(* IEC 61131-3 sources: ml2plc/benchmarks/st (part 6) *)

    weights_3_u : ARRAY[0..4095] OF REAL := [-0.726234972, -0.82971102, 0.359873623, 0.467501462, -0.795098782, 0.642522633, -0.834418893, -0.800529778, 0.752689779, 0.406455636, 0.616274774, 0.617786705, -0.741933465, 0.632032633, -0.739187837, -0.503853142, 0.545782745, 0.567466497, -0.337621212, -0.339030087, -0.389321893, 0.674896181, 0.789721549, -0.746486127, -0.669301271, 0.820195556, 0.72258997, -0.971024632, -0.772712708, 0.568969786, 0.828069806, -0.664833724, -0.332123041, -0.638633251, -0.857070208, -0.492956102, -0.802621424, 0.136594638, -0.361942023, -0.667052031, 0.616791487, 0.744978189, -0.954466581, -0.57189548, 0.74708873, 0.656679034, 0.282293171, 0.660095751, -0.696134508, 0.818064272, 0.902193606, -0.636808872, -0.692610443, 0.638984621, -0.867889166, 0.462693274, -0.667061865, -0.625101268, -0.593671858, -0.351741135, 0.234290212, -0.588220656, -0.595141947, -0.701019764, -0.372747988, -0.607375026, 0.464761764, 0.530245066, -0.573789001, 0.530546367, -0.433061302, -0.461016506, 0.59694773, 0.0462750606, 0.332048684, 0.404971868, -0.498975754, 0.562286198, -0.327837288, -0.52094245, 0.35660404, 0.363930374, -0.340805382, -0.0284396466, -0.445062369, 0.1347083, 0.55759269, -0.618813932, -0.599301457, 0.350034744, 0.372941881, -0.528004527, -0.534632623, 0.234335199, 0.397439361, -0.0195646528, -0.0915857852, -0.0818935558, -0.397882402, -0.0978519842, -0.491226345, -0.166510537, -0.00829036627, -0.282786936, 0.626897216, 0.404613793, -0.491245329, -0.337422758, 0.430924863, 0.278444827, 0.0179173294, 0.231050387, -0.347322822, 0.3725501, 0.48292917, -0.507511616, -0.393044561, 0.602047801, -0.562717617, 0.321077079, -0.230540395, -0.587909281, -0.0499534346, -0.369197726, -0.169617653, -0.41201207, -0.260386378, -0.412834316, -0.803556919, -0.740769684, 0.440442294, 0.568141937, -0.475784481, 0.644459307, -0.596662343, -0.940275252, 0.656770587, 0.322523296, 0.875917017, 0.875438809, -0.816106558, 0.825712204, -0.592998028, -0.347098321, 0.495246083, 0.658055961, -0.403978735, -0.0876639634, -0.502450585, 0.64121145, 0.575357795, -0.643270314, -0.996893167, 0.557650566, 0.867267251, -0.850942194, -0.756620347, 0.329067886, 0.669194162, -0.383174628, -0.0802536532, -0.551262677, -0.718719363, -0.598996222, -0.631955266, -0.0989504158, -0.0885992125, -0.713463306, 0.518353522, 0.730688989, -0.800943017, -0.605422258, 0.701749504, 0.95046109, -0.0751864091, 0.87148875, -0.567332923, 0.663198709, 0.649199545, -0.935164213, -0.753644347, 0.803934813, -0.580185413, 0.378011674, -0.636774302, -0.702305377, -0.344566911, -0.367477775, 0.00891227275, -0.607614458, -0.661959112, -0.687778234, -0.625213504, -0.534323871, 0.356132567, 0.448352844, -0.662155986, 0.502999783, -0.572085738, -0.688427746, 0.490987062, 0.707427204, 0.605727017, 0.829243064, -0.728774309, 0.576677978, -0.878341854, -0.301144749, 0.548745811, 0.666547835, -0.0080199372, -0.474185884, -0.431044191, 0.850138128, 0.552011251, -0.779790699, -0.770057082, 0.645845652, 0.763373435, -0.612323225, -0.813291967, 0.79515928, 0.696035445, -0.785743177, -0.688787401, -0.600066721, -0.71572578, -0.727747619, -0.471354902, 0.656914413, -0.512712061, -0.605490208, 0.525177181, 0.528167665, -0.758861125, -0.702212036, 0.415254414, 0.783526659, 0.741826832, 0.719366014, -0.687756479, 0.683343053, 0.737960219, -0.525721431, -0.455234349, 0.570235014, -0.521014452, 0.321572721, -0.731491745, -0.51282382, -0.718585134, -0.164967939, 0.67603749, -0.509025753, -0.7481004, -0.456257671, -0.669510841, -0.814430475, 0.570815623, 0.526050806, -0.529686749, 0.621858954, -0.670453012, -0.304120302, 0.726401627, -0.0356775187, 0.260329664, 0.624240518, -0.748086572, 0.772515833, -0.125408188, -0.57220155, 0.498111188, 0.0558861159, -0.435518563, 0.303609818, -0.723968267, 0.32118696, 0.692383528, -0.775559604, -0.599537134, 0.294759721, 0.716790199, -0.824359059, -0.780710399, 0.106178224, 0.59846735, -0.206296533, 0.128306508, -0.146541059, -0.224539533, -0.0289100092, -0.765631378, -0.220809624, 0.142412528, -0.384071648, 0.592445076, 0.540259898, -0.638875484, -0.205305457, 0.619496822, 0.442066103, -0.0485938378, 0.466518402, -0.158942863, 0.672467291, 0.807129443, -0.740897119, -0.669203401, 0.666509151, -0.744766951, 0.648471951, -0.381909788, -0.573550165, 0.188253239, -0.540039003, -0.318327606, -0.523213089, -0.323695183, -0.519757688, -0.785824299, -0.818390846, 0.508213222, 0.483413875, -0.783533275, 0.773789883, -0.734820127, -0.79764092, 0.595962107, 0.348774403, 0.728198171, 0.80280596, -0.905285239, 0.696726441, -0.556371629, -0.303590208, 0.505447924, 0.654682875, -0.246009961, -0.223182008, -0.24971877, 0.70417136, 0.801208556, -0.83401686, -0.837068319, 0.727295339, 0.710075676, -0.732324839, -0.919261158, 0.631765366, 0.908012867, -0.489900053, -0.275408089, -0.695942461, -0.762747347, -0.440948963, -0.733398139, 0.183654517, -0.027274197, -0.62028116, 0.811902761, 0.743571997, -1.0051589, -0.525409877, 0.59080416, 0.890070081, 0.162616029, 0.72517395, -0.71613127, 0.769188046, 0.83349818, -0.766713858, -0.669896007, 0.711548209, -0.647645533, 0.33983916, -0.509689867, -0.800435543, -0.344411999, -0.346289754, 0.314366817, -0.663431704, -0.645073771, -0.560695171, -0.580787599, -0.820379198, 0.494530648, 0.398333371, -0.511259377, 0.692627907, -0.654955804, -0.870129108, 0.622329593, 0.41138804, 0.681844473, 0.7009812, -0.699940562, 0.538193107, -0.626960039, -0.446550846, 0.611533403, 0.669651389, -0.173716933, -0.318383664, -0.307127029, 0.626539707, 0.756940067, -0.76652962, -0.840944767, 0.790242732, 0.646067619, -0.767073929, -0.862344623, 0.598574519, 0.593686044, -0.577582955, -0.0423634201, -0.574055374, -0.77169019, -0.707057357, -0.778539598, 0.205691278, -0.00679121865, -0.854793429, 0.703709006, 0.763270438, -1.00914109, -0.775699973, 0.657759905, 0.725754857, 0.0530802906, 0.774340749, -0.833031714, 0.78519094, 0.71297121, -0.876600504, -0.740658998, 0.718503237, -0.687330544, 0.385003448, -0.725991547, -0.754310906, -0.279794812, -0.459310025, 0.188008204, -0.733313024, -0.775156617, -0.419203967, -0.273565292, -0.338725805, 0.221741572, 0.281494081, -0.342794389, 0.295483947, -0.291649103, -0.420268297, 0.387898266, 0.168785974, 0.339827657, 0.513234437, -0.494564533, 0.233384728, -0.230191156, -0.308273941, 0.325547248, 0.405156314, -0.0751813129, -0.066444248, -0.128334582, 0.244734526, 0.429480523, -0.436590225, -0.505181551, 0.468694657, 0.35836184, -0.543859482, -0.418227315, 0.220673606, 0.348470032, -0.428927124, -0.277986884, -0.291793585, -0.206854329, -0.250032306, -0.438212544, 0.218785331, 0.0412712507, -0.282670617, 0.316561878, 0.467533499, -0.459543943, -0.365904897, 0.383837134, 0.291643828, 0.1889994, 0.21689266, -0.294608653, 0.276400536, 0.293337226, -0.420555532, -0.405189395, 0.228911266, -0.250243455, 0.240290195, -0.447692513, -0.475426018, -0.201851323, -0.297056526, 0.137493655, -0.48626101, -0.345898688, -0.396780074, -0.780549526, -0.823537588, 0.542945087, 0.354397655, -0.507387161, 0.698669791, -0.818379283, -0.727007926, 0.678681433, 0.212808281, 0.604210854, 0.803043723, -0.779703319, 0.685046077, -0.663781881, -0.521312237, 0.596160948, 0.652478755, -0.35376817, -0.15544413, -0.422452629, 0.534026861, 0.805908442, -0.847195268, -0.851938188, 0.799646616, 0.857016563, -0.839247882, -0.884811521, 0.510792196, 0.88849473, -0.392984003, -0.261963129, -0.586921692, -0.646880448, -0.462142944, -0.818890929, 0.035946276, -0.281571209, -0.74871695, 0.613813758, 0.680141926, -0.949269414, -0.684969604, 0.565539658, 1.00042653, 0.150313571, 0.684495986, -0.722136557, 0.778911769, 0.782094896, -0.730289161, -0.794239044, 0.885579526, -0.69606334, 0.444901079, -0.845269442, -0.598321259, -0.542192876, -0.288296878, 0.215937302, -0.722411454, -0.702072799, -0.705431938, -0.71226716, -0.786647379, 0.531604886, 0.609665036, -0.597535908, 0.666882694, -0.793303609, -0.787642837, 0.698806942, 0.348492414, 0.540394783, 0.626096666, -0.706491232, 0.829213083, -0.538429081, -0.65759629, 0.687242925, 0.430694371, -0.264121145, -0.216645733, -0.692179024, 0.672817349, 0.805104256, -0.622378051, -0.844789565, 0.451787233, 0.719521761, -0.836445928, -0.842959404, 0.355159968, 0.653186679, -0.37796697, -0.291634262, -0.63452822, -0.671194732, -0.504214764, -0.844722986, 0.306022525, -0.0711536258, -0.702196002, 0.737235725, 0.809727132, -0.613162577, -0.383354962, 0.606713057, 0.591403484, 0.339256108, 0.54715246, -0.473906338, 0.783900678, 0.663366318, -0.75187254, -0.493442833, 0.800020874, -0.789069772, 0.564043283, -0.611755073, -0.86263907, -0.336834759, -0.462656617, 0.237991378, -0.707368851, -0.405766249, -0.630902052, -0.821267247, -0.829749942, 0.509847701, 0.460671842, -0.807606995, 0.74302882, -0.736985207, -0.782585621, 0.754141986, 0.416912496, 0.794934273, 0.86178571, -0.872833729, 0.614410043, -0.788762808, -0.349991858, 0.646541595, 0.541881561, -0.174803972, -0.426443964, -0.381490558, 0.821741939, 0.750299513, -0.836915433, -0.74960041, 0.727819622, 0.92942059, -0.863370955, -0.941732585, 0.573167384, 0.670918107, -0.577338278, -0.318402857, -0.76259917, -0.771713018, -0.665239751, -0.721295357, 0.246406525, -0.497510284, -0.683297992, 0.660865605, 0.732286155, -0.704380989, -0.739708781, 0.889108539, 0.684882641, 0.533998311, 0.649343133, -0.691442072, 0.747027636, 0.723184109, -0.669957519, -0.683325231, 0.681482494, -0.914686978, 0.17408444, -0.640013218, -0.716807425, -0.482498884, -0.154035002, 0.310868859, -0.874958694, -0.748723865, -0.56742239, -0.887781858, -0.652014136, 0.452641785, 0.549586773, -0.645061731, 0.63546443, -0.579267085, -0.748191714, 0.554392397, 0.467173159, 0.758127451, 0.917132854, -0.757915795, 0.769090831, -0.851054728, -0.255667329, 0.637966394, 0.573545754, -0.222050503, -0.438768119, -0.314697772, 0.606786788, 0.856207848, -0.851828158, -0.720914125, 0.806266189, 0.729975462, -0.809783995, -0.858449399, 0.63611263, 0.791059971, -0.416043282, -0.307958245, -0.517980218, -0.714065015, -0.545959234, -0.723166049, 0.29447791, -0.254560858, -0.749505579, 0.825292349, 0.793439567, -0.854955912, -0.56521672, 0.660036385, 0.849229217, 0.315747947, 0.638653874, -0.577628732, 0.616680264, 0.968390405, -0.862338424, -0.541128039, 0.630861163, -0.679648817, 0.262172341, -0.719775438, -0.644159377, -0.345081747, -0.21565415, 0.271060109, -0.728009224, -0.683839321, -0.481576353, -0.570552051, -0.777552724, 0.622478604, 0.579048872, -0.596874118, 0.700840712, -0.657557487, -0.895704746, 0.521527052, 0.291102052, 0.669102132, 0.621534884, -0.792802751, 0.641864598, -0.615286052, -0.564382076, 0.658665776, 0.569696784, -0.29823938, -0.0890338346, -0.522620618, 0.498231977, 0.794570863, -0.825930715, -0.709672213, 0.49634099, 0.715287268, -0.878186584, -0.740223408, 0.342125803, 0.71430409, -0.333702475, -0.176821321, -0.435841233, -0.795084834, -0.508588672, -0.649351716, -0.0135515844, -0.00657207659, -0.628678024, 0.758297741, 0.722372234, -0.989041865, -0.492844343, 0.558204472, 0.986102402, 0.104362853, 0.769734919, -0.783679724, 0.814909697, 0.65221858, -0.909674704, -0.94838649, 0.790295839, -0.832857609, 0.358761221, -0.695959747, -0.763435304, -0.301868916, -0.560335457, -0.073698774, -0.803123415, -0.589908421, -0.699640691, -0.89512831, -0.89859134, 0.456811368, 0.526388049, -0.883316159, 0.668905437, -0.864467144, -0.77936691, 0.668658853, 0.686980963, 0.708051503, 0.897727907, -0.782424867, 0.870139658, -0.710069895, -0.290644497, 0.861719429, 0.686867714, -0.0812829584, -0.515805244, -0.619343758, 0.87452513, 0.647835255, -0.735748649, -0.724878669, 0.730390191, 0.706322849, -0.945946515, -0.875465572, 0.565879285, 0.718600035, -0.742332637, -0.467122614, -0.813044608, -0.77358681, -0.570550144, -0.745883226, 0.471848935, -0.442510426, -0.769583106, 0.646922112, 0.724060833, -1.03937078, -0.738261163, 0.878113747, 0.91464299, 0.451797158, 0.864410758, -0.641917169, 0.683274686, 0.916965365, -0.788966, -0.736622751, 0.830067337, -0.689770639, 0.21498701, -0.684152961, -0.942618608, -0.576527417, -0.366254419, 0.413313627, -0.873114645, -0.718489408, -0.583863616, -0.729837894, -0.627582729, 0.446807176, 0.410488844, -0.707820356, 0.574976921, -0.890346527, -0.6144858, 0.741384029, 0.301623613, 0.731503785, 0.6993469, -0.782861829, 0.707979858, -0.698563576, -0.491824239, 0.807846844, 0.705500066, -0.118933909, -0.514284432, -0.541995108, 0.544251263, 0.638027668, -0.623156488, -0.679441869, 0.760259151, 0.714749157, -0.856507719, -0.740746558, 0.407242507, 0.653954327, -0.48238948, -0.237410322, -0.433872312, -0.78880173, -0.499718726, -0.948717713, 0.38727656, -0.382465541, -0.525140166, 0.694271028, 0.800766528, -0.854491174, -0.519459486, 0.69115299, 0.829451561, 0.367598891, 0.702863634, -0.566851914, 0.780456722, 0.797254324, -0.647499442, -0.79959631, 0.792972267, -0.824902415, 0.502618432, -0.768850267, -0.846130311, -0.492772669, -0.54319489, 0.261164606, -0.788439989, -0.598921239, -0.816673398, -0.778527617, -0.844715834, 0.340323418, 0.428646266, -0.54244858, 0.792509854, -0.643731296, -0.842107594, 0.733490527, 0.408700466, 0.724223852, 0.683781266, -0.885363996, 0.572960675, -0.702454209, -0.350052059, 0.623003006, 0.453214765, -0.112270817, -0.282705426, -0.403194994, 0.685073912, 0.766042054, -0.868627787, -0.765646458, 0.69943887, 0.751629233, -0.739947796, -0.768767118, 0.463029802, 0.651656747, -0.593756258, -0.41636619, -0.488620043, -0.625012338, -0.534433126, -0.712874651, 0.208950907, -0.133826539, -0.598224044, 0.815514505, 0.730447471, -0.830714822, -0.623293459, 0.772215545, 0.647283673, 0.318770945, 0.789138079, -0.700474203, 0.864484668, 0.667024732, -0.678884387, -0.587849855, 0.697911382, -0.829990804, 0.179155171, -0.727644086, -0.696924448, -0.538560808, -0.416034847, 0.502129376, -0.694367468, -0.645184517, -0.723423243, -0.49315697, -0.625419617, 0.38362208, 0.653656721, -0.661024809, 0.622956514, -0.517229497, -0.238649622, 0.600716591, -0.0996971205, 0.362163216, 0.714113176, -0.630294204, 0.537375927, 0.00633827038, -0.446282089, 0.578546643, 0.0746347681, -0.4034895, 0.143355817, -0.42931506, 0.271517873, 0.443827868, -0.597008765, -0.408510149, 0.279152721, 0.637251139, -0.680869997, -0.600134134, 0.105825603, 0.446815252, -0.0732483864, 0.131000474, -0.18368794, -0.113074012, -0.129835978, -0.52116704, -0.341600209, 0.373502314, -0.0196969714, 0.633913875, 0.636404634, -0.549856961, -0.143283263, 0.693931937, 0.384506464, -0.140485421, 0.332994014, -0.210686848, 0.494369686, 0.509069741, -0.465097696, -0.556577265, 0.584524512, -0.634896696, 0.527375817, -0.277327806, -0.727154315, 0.244570479, -0.380336553, -0.229002371, -0.681452513, -0.141134918, -0.518900514, -0.655364513, -0.729059339, 0.458059072, 0.374501973, -0.576015532, 0.421382129, -0.445639879, -0.613623679, 0.323306084, 0.220022663, 0.765763342, 0.710305631, -0.466584563, 0.642416716, -0.566652477, -0.159625024, 0.368171424, 0.560183525, -0.0803456977, -0.244403571, -0.230083123, 0.565429151, 0.444226772, -0.678660274, -0.834407389, 0.453305334, 0.794850767, -0.623285592, -0.748075902, 0.327078044, 0.546659946, -0.332765788, -0.0947347432, -0.348671585, -0.549773335, -0.498938233, -0.791302204, -0.0774794742, -0.111681581, -0.462142825, 0.601308405, 0.524632215, -0.952877581, -0.464764923, 0.449773759, 0.883271515, 0.108514138, 0.694043458, -0.71735549, 0.57161361, 0.592660844, -0.839791715, -0.60587889, 0.749918222, -0.508633018, 0.236129105, -0.743721902, -0.476489544, -0.195013925, -0.282672107, 0.0493622757, -0.517781019, -0.535562217, -0.329918176, -0.847776532, -0.732566774, 0.510883033, 0.623402357, -0.765968084, 0.828452766, -0.703445256, -0.628907382, 0.866131842, 0.509048045, 0.585640192, 0.649587214, -0.69290334, 0.82051605, -0.58204633, -0.753176332, 0.677423954, 0.538980126, -0.343862832, -0.418356091, -0.545816958, 0.605414629, 0.631203949, -0.595712364, -0.771879792, 0.87947458, 0.71730864, -0.630509079, -0.781133711, 0.537814319, 0.850713968, -0.634746552, -0.460097373, -0.737617075, -0.642009556, -0.758920729, -0.581466377, 0.621308506, -0.58778739, -0.690724969, 0.78928262, 0.867532611, -0.669017315, -0.833978355, 0.562109888, 0.721790433, 0.676322162, 0.621345937, -0.854133487, 0.876233518, 0.645316303, -0.745479703, -0.547867, 0.74179703, -0.88884449, 0.478366524, -0.884673536, -0.711467445, -0.470088303, -0.41912964, 0.452502936, -0.781383872, -0.814150214, -0.541235626, -0.710442781, -0.681503534, 0.536275685, 0.384036362, -0.749922991, 0.711969078, -0.740409434, -0.725102127, 0.727339864, 0.341918498, 0.818270028, 0.627205968, -0.632465899, 0.722316206, -0.669062614, -0.375851154, 0.657044291, 0.446246296, -0.219635457, -0.43148765, -0.558377326, 0.569771409, 0.593329668, -0.695811629, -0.849102795, 0.527087867, 0.578450203, -0.888826013, -0.785208881, 0.582609951, 0.618132293, -0.591299593, -0.327320755, -0.447967768, -0.604386806, -0.402412832, -0.758327961, 0.391073734, -0.389803439, -0.66774869, 0.692318916, 0.817701697, -0.829085171, -0.63115406, 0.610895157, 0.692555726, 0.369530261, 0.619796872, -0.578089237, 0.65516305, 0.839975417, -0.714050353, -0.745283663, 0.742054462, -0.830090344, 0.18377535, -0.664344668, -0.776352465, -0.420603633, -0.384506494, 0.312064558, -0.62918669, -0.657724321, -0.738200486, -0.94836539, -0.778746307, 0.483145922, 0.703871608, -0.854615748, 0.926780462, -0.809766114, -0.760736287, 0.686831355, 0.42373687, 0.84679538, 0.906513274, -0.940874815, 0.677461803, -0.703147888, -0.676685631, 0.776708007, 0.517841399, -0.369472772, -0.478993565, -0.632530391, 0.686751187, 0.770708263, -0.658292234, -0.901899755, 0.63416034, 0.723803461, -0.916967928, -0.851831198, 0.582687438, 0.92195642, -0.693708897, -0.417580545, -0.636184752, -0.802806199, -0.494223386, -0.753114402, 0.482324481, -0.390217453, -0.83683461, 0.722103834, 0.941145539, -0.733774066, -0.697950721, 0.84744823, 0.903916419, 0.276334882, 0.747675598, -0.871818721, 0.641804755, 0.958486736, -0.652596593, -0.662544787, 0.954618335, -0.931458354, 0.38261348, -0.618713975, -0.795758426, -0.476883709, -0.321306169, 0.372669131, -0.628606498, -0.773585498, -0.705211937, -0.513652921, -0.564952254, 0.429203838, 0.631790817, -0.424225926, 0.703489482, -0.739444435, -0.327212363, 0.65977639, -0.0436902121, 0.294750094, 0.699085772, -0.498512357, 0.707677662, -0.0511214808, -0.666952133, 0.649589896, 0.0616720095, -0.373967946, 0.316006213, -0.487739474, 0.341629297, 0.508030772, -0.795359671, -0.532108784, 0.133212075, 0.792977333, -0.843702078, -0.695294678, -0.0300426763, 0.527421176, 0.148822859, 0.274006784, 0.132002801, -0.177068904, -0.123832136, -0.813948452, -0.385466427, 0.25638929, -0.201113567, 0.684263825, 0.479077369, -0.674763739, -0.0226189308, 0.537450373, 0.612549424, -0.166918933, 0.320700228, -0.0951954722, 0.679965496, 0.61227119, -0.840546191, -0.634014845, 0.692002535, -0.720923662, 0.471729636, -0.273466438, -0.487667233, 0.221207723, -0.483702719, -0.364673913, -0.528105438, -0.20860064, -0.63447243, -0.864778221, -0.824272394, 0.263325602, 0.499057829, -0.529165149, 0.692652166, -0.723354042, -0.789388597, 0.558536112, 0.540036798, 0.613343656, 0.787046909, -0.741134465, 0.784529388, -0.635947287, -0.409773231, 0.533056259, 0.652541399, -0.0424025841, -0.277122438, -0.57015878, 0.5594275, 0.703241646, -0.675032914, -0.726343215, 0.618670523, 0.695467234, -0.891808033, -0.895254016, 0.585447133, 0.828479052, -0.423756212, -0.361082226, -0.632846653, -0.778389513, -0.574056745, -0.610268235, 0.310293734, -0.219143718, -0.781860769, 0.745597601, 0.836865366, -0.806676924, -0.710307598, 0.765738964, 0.700198293, 0.134091407, 0.606047928, -0.828570783, 0.783700168, 0.885118484, -0.847240925, -0.601313412, 0.667737484, -0.857893348, 0.206913203, -0.656649649, -0.590756834, -0.591427386, -0.167132616, 0.210622162, -0.674396753, -0.735662997, -0.550461888, -0.438653499, -0.484567106, 0.0423764028, 0.402782738, -0.39615652, 0.527801216, -0.405160308, -0.540103197, 0.317408293, 0.758783579, 0.668566465, 0.7315467, -0.478771001, 0.391726941, -0.548839748, -0.151168957, 0.532397807, 0.801022947, 0.0191140678, -0.552368999, -0.369526327, 0.842350483, 0.593827605, -0.494756907, -0.704736352, 0.812934518, 0.552430868, -0.62915194, -0.752106965, 0.56200552, 0.59557122, -0.596497178, -0.491576523, -0.77894181, -0.697859466, -0.540353298, -0.392811835, 0.589950562, -0.50101465, -0.765250444, 0.439478427, 0.486397952, -0.583910704, -0.842351794, 0.298052102, 0.800410271, 0.721171498, 0.577043176, -0.711164594, 0.529448986, 0.579870582, -0.761946082, -0.334211707, 0.426836669, -0.544145286, -0.0236858372, -0.72631222, -0.269898385, -0.546507418, 0.150488898, 0.486382157, -0.541724324, -0.581802309, -0.334866315, -0.60239023, -0.679095268, 0.433860898, 0.470565766, -0.718216181, 0.62314868, -0.704164386, -0.857846975, 0.596488595, 0.312603414, 0.859928668, 0.779130697, -0.86165446, 0.697177708, -0.553644001, -0.406514913, 0.730294526, 0.61478579, -0.251439095, -0.25065136, -0.441192597, 0.799790978, 0.852701426, -0.738498449, -0.6936149, 0.683245599, 0.889102221, -0.760666132, -0.890614629, 0.408153266, 0.693063498, -0.6267699, -0.428469628, -0.436086804, -0.851893008, -0.408915699, -0.692253232, 0.288505495, -0.284870684, -0.728752315, 0.845336199, 0.715213299, -0.94300127, -0.678461432, 0.612001181, 0.698265493, 0.415461838, 0.657033384, -0.831675112, 0.581083179, 0.632179201, -0.819402874, -0.801949084, 0.665694177, -0.723644853, 0.517686546, -0.691868901, -0.683371305, -0.526625633, -0.533140421, 0.305379122, -0.800289869, -0.615729034, -0.727103829, -0.730080843, -0.748888373, 0.515534759, 0.503465474, -0.710360944, 0.838060856, -0.988474727, -0.781527102, 0.7566365, 0.654545665, 0.769656599, 0.813188851, -0.902251959, 0.723203838, -0.624532938, -0.469336659, 0.796414196, 0.521895111, -0.162911385, -0.668885231, -0.52628547, 0.751163602, 0.890729189, -0.839278996, -0.962187886, 0.834596097, 0.762223721, -0.883046627, -1.05751264, 0.684665084, 0.961484551, -0.749053955, -0.341711491, -0.637594283, -0.957236946, -0.551831722, -0.882907093, 0.296203643, -0.431090772, -0.767115414, 0.733907461, 0.938528359, -0.9906919, -0.751880229, 0.84377557, 0.96890384, 0.506706834, 0.656855583, -0.781019568, 0.857784092, 0.918415487, -0.857643902, -0.841950774, 0.787070394, -0.750242233, 0.40217787, -0.849638402, -0.753489494, -0.758095026, -0.606765985, 0.335884303, -0.65856272, -0.808486819, -0.885119617, -0.671191096, -0.675404072, 0.322195232, 0.439209133, -0.442668408, 0.53856045, -0.609920025, -0.924227893, 0.699789643, 0.167366132, 0.90906626, 0.814170897, -0.704245687, 0.716417432, -0.437005758, -0.315517783, 0.643189311, 0.343112886, -0.193849027, 0.0624860041, -0.579222381, 0.521086574, 0.524299681, -0.84888345, -0.956672847, 0.606286645, 0.658358991, -0.964612246, -0.787381589, 0.4372302, 0.825733185, -0.355769753, -0.0480801389, -0.540993035, -0.848746598, -0.410088539, -0.820118845, -0.0829904303, -0.0389961936, -0.661750019, 0.672849178, 0.670697868, -1.06788826, -0.460059553, 0.770552814, 0.940687656, -0.152831227, 0.7278862, -0.698670506, 0.82937777, 0.663784087, -0.84242171, -0.728216648, 0.728243887, -0.673153818, 0.513519049, -0.753371477, -0.562419951, -0.0328404419, -0.560846388, -0.160596967, -0.750968993, -0.493129641, -0.480887413, -0.471878946, -0.570706725, 0.190867126, 0.619297624, -0.657996356, 0.641835988, -0.615748346, -0.727557659, 0.42367655, 0.645834148, 0.564158618, 0.677742243, -0.760552824, 0.562094748, -0.760540366, -0.518487215, 0.581878543, 0.531943381, 0.139630035, -0.56694454, -0.510860264, 0.56850177, 0.45130375, -0.611318827, -0.780234337, 0.677732229, 0.788224757, -0.521191955, -0.696267605, 0.604700446, 0.697250664, -0.558842182, -0.64243567, -0.664067626, -0.567382276, -0.541549802, -0.474666208, 0.383841902, -0.483801514, -0.742288053, 0.706105828, 0.699141741, -0.677887678, -0.724218667, 0.462450176, 0.588963926, 0.647865117, 0.79887259, -0.558031619, 0.72386378, 0.548757076, -0.627694726, -0.449682295, 0.678358495, -0.781508863, 0.34308818, -0.572469234, -0.358995378, -0.657875001, -0.091854915, 0.417881787, -0.64309746, -0.650072634, -0.474960387, -0.807871401, -0.87663269, 0.600731075, 0.540997148, -0.502753854, 0.50888139, -0.656033993, -0.746612072, 0.48891297, 0.265826792, 0.717237949, 0.908482969, -0.633575022, 0.726195335, -0.622035325, -0.438288063, 0.762185693, 0.634955287, -0.34310177, 0.0347639322, -0.351194203, 0.716493368, 0.632564485, -0.630600393, -0.802460313, 0.60208261, 0.898235619, -0.893882751, -0.721909344, 0.53441304, 0.595046163, -0.477534801, -0.00178506097, -0.564549625, -0.836093783, -0.445003271, -0.642233789, -0.102366239, -0.127859131, -0.575787961, 0.552174449, 0.811557174, -0.839536726, -0.513024151, 0.73071909, 1.03467178, 0.0279106591, 0.767786324, -0.663220465, 0.635928929, 0.696484566, -0.909432828, -0.634868801, 0.831269205, -0.811127245, 0.419034213, -0.797002971, -0.720269203, -0.443168491, -0.527125359, 0.078103736, -0.729779184, -0.62820518, -0.514111221, -0.945336878, -0.896292031, 0.628046334, 0.775375545, -0.839837193, 0.991284788, -0.87743324, -0.702488542, 0.801653445, 0.591093957, 0.845495939, 0.995687902, -0.867820919, 1.01508343, -0.592688203, -0.701304674, 0.719586432, 0.5491395, -0.42802316, -0.381718159, -0.723167658, 0.615308344, 0.778011024, -0.982355416, -0.971625388, 0.562777638, 1.04408884, -0.874234378, -0.8119753, 0.475267857, 0.857940078, -0.537086546, -0.357432067, -0.619285464, -0.798609316, -0.472768217, -0.919322491, 0.0175475124, -0.268886387, -0.639463007, 0.971882164, 0.976396561, -0.829320788, -0.662895501, 0.989574671, 0.921676993, 0.285999775, 0.725146711, -0.858463764, 0.864225805, 0.83296448, -0.995106757, -0.909235537, 0.770166218, -1.03288674, 0.830250442, -0.810505748, -0.901980817, -0.35455966, -0.747324765, 0.103498332, -1.01383245, -0.698522568, -0.989441216, -0.875591397, -0.758631289, 0.534163296, 0.593221068, -0.766667783, 0.581122577, -0.680642247, -0.748880625, 0.813236117, 0.420501381, 0.509810269, 0.633358181, -0.721417844, 0.870527506, -0.716211557, -0.643129826, 0.594161093, 0.48839438, -0.380239099, -0.440621912, -0.62062639, 0.536787987, 0.760927856, -0.586608708, -0.759728014, 0.663005352, 0.621978164, -0.739436448, -0.795778632, 0.38639766, 0.865861237, -0.483696818, -0.289453, -0.495639235, -0.718874395, -0.537962198, -0.53384608, 0.151461318, -0.205503523, -0.568728864, 0.866042733, 0.695957661, -0.820673227, -0.581232011, 0.865490794, 0.787113965, 0.371780962, 0.685358405, -0.609164536, 0.741983473, 0.676958382, -0.71614629, -0.689819038, 0.870664418, -0.796582878, 0.421531945, -0.676896632, -0.780096352, -0.479086488, -0.28850174, 0.189821914, -0.569561064, -0.613025904, -0.847247124, -0.753034234, -0.821277082, 0.352717817, 0.437189221, -0.591018021, 0.58764863, -0.836360037, -0.888586044, 0.62162894, 0.591918111, 0.696287513, 0.847621679, -0.901061475, 0.817827344, -0.919304192, -0.302406639, 0.495800436, 0.577167511, -0.294019133, -0.506304026, -0.355751038, 0.810717702, 0.767890096, -0.919171154, -0.83949095, 0.7900666, 0.805035353, -0.773693919, -0.883592606, 0.62864089, 0.692126155, -0.61671406, -0.191977829, -0.642546952, -0.862159908, -0.621910453, -0.652162194, 0.276267111, -0.120133847, -0.741554439, 0.571325481, 0.715305507, -0.94157517, -0.67414248, 0.568462908, 0.840916693, 0.100790963, 0.655533969, -0.888875723, 0.739804924, 0.701006174, -0.979101002, -0.886520743, 0.66766119, -0.816392601, 0.455491394, -0.83178401, -0.57834661, -0.482791305, -0.331682682, 0.252267569, -0.64348048, -0.603320003, -0.503108501, -0.673919201, -0.674786091, 0.321125358, 0.282516241, -0.41301924, 0.49846524, -0.644164741, -0.556176603, 0.414570183, 0.0295571964, 0.532456696, 0.744642496, -0.728139222, 0.638748229, -0.241313726, -0.446577042, 0.373588115, 0.214588135, -0.42782855, 0.23797965, -0.436457992, 0.29760024, 0.471895516, -0.613751709, -0.756712735, 0.247900277, 0.544378281, -0.757288158, -0.742842615, -0.00422132853, 0.727512598, 0.127632841, 0.216005534, 0.00528804818, -0.24746415, -0.042836979, -0.481200725, -0.232504398, 0.312444508, -0.129482701, 0.689032257, 0.538662612, -0.663054168, -0.346863031, 0.631804407, 0.696779668, -0.141457081, 0.54328084, -0.213508695, 0.721033394, 0.469021231, -0.680828452, -0.671968102, 0.426979959, -0.451262534, 0.405148834, -0.477650434, -0.577977121, -0.0180714726, -0.595816553, -0.234744281, -0.677820146, -0.210872546, -0.35164547, -0.752111197, -0.592380166, 0.384332597, 0.38259539, -0.623815179, 0.696658492, -0.568687916, -0.668709636, 0.438631833, 0.0161281209, 0.541475534, 0.812331438, -0.739946544, 0.670636892, -0.569358468, -0.539536774, 0.564501464, 0.410508871, -0.434464753, -0.06972415, -0.520966589, 0.541325152, 0.586624146, -0.600775838, -0.951261282, 0.725977182, 0.881927729, -0.653428972, -0.739407599, 0.505920291, 0.819680393, -0.280781657, 0.0477778353, -0.529438376, -0.519729137, -0.478428662, -0.771895468, -0.115888581, 0.041262541, -0.501470804, 0.754126072, 0.655037463, -0.79851985, -0.617849946, 0.508627951, 0.937227786, 0.0741532892, 0.752697289, -0.638364196, 0.679024935, 0.573970377, -0.784812629, -0.628459752, 0.786691964, -0.724843383, 0.5313223, -0.691406608, -0.75389111, 0.0104060043, -0.52564913, -0.188856304, -0.619440973, -0.435179591, -0.541983306, -0.690828145, -0.742705524, 0.616703749, 0.559063494, -0.721412361, 0.819967091, -0.772261322, -0.781257987, 0.631072998, 0.380338579, 0.878968239, 0.641927123, -0.675080061, 0.797613561, -0.481859565, -0.588425994, 0.635215223, 0.529319406, -0.18409355, -0.104161449, -0.584507048, 0.729360759, 0.677086115, -0.91838634, -0.699541748, 0.733176768, 0.760962009, -0.877713263, -0.714370131, 0.56864804, 0.716714859, -0.351008207, -0.0716526881, -0.416153759, -0.674840271, -0.38810128, -0.85689503, 0.106242314, -0.125452623, -0.578308284, 0.581332147, 0.908393562, -0.947099328, -0.463029057, 0.596999586, 0.669750869, 0.124098182, 0.834454834, -0.625547647, 0.756004095, 0.855139315, -0.944711149, -0.826468945, 0.742309391, -0.644201279, 0.416745484, -0.830237687, -0.879375517, -0.241261527, -0.518852293, 0.208572835, -0.896292627, -0.489128619, -0.791282713, -0.693568945, -0.740639925, 0.372672617, 0.433634013, -0.574363589, 0.647077322, -0.755927563, -0.905629396, 0.704541504, 0.472369015, 0.741631627, 0.888307929, -0.764778197, 0.816288471, -0.639776289, -0.400392085, 0.648703933, 0.462509871, -0.321077108, -0.397640973, -0.265255511, 0.60962826, 0.817197382, -0.608798206, -0.813515663, 0.745844901, 0.767741144, -0.782118082, -0.976574183, 0.521064103, 0.811404645, -0.550130546, -0.200923726, -0.801614046, -0.7105757, -0.534501076, -0.834816158, 0.108991764, -0.284213603, -0.598311722, 0.634516656, 0.662789702, -0.961711645, -0.55547899, 0.689463377, 0.925820708, 0.321004957, 0.651610434, -0.788481355, 0.839279532, 0.896962583, -0.826938093, -0.625647545, 0.783975482, -0.765987933, 0.290778339, -0.697226048, -0.772948563, -0.520532966, -0.302889884, 0.307582259, -0.853788257, -0.661415219, -0.415231556, -0.766534269, -0.880717814, 0.779176176, 0.573440909, -0.80526334, 0.675502658, -0.7605474, -0.908923686, 0.559892893, 0.478005707, 0.702541709, 0.698307514, -0.663857162, 0.71693635, -0.757445753, -0.617220759, 0.647994876, 0.76613915, -0.380599052, -0.476907998, -0.581870794, 0.834186792, 0.627154231, -0.657073915, -0.671102643, 0.841464877, 0.697518826, -0.738666475, -0.81698674, 0.449527919, 0.859983444, -0.57618016, -0.373709887, -0.46734497, -0.819586575, -0.523836017, -0.880162895, 0.242388174, -0.180107474, -0.741554737, 0.631468177, 0.889757693, -0.787249923, -0.486703157, 0.765184164, 0.743254244, 0.429390669, 0.710775793, -0.826795936, 0.700413525, 0.743750095, -0.841565013, -0.796144485, 0.741605341, -0.869812429, 0.636555493, -0.769874454, -0.753798962, -0.390066355, -0.462443918, 0.316380143, -0.839541554, -0.594413042, -0.820055544, -0.386250556, -0.766966522, 0.356104404, 0.458123624, -0.598576725, 0.611094415, -0.385008574, -0.720398903, 0.598801851, 0.609170914, 0.564221084, 0.761261463, -0.569838047, 0.671205938, -0.59444052, -0.273799837, 0.431002319, 0.572460234, 0.0684290826, -0.524966538, -0.33802247, 0.701965511, 0.488980323, -0.526777029, -0.605396628, 0.653136611, 0.723090231, -0.658642232, -0.569547355, 0.67019093, 0.650734484, -0.830076218, -0.439730167, -0.690865159, -0.595351458, -0.777168036, -0.59454143, 0.50659126, -0.472202897, -0.82173121, 0.476545066, 0.708236814, -0.645752132, -0.83805418, 0.645649672, 0.63295567, 0.571810722, 0.601033151, -0.722490191, 0.507057011, 0.666704178, -0.780126572, -0.54492557, 0.49361372, -0.570636034, 0.139321253, -0.648267686, -0.601916194, -0.568152547, 0.00459315116, 0.585618138, -0.604337692, -0.612028778, -0.489147723, -0.673163533, -0.82612592, 0.331939816, 0.503432572, -0.595406413, 0.775024772, -0.601431549, -0.774770617, 0.696077585, 0.491742283, 0.826150775, 0.60972935, -0.617925227, 0.681661546, -0.496898532, -0.407171398, 0.738607049, 0.521275997, -0.164188981, -0.427779019, -0.57765162, 0.497248143, 0.58968693, -0.774330497, -0.724048913, 0.561790466, 0.901737273, -0.811422408, -0.920115411, 0.60594362, 0.844089687, -0.510447741, -0.0845303088, -0.505962789, -0.722236633, -0.588820279, -0.905805886, 0.161147177, -0.0675906166, -0.613443792, 0.805045784, 0.740983009, -0.795017958, -0.657744527, 0.771991968, 0.768809021, 0.0715370178, 0.730388463, -0.757172644, 0.610588789, 0.921177149, -0.660802126, -0.704743028, 0.894296169, -0.776598215, 0.40083468, -0.766098022, -0.631082892, -0.482050449, -0.456523091, 0.204471916, -0.742328823, -0.618026674, -0.582585573, -0.582920492, -0.821842253, 0.319727004, 0.406875104, -0.6655913, 0.455741823, -0.710364878, -0.664153576, 0.508424401, 0.288870007, 0.550063491, 0.808270574, -0.626519382, 0.581452131, -0.569593787, -0.476818293, 0.457556635, 0.445561707, -0.0485610664, -0.24738045, -0.444985181, 0.649168253, 0.600435913, -0.82338953, -0.819419324, 0.621534169, 0.59906435, -0.827731371, -0.725520134, 0.373910338, 0.621072352, -0.55123657, -0.122939125, -0.528970182, -0.661496878, -0.421430945, -0.704984426, 0.136317551, -0.129085422, -0.465678006, 0.711385965, 0.720281601, -0.808288276, -0.476439506, 0.492560297, 0.800636828, 0.0788417608, 0.539779246, -0.795838237, 0.750571787, 0.759191751, -0.687685132, -0.687194109, 0.655379653, -0.739059687, 0.418908745, -0.578194499, -0.621934414, -0.250479013, -0.307500094, 0.276355982, -0.756483793, -0.476955831, -0.580926478, -0.880090296, -0.903894961, 0.526468813, 0.438662648, -0.586907506, 0.774678111, -0.848770678, -0.704209864, 0.764953375, 0.166147113, 0.688481331, 0.632664442, -0.728086412, 0.752528667, -0.55796206, -0.527783811, 0.602526486, 0.365419745, -0.382094741, -0.275969684, -0.543003142, 0.763042033, 0.673357308, -0.731986105, -0.954332829, 0.553861737, 0.776516736, -0.868581176, -0.702298999, 0.566449225, 0.738316536, -0.300097197, -0.0250236187, -0.584532082, -0.83366096, -0.365447819, -0.682086706, 0.0813199356, -0.108937353, -0.510033131, 0.831014156, 0.854750335, -1.01503098, -0.408001602, 0.596535981, 0.956232905, 0.0837642699, 0.824545801, -0.576045811, 0.599528611, 0.737659991, -0.831438065, -0.805607975, 0.676522672, -0.821888208, 0.54248637, -0.770706773, -0.587351501, -0.341309696, -0.550333679, 0.254630625, -0.784025252, -0.434925675, -0.583545804, -0.700247288, -0.623690605, 0.747710407, 0.651148736, -0.629630804, 0.811769664, -0.966323435, -0.811420202, 0.80123955, 0.470187068, 0.941537738, 0.727977037, -0.844709992, 0.78723067, -0.710786164, -0.578857183, 0.682575226, 0.577266693, -0.361889452, -0.41349709, -0.478509456, 0.63676703, 0.808829844, -0.806750596, -0.78288722, 0.738270819, 0.718547761, -0.728419125, -0.906690955, 0.564367294, 0.700948358, -0.680756569, -0.20343551, -0.651196122, -0.70710212, -0.679091752, -0.882806182, 0.201177254, -0.296743393, -0.753044188, 0.663322151, 0.83742255, -0.941375911, -0.575195432, 0.874027967, 0.684853911, 0.138523683, 0.814414501, -0.620623648, 0.827720344, 0.946218967, -0.781000137, -1.07697952, 0.815017819, -0.788599968, 0.502321661, -0.839025795, -0.750845373, -0.573712826, -0.620826781, 0.376246095, -0.650368869, -0.546986699, -0.63691777, -0.535458803, -0.661363959, 0.64222914, 0.445760667, -0.650036573, 0.552645326, -0.524723887, -0.470716357, 0.408812314, -0.0521448217, 0.302379608, 0.754069269, -0.734246969, 0.649500787, -0.14728868, -0.611519575, 0.548350036, 0.180664763, -0.329953641, 0.404439777, -0.46179083, 0.233125389, 0.667019188, -0.667292356, -0.578000605, 0.143258646, 0.561079979, -0.572558224, -0.53526473, -0.0906038955, 0.554567277, 0.0830396116, 0.345211923, 0.0422255769, -0.379443973, -0.0188870002, -0.753450751, -0.27103126, 0.269124418, -0.0796215534, 0.622003257, 0.532311082, -0.766920328, -0.0959044099, 0.416122735, 0.438820273, -0.333582342, 0.313035697, -0.136017337, 0.698964596, 0.491872907, -0.490498453, -0.610670626, 0.61041522, -0.681962848, 0.608779311, -0.297278106, -0.602056086, 0.0237780996, -0.524540901, -0.168225974, -0.601503134, -0.0488869548, -0.614751041, -0.709879696, -0.81053257, 0.618391991, 0.481366783, -0.586239636, 0.48582685, -0.760471582, -0.698308468, 0.743673205, 0.227188304, 0.817469895, 0.748536706, -0.744036376, 0.707273901, -0.468130052, -0.512849033, 0.601515889, 0.481829971, -0.287206113, -0.275168508, -0.35080409, 0.626506507, 0.646277785, -0.783339739, -0.864806712, 0.626492918, 0.712349594, -0.698523939, -0.916393638, 0.532894731, 0.861266494, -0.355742395, -0.180526912, -0.492354751, -0.73325032, -0.52450633, -0.812147796, 0.287403464, -0.0731531456, -0.694485307, 0.76377815, 0.586709619, -0.750046194, -0.631363273, 0.649213135, 0.623009562, 0.316970795, 0.730307519, -0.562623203, 0.680675983, 0.778665662, -0.632263839, -0.766701758, 0.748266935, -0.644944012, 0.483556539, -0.655284286, -0.631178498, -0.288947672, -0.524350405, 0.161109626, -0.751300216, -0.568219364, -0.631061614, -0.459654063, -0.453424454, 0.4379327, 0.246354833, -0.393866688, 0.473403245, -0.224508211, -0.136230782, 0.454040915, 0.0736969262, 0.0650235489, 0.224952474, -0.245984912, 0.263276607, -0.10896042, -0.407990217, 0.373538494, 0.0658154264, -0.202472121, -0.0177803878, -0.376174629, 0.212074891, 0.204538375, -0.389253467, -0.273314506, 0.14198412, 0.442196608, -0.42727685, -0.368806392, 0.0250752289, 0.319224954, -0.0275438055, 0.153941676, -0.128593057, -0.0405203588, -0.00136987807, -0.258995146, -0.129632786, 0.0687909126, -0.178865761, 0.272538632, 0.291231513, -0.438901156, 0.0344174653, 0.234318942, 0.240363508, -0.0146555128, -0.0116621116, -0.152764007, 0.43221733, 0.293311298, -0.371143252, -0.293728679, 0.235918984, -0.391553432, 0.233665392, -0.0871992037, -0.456803441, 0.10449788, -0.356044739, 0.00685795257, -0.384432673, 0.0964239314, -0.377044171, -0.885274708, -0.881318748, 0.253104359, 0.446624637, -0.68234092, 0.765807927, -0.643134177, -0.718705595, 0.599717915, 0.561697781, 0.792307496, 0.936580896, -0.690402985, 0.773174942, -0.745944798, -0.402243197, 0.582286894, 0.654970646, -0.142961577, -0.536586404, -0.349747986, 0.59360075, 0.916892231, -0.862155676, -0.807970583, 0.872830153, 0.995110512, -0.833628416, -0.78662163, 0.503455997, 0.867108881, -0.557180941, -0.245067909, -0.628006876, -0.778172553, -0.509984016, -0.902629256, 0.221031204, -0.410905778, -0.60523653, 0.781412959, 0.710905313, -0.821959317, -0.540201783, 0.886811733, 0.900645852, 0.404937506, 0.868565142, -0.854416847, 0.824203849, 0.960867167, -0.978561938, -0.785064995, 0.911447525, -0.702819347, 0.223130912, -0.829280257, -0.814641654, -0.484858781, -0.269801229, 0.268610418, -0.649877191, -0.747808099, -0.815822065, -0.656320214, -0.815543652, 0.276486754, 0.287251383, -0.579886198, 0.543531537, -0.69070071, -0.550088942, 0.576355577, 0.166552976, 0.545751989, 0.793423891, -0.554714322, 0.671759546, -0.616303027, -0.177101985, 0.416990668, 0.419458419, -0.263717473, -0.386263788, -0.426950902, 0.729058325, 0.717306614, -0.584142983, -0.870174706, 0.662294269, 0.703803718, -0.8443048, -0.807497203, 0.302130997, 0.640786469, -0.328456789, -0.208200663, -0.435652047, -0.798655868, -0.473939508, -0.58023721, 0.108643815, -0.151288792, -0.425067931, 0.54358995, 0.489806861, -0.955569923, -0.523314834, 0.548543096, 0.705176771, 0.269364238, 0.721559882, -0.485653043, 0.738701642, 0.556263268, -0.65787977, -0.59525764, 0.704077065, -0.578215659, 0.406451851, -0.627702355, -0.429527014, -0.364257008, -0.394973516, 0.261529177, -0.649741352, -0.676808894, -0.584805846, -0.629884362, -0.771311998, 0.469886601, 0.661175489, -0.873140037, 0.717514813, -0.739519358, -0.585066617, 0.757585883, 0.374872744, 0.537243068, 0.78802067, -0.637313068, 0.84425354, -0.633909047, -0.645332694, 0.598048151, 0.486647695, -0.390491188, -0.397720188, -0.545434415, 0.514657676, 0.814876378, -0.687656522, -0.646742165, 0.669502914, 0.751603901, -0.918543041, -0.719638765, 0.509990275, 0.652769685, -0.355132073, -0.333902717, -0.650711894, -0.57162106, -0.634329498, -0.857199669, 0.319073766, -0.193643615, -0.664176762, 0.715555668, 0.724739909, -0.88206625, -0.446540654, 0.897243142, 0.653189182, 0.292568058, 0.775917113, -0.535787761, 0.790724456, 0.658093572, -0.880992055, -0.838543773, 0.637600482, -0.809378326, 0.59145391, -0.600317597, -0.659047484, -0.531531334, -0.40995428, 0.377802968, -0.835502625, -0.444133312, -0.715831339, -0.659778833, -0.909406066, 0.34459123, 0.36241433, -0.573488176, 0.676793218, -0.925030172, -0.666074097, 0.750683963, 0.34170568, 0.745981514, 0.661837518, -0.658390462, 0.661465526, -0.844284654, -0.362855017, 0.820108414, 0.573328674, -0.245461404, -0.388630271, -0.492695957, 0.665697277, 0.839606345, -0.945376277, -0.834185362, 0.704771042, 0.984751403, -0.802317083, -0.847898126, 0.512270451, 0.934234083, -0.548366427, -0.196056202, -0.769618511, -0.91448462, -0.586469769, -0.686836421, 0.324442148, -0.226726711, -0.699259937, 0.787815928, 0.77986908, -0.906870186, -0.622646213, 0.664633512, 0.965379953, 0.261142105, 0.739521444, -0.882350028, 0.77965039, 0.866730452, -0.685767531, -0.897825956, 0.885700345, -0.851926386, 0.341880292, -0.788809717, -0.90377146, -0.634577394, -0.18189238, 0.202429622, -0.838257372, -0.587727785, -0.792346656, -0.633845747, -0.631282032, 0.230794728, 0.35575673, -0.635922968, 0.522366881, -0.589991629, -0.824365258, 0.563995719, 0.270632148, 0.520304382, 0.719724059, -0.703722715, 0.76465863, -0.446904123, -0.332921058, 0.617324591, 0.460172296, -0.0889797881, -0.414205134, -0.221735567, 0.722010136, 0.666653395, -0.727845311, -0.6857512, 0.691950381, 0.679212689, -0.729128301, -0.873222232, 0.429747105, 0.632395744, -0.502513945, -0.101058438, -0.613713026, -0.658724427, -0.465612978, -0.710263848, 0.206008941, -0.206594348, -0.643254042, 0.460749328, 0.692132831, -0.723083198, -0.489309937, 0.447513372, 0.885030866, 0.076142408, 0.641402721, -0.516031563, 0.681621075, 0.613610268, -0.655405343, -0.622511804, 0.722302198, -0.58512634, 0.152508721, -0.619448543, -0.672749519, -0.371426702, -0.178846836, 0.37492907, -0.680418432, -0.441070706, -0.510757267, -0.880476117, -0.724268019, 0.34619385, 0.431624055, -0.714189768, 0.486258388, -0.851258337, -0.823630869, 0.649866939, 0.534181118, 0.621223152, 0.763567924, -0.879760146, 0.846098661, -0.704669833, -0.378155023, 0.670836568, 0.726910651, -0.0993666723, -0.348512292, -0.376732111, 0.773108244, 0.582655966, -0.71459043, -1.00996244, 0.590018034, 0.840767682, -0.798443496, -0.759210229, 0.501235783, 0.751499772, -0.490923017, -0.199188262, -0.675305605, -0.689773262, -0.431640506, -0.647069097, 0.341923743, -0.18180503, -0.608682752, 0.557936788, 0.64294225, -1.08424616, -0.781532526, 0.771675706, 0.852573812, 0.121008001, 0.86827153, -0.730012476, 0.685991526, 0.905628443, -0.957201123, -0.886822999, 0.832894027, -0.599573195, 0.327064723, -0.733655334, -0.730279922, -0.53496325, -0.240384325, 0.448531389, -0.614097893, -0.794672966, -0.706376314, -0.74544096, -0.773173034, 0.570546448, 0.427514106, -0.444615722, 0.438615471, -0.742748201, -0.663514256, 0.441997886, 0.223081052, 0.768652141, 0.767352939, -0.82819891, 0.591905892, -0.502386332, -0.232138827, 0.458612621, 0.483412117, -0.339043438, -0.297307998, -0.31513688, 0.685150385, 0.517466128, -0.757387996, -0.79981643, 0.646684349, 0.64423269, -0.863603234, -0.77957648, 0.457524031, 0.581705213, -0.500070035, -2.3287168e-05, -0.416274309, -0.822454572, -0.494968981, -0.724004745, 0.151759654, -0.0470242016, -0.458320737, 0.487453431, 0.58742553, -0.985899448, -0.524392545, 0.619049549, 0.672451138, 0.015001921, 0.548505127, -0.609336197, 0.618811011, 0.609387755, -0.616203606, -0.868938386, 0.648502886, -0.706217647, 0.422117949, -0.607814133, -0.69769448, -0.282395065, -0.329915673, 0.270893067, -0.620717227, -0.434449941, -0.541051507, -0.624369562, -0.558936834, 0.36058712, 0.244339034, -0.509721339, 0.602007687, -0.488616526, -0.82423687, 0.558339775, 0.303887308, 0.681071222, 0.791698992, -0.639396489, 0.540880263, -0.672880232, -0.230734691, 0.612652302, 0.298571467, -0.315639675, -0.207863599, -0.476127803, 0.528039217, 0.636137307, -0.730558574, -0.918804824, 0.500870228, 0.709573925, -0.729761302, -0.659218788, 0.32433477, 0.783052802, -0.398996264, -0.198050335, -0.539138496, -0.606561542, -0.257705718, -0.749406338, -0.010693701, -0.0518695638, -0.626358807, 0.694365501, 0.568448782, -0.773178041, -0.513458908, 0.596947312, 0.637067676, 0.0874893591, 0.553110361, -0.563885927, 0.559856832, 0.688722372, -0.619764328, -0.72137177, 0.548958659, -0.621736526, 0.505205154, -0.535925269, -0.674300134, -0.40449509, -0.399067283, 0.189447448, -0.615793705, -0.604717553, -0.589698255, -0.838647723, -0.752080619, 0.788835049, 0.69460237, -0.737440825, 0.753825486, -0.866874754, -0.553911388, 0.60568279, 0.381400913, 0.799542606, 0.658922553, -0.826175392, 0.763886094, -0.750403881, -0.513383687, 0.743360698, 0.473003924, -0.250108391, -0.416798174, -0.682477057, 0.493673325, 0.894135594, -0.72825706, -0.762408912, 0.562559485, 0.661762416, -0.776120186, -0.684534967, 0.593696475, 0.69683367, -0.48964873, -0.251934528, -0.473286778, -0.553586721, -0.571152627, -0.764987946, 0.285947382, -0.152190328, -0.743868053, 0.636850536, 0.654663205, -0.828935623, -0.457564354, 0.71596992, 0.879196167, 0.17749086, 0.76696682, -0.50241363, 0.749014556, 0.827994943, -0.729129791, -0.730309308, 0.760133088, -0.803988159, 0.462360501, -0.660810411, -0.764885366, -0.571637869, -0.578510582, 0.438658893, -0.750849068, -0.506327748, -0.822021663, -0.714650154, -0.825934231, 0.539240301, 0.631770253, -0.681773484, 0.768352687, -0.684669495, -0.826654851, 0.555521011, 0.298306823, 0.615761995, 0.853095591, -0.768198848, 0.748523414, -0.433759421, -0.60152334, 0.576286256, 0.399834365, -0.356214404, -0.0477745645, -0.466592401, 0.760694146, 0.791846514, -0.755647898, -0.994643748, 0.675257623, 0.823906958, -0.849487364, -1.06035781, 0.467603236, 0.874277651, -0.267676383, -0.0789039806, -0.523667037, -0.837654352, -0.370442241, -0.746147215, -0.193121627, 0.109492853, -0.508127868, 0.706793606, 0.760867774, -0.912249506, -0.614453435, 0.621820748, 1.05616903, 0.0724092796, 0.778449535, -0.600701749, 0.685213864, 0.713173747, -0.947834909, -0.92477721, 0.782118082, -0.910845876, 0.557262957, -0.642096281, -0.901124358, -0.165086895, -0.645973027, 0.0933399722, -0.692308605, -0.448648006, -0.55952388, -0.670140684, -0.905963659, 0.306854993, 0.531633437, -0.750165701, 0.758622468, -0.742368817, -0.650009394, 0.735341311, 0.507363021, 0.553088129, 0.789965332, -0.782577038, 0.722765386, -0.613248527, -0.515472889, 0.760704994, 0.620433271, -0.181457773, -0.292714357, -0.51450026, 0.712335289, 0.832214117, -0.617399156, -0.663556159, 0.709122777, 0.762562096, -0.86058712, -0.972798586, 0.637008429, 0.631769896, -0.386212826, -0.238182008, -0.503032207, -0.731764913, -0.542757154, -0.684528172, 0.145795241, -0.26232785, -0.694706678, 0.654279888, 0.848053336, -0.869346499, -0.627607524, 0.800941706, 0.792691588, 0.164885432, 0.642134964, -0.732307255, 0.851825595, 0.661572695, -0.66988337, -0.766816974, 0.838316202, -0.917763174, 0.210481569, -0.714864135, -0.621068001, -0.369671047, -0.29421562, 0.194236115, -0.648427188, -0.541722834, -0.700538337, -0.609870732, -0.713482261, 0.533526957, 0.505420506, -0.761462092, 0.605680764, -0.736602604, -0.675286412, 0.51925087, 0.31862694, 0.556803346, 0.868467152, -0.661071837, 0.84828496, -0.618372321, -0.331619322, 0.755493104, 0.53644377, -0.376695037, -0.236938447, -0.668599784, 0.671508372, 0.717017174, -0.700174928, -0.876824677, 0.544158936, 0.644148827, -0.691998482, -0.885807157, 0.352006167, 0.70680356, -0.399598837, -0.373940706, -0.555352867, -0.686695516, -0.39205569, -0.804119766, 0.0855121389, -0.205437869, -0.432054162, 0.737186611, 0.873384297, -0.78546083, -0.479268819, 0.852739275, 0.745189786, 0.145215303, 0.592113376, -0.56983906, 0.796408176, 0.626489222, -0.890051663, -0.761890113, 0.804768026, -0.804488063, 0.562567174, -0.607810378, -0.657597065, -0.401996285, -0.353776366, 0.306756914, -0.631820917, -0.519993901, -0.519025266, -0.517664015, -0.691131711, 0.36419484, 0.609319508, -0.437314779, 0.45794186, -0.695542932, -0.202282354, 0.521171153, 0.0124146258, 0.248000398, 0.515286684, -0.462535262, 0.584330499, -0.0601333044, -0.483984798, 0.579564869, -0.00630701752, -0.440996796, 0.221724525, -0.497643888, 0.241753414, 0.429231167, -0.594967127, -0.696366668, 0.21122545, 0.76387006, -0.725295663, -0.682499707, 0.136870936, 0.640352666, 0.0971844271, 0.181079447, -0.093014814, -0.118214674, -0.0885042697, -0.630984008, -0.38630563, 0.343149573, -0.0148162777, 0.457977355, 0.722049475, -0.770289063, -0.171033204, 0.526406705, 0.489453018, -0.127697423, 0.378924906, -0.278416127, 0.67813158, 0.445674479, -0.490538061, -0.587413192, 0.50061655, -0.601593077, 0.658657491, -0.124319792, -0.475965083, 0.11623431, -0.622034311, -0.248465717, -0.683995664, -0.246266603, -0.596609175, -0.596734047, -0.608198345, 0.417361289, 0.346513689, -0.668772399, 0.571508229, -0.553525627, -0.786572993, 0.699519455, 0.47918123, 0.805457294, 0.825717449, -0.587299824, 0.721440732, -0.770340621, -0.458128452, 0.456814826, 0.534690917, -0.0717943162, -0.355185479, -0.490397304, 0.768769026, 0.620793104, -0.702713192, -0.69406867, 0.731720805, 0.685039222, -0.709784985, -0.866937339, 0.600554228, 0.894621968, -0.39824304, -0.373409122, -0.528678238, -0.57516098, -0.451306015, -0.687205434, 0.157774508, -0.212319404, -0.774072707, 0.5095281, 0.78033942, -0.855686426, -0.435578614, 0.479955196, 0.731096566, 0.0855724514, 0.790767193, -0.728350103, 0.576205313, 0.839295089, -0.918894947, -0.518834651, 0.634736121, -0.622217238, 0.191857859, -0.624470174, -0.80250901, -0.496632963, -0.225754946, 0.297484487, -0.741780341, -0.711499035, -0.498131931, -0.770092607, -0.841350377, 0.710871935, 0.60860157, -0.634379983, 0.62338388, -0.786254048, -0.743752658, 0.778513968, 0.380605906, 0.741564929, 0.70950824, -0.632787704, 0.81374234, -0.680804193, -0.592398763, 0.656908572, 0.738384008, -0.337080717, -0.0387269668, -0.671773136, 0.562348604, 0.677132905, -0.871127427, -0.902743757, 0.662843525, 0.642007768, -0.722330868, -0.686625183, 0.543022215, 0.852080941, -0.396655589, -0.234145701, -0.704787552, -0.892564118, -0.563664794, -0.700944304, -0.0499284975, -0.100071982, -0.824975193, 0.785685837, 0.733327806, -0.985789955, -0.494533747, 0.569079041, 0.995475829, 0.0173491687, 0.716639459, -0.597337127, 0.716359913, 0.881419241, -0.705274582, -0.763357162, 0.788009644, -0.671955466, 0.600070059, -0.857818961, -0.832677364, -0.356224716, -0.592254996, 0.16872856, -0.698387325, -0.623712182, -0.604543328, -0.763082504, -0.834628224, 0.306040227, 0.354302883, -0.690976858, 0.498179018, -0.558686435, -0.842178226, 0.438858449, 0.357613653, 0.620885849, 0.764080763, -0.636522174, 0.613910079, -0.523531854, -0.403488576, 0.608101547, 0.396393418, -0.371086329, -0.102414593, -0.344746709, 0.537199318, 0.770033062, -0.823680878, -0.7562536, 0.477918386, 0.816444635, -0.855723262, -0.935863197, 0.25004217, 0.567221284, -0.451333195, -0.189253494, -0.313493073, -0.591894507, -0.536549568, -0.795074642, -0.0487271845, -0.081170328, -0.453078747, 0.655549645, 0.607715666, -0.960428238, -0.330212355, 0.587273061, 0.872655749, -0.066790849, 0.751874685, -0.540155113, 0.666716278, 0.634060979, -0.762022197, -0.850647628, 0.606674075, -0.552743554, 0.432056487, -0.705360293, -0.635362208, -0.265966207, -0.312942952, 0.163740516, -0.781231821, -0.646184325, -0.497765034, -0.594749868, -0.651977241, 0.510962903, 0.48331815, -0.711388707, 0.794482172, -0.634144604, -0.600354552, 0.771782517, 0.279378742, 0.664090395, 0.772180378, -0.86859268, 0.664606512, -0.463581741, -0.459145635, 0.745127141, 0.625650525, -0.388047993, -0.26752314, -0.356980205, 0.603207767, 0.558677435, -0.837008119, -0.860293925, 0.733782053, 0.654158711, -0.948712885, -0.706182182, 0.542136014, 0.795793593, -0.578172207, -0.244856983, -0.551398873, -0.859765828, -0.471795768, -0.957506418, 0.00114870397, -0.14141044, -0.672573149, 0.543505609, 0.854262054, -0.974989355, -0.570677876, 0.592236638, 0.753340125, 0.258676648, 0.774816573, -0.561520278, 0.720794737, 0.861506224, -0.818280399, -0.816248298, 0.660308182, -0.783487797, 0.472559541, -0.567909062, -0.769841135, -0.36992982, -0.44512248, 0.211672798, -0.85831058, -0.564784288, -0.736187398, -0.856575489, -0.688995361, 0.528019369, 0.580864489, -0.717701197, 0.575223446, -0.840357184, -0.644141495, 0.560073078, 0.418458194, 0.813837826, 0.743292391, -0.85651195, 0.694204092, -0.666799128, -0.335520416, 0.796116233, 0.490970165, -0.245439738, -0.314309359, -0.502725542, 0.765975296, 0.652717173, -0.740998805, -0.803605855, 0.834221482, 0.872561216, -0.75937748, -0.92128849, 0.614450514, 0.732889235, -0.589897335, -0.390999287, -0.749984324, -0.617868781, -0.692896664, -0.862923086, 0.263996333, -0.164384902, -0.605936825, 0.638017118, 0.914242387, -0.919540823, -0.641202629, 0.672807336, 0.821525395, 0.146091089, 0.731206298, -0.78296268, 0.688082337, 0.840435922, -0.965001762, -0.908083916, 0.851012588, -0.926303267, 0.385692447, -0.648626029, -0.831952035, -0.507010758, -0.316051006, 0.214994669, -0.90746206, -0.628715456, -0.815836489, -0.741105139, -0.597110569, 0.524019599, 0.573146105, -0.56936115, 0.471742421, -0.512584746, -0.495997608, 0.447572201, -0.0882092565, 0.514143169, 0.578645289, -0.544580996, 0.523378611, -0.346962571, -0.357619643, 0.54893893, 0.158550799, -0.386341751, 0.198253721, -0.508448303, 0.405493885, 0.60287261, -0.553333104, -0.846876681, 0.306857377, 0.784080625, -0.839027166, -0.768278539, 0.38080126, 0.679028571, -0.257493436, 0.00781017542, -0.178098157, -0.550591588, -0.229759976, -0.516107321, -0.101500362, 0.332074463, -0.374716163, 0.481380939, 0.503152072, -0.742745996, -0.411417663, 0.519585848, 0.61863476, -0.272574306, 0.530502439, -0.326629937, 0.633793116, 0.552621722, -0.820581615, -0.661003768, 0.581622362, -0.710823774, 0.636210501, -0.430048436, -0.610860944, 0.161980703, -0.536463141, -0.158715799, -0.59583956, -0.228576854, -0.652957439];
    recurrent_3_u : ARRAY[0..4095] OF REAL := [0.0300211906, -0.0726404935, -0.0737517402, 0.158155724, 0.101881593, 0.0459016934, 0.106127605, 0.0329704545, -0.0344988927, -0.0758979842, -0.0294167735, 0.0405295789, 0.0192210935, 0.113318145, 0.0260757133, -0.0657523498, -0.0224163197, -0.134512767, 0.00873535872, 0.0424721651, 0.103415355, -0.0688372254, 0.084060438, 0.0470905825, 0.0343437381, -0.0326196477, 0.0298775509, -0.0407948419, 0.101322442, 0.0656937957, -0.142149746, 0.015102867, -0.0493602864, -0.0175211914, -0.0303692408, -0.197288126, 0.14125213, 0.0856058896, 0.0221487749, 0.0296264663, -0.0948507115, -0.0278902445, -0.0167066362, -0.0772125348, 0.0345653631, 0.113668807, 0.119799644, 0.109393142, 0.0327464528, -0.112259045, -0.132422939, 0.116845936, -0.0464105122, -0.0504373275, 0.148030668, 0.12590833, 0.0312110968, -0.0305655356, -0.00114641618, -0.00481387228, -0.00148997642, -0.0140454788, -0.043380253, -0.0010807598, -0.014458037, 0.0159579515, -0.0403428823, -0.014772784, 0.0942004994, -0.082610406, -0.0322015435, -0.00887908973, -0.0458164886, 0.0110293124, -0.0739976466, -0.0362581946, 0.0755177662, 0.10764505, -0.100206763, -0.0479895957, -0.111544885, 0.11783307, -0.0622494444, -0.0618790276, -0.126783609, -0.111381091, -0.0407576784, -0.130454913, 0.0215890706, -0.0911371484, -0.0917792618, -0.130048037, -0.0297309868, 0.0877916068, -0.000393094262, -0.0588469468, -0.0297936685, -0.0971366912, 0.0301536247, -0.0722011104, -0.0837551877, -0.0260783099, -0.0586579666, 0.108883359, 0.0492240526, -0.16584681, -0.00450916216, -0.0253114011, -0.142470971, 0.0402365401, 0.0252783075, 0.0431143455, 0.0667134449, -0.10590326, -0.0664104894, 0.019558616, -0.0875182301, 0.033093445, 0.0697155371, 0.137690231, 0.0145864999, 0.0742130131, 0.150406629, -0.048722323, -0.0507028066, -0.0139164925, 0.0272116177, 0.0848037228, 0.103041291, 0.133840501, 0.128629327, 0.114150807, -0.0149933994, 0.136328578, -0.00714633893, 0.0632263646, -0.00389948674, -0.0373136587, -0.0361660421, -0.0706003681, -0.0132233119, 0.102651268, 0.0970900208, 0.0556763969, -0.0266075041, 0.16801855, 0.122122914, -0.0653990805, 0.0837429464, -0.0436800718, -0.0256232154, 0.102124937, 0.0752657056, 0.154713422, 0.0260666274, -0.0506237373, -0.0284463856, 0.0192195773, -0.00573915523, 0.0273115728, -0.00244970806, -0.138179153, -0.151856139, -0.0549204648, 0.0667010546, 0.0133919455, 0.0681342036, 0.083140105, 0.0790066496, 0.101608828, -0.0148200337, -0.0527088344, 0.0216680504, -0.126744986, 0.0727042332, -0.0177761577, -0.0781563297, -0.0114615867, -0.101109624, -0.134685636, 0.0576641485, -0.147509247, -0.0655705184, -0.0140403695, 0.099234961, 0.00335595477, 0.0481827967, 0.00108642969, 0.0677736476, -0.0509829633, -0.0663982257, 0.0251895357, 0.0575018488, 0.0351390764, 0.0143772382, 0.0510687828, 0.128724203, -0.0524879545, 0.0846009701, 0.0215634666, 0.0215874463, -0.0228919853, 0.136334121, -0.0845987946, 0.0723666176, 0.0102376565, 0.00383732724, 0.0103866477, -0.0431142226, 0.124460228, 0.200107276, 0.0479671881, -0.0755812079, 0.0902619064, -0.142843604, -0.0545342304, 0.0527493209, -0.0541797392, -0.0768503621, 0.0616208948, 0.0837951601, 0.00714502344, 0.0858522058, -0.0840131864, 0.0268256329, -0.0438843518, 0.0573481992, 0.0930459574, 0.0372035205, -0.143966675, 0.00481981924, 0.0248197056, 0.0165912248, -0.0476145633, -0.0617588572, -0.0879868492, 0.0660810098, 0.100188769, 0.0131307421, 0.0687118918, 0.02752617, 0.0834473521, -0.0857155919, -0.0603220463, 0.0110164033, -0.0817635432, -0.0143848229, -0.0562525913, 0.104724899, 0.0878890306, -0.0319999419, 0.123851545, 0.089456372, 0.028816184, -0.0516834185, -0.0678242892, -0.000487238081, -0.0662352368, 0.0014590444, -0.0246563964, 0.0686305761, 0.00554418843, 0.0282515567, -0.0481138304, 0.109705061, -0.106394254, -0.0443215072, 0.0999002159, -0.139139235, -0.00928665511, -0.0397253111, 0.0938298702, -0.0839995667, 0.0965257809, 0.0854988843, -0.00975783449, 0.0243535042, 0.0170450639, 0.0159549676, -0.100652389, -0.0341138393, 0.109760039, 0.0544666052, -0.118620828, -0.129411712, 0.125624835, -0.00942844898, 0.0457218885, -0.0322152488, 0.154747665, -0.0719875544, 0.0825248212, 0.0222184435, -0.107487805, 0.0240580626, 0.0342749134, 0.0545804426, 0.118475847, -0.0381727219, -0.0196922328, -0.0122831464, 0.0579704605, -0.102477662, 0.0445675552, -0.0130214822, -0.127181083, 0.0127406744, -0.0519533753, 0.0756189078, -0.0517086349, 0.0865597799, 0.108242944, -0.026486462, 0.0976301357, 0.0297792871, 0.089461118, 0.111656331, 0.11560344, 0.0867624208, -0.100683779, -0.0620547384, -0.00687698228, 0.0556412488, 0.0257217046, -0.12562339, 0.0703864098, 0.00830022153, 0.0186630096, 0.0221271738, 0.00233624596, -0.0128272325, -0.107483052, 0.115353957, 0.0140514653, 0.00380971842, -0.0164475031, 0.0248292983, -0.0229293928, -0.0233162344, -0.0321218781, -0.038253095, -0.0523340404, -0.0502889566, -0.0859642029, -0.0186352953, 0.0504419096, 0.212066144, 0.030847637, -0.0039832443, 0.20387359, 0.0830581039, -0.0162938889, -0.052821219, -0.0775873214, 0.0432782136, 0.00630828878, -0.0598597825, -0.0590133592, -0.0160276555, 0.0762145072, 0.0913062766, -0.0763732195, 0.0536984429, 0.126260594, 0.166124925, 0.0996124595, -0.0353368782, 0.0919128805, -0.0817618892, -0.13060537, -0.0492496602, 0.0797692761, -0.0509658232, 0.0341931991, -0.0244456176, -0.144371673, 0.016945241, 0.0437188074, 0.17513822, 0.161979482, 0.0447574817, 0.0721322522, 0.0259358902, 0.0513263829, -0.00340208528, -0.0856347457, 0.0574826561, -0.0435986854, -0.0393212289, 0.0103515256, 0.0027629137, 0.0590720773, 0.161202669, 0.0285558328, 0.042487599, -0.0245804042, 0.0756384581, -0.0490016155, -0.0437188633, -0.0879897624, 0.0908604413, 0.132594928, -0.0411755107, 0.0144351618, -0.0396872498, -0.0632711202, -0.0996934697, 0.079484418, 0.0767583698, -0.0284296796, -0.0203310624, 0.0465131924, -0.0777078941, 0.0394401476, -0.110213131, -0.0243016966, -0.0619608201, -0.00736968173, 0.0807653293, 0.0781108961, 0.0670029446, 0.0359667651, -0.17489022, 0.106508911, -0.0314920023, -0.0596255064, 0.0357943326, -0.0147969089, -0.0322091728, 0.121625692, 0.0630649924, 0.0156011377, -0.154010162, 0.156323478, 0.0521048158, -0.0744174048, -0.0438708104, -0.0274148509, -0.0384579822, -0.0622124374, -0.0403489545, 0.0828858912, 0.0269311965, 0.0437574945, -0.0243850574, 0.0194006916, 0.0877681375, -0.00616865419, -0.0443016589, -0.151599303, 0.0342801288, 0.1373882, -0.118570536, 0.0311327502, -0.0471654721, 0.0557361841, 0.0510144457, 0.167004779, 0.0370514207, -0.176691324, 0.10364899, 0.175244823, -0.0285309106, 0.0586183444, -0.137841046, -0.0251355357, 0.0926762149, -0.00946547836, 0.0714036003, 0.0133831464, -0.0166843832, 0.104796365, 0.0341226198, 0.0298807379, 0.0892409384, 0.0160754696, -0.0776526034, 0.0406826064, 0.00695893914, 0.00179352146, -0.0359312594, -0.0307491533, 0.0842620283, 0.0597327799, -0.058489684, 0.0652802438, 0.120634273, 0.00839943811, 0.0148034543, 0.0289159715, -0.181493834, -0.0612624437, 0.0701209456, 0.124627896, 0.0699967667, -0.0332627669, -0.00146601256, 0.0155480355, 0.0124639738, 0.101679124, 0.0661147386, 0.0655676425, 0.032507211, -0.00537183508, -0.116009071, -0.0426227786, 0.0338342711, -0.133613735, 0.103789069, 0.0237721466, -0.0146712111, 0.00209892727, 0.0812517703, -0.0960010216, -0.0398812182, 0.0841294602, 0.171301529, -0.0616740137, 0.0314620994, 0.0257012378, 0.138789892, 0.07173419, -0.0192908831, 0.0400421247, -0.0696838275, 0.00150038349, 0.0377930924, -0.113104664, -0.134451911, 0.0513372198, 0.00518697686, -0.00657348242, 0.131591082, 0.142681986, -0.166281387, 0.0281995982, 0.0722631142, 0.0553090014, -0.118525259, 0.0537127964, -0.0449562706, -0.0177839696, 0.0959131941, -0.0462499596, -0.0772643313, 0.235673472, -0.0921119079, -0.0824815929, -0.128127351, 0.0130128087, 0.0265209489, 0.00377602875, 0.133012831, 0.019820774, -0.065849863, 0.0459060445, -0.0681104958, 0.176234603, 0.0335450768, 0.000476682559, -0.134560227, -0.068593353, 0.059597306, 0.061161451, 0.089002952, 0.0547687411, 0.0282784533, -0.0931563526, 0.0148324687, 0.0850364491, -0.0328171328, -0.0634967685, 0.0538393185, -0.097870335, 0.0359249488, -0.0242960434, -0.0517275594, 0.0977952927, 0.0730445832, -0.0189512577, -0.030794397, -0.0424824655, 0.084905915, -0.0634760335, -0.0200301968, -0.0350165367, -0.0351203829, -0.0237792451, -0.0402107127, -0.0557167828, -0.0084409751, -0.015320668, -0.0336955488, 0.0718489289, 0.0624024086, -0.0760541111, -0.0849370658, -0.0865568519, -0.022664452, 0.045539435, 0.019727692, -0.00562720094, 0.00124942325, 0.128961012, 0.0534549765, 0.0855579302, 0.135221332, 0.0438616425, 0.0642335489, 0.0753047913, 0.0217456222, 0.0435579643, 0.0114335567, 0.00198130636, -0.0206198171, 0.0332672745, -0.0287975669, -0.0422020666, -0.0687767342, -0.0427560359, -0.136115283, -0.035427317, -0.0615837239, -0.107946299, -0.0263088681, -0.0157322623, -0.148495913, -0.0870623365, -0.0430138223, -0.0760763884, 0.012971051, -0.0292470958, 0.100048348, -0.019314222, 0.043334052, -0.0361490287, -0.125617921, -0.00180942146, -0.0627233908, 0.0159676187, 0.06812042, 0.115724817, 0.0870643035, 0.089640528, 0.0293276422, -0.0362524278, -0.0057851607, 0.079749383, 0.0676407516, -0.0731888264, -0.0598182678, -0.0336906984, 0.134522706, -0.0538420193, -0.0105081927, -0.0904522911, -0.0529807955, -0.115023464, -0.038046483, 0.0693064481, 0.0703464672, -0.101286009, -0.0829353929, 0.0810176209, 0.0267352816, -0.101998039, -0.0210474525, 0.0896722525, 0.0948957875, 0.0764785707, 0.0969453454, -0.044386968, 0.0178281143, -0.0157930516, 0.0637591705, 0.0534478016, -0.081791535, 0.0674777701, -0.0889050141, -0.0679636002, 0.227865309, 0.0386979356, 0.0846257955, -0.0238306765, 0.06915465, -0.0421275944, -0.0846743137, -0.0721803308, 0.0645987764, 0.0114659499, -0.0156908818, -0.0076075457, -0.0451015644, 0.0247296635, 0.0169328228, 0.101324432, -0.0569279343, 0.0550814345, 0.0642896295, 0.0399167463, -0.112161696, 0.000747356564, 0.0287158061, 0.00583758857, -0.0576586165, -0.177706122, -0.0233383477, 0.0158482641, 0.0426830277, 0.0378117561, -0.0384511724, 0.096626699, -0.0304281991, -0.0344576202, -0.068981126, -0.00999236107, -0.145686835, -0.018794328, 0.0549363159, 0.124868475, -0.0528515503, 0.00542497449, -0.00926763751, 0.00520887785, -0.0385200195, 0.105377898, -0.0153157115, 0.0096886605, 0.00409470033, 0.0240849257, 0.0299824476, 0.160701066, -0.00693662558, 0.110601895, 0.00107865594, -0.0841737986, 0.136813968, -0.0556525066, 0.0395123363, -0.0475255772, -0.00245102565, -0.0300234612, -0.0887759477, 0.0292069353, 0.0324145108, -0.0729678869, -0.144896433, 0.0627085492, 0.121023059, 0.101523846, 0.0460572615, -0.0130476011, -0.00442671869, 0.0776944309, -0.0256401189, -0.0258534029, -0.0875134617, 0.0316531472, 0.0134338001, 0.0183724258, 0.0910221785, -0.0448424555, -0.0671966597, 0.0819778144, -0.0927601233, 0.00420876965, 0.158277199, 0.0418164693, 0.029462399, 0.00131501374, -0.0552261472, -0.0408456959, -0.0457095131, -0.0668665469, 0.0422913805, 0.0386807621, 0.0470974259, -0.0555757433, -0.0114802998, -0.0459007248, 0.074424386, 0.0140240137, 0.0515092053, 0.109739125, -0.0375749506, 0.0098653771, 0.0736354217, -0.122812606, 0.0480498485, -0.0437185392, 0.0702512339, -0.0894126296, -0.0827951878, 0.0436093435, -0.0645922944, 0.0789797977, 0.0291797891, -0.0355316103, 0.101332135, -0.198943242, -0.104029313, -0.0112727433, -0.0789091587, 0.0118773729, -0.000342540676, 0.00273814611, -0.0632523596, -0.0654634759, -0.14086774, 0.136601105, -0.00821176264, -0.05583781, -0.0290638618, -0.0186112896, 0.106708393, -0.00524609815, 0.111985132, 0.0159759019, -0.0196489394, -0.0310848951, 0.0919062495, 0.00128706126, -0.0524096899, -0.0410058796, 0.0994544774, 0.0383059569, 0.001709793, 0.0270505175, -0.0850914195, -0.0341122113, 0.0382801443, 0.0187875647, 0.03861361, -0.0111816321, 0.0419666916, -0.00145811588, -0.0587432943, 0.0371218286, -0.00978743471, -0.0155214313, 0.0722185299, -0.0625950396, -0.051668454, 0.00635217084, -1.98557973e-06, 0.0266079903, 0.0965104178, 0.0593874231, 0.0157394018, 0.0291254073, 0.0470053293, 0.0284078233, 0.0667273998, 0.0530054197, 0.0479614139, -0.0406582095, -0.0848233402, -0.00881057326, -0.0390305854, 0.0470714867, 0.0330141634, 0.00621182565, -0.0400558338, -0.0110622616, 0.0188171957, 0.0332569443, -0.0973213315, 0.0514376462, 0.020230297, 0.00126702804, -0.109365977, -0.0354114696, 0.00999673083, -0.0252558291, -0.0149314767, 0.00663108286, -0.0941324905, 0.0610380322, -0.0831719339, 0.140592024, 0.0717088357, 0.0179549288, 0.0568820946, 0.0589482784, -0.00344366487, 0.0709155127, 0.0246975198, 0.0629138201, 0.0472637042, -0.0260836314, 0.0358886868, -0.0351610072, 0.0206064209, -0.0899197832, 0.0360539705, -0.0156198898, -0.0287199263, -0.0237169545, 0.140227064, -0.0215220582, -0.0155000035, 0.0248110592, -0.0333273523, 0.0362003744, 0.120821871, -0.0120896529, 0.0651367903, -0.104569778, -0.0685840696, -0.0592691414, 0.0800046921, 0.0394370072, 0.0483403578, 0.0630822927, -0.0838180184, 0.0636225641, 0.0329086259, 0.0978200436, 0.0213489477, -0.0855389982, -0.0740655288, 0.0161811933, 0.151725888, -0.0902655944, -0.0280115698, -0.0420006812, -0.0466880724, -0.0898003578, -0.141560018, 0.0149214026, 0.039345447, 0.0207163505, -0.0258197337, 0.0121819992, 0.0104798116, -0.019134406, -0.0742832571, -0.0608402789, 0.00371132605, -0.0716577843, -0.0102680735, -0.0282074492, -0.013085071, 0.00696290471, 0.00381721556, 0.052351106, -0.104948543, -0.00349350553, 0.0223676227, 0.00554437935, 0.0151917338, -0.0154319704, 0.0451491438, -0.0366223976, 0.0613482259, 0.00938831456, 0.12777096, -0.111735135, -0.0348628685, 0.0266387966, -0.0848575756, 0.0460705794, 0.00341442367, 0.0079893088, 0.00728575746, 0.0120959003, -0.103442483, -0.0214767233, -0.0122043844, -0.104347214, 0.0350893177, 0.113822937, -0.00995320454, 0.0689455718, -0.0145815704, -0.0428336859, -0.0286409333, -0.0811021999, 0.125193283, -0.0192737803, 0.0276477393, -0.00993182324, 0.0471581817, 0.0231339596, -0.109355502, -0.117305204, 0.144997433, 0.0151157714, 0.0844534338, -0.0343651734, 0.0428620316, -0.00809036475, -0.0672432184, 0.0611731224, -0.0845748857, 0.0148144085, 0.0099927634, -0.109748997, -0.0800439194, 0.0179431085, 0.0386479609, -0.0328162126, 0.0233447067, 0.000507566147, -0.0540861897, -0.0436197668, 0.136744231, -0.0723383427, 0.120576993, 0.0313198715, 0.0151343495, 0.00956058688, 0.0441376679, -0.0929630175, 0.0826271847, -0.0876522288, 0.0497241579, -0.0532637313, 0.0360197909, -0.120650068, 0.0634097308, -0.0932886973, -0.152571946, 0.0495552868, 0.0512149744, -0.0588000938, 0.00934654661, 0.00886407867, 0.120594025, 0.0621935613, -0.0745492056, -0.00351090031, -0.0503250659, 0.0951018482, 0.0218997821, 0.0429161862, 0.00255380943, -0.192196816, 0.00421994459, 0.0331431404, 0.0209429264, -0.0102446675, 0.065385744, -0.00934347603, -0.0778645501, -0.0742510259, 0.0279874597, 0.00824572891, 0.022834558, 0.0787923485, 0.068176806, -0.142575294, -0.0214019455, 0.0431722999, -0.00839523599, 0.0336834826, -0.0530726165, -0.0890816003, 0.0272959881, -0.0813687444, 0.0251530595, -0.0454012901, -0.0119484328, 0.0687285289, 0.0111977039, 0.042694129, -0.0184652433, 0.0290676206, 0.120775983, 0.0462502204, 0.0458604582, 0.0991594046, -0.0471682623, 0.0169123765, -0.0223320536, 0.0584361143, 0.0313238092, 0.0598582178, 0.0452558696, -0.0473417453, -0.0160958096, -0.0382179171, -0.113199547, 0.0429387018, 0.0126064243, -0.141708672, 0.0561275259, -0.0514974706, 0.0028870441, -0.00186583144, 0.0542809814, -0.133144855, 0.13110131, -0.0619775467, 0.0667550638, 0.00407430343, 0.0933402628, -0.0220654439, -0.0276085194, 0.0261877533, 0.0389356427, 0.0085213501, -0.119906865, 0.0741268024, -0.0328141563, 0.0718610287, 0.0872857198, -0.0447113216, -0.110671438, -0.0578399003, 0.0857168809, -0.03271107, 0.0738816559, 0.108883522, -0.0343707502, -0.00753945531, 0.0515688322, -0.0147661353, -0.0524580479, 0.0608402789, 0.0445684753, 0.0285523068, -0.109277993, 0.070337534, 0.0272401553, 0.0353941433, 0.0222975779, 0.0128672598, -0.00301552005, -0.0973205864, 0.10792546, 0.018098237, 0.104823112, -0.0538132042, 0.141909778, 0.0314420238, -0.0277270172, -0.0402160212, -0.015063649, -0.0499392673, 0.090666987, 0.10393694, -0.0378711149, -0.0596093759, 0.0535159633, -0.130450368, 0.0946984887, -0.0148644941, -0.0580188856, -0.0506390184, 0.0958756357, -0.00710751256, 0.04835172, -0.00110983336, 0.0637535378, -0.0741288438, -0.0353915319, -0.0536486879, 0.0236730259, -0.01360323, -0.0201059133, -0.197702736, 0.0104328562, 0.0219679624, 0.0193600822, -0.0580621734, 0.000722768717, 0.020218214, -0.0416449681, -0.0252169892, 0.0284183025, -0.0408081897, 0.0971229225, -0.0989613086, 0.0676739514, -4.57838178e-05, -0.0325548425, 0.124891654, -0.0249339845, -0.0448648669, -0.0860858411, 0.135519788, -0.0126024559, -0.00650942046, -0.0178682227, 0.0157775246, 0.0321179777, 0.0359329842, -0.154746488, -0.0417040624, 0.0106083816, -0.0687999204, -0.04342594, -0.00977691263, -0.114951603, -0.167931125, 0.130631298, 0.180089399, 0.0460239872, 0.00140842423, -0.0103462273, -0.0837078989, 0.203594267, -0.139691621, -0.0553071611, 0.0519921556, 0.0752987489, -0.02307266, 0.0217926558, 0.0384444743, -0.0378084481, -0.00622680411, -0.0154887512, 0.0137523329, 0.02744684, 0.0529851243, 0.00022099771, -0.0210061241, -0.0213450324, -0.00144641288, -0.0338753499, 0.0976678208, 0.0839371234, 0.00644144183, -0.0212083384, -0.00823141076, 0.00303189107, -0.0606096461, 0.0214796457, -0.0091151977, -0.149327904, -0.0816511363, -0.00109600648, 0.160985664, -0.0915080979, -0.0764324665, -0.0513857156, 0.0188563056, -0.0482605658, 0.0110944454, 0.00537128374, 0.00916528888, 0.111269832, 0.0517503619, -0.00489495322, -0.0374845117, -0.00212028786, -0.0960891694, -0.0880883113, -0.0025981334, 0.0541328788, 0.0289277323, -0.0322767906, -0.0763743296, -0.124166809, 0.0541787446, 0.0224841125, 0.10735859, -0.112267554, 0.0613304041, -0.0375550166, 0.0711611584, 0.0157942362, 0.0914436802, -0.0144078666, -0.0181604102, 0.0121784825, 0.00565243559, -0.0955590308, 0.0696517527, 0.0795066208, -0.00259897113, -0.0420458987, 0.0728832036, -0.0184523873, -0.202795371, -0.0350662023, -0.0611995086, -0.0217991471, 0.0101415236, 0.0153950425, -0.0374389775, 0.0952190459, -0.0143837286, -0.0147394054, 0.0437798947, -0.140954733, -0.0967265069, -0.00696234219, 0.00492353737, -0.0288501102, 0.0016134372, 0.00987270288, 0.0545649603, 0.183393598, 0.0611884519, 0.0782967359, 0.0560247451, 0.0338543355, 0.00486933626, -0.0185989141, -0.127538711, -0.112394586, 0.0266220234, 0.0501661748, -0.238818854, 0.075178951, -0.0953118056, -0.0361153409, 0.0358236432, -0.192152649, -0.091668129, -0.0130089419, -0.00927320961, -0.0107419714, 0.0461085662, 0.0165692661, -0.0513927191, 0.00370220933, 0.0259465929, -0.100428723, 0.0388426632, -0.0524522066, -0.025584789, 0.0589909889, -0.00583225675, 0.0193980969, -0.0032009799, -0.0188045986, 0.0178497285, -0.0385144688, 0.081183672, 0.061315082, 0.0825035498, -0.0108325351, 0.0939969048, 0.118712887, -0.110002652, 0.0159510095, -0.0272368379, 0.0272152591, 0.075575456, 0.0401944853, -0.139272094, 0.0121700456, 0.0693234056, 0.067877762, -0.0503801927, -0.0100093447, -0.0268891584, 0.0517582633, -0.0206706841, -0.035483554, -0.0586260855, -0.0300630294, -0.119854912, -0.0620919578, 0.100395717, 0.113561206, -0.0681952164, -0.112974942, -0.0581537336, -0.00899193622, 0.0414297767, -0.0132136792, -0.027603507, -0.022939615, 0.134260103, 0.134957984, 0.020267915, -0.0543925762, 0.00606182963, -0.0194226392, 0.00143498369, -0.180657759, -0.010997694, -0.0365972891, -0.0676313266, -0.137266397, 0.0148993051, -0.133080408, 0.0260280091, -0.00607299339, -0.0297786333, 0.0242825039, -0.0418978855, 0.0773347393, -0.000944940373, -0.0122882165, 0.134246141, -0.181817785, -0.00448207185, -0.0666503161, -0.000194192515, 0.0506850034, -0.182508036, -0.0106826015, 0.0565887913, -0.163172677, -0.000436317176, 9.17259604e-06, 0.00623785146, -0.213638961, -0.11311245, 0.114885837, 0.136188999, -0.0547634289, -0.0319928341, 0.063556686, -0.0383523665, 0.0233660601, 0.0244582798, 0.0156256612, 0.0102286264, 0.110123917, 0.0108919647, -0.00318586268, -0.0345591418, 0.02237924, 0.0220686905, -0.100356959, -0.0868106857, 0.0951698795, 0.0631417334, 0.0195696782, 0.0197948851, 0.046977967, 0.111540154, -0.0389526747, -0.124880537, 0.0932635069, -0.0240721647, 0.0736240447, -0.0713330284, -0.100934051, -0.0332081206, -0.056899704, 0.0142954942, -0.00425576791, 0.0407140888, 0.0232541263, 0.0660687611, 0.055978965, 0.205581218, -0.0522601232, -0.0177105553, -0.0709572136, 0.042501092, 0.136781737, -0.0591489449, 0.10280785, -0.0286009647, 0.0203699283, 0.0684441179, 0.0151023567, 0.00649720803, -0.011614088, -0.0292001143, -0.145675272, 0.0745430589, -0.0365434624, 0.0497663878, 0.0714009777, 0.0432593264, 0.000566895586, -0.0398042239, 0.0387506709, -0.01325492, 0.00306883641, -0.00806504115, -0.0631631538, -0.0358932018, 0.00865605939, -0.00388304912, 0.0228559636, -0.0118870949, -0.0144958608, 0.173925027, 0.0152818449, 0.0460042655, 0.0929632485, -0.11597693, -0.0457302704, -0.00481079146, 0.00812531728, -0.0175451841, -0.0146273216, -0.0324932411, 0.0914042816, 0.0152572189, -0.0973307192, 0.0300447084, -0.0236581732, -0.00614617858, -0.0062218681, 0.0844372511, -0.0257651359, 0.0486652851, 0.0117939711, 0.0269584842, -0.130671054, -0.0907182097, 0.0558942333, 0.0269881673, 0.0672956035, -0.0295029841, 0.0920254141, 0.00585082732, 0.00767091569, 0.0626625121, -0.0814452693, 0.062444672, -0.064830482, -0.153269723, -0.0444657467, 0.004085619, 0.0561959743, -0.0803028196, 0.0606159419, -0.0403594561, 0.0761666894, 0.0986458734, 0.0105678514, -0.0817268714, -0.0271067526, 0.123596549, 0.00231281528, 0.0176865272, -0.0248383991, 0.115191989, -0.0942414999, -0.0389549807, 0.059627112, -0.0159614347, -0.0179036092, -0.132311836, 0.0365776531, -0.00939529575, 0.0188696757, -0.0315882787, -0.138933256, -0.0103765316, -0.00589833222, -0.0435589291, -0.0838890523, -0.0195166953, -0.00982258283, 0.0193074346, -0.0212550163, 0.0524057858, -0.0268558655, -0.0110593773, -0.0858485326, 0.136565596, -0.0338770412, 0.0230880268, -0.0766331553, 0.0936120376, 0.0894639641, -0.00722966157, 0.0693049431, -0.0281773955, 0.0802517757, 0.0316463821, 0.0451297984, -0.117503449, 0.0870215446, -0.00771393441, 0.109934144, -0.0832953006, 0.058644902, -0.0155102331, 0.131189704, 0.0246528871, 0.0168847498, 0.0417052768, 0.0578640252, 0.12534298, 0.00086741522, 0.0603443943, -0.0755436271, 0.018010933, -0.0159134269, 0.0909223482, 0.105587371, -0.0225883648, -0.018136058, -0.00429809093, 0.0648536384, 0.00792603102, 0.100273214, 0.0426818356, 0.0358592942, -0.019300919, -0.099387452, -0.0207134746, 0.0274422728, -0.106460415, 0.0799673796, 0.00366885494, 0.0256798808, 0.0333483554, 0.0427413732, -0.000553729013, -0.0421616882, -0.0394642055, -0.0127464496, -0.00283724372, -0.0142694162, -0.00163088657, -0.105811559, 0.038578026, -0.111376107, -0.0123410979, 0.000582673354, 0.0306444187, -0.0510375798, -0.0955996513, -0.0337491222, -0.0427375436, 0.0668885112, 0.0387860388, 0.0303316265, 0.0527413785, 0.0891910344, 0.0156252384, -0.0414381102, -0.0514662415, 0.0876697078, 0.143676057, -0.00428622402, 0.131740123, 0.0262013078, -0.0214228537, 0.0162912421, 0.0362434909, 0.0137105649, -0.0189073104, 0.0995535105, -0.0660979897, -0.102600813, 0.0476988591, -0.0180132743, 0.0930725336, 0.0458689667, -0.0532454103, -0.000116987154, 0.0197553188, -0.0316911414, -0.0152121885, -0.0904175863, 0.0844524279, -0.165547609, -0.0619317517, 0.12770927, 0.0103618838, 0.066581279, -0.00753936358, 0.0160168111, -0.082596615, -0.0370407775, -0.0138111124, 0.0578644872, 0.0567265712, -0.00937330443, -0.0208524279, 0.00568321673, 0.0352295525, 0.0316374637, 0.0383372568, -0.00410140678, -0.0159495249, -0.119643256, -0.0967994928, -0.00457899366, -0.0840825886, -0.00609358307, 0.189631119, -0.00772488676, -0.0562163219, 0.116063178, -0.0523985811, -0.00439142808, -0.0318450294, -0.0286335051, -0.102702357, -0.0878510252, -0.0354822725, 0.113764897, -0.03534621, -0.104682565, -0.067143932, -0.018403139, 0.0943159834, -0.0787311271, -0.00701456051, -0.0965824127, 0.119348221, -0.0734687448, 0.0549593791, -0.06867522, 0.0889204815, -0.121300004, 0.0857042074, 0.0114896242, 0.125987515, 0.131136298, 0.0701710731, 0.0439608805, -0.047840327, 0.0277401656, 0.0564279035, 0.0779915899, 0.136212945, 0.00460846862, -0.0677497759, -0.0715289786, 0.0150211751, -0.0407311581, -0.0127222119, -0.042455323, 0.0607895777, 0.173657656, 0.104650997, 0.00195117109, -0.0108929705, 0.00134520046, 0.0316501334, -0.0480045862, 0.0740273222, 0.107059404, -0.0139094181, 0.0933045521, 0.0341952369, -0.110332601, -0.0287618712, -0.0501488298, -0.0959062278, 0.0929894671, 0.0538922958, 0.0178117007, -0.072513625, -0.0560367592, 0.0946408361, -0.0176601652, -0.0623949431, 0.11369361, 0.0758318007, 0.00737708248, -0.0665262491, -0.0557445325, -0.108372115, 0.00145903183, 0.124586642, 0.0352536514, -0.0335065126, -0.0505453572, 0.15350382, 0.102788538, -0.0545426793, -0.0371701829, -0.117617652, -0.0163915269, -0.0635081977, -0.0985327736, -0.0312759466, -0.0946389213, -0.101049721, 0.0435979217, -0.00786320865, 0.0426449627, 0.0169741418, 0.0111421272, 0.0265836753, -0.17795454, 0.0141290557, 0.0903434753, 0.0691457242, -0.0120085133, -0.0327966586, 0.00159727596, 0.0406891368, 0.0370729789, 0.0657485276, 0.10091044, -0.0109258816, 0.0501286685, 0.00371955708, -0.0208817869, -0.0126140974, 0.0867753923, -0.0718555823, -0.0448352732, -0.0100010429, 0.0135794897, 0.0442451313, -0.0854981244, -0.0428287387, 0.0145759936, -0.122173212, 0.0869320706, -0.025685735, -0.056249842, -0.039507661, 0.0238149613, -0.14451392, -0.0123944217, -0.0103876553, -0.0339916646, 0.046212513, -0.0512748808, -0.0487293378, -0.0314902849, -0.0570745468, 0.0528965704, 0.0513674095, 0.0355832055, -0.156722128, -0.0745223165, -0.054123722, 0.07634902, 0.0399962068, 0.0753087252, -0.0408569351, -0.0402079448, 0.0424394347, -0.180192992, 0.0247934405, 0.00698059797, 0.0393613018, -0.0503891483, -0.00118991546, 0.00325610489, 0.0749366581, 0.0247755647, 0.0585099757, 0.0318140201, -0.0235114805, 0.0815698281, -0.00935976766, -0.153780609, 0.143829837, -0.000695410185, -0.0505319089, -0.0805246457, 0.0407051295, -0.0339464992, 0.0287359748, 0.0735844597, 0.0347057283, -0.0256676152, 0.0358682089, 0.0351833589, 0.0243087821, -0.0101794899, -0.070938468, 0.0585412085, 0.0242326297, -0.0373695157, 0.0499537587, 0.0148751428, -0.0247470364, 0.0399893373, 0.00381147163, 0.0228822287, 0.0986248404, -0.0894921198, 0.106893569, -0.119953528, 0.0489409491, -0.0408462174, -0.05191724, -0.0571553521, 0.0414567068, -0.047445152, -0.0349077731, -0.0283654295, 0.0597603917, -0.0224978384, 0.030724559, 0.0843390897, 0.0264454894, 0.0966515765, 0.167522177, -0.111903526, 0.00882041454, 0.113430358, 0.0291332863, -0.0260825232, -0.0793373361, -0.0346951112, 0.0396763645, -0.0837606937, 0.00599098578, -0.0700120628, 0.0362895653, -0.201220602, -0.0652408451, 0.0983557552, -0.0305539519, -0.0905546769, 0.0781318843, -0.092222698, -0.103067264, 0.0987830758, 0.045919463, 0.0908412114, 0.00743933767, -0.000903667882, 0.0673883334, -0.00918021053, -0.0279686786, 0.0120513588, -0.0784084052, 0.0919407234, -0.000809054822, -0.0930619985, 0.00232095132, -0.0435902402, -0.066131644, 0.00156507734, 0.00279734842, -0.00235813973, 0.0383707695, -0.0504254848, 0.00257976586, 0.0383168086, -0.0559064522, -0.0534450486, -0.0758779496, 0.0953854695, 0.132303834, -0.0230809674, -0.0412184075, -0.017347794, -0.0476713926, -0.0258203596, 0.167052031, -0.0768064409, 0.0581221543, 0.0832431465, -0.0756253675, 0.073915869, -0.0277787428, 0.0670492351, -0.126199961, -0.0692963228, 0.0618876591, 0.061215423, 0.0948523879, 0.102515221, 0.0105340537, -0.0490158424, -0.066204682, -0.0114222281, -0.0259333961, 0.0268512424, -0.0240285192, 0.0975229889, 0.0199942347, 0.00509725977, 0.0178026408, -0.110453472, -0.145900846, 0.0381931141, 0.0195362102, -0.0643835962, -0.0124122482, -0.0106626721, 0.0120995101, -0.0803319365, -0.0431276858, -0.0610677041, 0.0589038916, 0.00969081745, -0.0979269892, -0.160353616, 0.00215788186, 0.0276951697, -0.00386547297, -0.0402911752, -0.0883995518, 0.0351082012, 0.00981349126, 0.0510662273, -0.0526945964, -0.0314154886, -0.125641719, -0.0229007266, -0.0723547637, -0.0714586675, -0.218625143, 0.0324526206, -0.00133723952, 0.0972320512, -0.0218060166, -0.0243024211, 0.068929255, -0.0148029383, -0.0295722019, 0.00892486051, 0.0101208016, 0.0139173307, 0.00760096917, -0.0666164532, -0.0561370701, 0.0248976778, 0.0537908785, 0.0947454348, -0.0378669389, -0.129367724, -0.171187624, -0.0988218933, -0.0418063924, 0.117174529, -0.08213377, 0.101846017, -0.0128666349, 0.0666807964, -0.0470159426, 0.000867781462, 0.130794257, 0.0302610211, -0.0359856896, 0.0312333647, -0.0520480908, -0.0232087225, 0.126273811, 0.0212589353, 0.00844010152, 0.0702419132, 0.069330968, 0.140420675, -0.0790618658, 0.0982266888, 0.0279324092, -0.021764446, 0.0403622873, 0.0360463038, 0.0522308312, 0.0263859164, -0.0660897195, -0.0260122716, 0.0587906465, -0.0165068898, 0.0118215568, 0.116144128, 0.0262203328, -0.129264325, 0.0846690685, -0.082121931, -0.0407930762, 0.110639967, -0.0203457363, 0.0497394279, -0.076648578, -0.109537818, -0.0968411043, 0.0174954198, -0.0489697829, -0.000839303248, 0.00780601799, -0.0506865941, -0.0235634819, 0.0124392062, 0.0553957298, -0.0309087858, -0.0106674321, -0.0123102777, 0.0587912202, 0.0771834254, 0.0601142459, -0.0440628566, -0.105514377, -0.0222603045, -0.0444181077, -0.118177205, 0.0587717034, -0.0497949123, 0.057883665, -0.0269314721, -5.55440784e-06, -0.0486246347, -0.0606392771, -0.0122536812, -0.180696011, -0.0932258815, 0.0564828068, 0.0683011413, 0.0668136999, -0.106748983, -0.034203209, 0.0697825253, 0.0776619911, 0.0430945531, -0.0202588513, 0.0135798603, 0.0685243011, 0.0470924824, 0.050038483, 0.0260951351, -0.0188981667, -0.05626598, -0.0308555029, 0.00269413646, 0.0321046747, 0.0673542842, 0.0152772674, 0.000534251332, -0.0957631543, -0.0416444466, -0.0481545255, -0.00117808534, 0.0869539008, 0.00363457063, -0.0844588056, 0.146690086, 0.00341843953, -0.0287580416, -0.131334633, 0.128242806, 0.0793444216, 0.0350410119, -0.122858815, -0.0029347213, 0.0196148157, -0.0958061218, 0.139851466, 0.178974509, 0.0849440545, 0.0649157688, 0.161671922, 0.0135882776, 0.102754846, -0.0809206069, 0.0411005467, 0.00458120648, 0.0303182937, -0.00111264363, 0.0546225011, 0.116480209, 0.0340099819, 0.0191972926, -0.0349055603, 0.0488266423, 0.0599862598, 0.0659702495, -0.0212834459, 0.155259833, -0.0356789827, -0.0589237735, -0.012385048, -0.0444460176, 0.0270156488, -0.0360074714, -0.0231806543, 0.0205656234, -0.0253960565, 0.0225299336, -0.0817852765, -0.0741998404, -0.0744033605, 0.08136262, 0.0998105779, 0.0145104919, 0.13637574, -0.0184606779, 0.112999789, -0.0340401269, 0.0372141972, 0.128838018, -0.0560116619, -0.054176271, 0.0386753529, 0.0168194808, 0.106321022, 0.0782190487, 0.0210235976, -0.109597981, 0.114914745, -0.100452952, 0.00199358165, -0.119633958, 0.0552967116, -0.00784056261, 0.085729368, -0.0139441267, 0.0154473465, 0.0230699964, 0.0630311817, -0.0285764374, 0.0794003531, -0.0662526786, -0.0403759107, -0.0215331204, 0.0585868806, 0.0641366914, -0.0714779049, -0.0516804829, -0.115252681, 0.03934066, 0.0521539487, -0.0521697477, 0.0632954016, 0.0472986735, 0.0540311188, -0.079566434, 0.0109893093, -0.0508477949, 0.0969278961, -0.0280641764, -0.0909949988, -0.0146755213, -0.00297376886, -0.00317909941, 0.0654218569, -0.055034548, -0.0476058871, -0.114990205, 0.0453802086, 0.0516088717, 0.131197974, -0.13477245, 0.0250613429, 0.0154938037, 0.0192972422, -0.00781201199, -0.0932095498, -0.115033433, -0.0839962438, 0.118021339, 0.0362724736, 0.0669088662, -0.0141215641, -0.00995045155, 0.0379489101, -0.0162990056, 0.0602151752, 0.099577032, -0.067778185, 0.0149203511, -0.00255671958, -0.113436691, -0.0915586203, 0.0136897275, 0.0411932655, -0.00953338202, 0.0263220593, -0.0732731596, -0.118662558, 0.0749758258, -0.0214597844, -0.0393433496, 0.0138760433, 0.0184391588, -0.208835825, 0.125120178, 0.0977995098, 0.0527613461, -0.120004192, -0.000734303147, 0.00713940524, -0.0657053888, -0.0646293834, -0.0411789007, -0.0304559097, 0.0198378935, -0.0110937105, 0.0679421574, -0.00985591859, -0.00248605758, -0.043492876, -0.0291730724, -0.0291538015, -0.0849319026, 0.0157827307, 0.0133116934, 0.0607607402, -0.0812886655, -0.0553325936, -0.0242931135, 0.117785767, 0.0170826335, -0.0091655273, 0.0149460379, 0.123396315, -0.0602605939, -0.0471653678, -0.0144482926, -0.0235987809, 0.00425107218, 0.0347998813, -0.025054194, -0.0339833088, -0.0931314826, -0.0289532151, -0.100628607, 0.00409202278, -0.0470786206, 0.0112245418, 0.0831836164, -0.0807382613, 0.0457447581, 0.0371434726, -0.00157180824, 0.0330429412, 0.0785487518, 0.117080823, -0.00489734113, -0.0406062566, 0.0132249352, 0.0562938564, -0.127077758, 0.0887920111, -0.00685449317, 0.139241233, 0.0873695537, -0.100828312, -0.0187399201, 0.115055084, -0.0487159081, -0.0302133579, -0.0768338293, 0.109716788, 0.0370821282, -0.0287049375, 0.0339346826, -0.0768983513, 0.0506638214, -0.0337555222, 0.0354681201, 0.11514692, -0.124518529, 0.0959410667, -0.0218171068, 0.024832489, -0.0312339403, 0.129222929, -0.0300681666, 0.0334382914, -0.0897566751, -0.0120510366, 0.0624336302, 0.0457688347, -0.0506006442, 0.137060016, 0.0133634377, -0.0277635027, -0.0519386791, 0.138215795, -0.0255931355, 0.0637193248, 0.0782612711, 0.043704588, -0.0706363916, -0.0867473483, -0.0280122384, 0.0143328644, -0.185355306, 0.050373856, -0.0229333751, -0.066549696, 0.0259219687, -0.0110726804, -0.0339643508, 0.0199308693, -0.0870389342, 0.0375659764, -0.133983865, -0.0622325093, 0.131928563, 0.0606075227, 0.068603076, -0.150959507, 0.0186037701, 0.0163800921, 0.0321337283, 0.00117886369, 0.000826181844, 0.0113856308, -0.0348047912, -0.0119585209, -0.0290229712, 0.0411998257, 0.0409038179, 0.118324578, 0.0484670438, 0.131134927, -0.047241576, 0.0746052638, -0.0132506397, -0.00523084402, 0.0403868295, -0.0415815935, -0.000496421009, 0.0481602177, 0.02978421, 0.0564897209, -0.0941936523, -0.0705231503, 0.0620953739, 0.0165946558, -0.0201972723, 0.00739394873, 0.0693807825, 0.152135521, 0.0163156874, -0.07376571, -0.149465919, 0.0617062971, -0.0557777435, 0.140250653, 0.0829453617, -0.0322103314, -0.0854051635, 0.0221399292, 0.00541131804, -0.119276442, -0.0918929577, -0.0844398737, 0.0397989228, -0.063847065, -0.054408513, 0.0407775901, -0.0566180088, 0.0307342559, -0.0669313669, 0.0502063967, 0.0694551468, 0.0186264273, 0.141365051, 0.208998054, 0.0882838815, 0.0431206562, -0.106544271, -0.025726106, -0.124994293, -0.108791724, -0.00610821694, 0.0892394409, 0.0467048548, -0.0183123369, -0.0259367432, 0.0793271884, 0.0753387809, -0.01059209, 0.150667146, 0.0324033499, -0.0317094512, 0.0576882437, 0.0694558024, 0.109828189, 0.11538896, 0.085645929, 0.031709671, 0.000370375812, 0.112622947, -0.0891636685, -0.0968724787, -0.144358069, -0.0474674366, 0.00848028064, -0.0375958011, 0.0430304445, 0.00660038553, -0.0156454258, 0.056116946, -0.0557026677, -0.0476781391, 0.0235502943, -0.125562862, -0.0046607703, -0.000461176038, -0.00376228988, -0.00742668286, -0.0267891437, -0.0796516612, -0.0622754246, 0.0241216607, -0.00720124412, -0.0482311323, 0.0269438699, 0.0341051444, -0.00857788976, -0.0618463457, -0.0687971115, 0.0168338753, -0.0437239334, -0.0133013222, -0.126889855, -0.0678971708, -0.0325310044, -0.158968776, -0.0658790767, 0.137922496, 0.159343541, 0.0599740259, -0.0736397728, 0.115832753, 0.00552628655, -0.159536272, -0.108788006, 0.0292282421, 0.0619180948, 0.0232697465, 0.0114452057, 0.00564116426, -0.0352590159, -0.0244480371, 0.120290115, -0.173366487, -0.0393587053, 0.131349578, -0.0242320467, 0.0382967778, -0.0374716818, 0.131232351, 0.00148183596, -0.0862775669, -0.0387868658, 0.0471384004, 0.0219578557, 0.025387682, -0.014806807, -0.0119337738, 0.0113282539, -0.0756373405, 0.0581592396, -0.0075218454, -0.068835184, 0.0475200154, -0.0637260675, 0.193392813, -0.0613547042, -0.00515126996, -0.107052475, 0.11569576, -0.119802773, -0.111610524, 0.0550946966, -0.0737449825, -0.045266822, -0.0353542194, -0.105106704, -0.1943589, 0.0179066919, 0.11703974, -0.0468418822, -0.013253523, 0.0484630913, 0.0434607863, 0.0510577559, -0.0305536259, -0.148791358, 0.0887724161, -0.097481668, 0.0422660895, -0.0535485707, 0.00857671537, -0.0413352959, -0.0438640192, 0.0100388546, 0.0508824401, -0.0646590143, 0.057626307, -0.0195472836, -0.0699712262, 0.115772441, 0.0393819921, -0.0359452814, -0.0358799808, 0.067502439, 0.0392773449, 0.0120418202, -0.177543595, -0.0146268904, -0.0204802621, 0.0016590287, -0.0298607051, -0.0187359713, 0.100402273, 0.115794286, -0.0648050606, 0.138902277, 0.0666446462, 0.0184744634, 0.0240013637, -0.0266780537, 0.0688692182, 0.0461845919, 0.0567253493, -0.0309719369, 0.0898457766, 0.0817998946, -0.0356795192, 0.0649556443, 0.106682301, -0.166588888, -0.00919233076, 0.141001731, 0.0420306027, -0.0658727512, -0.00433288515, 0.0317629911, -0.0550467074, -0.00407661311, -0.0857384354, 0.0598526224, 0.00708718784, 0.0864894912, -0.0628462583, 0.0308408234, -0.000600259751, -0.120377198, -0.0287705027, 0.0112019461, -0.0801755488, 0.0116645917, -0.078481406, 0.0767025799, -0.075545013, -0.140401378, -0.0802578405, -0.120694712, -0.0216989685, -0.0317520089, 0.0420968048, 0.070038408, 0.00442051981, 0.0610248409, 0.139262721, -0.0418416671, 0.050451614, -0.0104785236, 0.0406922102, 0.110013396, -0.0490329191, 0.12251652, 0.00627331156, -0.0276043098, -0.0187224839, 0.0982051641, 0.0293273591, 0.0450135656, -0.0379322655, -0.0112920254, -0.107056648, -0.0681236461, 0.118041284, -0.0493883193, -0.00300544873, -0.0748077631, -0.0504209548, 0.0146083888, 0.0419397876, -0.00454512984, 0.0104878852, -0.187521726, -0.0824201331, 0.0579334982, 0.0474240631, -0.0432562158, -0.0197104309, -0.0446122512, -0.0378362015, -0.00945643149, -0.0539182052, -0.00146937557, -0.111218169, -0.0110235699, 0.0074978359, 0.161174268, -0.0650610924, 0.0904625505, 0.0807929561, 0.0915387943, -0.00764246192, -0.0486331359, 0.0369200967, 0.118042879, -0.00210989453, -0.0401251242, -0.12022458, 0.0929566175, -0.0149899637, 0.0888923258, -0.162864044, 0.098613888, 0.0444668122, 0.00797554664, 0.0253885258, 0.0782689527, -0.0126456572, -0.0217401646, 0.132580444, 0.059950754, -0.00834976509, -0.0496116169, -0.037995778, 0.132465795, 0.0355909914, 0.027968524, 0.0530179814, -0.0166351162, 0.0771531537, 0.0245379992, 0.057781186, 0.0145554598, 0.0339131877, 0.188989908, 0.063147679, -0.025067037, 0.0142894313, 0.0364510752, 0.0422343612, -0.00567561947, 0.0124436766, 0.00300999358, 0.00380477495, 0.0679786354, 0.051919803, -0.0499886312, -0.144870698, 0.139361382, 0.0195103325, -0.0856847316, 0.0278958902, -0.00421368703, 0.00291786436, 0.0304587819, 0.0217464864, -0.0125341946, 0.0506761521, -0.0362862945, -0.0923682898, 0.0533040985, -0.00371540152, 0.000961206853, 0.0589806214, 0.000787030905, -0.131475985, 0.054873541, 0.0949562043, 0.0810329914, -0.0336201787, 0.126859963, 0.15160881, -0.0486177132, 0.0335220993, 0.0558877923, 0.0428225473, -0.0423192233, -0.0434767045, -0.0189460516, -0.107544094, 0.000446313992, 0.00141296652, 0.0334832147, -0.204021677, 0.178792879, -0.0609032884, 0.0193695966, 0.0513797626, -0.0362374894, 0.047803212, 0.0560990237, 0.0023830561, 0.0802260116, -0.0867181197, -0.0223791339, -0.047827974, 0.0230495315, -0.0701122582, 0.183097705, -0.0689380169, 0.105148278, 0.0907316059, 0.0237972438, -0.0149131007, -0.0549703613, 0.137934983, -0.0971860141, 0.0100527536, -0.110943921, -0.0569062233, 0.0577629618, -0.0443707705, 0.175148338, 0.0470523536, 0.0229153782, -0.108078659, 0.0912545621, -0.0411299206, -0.0125831012, -0.014442116, 0.0116702914, 0.0116804931, 0.00841268525, 0.00972991809, -0.0457131639, -0.0640593246, -0.0764123499, -0.0467268825, 0.0948646963, -0.110118203, 0.104310952, -0.0200548321, -0.00133190304, 0.112414286, -0.00887494348, -0.0175741073, 0.0546413921, 0.0407879762, -0.137215406, -0.0960658342, -0.0782571658, -0.0324235559, 0.0907090008, -0.0478524938, 0.030605752, 0.0432760715, 0.0325544327, -0.0496563055, -0.034460105, -0.0536670089, 0.00116366334, 0.061855834, -0.0359185711, -0.114783369, -0.0068679899, 0.0400654972, 0.0265578609, 0.0767074376, -0.072686851, 0.132775396, -0.0462088808, -0.0183823705, 0.00448135519, -0.0202818383, -0.065671809, -0.0463726036, 0.0428554304, 0.0909213647, -0.0419094712, -0.106354974, 0.0316834077, -0.0306691602, -0.0556162484, 0.142710477, 0.0494344719, -0.103703126, -0.059927728, 0.0554858632, -0.120031625, 0.0450445749, 0.0475841835, -0.0595748462, -0.00376545638, 0.0586875342, -0.0307709053, 0.0238728747, 0.0150918737, -0.000204436481, -0.00262482837, -0.0332630686, 0.102440573, 0.0357867703, 0.125794888, -0.112869285, -0.0243463106, 0.101468235, -0.12973693, -0.0667174682, 0.00922841486, 0.0572887175, -0.0303817522, -0.0662079304, 0.066669099, -0.129647031, 0.0546359047, -0.128584623, 0.010580454, 0.0101046814, -0.0312611423, 0.0791293904, -0.0426313728, -0.0680926144, 0.0335913859, 0.0148151731, -0.00421966705, -0.0111462269, -0.0224630907, -0.000497120433, 0.0246174708, 0.0833309144, -0.129092276, 0.0678693354, -0.131356567, 0.0588797405, 0.00920473225, 0.0612161979, -0.0848389193, -0.0071021202, 0.080742918, 0.0552304089, -0.0345649272, -0.00250155292, 0.0574286059, -0.0959362164, -0.135212213, 0.00283145555, -0.0284595434, 0.0140521834, 0.0576984659, 0.0464126095, 0.063174352, 0.040335957, -0.118675485, 0.135154814, 0.0202042088, 0.0609128438, -0.135530487, -0.0496266671, 0.00842737779, 0.107638665, -0.0529136173, -0.065190509, 0.0396431759, 0.0686914623, -0.131918639, 0.103470311, -0.016866155, 0.0228836238, -0.180925727, 0.0224847198, 0.0532157496, 0.172246039, 0.0417397097, 0.00659351051, -0.00833398104, -0.027996242, 0.0823713541, -0.0462665185, 0.00943694916, 0.0314624496, -0.0479518138, 0.0495952778, 0.0898738652, 0.00436242763, 0.0604423732, -0.0349833779, 0.0444733836, 0.0104675815, 0.0487625673, 0.0547988042, 0.122417681, -0.103307828, 0.0407392383, -0.0402793512, -0.0260798652, 0.0149922073, 0.0195754189, -0.05040773, -0.0902734175, 0.00871187635, -0.00195848197, 0.0102583338, -0.0978202, -0.0685906112, -0.139993802, -0.0051469449, -0.100025199, 0.00589732686, -0.0337264985, 0.215451062, -0.0984086841, -0.00606664969, 0.0359480307, 0.0565156266, 0.105717048, 0.0267035998, -0.0242278166, -0.00569936121, -0.0918593109, -0.0523912534, -0.0822795704, 0.113297582, 0.014958689, 0.0333733894, 0.117265664, 0.0192012917, -0.0707047284, -0.105211809, -0.0132810213, -0.071634531, -0.0505304076, 0.0251308717, -0.11762315, 0.030193273, 0.00410067569, 0.0369552188, -0.031379018, -0.0473172627, -0.0846178234, -0.0176126845, 0.0762565881, -0.0263493359, 0.0386259109, 0.00295338058, -0.0766040608, -0.0461957157, 0.085407868, -0.0253898911, 0.0454309508, 0.0543058626, 0.15222469, -0.0694000125, -0.150859237, 0.0406388752, 0.0129035041, -0.0507414937, 0.0925635695, 0.0131557621, 0.00173948146, 0.0527211428, 0.0082938252, -0.0199036524, 0.0526379533, -0.0866013691, -0.0417134427, 0.040677879, -0.0628831312, 0.082594268, 0.0365447104, -0.0956738889, 0.014216762, 0.0195986778, -0.0878263563, -0.0386111587, -0.0719939172, -0.0631440058, 0.161196768, -0.0623713508, 0.0674361512, -0.0172760263, -0.117272392, 0.0254153721, -0.189543292, 0.0338623449, -0.0333566591, -0.0785432607, -0.0825426802, 0.0212335829, -0.00181452557, 0.0224282667, -0.0112977102, -0.0815744847, -0.078524895, -0.0774800107, -2.10814178e-05, 0.0677622408, 0.0377039611, 0.043813847, -0.0690885931, 0.0389433466, -0.209852159, -0.00648564193, 0.016548641, -0.0730931088, 0.0825504363, -0.0176654309, 0.0567998029, -0.051393047, 0.0608661249, 0.0974092633, -0.0341625921, 0.0777445063, 0.0798430741, 0.0532468259, -0.066051513, 0.0264353119, 0.163517594, -0.0298399553, -0.0835821703, 0.0212889966, 0.0603696071, -0.0551470481, -0.0349132493, -0.073651202, 0.0817477852, -0.0104334783, -0.0674619302, 0.0600917898, 0.0395211875, -0.0919675902, 0.0394610986, 0.0600610226, -0.0318777189, 0.124784738, 0.0569640696, -0.089247331, -0.0424785838, 0.0129063651, 0.0959335864, -0.105632305, -0.0349580944, 0.124290213, 0.00742910523, -0.0856474265, -0.0649904013, 0.0538651571, 0.102797888, -0.0986762345, 0.0703774765, -0.0206485633, 0.0402970538, 0.0192304533, -0.00283538736, -0.056690678, -0.0873244852, -0.055459749, -0.00415593386, -0.0918343961, -0.0803622529, 0.108468682, -0.157544032, 0.0120868664, 0.0939099938, 0.132997841, -0.00674599037, -0.0179110896, 0.129941925, -0.0587300844, 0.0247610286, 0.0774628744, 0.0160910618, -0.0476965532, -0.102211349, -0.0750115514, -0.00666426728, 0.0836928189, -0.0767372474, 0.00125703483, 0.0226993021, 0.0866479278, -0.0185180958, 0.0609958544, -0.00676918775, 0.00245276652, 0.104882963, -0.0618118271, 0.0347103737, 0.0706075057, 0.0598387346, -0.0084846206, -0.0362102054, -0.108916335, 0.0123542259, -0.0172353536, -0.0278785471, -0.163362816, -0.0573998764, -0.085427314, -0.11744605, -0.103283063, -0.0401511155, -0.0180830099, 0.0555042364, 0.115041502, -0.0738493353, -0.00529451668, -0.00972217508, -0.0345094875, -0.0759169757, 0.103236079, -0.00818775874, -0.067956008, 0.0146953929, 0.13305375, -0.0778180435, 0.0579100139, -0.00344126951, -0.119493879, -0.0432206392, -0.0199865401, 0.0835982263, -0.00647525303, -0.0163019374, -0.0838292018, -0.00633716583, -0.0312179942, -0.0265295058, 0.0268367082, 0.115729399, 0.0971110016, -0.00338013656, 0.0156162735, -0.0879468098, -0.0433894545, 0.0345592611, 0.0536117218, -0.0351378322, 0.0382302962, 0.0127161127, -0.00957513787, 0.11938367, -0.0673539117, -0.0369861275, 0.0134010594, 0.0141588133, 0.105023503, 0.0664163977, 0.029922653, -0.117293611, 0.039896138, -0.0773853213, -0.0897473469, -0.0697960109, 0.0581272244, -0.107994184, -0.0148722082, 0.0915718973, -0.0251923297, -0.0658146143, -0.000552773476, -0.0682300031, -0.144395769, 0.0585696325, 0.0236287657, -0.0936093181, 0.00539004151, 0.0615960807, 0.0584734455, 0.00777017325, 0.0802931711, -0.106316745, -0.0129972901, 0.0404598229, -0.0114201587, -0.0783428848, -0.100179978, -0.0737028867, -0.0314852335, 0.00265409378, 0.0352568403, 0.094788298, -0.0325277448, -0.0307070017, -0.068057254, -0.00465865992, -0.0122316107, -0.0948953703, 0.208852217, 0.0282319412, -0.0256948993, -0.0362353139, -0.00716653233, -0.0289362669, 0.168159798, -0.0553451665, 0.0347298011, -0.0679618493, -0.0605969317, -0.0318555869, -0.0855532736, 0.0666620955, -0.119269513, 0.0350951627, 0.142051041, 0.0425311662, -0.0091514783, 0.0184900872, -0.0630475134, 0.133693263, 0.00296160299, 0.0309478026, 0.0415407345, 0.170553029, -0.0490989387, -0.135096058, 0.126458749, 0.0118405139, -0.0247989483, 0.00372360437, -0.023267014, 0.0483793914, 0.0218263846, 0.00648327172, -0.104708791, -0.0632834136, -0.0144017916, 0.038995266, -0.0494858362, 0.118353747, -0.00793843158, 0.0208233427, -0.08309789, -0.0353376158, 0.0120601878, -0.161479384, -0.0884625912, 0.0657360554, -0.0234829895, -0.0697832555, -0.0651538819, -0.056885317, -0.109124765, 0.0493674688, -0.00817315932, 0.0100291241, -0.0481616072, 0.000424249098, 0.0191879421, 0.0442795306, 0.0166311134, -0.118633807, 0.0365566425, 0.0225939676, -0.00260969903, 0.114157684, 0.0262636915, -0.0418700352, -0.083099097, -0.0560676157, -0.119343206, 0.0361770205, -0.116154544, -0.13569513, -0.0284458604, -0.025453655, -0.0674404427, 0.017628219, -0.0759436861, -0.0249355529, 0.0292041786, -0.0493779406, -0.0167716984, 0.108655222, 0.0311130378, 0.0179302357, -0.135022163, -0.0417784788, -0.0570391379, -0.135354355, 0.0101753296, -0.00823653676, 0.118374012, -0.057753209, 0.0182850026, 0.0976908654, -0.0130774835, -0.0517067276, -0.0648995489, 0.0260742195, 0.0781308338, 0.0817104727, -0.00144365057, -0.00840477273, -0.0647739768, -0.0124128386, 0.123619005, 0.00500325579, 0.126719385, -0.0177009441, -0.0213475171, -0.0480079725, -0.0449275188, -0.0113018146, 0.00201481557, -0.139193699, -0.0132091753, -0.0924841762, -0.0141410977, 0.0912420899, 0.0638051257, 0.0620417744, -0.0886238888, 0.0261636358, -0.189361647, -0.077522859, -0.113367982, 0.19848153, 0.0629237592, -0.0115735661, 0.0534239337, 0.0523569807, 0.0614056997, 0.017402282, -0.0137614813, 0.128127381, -0.0507759713, -0.0122432224, -0.137505561, -0.0140329935, 0.175129205, -0.0474996269, -0.0126683433, 0.0954533815, 0.0182087515, 0.102476642, -0.00505503453, 0.0445043184, 0.0157436822, -0.000684835017, -0.0446982607, -0.0160516407, -0.0268566143, -0.034871392, -0.0723624006, 0.0276829042, -0.106894553, 0.0297245849, 0.148517668, 0.0306119043, 0.024480788, 0.057873264, -0.0542904139, -0.0187257193, -0.0268429592, 0.0347781479, 0.182711676, 0.0387707427, -0.0413666219, -0.0304399971, -0.0249730311, -0.0115301311, -0.0225001946, -0.0538630486, -0.0358827002, 0.153448954, -0.016551502, -0.0279785749, -0.0211092904, 0.0145989303, 0.114712067, -0.0959315822, -0.0200077035, -0.00496096537, 0.0531129092, -0.00461301208, -0.092136547, -0.019290518, -0.0976062939, 0.0286135897, 0.136693239, 0.0312552676, 0.117106304, -0.122289285, -0.0588494167, 0.0291798022, 0.0087381117, 0.0761296526, 0.0589485057, 0.161292061, -0.0534005016, -0.0545016713, -0.0542927757, 0.0473307259, -0.026263196, -0.0648127347, -0.0510592088, 0.122262836, 0.0621393174, -0.00620839931, 0.120539084, 0.143868059, 0.00991750322, -0.00703470968, -0.133466795, -0.0672097951, -0.0992771462, 0.0398608893, 0.0112410393, -0.0732283741, 0.0225866288, -0.0965754241, 0.0600055791, -0.0412300713, 0.0300039612, -0.147102296, 0.145886332, 0.0533294939, -0.087719366, -0.11787077, 0.122798428, -0.0632750094, -0.0133608114, 0.0397222638, -0.120839655, 0.0279717967, -0.0290077776, 0.0442973301, -0.0888298824, 0.0969517604, -0.0830697343, 0.0314744674, -0.0240058973, -0.0318419263, -0.0793337822, -0.145824462, -0.0259806756, -0.056130074, -0.00145428069, 0.0159080252, -0.0695925355, 0.0958659872, 0.067442283, 0.0224857777, -0.0833125859, 0.0308842678, -0.0480967164, 0.253588706, 0.00488279015, 0.00748084858, 0.010573877, 0.105883926, 0.0911075398, -0.0282798465, -0.0420237556, 0.0919920504, 0.0166334547, -0.0042803511, 0.0474388972, -0.0794579312, -0.12708059, 0.0714929402, -0.116839588, 0.0495442934, -0.115805045, -0.0915021449, 0.0321426913, 0.00533871911, -0.149284571, 0.105603233, -0.159845412, -0.0764946789, -0.0513117686, -0.0528372861, 0.0752885342, 0.155340552, 0.00743776234, 0.0421962626, -0.120706692, -0.0271855444, 0.0263345502, -0.0189696793, -0.0801173896, 0.03058137, 0.0575154275, -0.0212100595, 0.0674094707, -0.0577037409, 0.0451060459, 0.00919431448, -0.101748303, -0.127133489, 0.00121978298, -0.0936859027, 0.144394696, 0.0653232187, -0.0212536044, 0.16899395, -0.000152459368, -0.0977137461, 0.0033859238, -0.117419414, -0.0493396297, -0.035705924, -0.024119677, 0.0573134907, 0.0069703497, 0.0261702631, -0.116585165, 0.00808379799, -0.146062806, 0.0126314852, 0.0150787905, -0.132542253, 0.0098644346, -0.0288225487, -0.010356755, 0.0386339724, 0.0684816912, -0.0271345451, -0.0483281352, -0.0399376117, -0.0557099693, -0.100194566, -0.102490455, -0.0575878583, -0.0679349005, 0.0249807127, -0.0806581378, -0.00437785126, -0.0550510548, -0.0687842146, 0.0311038904, -0.00495552784, 0.00638894085, 0.0355049297, -0.0132802539, -0.0234391242, -0.0858439803, 0.0587111451, -0.0252123624, -0.0960020944, -0.0448848084, -0.0496538766, -0.00416004006, 0.016414592, 0.0572075024, 0.0184295736, -0.0296163149, -0.026117295, -0.039015539, -0.137685612, 0.0715054572, -0.0219773948, -0.0229666159, -0.0302200988, 0.0363391303, 0.109770469, -0.0656398833, 0.0457481146, 0.094116956, -0.0773075968, -0.0314593501, -0.159501195, -0.110025816, -0.0458520651, 0.0304925535, 0.0181574859, -0.0170991682, -0.146890998, 0.0161250383, -0.204725102, 0.0404614955, 0.00172442512, -0.0773060024, 0.0338327289, -0.111908913, 0.0843269378, 0.0417656079, 0.0236102529, -0.0767799839, -0.0120361708, -0.0634715706, 0.00617155805, 0.0768341199, 0.15493007, 0.00329212658, 0.029349409, 0.125606447, 0.0361124091, -0.0804133043, -0.137538493, -0.0659092069, 0.0318373069, -0.160256818, -0.0132932011, -0.11344295, 0.0680131912, -0.0408285931, 0.0277636871, 0.0435267016, 0.0119331479, -0.0301122367, -0.0860860273, -0.0477272347, 0.0555923842, 0.0643539429, 0.0257913917, 0.0240713283, 0.148189276, -0.0128130158, -0.120931864, 0.094560191, 0.0486292243, 0.0279901735, 0.0159090422, -0.109461352, -0.00390604138, -0.015810281, -0.0487371013, -0.0140297767, -0.000135540962, 0.0851485655, -0.0680190176, 0.118419319, 0.0645026565, 0.0795653462, -0.0313418992, -0.0489860103, 0.0370845869, 0.0840737447, 0.00726946816, -0.0644930378, -0.0160436202, -0.0734778047, -0.218570292, -0.136610791, -0.0216169842, 0.135029256, -0.00319907814, -0.0150682442, 0.117365927, 0.0704264194, -0.0719463676, 0.0415127277, -0.0872843713, -0.0254714675, -0.0133848153, 0.0679500997, 0.0415262394, 0.0900941938, 0.0285563879, -0.00156569388, -0.0411640517, -0.0303782597, 0.000205819029, 0.00295572542, 0.0670176148, -0.137253135, -0.00285264291, -0.021808045, 0.0313622952, 0.0469728671, -0.0205262154, 0.00927074254, -0.0372303762, -0.0103757288, -0.0714906454, -0.157990828, 0.0343606398, 0.0954145193, 0.123222455, 0.0823525265, 0.117442392, 0.0234946515, -0.00873712823, -0.00445685443, 0.0669916421, -0.0227660593, -0.0154639501, 0.0184325259, -0.0205302611, 0.135972634, -0.06449496, 0.00152645307, -0.0575076118, 0.0527576469, -0.105739474, -0.187588841, 0.0853657201, 0.0738194585, -0.18257232, 0.00380814308, 0.0113347061, -0.0144741945, 0.0401724204, 0.0282401312, -0.0107867429, -0.0162548311, 0.155527055, 0.0126220174, -0.0744252354, -0.0558582246, -0.180569381, -0.123541631, 0.126075476, -0.13872765, 0.0357238427, 0.0408113226, 0.0505880788, -0.00524656894, 0.121458866, 0.228833333, -0.0176178459, -0.0455273241, -0.13362968, 0.109332412, -0.0374373719, -0.00115054101, 0.0354806446, -0.0877593532, 0.139906853, -0.0553748682, -0.0612836853, -0.0690333545, -0.120751485, -0.0274280068, -0.134869367, 0.130242035, 0.109948143, 0.0753683746, 0.0777142346, -0.037511088, 0.0469326377, 0.00097156316, 0.0486398265, 0.00589081924, 0.0846952945, 0.206510618, -0.0853412375, 0.0449974313, -0.0534627996, -0.0558119938, 0.0255994126, -0.0422267132, 0.0211019013, -0.101064906, 0.0302758403, -0.00200177729, 0.0577369705, -0.0173249096, 0.0458261706, 0.116266757, -0.0139172692, -0.0195216723, 0.0236957557, -0.00261176378, 0.102870516, -0.0350448191, -0.0415064879, 0.161883056, 0.10469836, 0.0162769742, -0.126410037, 0.0825980902, 0.0385107286, -0.0513081625, -0.0198488347, 0.0984914452, -0.114959389, 0.115681939, 0.0209397022, -0.0462179631, 0.0214058869, 0.105201021, -0.0764848813, 0.0111919772, -0.0412613116, -0.0272944085, 0.0146023501, -0.0598362722, 0.0309797414, 0.0782676339, -0.00873469189, -0.0515040122, 0.0926494226, -0.0146439606, 0.122180969, 0.0172243491, 0.096255213, 0.0478411429, -0.00864358619, -0.043324858, 0.0806294382, 0.0385359637, -0.110801741, -0.0747344047, -0.0966870263, -0.0405380689, 0.0107716825, -0.138293356, 0.0552434511, 0.0178805068, 0.027309062, -0.046948716, -0.0610931665, 0.088001661, 0.0763297454, 0.104673654, 0.0307341795, -0.0418299511, 0.0517079681, -0.0207884647, 0.117879823, 0.120932519, 0.0588165745, 0.112198956, 0.0273296181, -0.152703375, 0.0917826146, 0.0574529879, -0.127207488, -0.034267921, 0.038627021, -0.109168932, 0.103566602, 0.144766361, 0.0263313949, -0.00911980867, 0.025112465, 0.00483409502, -0.0115482705, -0.144090742, -0.0522341058, -0.0890554339, 0.123037137, -0.14432092, 0.0566201583, -0.0978538245, -0.0754307657, 0.0577240288, 0.115228221, 0.0717470497, -0.169151589, -0.0289260317, 0.0186712164, -0.0132641988, -0.0773575976, -0.13275443, -0.00525302626, -0.0448894016, 0.0724294782, 0.0305841565, -0.105213851, 0.0965616778, 0.0152161764, 0.0214027092, 0.0398187488, -0.124009691, 0.0709653571, 0.128675655, 0.0161593743, -0.0553461984, -0.0716221556, -0.0192435756, 0.0274756961, -0.0260479618, 0.0247825366, -0.0331113636, -0.0272251852, 0.067591548, -0.103237525, 0.00457238592, -0.0378931724, -0.0647895262, 0.111099169, -0.0802518725, 0.0201167539, 0.0551374778, 0.0205719061, -0.0536681078, -0.0430784672, 0.00408056565, 0.125642642, 0.124837883, 0.0629464313, 0.0523719788, -0.0555003472, -0.0356114469, -0.0642954111, -0.0556642935, -0.0128267063, -0.112548143, -0.0343009867, -0.0197926443, 0.032527376, -0.027550457, -0.0483105481, -0.1111186, -0.0533099994, 0.0897685438, -0.176952422, -0.111487359, -1.16974115e-06, -0.0101449145, -0.101750091, -0.0680906251, -0.0606357791, -0.00741220964, 0.130814746, 0.00218121661, 0.00785925984, 0.0854899511, 0.0221307538, -0.0848427489, 0.0814598054, -0.0656011105, -0.00223445706, 0.0759817585, -0.04201537, 0.000538141001, 0.155041024, 0.00807041302, -0.0581379309, 0.0459022969, -0.041241359, 0.175478607, 0.0606626831, -0.152528405, -0.00659666769, 0.0296979882, -0.0253408607, -0.0210521482, -0.00938495249, -0.0788428262, -0.0433672257, -0.0670581684, -0.0472778715, -0.0580407344, -0.0635472536, 0.105501935, -0.025068542, -0.114852771, -0.078055203, 0.0648784712, 0.0575545654, -0.115270779, 0.0121703502, 0.0322844461, -0.0923805609, -0.144185811, -0.0330828764, -0.0184293706, 0.0116816945, -0.13204585, -0.00187658332, -0.0570808128, 0.0447487347, -0.0320288502, -0.00365327112, -0.0644106045, 0.0492683053, 0.107609272, 0.020459529, -0.0907351226, 0.0351800546, 0.0128706573, 0.0705500469, -0.0460589565, -0.055538062, 0.0625325516, -0.00942290761, -0.0372318514, 0.0181166455, 0.0596277937, -0.0327496566, -0.0815372467, -0.143072665, 0.117885664, 0.0493902341, 0.0260507278, -0.0880189314, 0.0991055444, -0.124405935, -0.032854408, -0.018674368, 0.0103320964, 0.095204711, 0.0335261337, -0.0324110873, 0.0762193576, -0.0107756723, 0.0228998549, 0.0467691422, 0.0496879257, -0.00409949198, -0.134445935, -0.048339799, -0.0293532889, -0.0458019264, 0.0628730804, 0.070340015, 0.128977701, -0.0638133585, -0.00630695, 0.0475100204, 0.0443713255, 0.0790372193, -0.0519603938, 0.188868493, -0.0768636093, -0.0245793685, -0.0350950733, -0.0824217573, -0.100060083, -0.0734033883, -0.126760826, 0.145379573, 0.00923496857, 0.0131270029, -0.151082799, -0.042517446, 0.0937817767, 0.0573463663, 0.0198057704, 0.0535882413, 0.130594969, 0.162333325, 0.17903626, -0.0330195092, -0.00909163989, -0.0369175971];
    bias_3_u : ARRAY[0..63] OF REAL := [-1.01581478, -0.887849212, -1.0505383, -1.15503514, -1.07520187, -0.916982114, -0.917284429, -0.731233597, -1.29561114, -0.978517473, -1.07225573, -0.933320463, -1.01116836, -1.08638, -1.18247354, -1.04536152, -0.969618022, -0.833687901, -1.11044276, -0.937979698, -1.06253076, -1.03395391, -1.0668242, -1.07883251, -1.06569052, -1.17800641, -1.06056368, -1.06715477, -1.12462008, -1.39895415, -0.985698521, -1.04860067, -0.951921403, -1.17121184, -1.14114308, -0.945074677, -0.979631424, -1.1202879, -0.966821134, -0.93666774, -1.21267986, -1.05218196, -0.937734425, -0.909563243, -0.509452641, -1.04473948, -0.886089802, -1.02757108, -1.03394639, -0.899240732, -1.0388056, -0.880722702, -0.876731336, -1.037606, -1.27209771, -0.938842952, -0.941654742, -0.963986933, -0.950356603, -1.25041759, -0.941537082, -1.0247581, -1.06483781, -1.16372526];
    weights_3_r : ARRAY[0..4095] OF REAL := [-0.32606411, -0.305181414, 0.853710055, 0.643296003, -0.507959902, 0.360487521, -0.395130873, 0.414017469, 0.52319634, -0.479849488, -0.219426215, 0.15654248, -0.266728312, 0.461980253, 0.425416172, -0.556642294, 0.567818284, -0.549158752, -0.975931108, 0.67720896, -0.512712419, -0.328124523, 0.426616818, -0.443059117, 0.207611114, -0.310299754, 0.239883587, -0.236781195, -0.359037995, -0.36396715, 0.353712529, 0.408867657, 0.591968954, 0.530881524, 0.290289044, 0.594232917, -0.553219259, -0.784148693, 0.648065209, 0.490015626, 0.40664199, 0.315410346, -0.130245835, 0.343178451, 0.620505393, -0.133835554, -0.542454004, -0.264066935, 0.462930053, 0.207760662, 0.291069508, -0.347996682, -0.453460783, 0.382044703, -0.468908966, 0.723257065, 0.391256899, -0.62128371, 0.708973348, -0.712345123, -0.631182015, -0.333737373, 0.533903599, -0.446012765, -0.0378672406, -0.0479045957, 0.586389065, 0.264671922, -0.315799654, 0.208430871, -0.279002279, 0.175511852, 0.18931058, -1.05650055, -0.255715102, -0.00363925798, -0.0582851283, 0.244597003, 0.621904135, -0.331989348, 0.22773771, -0.47247237, -0.619856715, 1.33818412, -0.277933121, -0.213242188, 0.212933451, 0.106559314, 0.170447171, -0.224164695, 0.0732215643, -0.171327472, -0.0792607442, -0.611715198, 0.186487168, 0.723508537, 1.28295064, 0.690890372, 0.263711125, 0.478959203, -0.203083411, -1.04438186, 1.11608183, 0.370813042, 0.261939019, 0.276761144, 0.0417740121, 0.317641348, 0.114977218, -0.247694671, -1.47137809, -0.247703269, 0.447909325, -0.0339002497, 0.260987759, 0.177349597, -0.402403384, 0.156143531, -0.135770425, 0.510051191, 0.266276211, -0.167485476, 0.913470268, -0.461754829, -1.2195636, 0.077979736, 0.337161303, -0.141935438, -0.265271962, -0.035638582, 0.655573785, 0.537032127, -0.366385311, 0.203982592, -0.307501882, 0.381213546, 0.349319398, -1.1813004, -0.298807174, 0.0479753166, -0.37418431, 0.278960109, 0.840693057, -0.64014262, 0.474891245, -0.556242645, -0.614137411, 1.7334156, -0.526385307, -0.572337627, 0.248649359, -0.140956938, 0.119385995, -0.29798314, 0.244529814, -0.295158684, -0.300115496, -0.580093205, 0.226594269, 0.918142796, 1.74169719, 0.820151925, 0.248385459, 0.692447603, -0.396430552, -1.54747987, 1.38017225, 0.565111041, 0.392608315, 0.422911912, -0.119393133, 0.676306248, 0.460222095, -0.212124556, -1.80655181, -0.505402863, 0.301489621, 0.412834406, 0.181648746, -0.250534654, -0.471679151, 0.314968139, -0.233505979, 0.52545321, 0.381838292, -0.353975505, 1.25488007, -0.596149445, -1.74091864, -0.217042983, 0.638933122, -0.469897091, 0.245818049, 0.290093303, -1.08427835, -0.664157927, 0.370533347, -0.185779259, 0.533736944, -0.0601371452, -0.527724266, 0.60000211, 0.149180949, -0.224620834, 0.200513855, -0.258397371, -0.456327915, 0.949554861, -0.421606094, 0.376373112, 1.6443671, -0.485285401, 0.816311598, 0.243153811, -0.471630067, 0.139453158, -0.144242361, 0.317050517, -0.232827887, 0.255592555, 0.15091145, 0.247503817, -0.286755443, -0.362139732, -0.461967707, -0.363402843, -0.109364457, -0.491291016, 0.351950824, 0.639383376, -0.539893091, -0.424525499, -0.2290764, -0.199569568, 0.0934817418, -0.173082545, -0.35091725, -0.0301282555, 0.594287872, 0.188275486, -0.270237386, -0.136253968, -0.155206367, 0.0628562197, 0.550562918, -0.107881248, 0.202634931, -1.20844626, -0.0330623388, 0.419759899, -0.539858162, 1.55076027, 0.473937124, 0.114922389, -0.359740287, 0.358791083, -0.238371491, 0.0309315939, 0.379086971, 0.413848668, -0.293242633, 0.332917243, -0.141442761, 0.232743874, 0.242201135, -1.23438561, -0.296759665, -0.115022659, -0.164160192, 0.163818792, 0.685197115, -0.330099732, 0.304970264, -0.346489012, -0.779386997, 1.42712438, -0.523679256, -0.276608735, 0.150926173, -0.12271972, 0.232150823, -0.36957562, -0.0389995165, -0.138426706, -0.0751603991, -0.493225664, 0.166680902, 0.683986783, 1.75461292, 0.551047027, 0.17739968, 0.486676127, -0.162812993, -1.4567163, 1.28828633, 0.419575125, 0.305336416, 0.287140518, -0.0665183365, 0.310240835, 0.230046228, -0.329168618, -1.68186617, -0.129506499, 0.230660826, 0.191573709, 0.167725205, 0.0199827328, -0.31258601, -0.00548750907, -0.322434396, 0.417515099, 0.352410108, -0.267527252, 1.1229645, -0.469884247, -1.70649111, 0.0533591323, 0.396650195, -0.213872373, -0.247390494, -0.308249265, 0.885731876, 0.648571968, -0.310095698, 0.268737406, -0.389113486, 0.0871751979, 0.343963742, -0.485504836, -0.115139328, 0.23760289, -0.424925536, 0.500883222, 0.316645622, -0.702252448, 0.555773854, -0.386323303, -1.48340034, 0.66543299, -0.705020845, -0.37072435, 0.363651961, -0.446105599, 0.149830148, -0.358513474, 0.396215469, -0.265176088, -0.253546655, -0.286184102, 0.458667219, 0.252435833, 0.38352707, 0.340764135, 0.106404178, 0.436587185, -0.641245365, -0.495529294, 0.632080793, 0.337052464, 0.518227041, 0.220586628, -0.318199962, 0.406555504, 0.530345023, -0.155054793, -0.621839464, -0.295333445, 0.212138698, 0.228294671, 0.316329509, -0.364110976, -0.440465301, 0.486016542, -0.278429061, 1.33248186, 0.18339245, -0.53936249, 0.29928565, -1.45049202, -0.368015051, -0.349973351, 0.438491136, -0.403809279, -0.477971882, -0.304249853, 0.466022611, 0.498331398, -0.467597336, 0.348668754, -0.510163784, 0.410904944, 0.498593748, -1.05407882, -0.255845338, 0.185745597, -0.367634088, 0.333585799, 0.853473485, -0.660563707, 0.329295546, -0.603268206, -0.667021155, 1.56817055, -0.494137198, -0.403352022, 0.44587186, -0.295524448, 0.238873377, -0.393918365, 0.317173779, -0.151768267, -0.37963894, -0.579922795, 0.234902322, 0.674435318, 1.45155692, 0.716528475, 0.271678597, 0.764275908, -0.332182556, -1.46324396, 1.45741057, 0.597791016, 0.335873425, 0.256497473, 0.030166598, 0.484657943, 0.466247529, -0.41871053, -1.51203668, -0.494381219, 0.329711199, 0.293426394, 0.439302534, -0.11895518, -0.503041506, 0.27442047, -0.2831963, 0.558458626, 0.304881573, -0.32383275, 1.03910983, -0.792959034, -1.5608331, -0.257430762, 0.664614916, -0.501426876, -0.281351089, 0.0414545909, 0.447095424, 0.343832135, -0.255541176, 0.0612748638, -0.280172408, 0.177165255, 0.36193496, -0.925673783, -0.16850391, 0.0128063755, -0.0942704827, 0.134742722, 0.680249214, -0.383725584, 0.369982153, -0.395214558, -0.586839259, 1.06134593, -0.446925581, -0.405082673, 0.0176686663, -0.0800010785, 0.340114951, -0.200141653, 0.0898567736, 0.01082341, -0.143583834, -0.3846412, 0.0610680543, 0.750910878, 1.13939989, 0.655028045, 0.41650939, 0.57746464, -0.235219672, -1.15468717, 0.96712774, 0.269759059, 0.0998954624, 0.116918571, -0.0196392536, 0.38387078, 0.117413625, -0.302846849, -1.33640993, -0.398219466, 0.394320697, 0.0167492945, -0.0259594377, 0.0365658924, -0.192624837, 0.0477550216, -0.140257016, 0.48980245, 0.242636696, -0.0990151837, 0.977481246, -0.521247506, -1.034536, -0.171559945, 0.293284655, -0.237343356, -0.313935697, -0.232274383, 0.778067112, 0.62355727, -0.57867223, 0.428997576, -0.640505195, 0.250204235, 0.661255181, -0.649872541, -0.122935608, 0.126976743, -0.333370656, 0.507789612, 0.593846679, -0.838342011, 0.664126933, -0.352723658, -0.909550726, 0.843601286, -0.8069399, -0.315561473, 0.478078306, -0.322076082, 0.273690939, -0.423558116, 0.177327543, -0.399279118, -0.173438579, -0.431111574, 0.160768285, 0.451122195, 0.598117471, 0.364526689, 0.266648859, 0.584997833, -0.595889211, -0.674656212, 0.733342409, 0.516002715, 0.433507383, 0.472957939, -0.183722794, 0.407700777, 0.417470217, -0.197818443, -0.78360039, -0.190586895, 0.252519101, 0.269995302, 0.320930928, -0.201623842, -0.679484725, 0.476249129, -0.337365001, 0.729481757, 0.393714428, -0.458076656, 0.610665083, -0.840719402, -0.656802475, -0.316481829, 0.264371485, -0.371127099, -0.252732307, -0.239085466, 0.266183496, 0.417861938, -0.438964844, 0.221316725, -0.455889136, -0.13639456, 0.258295447, -0.0555382408, 0.164990604, 0.154210657, -0.170295238, 0.262882829, 0.0899999365, -0.248038337, 0.436610639, 0.148447692, -0.615800679, 0.150086999, -0.390931129, 0.154123083, 0.145448953, -0.182117596, -0.20823136, -0.00837396272, 0.134367272, -0.222348854, -0.404675871, 0.174651444, 0.138303235, -0.0794249997, -0.0343393162, -0.130718768, 0.00081770902, -0.0382439457, -0.424111843, -0.119458333, 0.230674118, -0.028081717, 0.415239364, 0.156845033, -0.163451418, -0.121806018, 0.408577055, 0.241918802, -0.0300814416, -0.0074230493, 0.0646340176, 0.324945062, 0.306441814, -0.211217076, -0.170305654, 0.242016852, -0.278236717, 0.575324535, -0.113995463, -0.432759374, 0.114849724, -0.533126533, 0.0167393349, -0.38273707, -0.0428678691, -0.28884092, -0.471949935, -0.268262804, 0.698775351, 0.698765576, -0.415175825, 0.310324371, -0.465906799, 0.294130713, 0.402897477, -0.594575763, -0.276606709, 0.336049944, -0.483903408, 0.384283513, 0.581177354, -0.83756572, 0.441531897, -0.380635679, -1.11072242, 0.831285536, -0.794558227, -0.485136062, 0.480796397, -0.478292763, 0.204729795, -0.229210749, 0.30153206, -0.166791767, -0.234277368, -0.397676736, 0.398091793, 0.483754039, 0.766412258, 0.511118889, 0.171075433, 0.313571274, -0.557242393, -0.641509473, 0.633744478, 0.381214678, 0.45218268, 0.479226977, -0.355552763, 0.230504155, 0.50238204, -0.196017981, -0.771038353, -0.19761245, 0.31358242, 0.489434212, 0.411978036, -0.132157326, -0.518997371, 0.482037663, -0.459952474, 0.861239672, 0.258370727, -0.446846068, 0.452018321, -1.01126957, -0.603265166, -0.195862025, 0.351056933, -0.368395925, -0.504480958, -0.367227137, 0.939662576, 0.660247386, -0.365831763, 0.541688263, -0.460847795, 0.307414412, 0.624971688, -0.344881892, -0.129336655, 0.271847337, -0.217659026, 0.245232657, 0.36421901, -0.855669737, 0.592403769, -0.393725753, -1.20529306, 0.547492087, -0.729086757, -0.410979331, 0.346642703, -0.328289866, 0.237400368, -0.295209855, 0.197553545, -0.485058933, -0.189968109, -0.304942578, 0.487791836, 0.54598552, 0.630286992, 0.37855649, 0.137780443, 0.480451822, -0.39389208, -0.634016931, 0.647453427, 0.214886963, 0.531250536, 0.445005357, -0.208312169, 0.374261469, 0.578697205, -0.139688984, -0.697460771, -0.35923028, 0.434657186, 0.464936823, 0.450845182, -0.302823961, -0.736231744, 0.452758044, -0.506413817, 1.14236045, 0.248236433, -0.505619764, 0.633802891, -1.08701026, -0.525048733, -0.285771459, 0.441548675, -0.56051898, -0.31927681, -0.324115783, 0.643988669, 0.405917078, -0.330453306, 0.375912219, -0.34731546, 0.176775172, 0.385320067, -0.976352394, -0.39451161, 0.302981526, -0.331505746, 0.394162476, 0.700016201, -0.629214704, 0.529205024, -0.680885017, -0.727290213, 1.39126933, -0.598196208, -0.611907423, 0.453459501, -0.260176986, 0.173567802, -0.294734448, 0.349817783, -0.168323874, -0.219119057, -0.633465707, 0.165119141, 0.66164422, 1.34298229, 0.864157617, 0.481791258, 0.551117599, -0.453588724, -1.33108592, 1.32759583, 0.400511742, 0.416378945, 0.210791215, -0.0152973225, 0.598210633, 0.338426322, -0.389807463, -1.30942619, -0.491540879, 0.587278724, 0.2986525, 0.20118694, 0.00159147358, -0.630330503, 0.450823069, -0.408089966, 0.715183794, 0.22981061, -0.406616211, 1.01547182, -0.78458935, -1.39109886, -0.209403127, 0.513578713, -0.506427526, -0.29192251, -0.365352601, 0.821260273, 0.799699843, -0.551483572, 0.347243428, -0.618902028, 0.104906209, 0.384635627, -0.678108811, -0.1532446, 0.366201997, -0.224698484, 0.291296363, 0.267117858, -0.721745253, 0.407198012, -0.250949353, -1.48795342, 0.745735586, -0.698526442, -0.408564717, 0.319990903, -0.258586496, 0.218047649, -0.279926717, 0.209587425, -0.461742342, -0.232960254, -0.45649752, 0.39823553, 0.316946059, 0.499801308, 0.365775526, 0.285763681, 0.410254568, -0.585092723, -0.758430243, 0.793517828, 0.347428501, 0.463376641, 0.282039613, -0.137573525, 0.201987252, 0.574360251, -0.147843152, -0.551913857, -0.105053365, 0.239548668, 0.268206239, 0.277595073, -0.292813897, -0.627250075, 0.332713664, -0.36461249, 1.09503412, 0.278442115, -0.570906878, 0.575401843, -1.14452851, -0.503782451, -0.222146109, 0.25390774, -0.435958177, -0.346188098, -0.287907928, 0.577285111, 0.625171602, -0.485937923, 0.279984206, -0.580171645, 0.304609418, 0.382132024, -0.720344841, -0.334448129, 0.338395119, -0.253193289, 0.320167184, 0.369183391, -0.75026536, 0.365687907, -0.602306545, -0.862038493, 0.716569424, -0.626643598, -0.529524446, 0.27669844, -0.231221542, 0.19715257, -0.364062011, 0.272420794, -0.193196043, -0.26943177, -0.40359816, 0.175001666, 0.61060524, 0.733311117, 0.647010386, 0.300696403, 0.531074643, -0.427513987, -0.991258919, 0.965829194, 0.505575061, 0.464456826, 0.370266259, -0.180219814, 0.514823973, 0.547894955, -0.30526337, -0.775482357, -0.277872801, 0.304864079, 0.438526511, 0.442127705, -0.185165703, -0.408223033, 0.372900993, -0.307785809, 0.803971171, 0.247336209, -0.346430957, 0.561486781, -0.784184873, -0.775968432, -0.33393088, 0.414071649, -0.414346129, -0.424316555, -0.228602037, 0.798046768, 0.589726985, -0.471872777, 0.375852257, -0.523459375, 0.312538296, 0.64948523, -0.564522266, -0.39429161, 0.392420679, -0.331350297, 0.406572282, 0.498701811, -0.538559735, 0.37152037, -0.500432014, -0.88565588, 0.814511836, -0.65060389, -0.32671982, 0.443832159, -0.366107523, 0.323150456, -0.431577086, 0.31207934, -0.443811983, -0.453019857, -0.491461039, 0.260425597, 0.649067998, 0.623069763, 0.515208781, 0.29761672, 0.553334832, -0.419336051, -0.74229908, 0.618693173, 0.562187016, 0.327073514, 0.328121513, -0.152062252, 0.258443296, 0.38306722, -0.219228178, -0.824401379, -0.364127398, 0.281175613, 0.228253767, 0.505391181, -0.260356188, -0.714000762, 0.434605122, -0.283382773, 0.759392858, 0.418259323, -0.480381697, 0.658830822, -0.828426778, -0.594255626, -0.434398293, 0.434758842, -0.475796342, -0.253429919, -0.151888281, 0.464026541, 0.447059274, -0.23363854, 0.234164312, -0.228685543, 0.108610779, 0.417265028, -0.949152887, -0.376021415, 0.127703905, -0.180501074, 0.241112828, 0.734871805, -0.522570789, 0.398032188, -0.564164639, -0.479930878, 1.43935657, -0.37222895, -0.455183208, 0.266491622, -0.0408120714, 0.311739117, -0.388832271, 0.182095289, -0.118631139, -0.00731076393, -0.43673858, -0.0472857542, 0.855252743, 1.33718526, 0.790244818, 0.398922116, 0.565711081, -0.20525077, -1.10990274, 1.13496363, 0.480120897, 0.20322676, 0.107450388, -0.0908780992, 0.300021589, 0.119640276, -0.191865563, -1.46495235, -0.298560351, 0.488960505, 0.0581271686, 0.0770600885, -0.103614494, -0.303027779, 0.0364120677, -0.139285401, 0.683296263, 0.190768391, -0.226745963, 1.05477059, -0.473936111, -1.46578884, 0.078238152, 0.489368916, -0.337299317, -0.444000721, -0.174462199, 0.626759052, 0.392545253, -0.330222338, 0.246465355, -0.421768636, 0.284421295, 0.400160909, -0.558163941, -0.282744735, 0.106122591, -0.385983437, 0.504063666, 0.545476139, -0.622974038, 0.304397136, -0.36480096, -0.651256442, 0.750828683, -0.651343167, -0.32135278, 0.462911516, -0.208699137, 0.344162047, -0.337207288, 0.166761756, -0.157386944, -0.209506616, -0.315502286, 0.185891688, 0.636180043, 0.588617742, 0.512386203, 0.317265481, 0.474550545, -0.591336787, -0.675465286, 0.629930377, 0.497780949, 0.283470303, 0.278181314, -0.152107403, 0.323860735, 0.300083309, -0.237705827, -0.707360804, -0.233611494, 0.298213273, 0.327645987, 0.474210054, -0.220958605, -0.43902716, 0.405127794, -0.285075426, 0.677587867, 0.197221667, -0.526327968, 0.604875863, -0.556873083, -0.553813517, -0.32801944, 0.378549248, -0.587617636, 0.21427089, 0.21984911, -0.875384271, -0.620468438, 0.364588082, -0.312358916, 0.41226685, -0.139815196, -0.175383493, 0.280132443, 0.102841973, -0.131755173, 0.0816493407, -0.245622069, -0.476292968, 0.712404072, -0.346726954, 0.30152601, 1.45562994, -0.407604456, 0.471377373, 0.0670249537, -0.208978981, -0.00896921568, 0.00792890228, 0.160337701, -0.126184568, 0.109025173, 0.0403974764, 0.385903925, -0.0472378358, -0.234496132, -0.592926741, -0.370333821, -0.015724184, -0.372033179, 0.464167625, 0.449376225, -0.561121225, -0.294491768, -0.269805431, -0.23032254, 0.113178119, -0.374025494, -0.24987562, 0.154645085, 0.500742376, 0.0921915993, -0.187845826, 0.00581417372, -0.133517161, -0.0244534146, 0.424528837, -0.286528796, 0.305054575, -1.10627806, -0.224664286, 0.403331935, -0.541942596, 1.32796419, 0.379160345, 0.156610399, -0.148328111, 0.27849111, -0.479717582, -0.416316181, 0.728976667, 0.47371915, -0.340526283, 0.425530344, -0.493184388, 0.196874604, 0.422890276, -0.734140754, -0.428865492, 0.295673072, -0.347783983, 0.275349826, 0.647607803, -0.740972102, 0.359515399, -0.355478734, -0.89868927, 0.693098068, -0.565694273, -0.45446521, 0.521305144, -0.423126072, 0.343195379, -0.36296463, 0.182377294, -0.3046498, -0.230392531, -0.479535222, 0.292608529, 0.443596572, 0.750985682, 0.678646863, 0.341219902, 0.37737909, -0.480458766, -0.824370861, 0.720338881, 0.468586832, 0.401706249, 0.337754607, -0.288740158, 0.38029319, 0.319494545, -0.25374651, -0.610306621, -0.489055008, 0.301279873, 0.242298141, 0.469092429, -0.316974074, -0.482820809, 0.29542467, -0.279328406, 0.800565243, 0.219063267, -0.567258596, 0.586478591, -0.836146533, -0.598628998, -0.277637094, 0.35739249, -0.349981159, -0.212868378, -0.132515892, 0.582968831, 0.245836794, -0.21859476, 0.248592272, -0.436507136, -0.0525316447, 0.219017044, -0.078199558, -0.0697035566, 0.325711846, -0.220956966, 0.382013202, 0.151345342, -0.482834786, 0.230038151, 4.8701273e-05, -0.896882534, 0.167872235, -0.556771755, -0.0531435348, 0.277634442, -0.303767294, -0.0111572994, -0.0296421107, 0.21856828, -0.113810413, -0.360011727, -0.141940147, 0.157705769, 0.144350186, 0.290767372, 0.136084914, -0.179874763, -0.0301123243, -0.427401155, -0.297967046, 0.323375195, 0.045945961, 0.229860306, 0.399075538, -0.240118444, 0.0239243489, 0.305032372, 0.043214988, -0.0338462107, 0.12562266, -0.0240930375, 0.38718912, 0.217619404, -0.29890126, -0.19797644, 0.214872062, -0.149662852, 0.862906933, -0.158315763, -0.35901013, 0.207159743, -1.03316343, -0.0435992517, -0.371495306, 0.0122571802, -0.222766235, -0.335296631, 0.00614431966, 0.442041367, 0.511820197, -0.271431029, 0.251062542, -0.354020029, 0.26408121, 0.380686581, -1.19595873, -0.199459553, 0.0512621887, -0.230785102, 0.121044502, 0.563847125, -0.476866037, 0.282984555, -0.610335827, -0.750677407, 1.48484993, -0.396005511, -0.4459984, 0.15016526, -0.165891528, 0.175520033, -0.253411263, 0.0663821399, 0.0307248328, -0.027399281, -0.577981889, 0.187904432, 0.716747284, 1.71462762, 0.719156265, 0.457143158, 0.491087288, -0.243744597, -1.26668429, 1.36153471, 0.529155016, 0.0915734097, 0.329717249, 0.151948646, 0.425810426, 0.218522847, -0.193444088, -1.54156172, -0.419055372, 0.324922889, 0.101474956, 0.0678244159, 0.0475526936, -0.368958205, 0.0250567012, -0.249778137, 0.567493558, 0.285005659, -0.29450646, 1.22011006, -0.566066265, -1.52908516, -0.0332701094, 0.39348945, -0.435152113, -0.279379427, -0.252164513, 0.88293618, 0.603829801, -0.557003856, 0.4126091, -0.611310482, 0.262114704, 0.39541617, -0.657683015, -0.419031233, 0.334631443, -0.439445496, 0.239912346, 0.594620764, -0.710724235, 0.625857174, -0.281924397, -0.94848001, 0.766416132, -0.573693395, -0.507681251, 0.455642968, -0.344042838, 0.120637521, -0.196149305, 0.187891915, -0.33866787, -0.461829305, -0.431388974, 0.473234236, 0.376484066, 0.671459436, 0.532400489, 0.414870739, 0.612779319, -0.447367132, -0.736575902, 0.608187616, 0.457972795, 0.391607225, 0.391642749, -0.270501822, 0.473758906, 0.371922523, -0.248366505, -0.516390562, -0.178563148, 0.301155925, 0.488553792, 0.470395386, -0.259697437, -0.604833424, 0.439455271, -0.526135087, 0.754391849, 0.213179052, -0.635523617, 0.726304114, -0.92388463, -0.556524396, -0.369461954, 0.522346735, -0.548059225, 0.257865012, 0.0679476708, -0.755721331, -0.416924179, 0.183604792, -0.196284577, 0.381534636, -0.153743476, -0.434020489, 0.365814686, -0.0303360354, 0.00483766757, 0.234462872, -0.1011682, -0.343322188, 0.688691437, -0.311507314, 0.243866593, 1.36334038, -0.447809219, 0.745755851, 0.321573853, -0.16720055, 0.0732166767, -0.0399155952, 0.141015455, -0.313092411, 0.0137336878, 0.160370693, 0.317644477, -0.166301489, -0.494622916, -0.501563907, -0.429580897, -0.0300284959, -0.421272367, 0.521287918, 0.609171689, -0.657234728, -0.159242377, -0.208006412, -0.282181531, 0.0125726322, -0.109527849, -0.450762987, -0.0350307785, 0.4969396, -0.00262273988, -0.0696354359, -0.0597759075, -0.103529476, 0.0310744941, 0.573780298, -0.313798845, 0.202677295, -1.02902234, -0.0767832696, 0.405816942, -0.357142836, 1.42817438, 0.576379418, 0.041038733, -0.40113923, 0.450059474, -0.249666899, -0.324406743, 0.645155787, 0.651951373, -0.335311472, 0.318877369, -0.377464861, 0.278273344, 0.577528358, -0.707005084, -0.454609185, 0.346883327, -0.375036657, 0.408443093, 0.604526222, -0.738248646, 0.488500953, -0.574646294, -0.803916037, 0.758122504, -0.623487353, -0.300931603, 0.519699752, -0.21979551, 0.182568133, -0.535689473, 0.355320454, -0.335205972, -0.333302468, -0.528201103, 0.384286255, 0.590183973, 0.814082682, 0.453687638, 0.449585825, 0.441816151, -0.566304922, -0.855111718, 0.909155846, 0.491852105, 0.46307838, 0.467540711, -0.180398166, 0.49356845, 0.508661568, -0.372565985, -0.889092684, -0.290327221, 0.393947303, 0.43914488, 0.396424651, -0.0341150574, -0.504731894, 0.242020696, -0.3221201, 0.611044109, 0.406554967, -0.525439441, 0.852771521, -0.805656016, -0.788086474, -0.3786515, 0.528430641, -0.327401429, -0.405131936, -0.401135057, 1.03028727, 0.547111273, -0.511407316, 0.484279543, -0.37078923, 0.317534953, 0.497445107, -0.566063821, -0.192737415, 0.17343004, -0.437663138, 0.27078265, 0.370668411, -1.03059494, 0.679856479, -0.484099001, -2.04160094, 0.550596535, -0.936203003, -0.326845407, 0.458781779, -0.330802292, -0.0390953943, -0.148416176, 0.282826245, -0.339116395, -0.44140628, -0.354241639, 0.373801202, 0.561958194, 0.471544474, 0.338501513, 0.190972656, 0.560675621, -0.60877955, -0.806209028, 0.740752816, 0.403585136, 0.44382149, 0.310492158, -0.165237129, 0.467229635, 0.639951468, -0.250467837, -0.719496429, -0.342186749, 0.346429437, 0.472102076, 0.423257083, -0.113565609, -0.611903667, 0.502099693, -0.454853475, 1.47754538, 0.192447752, -0.623071432, 0.622491539, -1.70403862, -0.689736545, -0.311849207, 0.346993446, -0.61403209, -0.32030949, -0.260404497, 0.606727421, 0.378895342, -0.522973001, 0.242676035, -0.503748238, 0.400032282, 0.409070313, -1.04656887, -0.23251985, 0.0598524436, -0.160751864, 0.267909467, 0.585713267, -0.53919065, 0.41407761, -0.638192773, -0.853965998, 1.66303492, -0.484024048, -0.597094715, 0.202447027, -0.31045422, 0.41164431, -0.37736547, 0.236909643, -0.288764238, -0.323797226, -0.65210408, 0.277571082, 0.785428286, 1.53385842, 0.603273511, 0.27001673, 0.734697819, -0.316855073, -1.2592355, 1.29509652, 0.566119313, 0.451303422, 0.450500518, -0.118251942, 0.5555861, 0.517378032, -0.212427497, -1.65542746, -0.387000918, 0.551443279, 0.295913428, 0.357824534, -0.0474563763, -0.501777112, 0.346730024, -0.255087167, 0.65019232, 0.233359382, -0.399132252, 1.20495582, -0.788980126, -1.47384763, -0.298721731, 0.547602355, -0.400281519, 0.415391237, 0.11500933, -0.764448643, -0.526417255, 0.471959233, -0.303978741, 0.411469579, -0.215374574, -0.552919745, 0.464531958, 0.180658236, -0.228912786, 0.307991862, -0.389285654, -0.357774109, 0.677281499, -0.538697839, 0.266804308, 1.55649245, -0.543816209, 0.663670182, 0.205055431, -0.306369811, 0.314960301, -0.0812868699, 0.244915798, -0.0972369686, 0.118134655, 0.228851423, 0.33507967, -0.178763539, -0.542017519, -0.440441757, -0.505637646, -0.00129357539, -0.469659418, 0.369825453, 0.763003647, -0.471925408, -0.229464024, -0.215304658, -0.216859743, 0.120160319, -0.403819114, -0.454149246, 0.198572591, 0.695058703, 0.091226548, -0.0968206972, -0.355034381, -0.354152858, 0.0810929313, 0.477759898, -0.261985332, 0.248434946, -1.40007436, -0.115490466, 0.2606875, -0.557928205, 1.54712737, 0.568113387, 0.0240328442, -0.371635526, 0.468986988, -0.3890315, -0.227186203, 0.558743656, 0.638008714, -0.2325169, 0.325430512, -0.360332191, 0.387367666, 0.388153821, -1.04519343, -0.269344211, 0.165706381, -0.168712839, 0.402218312, 0.652806342, -0.674834907, 0.41147843, -0.499225646, -0.734338701, 1.82643378, -0.444065362, -0.588895082, 0.455570638, -0.21291098, 0.110225089, -0.332531989, 0.181953952, -0.294583291, -0.264316112, -0.515410423, 0.162889913, 0.868188739, 1.86032271, 0.700357616, 0.513032436, 0.765919447, -0.49682951, -1.62329006, 1.45719647, 0.545549512, 0.451227427, 0.28905201, -0.142598704, 0.610706568, 0.444595754, -0.141367614, -2.04516983, -0.381730109, 0.318353266, 0.207129255, 0.14816165, 0.0522552989, -0.550924182, 0.407493293, -0.41661644, 0.614094198, 0.354451597, -0.451580673, 1.33644974, -0.551402748, -1.78111506, -0.0356309898, 0.558322489, -0.308785051, -0.253635705, -0.0270095747, 0.46169883, 0.35802564, -0.205481261, 0.318101376, -0.502353311, 0.353082567, 0.418376744, -1.11887336, -0.111144789, 0.117297441, -0.257290363, 0.253319979, 0.7175529, -0.568437874, 0.234085515, -0.576971769, -0.753595471, 2.22766876, -0.63931638, -0.406852841, 0.176097482, -0.0419444628, 0.108799115, -0.454771698, 0.139979661, -0.00126432185, -0.175606206, -0.553412139, 0.166107267, 0.923081875, 2.3204813, 0.596822083, 0.273973882, 0.590377271, -0.273627281, -1.66828382, 1.68053067, 0.356793612, 0.158161953, 0.292190343, 0.0725176632, 0.514080942, 0.25470531, -0.336534709, -2.26764321, -0.27513203, 0.21084933, 0.238806561, 0.319567502, 0.00441332161, -0.470187545, 0.247312322, -0.301804394, 0.539537251, 0.40202406, -0.321202397, 1.35585296, -0.678141296, -2.18601513, -0.156690359, 0.644770503, -0.447970003, 0.184947133, 0.0586535335, -0.842697203, -0.476564407, 0.326289117, -0.175858513, 0.337102354, -0.150091827, -0.393082768, 0.342845351, 0.0555129908, -0.0486602783, 0.266736895, -0.220026106, -0.269021273, 0.608967543, -0.186941519, 0.279839188, 1.1750114, -0.559024274, 0.393088549, 0.141963348, -0.172769904, 0.121606402, -0.110438086, 0.119224839, -0.16923289, -0.0105624478, 0.0515540726, 0.399702787, 0.0513814129, -0.278160423, -0.349841654, -0.216284662, -0.0206595752, -0.322790265, 0.407239199, 0.418390363, -0.452856183, -0.365659744, -0.303342491, -0.235371232, 0.132295564, -0.27970612, -0.363894314, -0.0102149583, 0.503446877, 0.252181977, -0.201562554, -0.140030086, -0.212522104, -0.102482498, 0.521413445, -0.0599606782, 0.317379594, -0.91857636, -0.0796753466, 0.374061078, -0.407837212, 1.13819242, 0.538435876, 0.0274906904, -0.203527272, 0.221570566, -0.585137784, -0.22554791, 0.897851586, 0.794410348, -0.348831713, 0.427135259, -0.493484974, 0.113772824, 0.674505949, -0.469446868, -0.368993729, 0.295242786, -0.40725553, 0.337209344, 0.473266065, -0.80423677, 0.664289951, -0.449214637, -1.27750874, 0.742842019, -0.766273737, -0.467851818, 0.290394068, -0.465311527, 0.238281116, -0.425370961, 0.435574234, -0.291806579, -0.428470105, -0.44762519, 0.277623832, 0.619269311, 0.458167434, 0.591054261, 0.323538482, 0.396119237, -0.537716269, -0.799658716, 0.515515029, 0.291549206, 0.352653205, 0.560084641, -0.245590121, 0.225990862, 0.502214193, -0.276380807, -0.484679371, -0.15336445, 0.211182415, 0.427163899, 0.443517625, -0.239297152, -0.777251482, 0.447269887, -0.335349888, 1.21866739, 0.410942733, -0.667268157, 0.692402005, -1.24103224, -0.534754515, -0.281618685, 0.307847261, -0.592071176, -0.17489098, -0.057309825, 0.622739553, 0.33250168, -0.18130222, 0.214820161, -0.32339251, 0.378621399, 0.253713369, -1.22676325, -0.325474322, -0.0511168316, -0.237608954, 0.160359859, 0.682873309, -0.438781857, 0.374165386, -0.598473728, -0.586400807, 1.50517404, -0.531930804, -0.505696177, 0.188739181, -0.0759081692, 0.322496235, -0.534777462, 0.0866990909, -0.220319897, -0.220647246, -0.589855194, 0.136748701, 0.710161626, 1.55659211, 0.811731458, 0.392696917, 0.581875682, -0.286527216, -1.25108588, 1.18614066, 0.594158888, 0.238403395, 0.324100316, 0.0939783454, 0.568623304, 0.285499305, -0.149848759, -1.64757788, -0.389623255, 0.426757812, 0.339580208, 0.224090979, 0.0706543475, -0.387865424, 0.149145648, -0.13083519, 0.49459061, 0.21732384, -0.269787997, 1.21367657, -0.599125087, -1.48657, -0.0794282928, 0.483454108, -0.495730668, -0.149702519, -0.12196622, 0.518101096, 0.498079419, -0.440585136, 0.377816558, -0.44399941, 0.298395574, 0.526369333, -1.3361609, -0.184671834, 0.198181227, -0.213837981, 0.227365643, 0.69264257, -0.642421722, 0.253970891, -0.459746599, -0.721164227, 2.0608139, -0.410998136, -0.295992911, 0.381521583, -0.0209507495, 0.356352538, -0.274228454, -0.0050154482, -0.0101287942, -0.149391398, -0.546611249, 0.244803205, 0.957121789, 2.423383, 0.761666834, 0.449197382, 0.818116665, -0.290270865, -1.38992047, 1.68735409, 0.584730566, 0.209530428, 0.390848577, -0.0938457027, 0.381666511, 0.222843274, -0.335909754, -2.28804636, -0.407721847, 0.495959103, 0.0609779879, 0.377927572, -0.000324302353, -0.402243406, 0.0875439867, -0.308821261, 0.752283812, 0.330103457, -0.535354733, 1.26573205, -0.805240512, -1.81103754, -0.212165743, 0.49315542, -0.27250576, -0.26895386, -0.23040916, 0.642885923, 0.658500731, -0.37262395, 0.37434265, -0.349618167, 0.240233302, 0.563242972, -1.00378811, -0.382425368, 0.209850684, -0.395602703, 0.19864963, 0.598141253, -0.55917263, 0.327447176, -0.54477936, -0.677006662, 1.02608597, -0.622659922, -0.374311239, 0.454068393, -0.1352209, 0.139970779, -0.393903822, 0.311810255, -0.347855955, -0.183584973, -0.613458753, 0.294341862, 0.695668757, 0.97671634, 0.629432797, 0.222873241, 0.576654196, -0.576174319, -1.17176938, 1.21802914, 0.463727653, 0.323104858, 0.385295808, -0.0564640015, 0.495977908, 0.560169458, -0.402570993, -1.24606681, -0.30742529, 0.446491867, 0.206024915, 0.378804684, -0.0637932569, -0.548548579, 0.264957011, -0.435918182, 0.714320481, 0.503891647, -0.490187079, 0.92835933, -0.653939903, -0.998602509, -0.234939784, 0.519885242, -0.345346838, -0.438330591, -0.199805692, 0.791778803, 0.772088349, -0.334469944, 0.533462465, -0.613139749, 0.273976594, 0.438189596, -0.5514853, -0.35970071, 0.340049952, -0.453285843, 0.468381822, 0.559531033, -0.710513115, 0.589847207, -0.400875419, -1.59320593, 0.761381209, -0.714087009, -0.386633068, 0.277693152, -0.341802031, 0.180621013, -0.407044262, 0.40718329, -0.343057722, -0.358702391, -0.242539018, 0.427075744, 0.438927263, 0.677350819, 0.34506014, 0.311973274, 0.431390852, -0.481903553, -0.805651665, 0.652924657, 0.382951111, 0.34651202, 0.547604501, -0.228527293, 0.320236057, 0.505470097, -0.118233278, -0.483198285, -0.175483301, 0.31151852, 0.390251815, 0.294036955, -0.243998915, -0.682308316, 0.409372777, -0.539528608, 1.08507121, 0.392528206, -0.633849263, 0.564027965, -1.2653687, -0.708535314, -0.37867108, 0.462343037, -0.63749373, -0.336225659, -0.354143858, 0.538114786, 0.575526595, -0.513737082, 0.226745903, -0.354042709, 0.321344256, 0.533973157, -1.00941694, -0.384838343, 0.116603948, -0.371144712, 0.309847772, 0.680324495, -0.464205742, 0.382111371, -0.518437624, -0.835754752, 1.296188, -0.719237804, -0.336357653, 0.317768604, -0.37401849, 0.148494884, -0.583994448, 0.362303764, -0.160795614, -0.393341154, -0.592710495, 0.422500819, 0.844100416, 1.22041082, 0.815548182, 0.259628803, 0.518015802, -0.441701949, -1.20411873, 1.26204193, 0.557317436, 0.330148011, 0.305774599, -0.166518152, 0.624247551, 0.459448367, -0.399693191, -1.16738927, -0.503780901, 0.536997199, 0.198219493, 0.41484648, -0.156464636, -0.587040901, 0.381635636, -0.46363765, 0.541935325, 0.447267145, -0.478802979, 0.919147849, -0.607068002, -1.34749579, -0.334636748, 0.49500072, -0.340175569, 0.353704125, 0.101251774, -1.02059579, -0.730872273, 0.478754908, -0.210190028, 0.556650937, -0.0836573839, -0.428684831, 0.475618631, 0.26693821, -0.0365147106, 0.349770874, -0.296871215, -0.461401045, 0.932147861, -0.574303329, 0.337240696, 1.84354556, -0.531826258, 0.684611261, 0.230101213, -0.265553534, 0.351761222, -0.155148238, 0.210944265, -0.266109228, 0.320440918, 0.119257875, 0.288138092, -0.342955351, -0.413885891, -0.525543213, -0.563633621, -0.26180914, -0.464125246, 0.587187707, 0.672474265, -0.593278229, -0.299270064, -0.353163183, -0.463583589, -0.00285831909, -0.251852244, -0.532872677, -0.0746277645, 0.717572629, 0.203225821, -0.289940834, -0.307978928, -0.279727012, 0.257997662, 0.563363969, -0.126924291, 0.392226875, -1.30514491, -0.0880905986, 0.494673967, -0.658143938, 1.59869182, 0.759586871, 0.277507126, -0.217861027, 0.398876876, -0.492357105, -0.282907367, 0.813215792, 0.627021313, -0.321904421, 0.363541245, -0.311341137, 0.114971392, 0.586712539, -0.438207448, -0.291453928, 0.183375284, -0.316651762, 0.33620429, 0.418325275, -0.810234189, 0.564028382, -0.281237781, -1.54698515, 0.64791584, -0.66442287, -0.140249655, 0.357892454, -0.271120518, -0.0289524198, -0.137522936, 0.168941945, -0.435024828, -0.443703264, -0.342307836, 0.250819564, 0.352735728, 0.470329642, 0.484651417, 0.17451258, 0.504986525, -0.489991665, -0.452524006, 0.48424527, 0.453603983, 0.420602649, 0.463263929, -0.239898235, 0.244296864, 0.545481205, -0.197661057, -0.449634731, -0.223071486, 0.32376349, 0.377509594, 0.199731633, -0.298727512, -0.554720581, 0.451484352, -0.285018682, 1.16988611, 0.0934815109, -0.358396918, 0.328986198, -1.4225142, -0.614723146, -0.273198545, 0.22736989, -0.557725787, -0.351461083, -0.262877256, 0.811221361, 0.416087955, -0.510921419, 0.461658508, -0.567678869, 0.33768183, 0.472564608, -0.607918084, -0.25393039, 0.224310562, -0.32430318, 0.35536015, 0.607146919, -0.650484383, 0.625925839, -0.362202227, -0.8074193, 0.735684514, -0.70511049, -0.265186429, 0.325658977, -0.412962407, 0.18513383, -0.42445606, 0.303192258, -0.305631042, -0.355679244, -0.420834124, 0.273631752, 0.425167948, 0.594565034, 0.507372856, 0.183894157, 0.542529643, -0.518569767, -0.60572201, 0.685898781, 0.293093473, 0.42061916, 0.299018055, -0.277766168, 0.450671166, 0.341782182, -0.327823669, -0.508060336, -0.290250212, 0.362154663, 0.246053413, 0.241558269, -0.251524419, -0.508265316, 0.250327438, -0.392809272, 0.668544412, 0.436275512, -0.586359143, 0.622453272, -0.81871587, -0.55931741, -0.30781436, 0.328269511, -0.407830954, -0.387682945, -0.0372718908, 0.546487033, 0.632412314, -0.494615287, 0.484569222, -0.335046232, 0.400614917, 0.409777731, -0.785230041, -0.35260576, 0.146089226, -0.41855368, 0.350596845, 0.767834604, -0.553323448, 0.557047486, -0.474052519, -0.851296663, 1.20988882, -0.479504496, -0.47507292, 0.252668232, -0.0768971816, 0.10374929, -0.491340846, 0.167298138, -0.135968253, -0.237201631, -0.539235413, 0.266471863, 0.764274776, 1.06963873, 0.64189136, 0.258160442, 0.773039699, -0.597770989, -1.18434858, 1.07148314, 0.604650915, 0.436439157, 0.245012432, -0.211310655, 0.393630803, 0.334076166, -0.392476201, -1.0658356, -0.247959822, 0.362116396, 0.347162098, 0.382426381, -0.0759491622, -0.601584256, 0.407191366, -0.328497529, 0.781683564, 0.318506658, -0.326974452, 0.927063286, -0.62534368, -1.00211442, -0.233628362, 0.503780782, -0.579641759, -0.510079503, -0.225645274, 0.714158595, 0.562757492, -0.41103372, 0.357707769, -0.349875361, 0.383057445, 0.474146307, -1.10002911, -0.351130009, 0.233985648, -0.387513161, 0.255342811, 0.734385729, -0.669323981, 0.4122141, -0.628313184, -0.787473977, 1.24135518, -0.668933749, -0.559095502, 0.493527651, -0.325537354, 0.203377366, -0.4349356, 0.218989521, -0.266290963, -0.250037432, -0.707569301, 0.145341069, 0.838765979, 1.36045778, 0.589600563, 0.41397813, 0.701046765, -0.613428831, -1.41070533, 1.2054882, 0.640872717, 0.36385268, 0.334897906, -0.143711925, 0.392348975, 0.496713519, -0.244517505, -1.36358345, -0.466609299, 0.50618273, 0.453114003, 0.209123433, -0.0101209115, -0.494866222, 0.45383361, -0.415456951, 0.557616353, 0.488063991, -0.589736938, 0.964533627, -0.786089599, -1.40910828, -0.219961941, 0.69679755, -0.42304343, -0.0751851201, -0.0158687998, 0.524854839, 0.382059753, -0.380647719, 0.296273112, -0.221393883, 0.295532912, 0.207258373, -1.01958632, -0.419472277, 0.119841956, -0.231918409, 0.127797827, 0.693200946, -0.596327722, 0.273448795, -0.444010764, -0.650002062, 1.56623471, -0.508645296, -0.322794497, 0.232511312, 0.0286838915, 0.123914391, -0.478893369, 0.0807095543, -0.0190814249, -0.138284802, -0.594440401, 0.161965251, 0.646832049, 1.39575422, 0.672821045, 0.266411602, 0.6013605, -0.208654016, -1.19242501, 1.31982136, 0.38568151, 0.303202957, 0.202859864, -0.0928090587, 0.347312659, 0.315423042, -0.12567246, -1.46938014, -0.267662674, 0.402740896, -0.0137400124, 0.0410433933, 0.104746483, -0.513144255, 0.184428141, -0.265233636, 0.507298529, 0.334750563, -0.241917416, 1.19321907, -0.509043217, -1.28002822, -0.154179201, 0.46423164, -0.425630748, -0.377833992, -0.308563799, 0.503439784, 0.566137612, -0.329539478, 0.425764769, -0.447303951, 0.275466025, 0.301733613, -0.909776688, -0.281282872, 0.19528611, -0.443917394, 0.446689099, 0.604748964, -0.472025454, 0.362883776, -0.586260378, -0.786115766, 1.10065484, -0.663078666, -0.53651011, 0.513481915, -0.268212765, 0.135437921, -0.293859124, 0.201443642, -0.263526827, -0.191120133, -0.507800221, 0.197312221, 0.61701107, 1.18685925, 0.58754468, 0.339690387, 0.543017268, -0.573801339, -1.25017965, 1.26668549, 0.644240022, 0.227935314, 0.239973575, -0.0955443829, 0.429756433, 0.310308695, -0.327461034, -1.12692904, -0.343368918, 0.404465795, 0.285750985, 0.347576022, -0.193942234, -0.509978712, 0.299390674, -0.408819109, 0.613180876, 0.50600493, -0.383563101, 0.823956847, -0.557829618, -1.04754567, -0.14566049, 0.683749676, -0.417017907, 0.141781881, 0.0743693039, -0.132111654, -0.194817632, 0.239561945, -0.203357652, 0.129579425, 0.243770778, -0.162329704, -0.120766371, -0.304414809, -0.100198939, 0.306472868, -0.205838069, 0.228253603, 0.0499281138, -0.0701815933, -0.350182891, -0.102613375, 0.308618367, 0.0602031201, -0.356271297, -0.215074703, 0.0202723313, 0.339929104, -0.35398379, -0.0955704078, 0.054202728, 0.199776128, -0.264065534, -0.272960156, 0.252726734, 0.197265312, 0.293150187, 0.241630673, 0.224784866, 0.0434284359, -0.270462722, 0.32273671, 0.330430359, -0.057046663, -0.11925932, 0.302505672, 0.173419356, -0.056487646, -0.131198362, -0.121880151, -0.250820816, 0.220319062, -0.0528289527, -0.267461002, 0.34639132, -0.068936266, -0.145081401, 0.209030926, -0.0336397141, 0.296665043, 0.0556676574, 0.282968313, -0.196078867, -0.392456293, 0.0977721214, 0.126284763, -0.0385491028, -0.536525786, -0.216324195, 0.917357683, 0.536329627, -0.551019132, 0.495584935, -0.356248587, 0.0713457093, 0.452945203, -0.551084518, -0.223783389, 0.23693043, -0.475640595, 0.480812252, 0.483833313, -0.90822643, 0.466743559, -0.492364109, -1.43452275, 0.66220808, -0.800147474, -0.287594885, 0.49357149, -0.400070131, 0.0161626022, -0.284491211, 0.356228054, -0.332562715, -0.46980533, -0.303855091, 0.407975286, 0.441551328, 0.45449084, 0.380961061, 0.376776457, 0.403666914, -0.517319918, -0.723441899, 0.774898529, 0.332766831, 0.347670108, 0.34094736, -0.253277391, 0.293842703, 0.526172578, -0.283712655, -0.712753057, -0.20704098, 0.165279225, 0.358801842, 0.494020849, -0.328629881, -0.772424579, 0.380714238, -0.42599535, 1.14401996, 0.355478346, -0.508070111, 0.439177215, -1.32407653, -0.469580084, -0.414156139, 0.241568148, -0.484124035, -0.276388198, -0.261566132, 0.653547585, 0.59162581, -0.422252506, 0.424493521, -0.599047959, 0.258712322, 0.441181451, -0.53624934, -0.186149001, 0.276645988, -0.383999735, 0.443050385, 0.489643008, -0.733591199, 0.614002407, -0.534607351, -0.705386817, 0.529855013, -0.53553319, -0.261432081, 0.310381442, -0.319335639, 0.267668366, -0.359064192, 0.182456613, -0.20163992, -0.45611757, -0.396166146, 0.226411417, 0.597525537, 0.497735977, 0.519696236, 0.393224806, 0.501320422, -0.6284495, -0.796498358, 0.649134874, 0.404830784, 0.374959826, 0.532537162, -0.0843869746, 0.495871365, 0.55207634, -0.153529882, -0.76127553, -0.440744579, 0.39312306, 0.434141517, 0.313946664, -0.260658473, -0.664929032, 0.20010671, -0.28246513, 0.68965894, 0.159476191, -0.541988015, 0.612759888, -0.686699986, -0.721419275, -0.159214392, 0.563255191, -0.451826155, -0.404601485, -0.129923105, 0.768116534, 0.457714319, -0.282415062, 0.518207252, -0.545926452, 0.202296808, 0.334579706, -0.539969027, -0.0623441637, 0.186650351, -0.314906806, 0.295887321, 0.349980056, -0.642017603, 0.412462145, -0.309073955, -1.63875937, 0.440417379, -0.617059648, -0.303727299, 0.303480119, -0.199189305, -0.0904858708, -0.247963756, 0.236305654, -0.32573244, -0.384526402, -0.379666358, 0.305572599, 0.2990233, 0.532991648, 0.44215709, 0.0943114758, 0.460006803, -0.413071066, -0.602228284, 0.655565858, 0.306779355, 0.375284523, 0.392729402, -0.31339851, 0.310526878, 0.321203232, -0.0857086107, -0.340077549, -0.158091217, 0.276746541, 0.313685209, 0.222494602, -0.0896148905, -0.662942171, 0.40668714, -0.226965919, 1.21436954, 0.116670243, -0.460618585, 0.379437119, -1.43157935, -0.497810781, -0.268609434, 0.2691257, -0.4374744, -0.544128656, -0.153738856, 0.806466758, 0.697766304, -0.308749884, 0.279687375, -0.616335094, 0.0378023386, 0.631812394, -0.61610961, -0.324923128, 0.246356532, -0.479753315, 0.498239189, 0.320099026, -0.879978836, 0.413096756, -0.27323848, -1.64678144, 0.718110323, -0.815286458, -0.438307106, 0.39924106, -0.232177705, -0.013364736, -0.314342916, 0.349587202, -0.35428375, -0.342492789, -0.488959461, 0.243335634, 0.580216885, 0.686432123, 0.512776315, 0.37325263, 0.457635701, -0.666968644, -0.518783569, 0.760379374, 0.273760647, 0.537627399, 0.460816681, -0.324044377, 0.370896131, 0.465907395, -0.0126787117, -0.595686376, -0.374347538, 0.222507402, 0.428265959, 0.479308754, -0.270265073, -0.590712905, 0.396659136, -0.344178051, 1.16334081, 0.384546846, -0.527725339, 0.435495198, -1.30978096, -0.696059883, -0.320203543, 0.229033664, -0.650147617, -0.273492187, -0.164835364, 0.668667018, 0.629295409, -0.522264779, 0.330360919, -0.60428226, 0.169723704, 0.471017838, -0.589739799, -0.172625318, 0.290637463, -0.357112855, 0.482530624, 0.596085727, -0.593576312, 0.496339232, -0.396099567, -0.791489959, 0.523505449, -0.698192954, -0.24262999, 0.361119211, -0.375197023, 0.307743907, -0.457079798, 0.203491971, -0.218809396, -0.207070023, -0.5566383, 0.21313338, 0.587665677, 0.590981603, 0.460330576, 0.381497055, 0.31396991, -0.406499654, -0.646273673, 0.782972097, 0.285102636, 0.433285028, 0.391306609, -0.333679378, 0.320724577, 0.434925884, -0.342287928, -0.727689326, -0.217701256, 0.270231545, 0.473350465, 0.303761214, -0.402583748, -0.546936989, 0.436739236, -0.509154141, 0.763270915, 0.269892544, -0.616448164, 0.659267008, -0.929162681, -0.668321013, -0.337674767, 0.440619588, -0.591116369, -0.563047826, -0.26057142, 0.969926476, 0.607192755, -0.409259439, 0.310617298, -0.471728027, 0.339939326, 0.551383674, -0.62580049, -0.172993213, 0.240941212, -0.26740551, 0.305900991, 0.347701877, -0.878069222, 0.515981078, -0.537627876, -1.17052972, 0.755907178, -0.639583409, -0.47517246, 0.346790433, -0.219063297, 0.0348705351, -0.292179734, 0.474882126, -0.386153251, -0.213677242, -0.456836134, 0.324294567, 0.331846178, 0.537104189, 0.436003745, 0.144273177, 0.530209661, -0.426131099, -0.735307217, 0.718763411, 0.453274429, 0.469704777, 0.321545869, -0.21566245, 0.424108654, 0.344189733, -0.0592800081, -0.521855295, -0.107721195, 0.317939609, 0.430018395, 0.457768142, -0.172899276, -0.612234235, 0.406998247, -0.448220253, 1.11257839, 0.191234738, -0.479058534, 0.481455982, -1.12707865, -0.648124576, -0.194276959, 0.345581084, -0.484572679, -0.343308598, -0.12794216, 0.672531426, 0.424719602, -0.302648067, 0.359854698, -0.400834858, 0.473584592, 0.422555357, -0.678353608, -0.261491418, 0.217765197, -0.171049848, 0.285351127, 0.513761342, -0.658162415, 0.46343568, -0.548393846, -0.617358863, 1.1439836, -0.508872807, -0.538265049, 0.477225065, -0.299464107, 0.22175248, -0.313081294, 0.371365666, -0.230835333, -0.145164087, -0.441226751, 0.414759785, 0.584097981, 1.06914091, 0.552144825, 0.320418417, 0.714488447, -0.354277045, -0.928710818, 1.1338594, 0.36863628, 0.266910672, 0.392667323, -0.0111860326, 0.355612755, 0.278948724, -0.428407669, -0.807357132, -0.262119412, 0.42804426, 0.205490455, 0.33340618, -0.288222104, -0.650719345, 0.412516952, -0.491195202, 0.773645103, 0.364975005, -0.519680321, 0.906551361, -0.524672151, -1.01487565, -0.39606598, 0.405813515, -0.563595951, -0.269886643, -0.350732118, 0.606613576, 0.384260803, -0.376138091, 0.508033037, -0.360961974, 0.466318488, 0.277735382, -0.66640687, -0.35502246, 0.109514922, -0.298087895, 0.355182439, 0.646670938, -0.632044554, 0.439749837, -0.382921994, -0.660431385, 0.893898308, -0.540391684, -0.321551055, 0.221916288, -0.160736755, 0.308179349, -0.26730603, 0.206497774, -0.225358516, -0.351685643, -0.558867693, 0.374778271, 0.612612009, 0.978533804, 0.607411861, 0.285413414, 0.51165098, -0.344507605, -0.921458423, 0.888002694, 0.500364721, 0.202447027, 0.380399704, -0.271877974, 0.380116731, 0.526907861, -0.218600065, -0.825426459, -0.240812227, 0.396916181, 0.264241874, 0.365629554, -0.171145856, -0.403258473, 0.408908993, -0.489471793, 0.606956661, 0.459666014, -0.463012695, 0.852094889, -0.780032933, -0.761940658, -0.291623026, 0.498924643, -0.302560419, -0.171400279, -0.33405292, -0.0493575782, 0.17232205, -0.110599153, 0.329337597, -0.357625425, -0.234940618, 0.152215123, 0.319324821, 0.43764329, 0.386182725, -0.177471906, 0.32160902, -0.474107057, -0.00973141473, 0.0944921076, 0.322700441, 0.0120441252, -0.451121688, -0.0308260825, 0.433692187, 0.224495098, -0.292792976, -0.511347592, 0.473475844, 0.262363851, -0.240330055, -0.421176165, 0.369746774, 0.432316303, -0.436458081, -0.277693868, -0.514254212, -0.520781636, -0.385244131, -0.155822918, 0.358417571, -0.188162878, -0.299654812, 0.237457052, 0.241685927, -0.423709124, -0.283290237, 0.1787242, 0.314056337, 0.152405173, 0.388397336, -0.299144179, 0.190873206, 0.425582856, -0.315479517, -0.129302844, 0.184376732, -0.328748405, -0.127442196, -0.323519915, -0.122181714, -0.446838707, 0.0990149751, 0.233083859, -0.313614875, -0.286455244, -0.108938903, -0.173898384, -0.154455885, 0.608990073, 0.639379859, -0.333209395, 0.214992166, -0.297589988, 0.255593807, 0.415786177, -1.06228507, -0.219749421, 0.0616546981, -0.0850304291, 0.217553958, 0.614582717, -0.527022839, 0.334150106, -0.680784225, -0.861281753, 1.82366407, -0.43191725, -0.372459769, 0.387694806, -0.0302853379, 0.131834209, -0.512922108, 0.107565053, -0.224938229, -0.319808245, -0.549067795, 0.112411819, 0.703112602, 1.82133305, 0.7760638, 0.212270632, 0.559252858, -0.326964855, -1.57775831, 1.69533455, 0.496235013, 0.351062626, 0.150329247, -0.0431579985, 0.518127322, 0.488872588, -0.182545111, -1.98710394, -0.428537518, 0.527171254, 0.13654837, 0.316436887, 0.0261419453, -0.339206904, 0.154128537, -0.293990165, 0.695450902, 0.270007789, -0.371297151, 1.1685667, -0.692904472, -1.70720041, -0.161414593, 0.542755067, -0.368743628, -0.271216959, -0.350861341, 0.879380643, 0.389808565, -0.462255955, 0.25825274, -0.287204325, 0.0223016348, 0.572541773, -0.368543565, -0.262212306, 0.345916182, -0.206542492, 0.198395595, 0.438706398, -0.680423021, 0.421501189, -0.225021601, -1.4016006, 0.453847796, -0.717998624, -0.333025008, 0.322651654, -0.387569427, -0.0341551788, -0.28112945, 0.37996915, -0.186973631, -0.203572124, -0.152209431, 0.34419021, 0.34519434, 0.446676373, 0.446126312, 0.0983296484, 0.314393342, -0.616695642, -0.579172671, 0.402942836, 0.259942979, 0.484394908, 0.313688248, -0.130447447, 0.179317132, 0.490951687, 0.0383905619, -0.331919551, -0.27869752, 0.304098934, 0.407192022, 0.405362815, -0.326767892, -0.457747221, 0.379286647, -0.478376925, 1.23467183, 0.119863309, -0.276864558, 0.246494442, -1.32616842, -0.403463274, -0.377959818, 0.28082931, -0.308996797, -0.425722748, -0.193674147, 0.78785944, 0.508327127, -0.248903885, 0.264103949, -0.357186317, 0.0147308437, 0.409206808, -0.194472671, 0.00276197912, 0.258905709, -0.166197851, 0.420497239, 0.329626769, -0.692572415, 0.47229892, -0.0915081054, -1.23548186, 0.432720244, -0.532778084, -0.293897599, 0.351049364, -0.116568863, -0.0321129113, -0.00978968013, 0.194032043, -0.305195987, -0.331068963, -0.151935816, 0.279666692, 0.18866615, 0.430132568, 0.327653021, 0.187172294, 0.219540179, -0.436067939, -0.488186747, 0.306090027, 0.0649880245, 0.295697391, 0.304286689, -0.220163599, 0.218568921, 0.42988044, 0.083551079, -0.21370098, -0.24988465, 0.119232155, 0.42408514, 0.367069811, -0.316671014, -0.37558344, 0.158022285, -0.264873117, 1.1731286, -0.00102446123, -0.327192366, 0.419644058, -1.28937852, -0.396725744, -0.142590478, 0.174560189, -0.52244091, -0.0736855492, -0.00405138312, 0.502723634, 0.257404685, -0.20088473, 0.338655323, -0.30681926, 0.248688862, 0.340052962, -1.18811226, -0.305723131, 0.132275894, -0.0452247262, 0.171353057, 0.583092511, -0.487280637, 0.196598664, -0.483296543, -0.69260937, 1.35671079, -0.436298639, -0.381194085, 0.213245317, -0.139961824, 0.242243573, -0.332228541, 0.162442148, -0.0164368581, -0.134004563, -0.395557404, 0.153602988, 0.805303276, 1.37767732, 0.616612911, 0.365305662, 0.650224328, -0.22939913, -1.2560699, 1.10163033, 0.357846498, 0.065071173, 0.181495398, -0.0377712026, 0.388611585, 0.213618428, -0.107306898, -1.31008828, -0.177096337, 0.321845561, 0.218017265, 0.206176892, 0.00983442646, -0.525239408, 0.240989879, -0.143164024, 0.669313908, 0.247989461, -0.351266146, 1.11758339, -0.531946778, -1.49604833, 0.02928463, 0.581405699, -0.440303475, -0.385143578, -0.396308482, 0.750951886, 0.57296735, -0.446412802, 0.455750138, -0.418437362, 0.0957896784, 0.501497984, -0.44672817, -0.237872884, 0.274565369, -0.42142725, 0.489412338, 0.56970638, -0.710014164, 0.450249612, -0.278510541, -1.0801419, 0.788323283, -0.569819212, -0.344335169, 0.542477369, -0.337672293, 0.236581355, -0.170987174, 0.246147275, -0.266410828, -0.17478773, -0.250558347, 0.252318501, 0.381735712, 0.602397978, 0.616476417, 0.217723235, 0.384022832, -0.377786189, -0.662218869, 0.57415092, 0.349585682, 0.339607358, 0.465482593, -0.295192808, 0.506696105, 0.317660213, -0.0275208782, -0.636613369, -0.173345938, 0.383084655, 0.39059639, 0.437923908, -0.362441689, -0.492392182, 0.304834664, -0.277102828, 0.780932546, 0.358055443, -0.35449028, 0.648201704, -1.02766812, -0.65746969, -0.290710598, 0.266317517, -0.487403065, -0.342292964, -0.214244977, 0.737149656, 0.448120058, -0.230806604, 0.422618449, -0.292649239, 0.168079019, 0.534740627, -1.16855597, -0.432713687, -0.0108646816, -0.126822308, 0.25649479, 0.770150781, -0.645632446, 0.403120458, -0.724118412, -0.859452844, 2.22503901, -0.64947921, -0.367921531, 0.358518481, -0.155806094, 0.193853229, -0.297354549, 0.120156467, -0.0946324617, -0.243912473, -0.472326577, 0.145495683, 0.832385361, 2.19498634, 0.778509676, 0.342008919, 0.848277271, -0.49624604, -1.69642162, 1.71654153, 0.588248074, 0.33258453, 0.344076008, -0.163638383, 0.56731528, 0.247680068, -0.354752421, -2.37261987, -0.398869097, 0.391421556, 0.352473855, 0.115878321, -0.112021856, -0.472907096, 0.381194562, -0.418286622, 0.543751717, 0.30754447, -0.280784011, 1.41610241, -0.798416913, -2.10225344, -0.185180351, 0.510154903, -0.323697358, -0.458895683, -0.348646909, 0.705939233, 0.538262188, -0.513440371, 0.475339651, -0.328043967, 0.384672582, 0.44323957, -0.761635363, -0.270843118, 0.261911571, -0.252113491, 0.381079525, 0.609498322, -0.450055778, 0.356651932, -0.491022676, -0.810506225, 0.82410872, -0.578057647, -0.521694124, 0.423432797, -0.246942252, 0.291828603, -0.274428874, 0.34558928, -0.163658366, -0.2072023, -0.667214453, 0.331220478, 0.769516528, 0.815972626, 0.761667073, 0.519886792, 0.735126495, -0.363234431, -1.01916885, 0.980866015, 0.465000719, 0.297353357, 0.268718481, -0.133869484, 0.596612692, 0.272900581, -0.374923646, -0.764245868, -0.400829643, 0.387301534, 0.411194116, 0.458122432, -0.0897585005, -0.611259997, 0.396098167, -0.514478326, 0.615652442, 0.469147056, -0.551474094, 0.677580595, -0.723048508, -0.958446622, -0.351297438, 0.5369609, -0.466082484, -0.392684519, -0.140763402, 0.738301575, 0.505346894, -0.551214337, 0.488818526, -0.464140445, 0.197854578, 0.394551396, -0.906450927, -0.236846372, 0.0841318369, -0.367447346, 0.449851722, 0.773675323, -0.738755822, 0.441427588, -0.654032588, -0.711928427, 1.18266237, -0.549853086, -0.460477382, 0.219276875, -0.149520844, 0.179480404, -0.431614518, 0.197724342, -0.272667557, -0.340881646, -0.565278411, 0.232482374, 0.804801285, 1.03302395, 0.805033445, 0.504528701, 0.587796926, -0.4402273, -1.21261656, 1.17494059, 0.443305463, 0.264766097, 0.316561788, -0.138892338, 0.65940237, 0.564585388, -0.31081444, -0.90176338, -0.471996456, 0.371961445, 0.158505559, 0.370738208, -0.0978980586, -0.373646945, 0.392568529, -0.308288038, 0.779628813, 0.232412338, -0.372803688, 0.794813037, -0.738244116, -1.15833187, -0.373204678, 0.6222229, -0.539139509, -0.443403453, -0.290466309, 0.819968641, 0.527707577, -0.413294584, 0.274637192, -0.467576206, 0.0177975688, 0.598754168, -0.495468289, -0.163562313, 0.17254664, -0.416864395, 0.243399248, 0.288690567, -0.750119209, 0.554691315, -0.208583638, -1.92795444, 0.496306002, -0.850651801, -0.344283283, 0.44015038, -0.395032018, -0.0522430316, -0.25097248, 0.401277214, -0.398269415, -0.220324293, -0.422234803, 0.186774373, 0.392636329, 0.649317384, 0.484548628, 0.120573297, 0.480113119, -0.571780026, -0.65580982, 0.513943195, 0.472561806, 0.326867461, 0.286692291, -0.303493977, 0.462431997, 0.504831314, -0.20678623, -0.445540279, -0.0930512697, 0.290064484, 0.194492519, 0.420097232, -0.199875414, -0.649175227, 0.197605386, -0.534060299, 1.32834315, 0.113373868, -0.361338526, 0.44961217, -1.64719367, -0.678484142, -0.303245872, 0.287665248, -0.575748205, -0.336794019, -0.0869292989, 0.432107985, 0.486114502, -0.221369773, 0.288731098, -0.318255961, 0.268310964, 0.240426511, -1.1222862, -0.309996933, -0.0533496514, -0.178539693, 0.306757689, 0.708717108, -0.463632852, 0.213827491, -0.629661322, -0.744728744, 1.77040315, -0.515126169, -0.487291873, 0.264207542, 0.00132249307, 0.323194981, -0.497462869, 0.182954505, -0.23436442, -0.187767476, -0.705290735, 0.164230332, 0.66266185, 2.02163887, 0.588158846, 0.303405881, 0.737843692, -0.390376419, -1.43576646, 1.54322898, 0.434838712, 0.145693526, 0.30881536, -0.0685351416, 0.342455328, 0.24507685, -0.27616778, -2.15865946, -0.287609041, 0.460926324, 0.190310925, 0.0574499927, 0.100047357, -0.557812035, 0.199095517, -0.114541799, 0.670535684, 0.32147494, -0.418899715, 1.15679395, -0.762430549, -1.66618228, -0.093862243, 0.486004472, -0.202861622];
    recurrent_3_r : ARRAY[0..4095] OF REAL := [0.00911375321, -0.00202236348, -0.0237983093, -0.0230638143, 0.0748881623, -0.0255280919, 0.032285504, -0.00382772577, 0.110893279, 0.0975007489, 0.0418522805, 0.0609153658, 0.0313407704, 0.0302556343, 0.0175146423, -0.0281471703, 0.0318852216, 0.0426676609, 0.0123656504, 0.1041703, 0.0541706048, -0.000886218622, 0.197626323, 0.0429425202, -0.0799675807, -0.00761905871, 0.00706546754, -0.0571719408, -0.0689751357, 0.0451986678, 0.0201027133, 0.0631553233, -0.129691571, 0.0320937745, 0.0302708726, 0.121609271, -0.112159126, -0.0793186352, 0.0803062767, 0.0614077896, 0.00459189387, 0.0504808798, -0.125838056, 0.176575303, 0.0082402043, 0.0200517774, 0.0343972668, -0.0574389771, 0.110039622, -0.0383961499, -0.114136584, -0.0274701472, -0.0615831465, 0.0620580614, -0.022973517, -0.00469653029, -0.0329369009, 0.0095978938, -0.056178797, 0.0776937082, 0.0561335124, 0.132600427, -0.100108549, 0.0226371828, 0.0583960861, -0.0655008852, -0.00749516673, -0.0113983564, -0.0423510447, -0.0797068775, -0.0199018288, 0.0782541484, -0.0776402503, -0.0815584138, 0.154344261, 0.116309933, -0.0853010118, 0.0429037586, -0.111408979, 0.0519659445, -0.0714104623, 0.0202703439, 0.0431506336, -0.0217190031, -0.0993405879, -0.0339033231, -0.0319767073, 0.0969930366, -0.0934475288, 0.0431513488, -0.0437430516, 0.0551541001, -0.102149546, -0.0419385284, -0.0510420054, 0.104995966, 0.00981811248, 0.054826092, -0.0460422263, -0.14945735, -0.0887676179, 0.0757255033, -0.0682021081, 0.067138575, 0.0527030081, -0.142467126, 0.00623679161, -0.081650205, -0.0217414498, -0.0519152284, -0.0114929061, -0.0353443436, 0.0697723329, 0.0216454808, -0.147972912, -0.0305027403, 0.00866494142, -0.0361279584, -0.0156128649, 0.0648681819, -0.0711312518, 0.0697998106, -0.0817103982, 0.0791503042, 0.167355821, -0.0372648276, -0.0513354391, 0.120582767, -0.0890771151, 0.0257072933, -0.123685598, 0.0827882737, 0.0198066384, -0.0830840692, -0.0058414354, -0.11684899, 0.11155083, -0.0375803076, -0.0860175788, 0.108100832, 0.00140646752, 0.00455251336, 0.00355935167, 0.104866102, -0.183338359, 0.19762516, -0.02773319, 0.0545151457, -0.0323703475, -0.0841021389, -0.020246096, 0.103897557, 0.0332882218, 0.122344576, 0.0356296748, -0.0390966535, 0.0482734516, -0.0153638236, -0.0705761611, -0.0545569919, 0.0216887072, 0.0146980723, 0.134173021, -0.0277683474, 0.108473256, -0.00895685516, -0.000122845173, -0.148091972, 0.00765258633, 0.112680122, 0.0627765208, -0.0699514449, 0.0579327606, 0.167391047, -0.0206126291, -0.0232587494, -0.0227806028, 0.164959013, 0.017952228, -0.029058177, 0.0931209773, -0.0905666649, 0.0297105536, 0.0643432513, -0.0572242662, 0.00399557408, 0.0640901178, 0.0284853913, -0.0532626435, -0.093953222, -0.116984934, 0.00363150612, 0.0778844729, -0.0534194075, 0.0356680602, -0.0513897985, 0.0127216633, 0.0420455039, -0.026197603, 0.047176417, 0.0816618875, 0.00285134348, 0.0223577488, 0.0966080576, 0.00698447414, 0.0076117944, 0.041453708, -0.0264793001, 0.0078772828, 0.0449370891, -0.114559084, -0.0222518574, -0.0767178088, 0.0344772972, -0.0263515487, 0.00535550434, 0.0400021747, 0.0447246432, -0.0108250044, 0.00396102015, 0.0204284508, 0.071688287, -0.0889900625, -0.0552459359, 0.0875648484, -0.0842856988, -0.0550064743, -0.101071484, 0.0326540209, 0.0544580296, 0.0738798827, 0.00837158598, -0.0739922822, 0.031114623, 0.0112157539, 0.047144495, 0.129318848, -0.037200179, 0.118786499, -0.0740327165, 0.0661123395, -0.0531371832, -0.0284307264, -0.108321421, -0.100672431, -0.029302977, -0.101315923, -0.177598029, -0.092394568, 0.0691574663, -0.0419421941, 0.0279376302, 0.158116013, -0.0253254287, 0.0146561749, -0.047278095, 0.033318989, -0.0360458903, -0.0600628331, 0.0303683579, -0.0589155927, -0.0240204073, 0.0839619339, 0.0034722772, -0.0770511553, 0.0292353425, 0.0550547764, 0.00291131251, -0.0408926569, -0.01090765, -0.0305658355, 0.141737267, 0.021275593, -0.123218119, -0.0334331989, -0.0504225008, 0.0127103962, -0.0695255473, 0.0296204053, 0.0265006982, 0.0580648482, 0.0501579717, -0.0626788139, -0.0789386332, -0.0628380179, -0.0720427558, 0.0320159942, -0.0315630734, -0.10637518, -0.0208138376, 0.00724740699, 0.0239238143, 0.0816971362, -0.0362997353, -0.10336107, -0.00830980577, -0.0301181413, 0.0565131381, 0.0499073453, -0.000258012209, -0.0084053874, -0.0921288431, -0.002275832, -0.114925586, -0.0470449179, -0.106850281, -0.0981545299, 0.0292031579, 0.127993435, 0.023694573, -0.0580891445, -0.108017705, 0.0432504714, 0.0474100932, 0.0421978645, 0.0362437442, 0.00868836232, -0.0331392735, -0.0259158984, -0.0993543863, -0.091642648, -0.0400814563, 0.0184793398, -0.0358050019, 0.143999591, -0.023802178, -0.0589483343, 0.0488821268, -0.0130757075, 0.0715813115, 0.0435160547, 0.0556875393, 0.0652761608, 0.000147297047, 0.0398971811, 0.0967640653, 0.0463042036, 0.00411752611, 0.00755714439, 0.0722247064, 0.0147378575, -0.147983626, -0.0114682335, -0.119335331, -0.0348146968, 0.0757440105, -0.0889739841, -0.171713427, 0.0727809593, -0.109121919, -0.0193136204, 0.107689202, -0.031507574, -0.0489449948, 0.0480983704, -0.0117908092, -0.0625669062, -0.0629829913, -0.0509033576, 0.14963536, -0.101753235, 0.0575250536, 0.0423747487, -0.135954604, 0.00802879781, 0.138046563, 0.203562587, -0.0937730521, -0.043450743, -0.0903653726, 0.0496570095, -0.101320013, -0.0425310731, -0.0388302952, 0.0215265229, -0.0114472369, -0.160118356, -0.0577234179, -0.056208618, -0.159860149, -0.130893126, 0.0153518021, -0.0469167009, 0.0170055293, 0.0609783083, -0.0040185065, 0.0274109729, 0.11365439, 0.00275870599, 0.00512488326, -0.0133355847, 0.094586432, 0.102978855, -0.0182318985, 0.0394562408, 0.024214007, 0.00501166517, 0.146497458, 0.0535710938, -0.167801186, 0.0870854333, -0.0367849171, 0.127105713, -0.0133330319, 0.0571585521, -0.131522089, 0.0820833668, 0.0694639385, -0.00270178728, 0.0746649206, -0.0351437517, 0.0531759933, 0.107341737, -0.0166541357, 0.0899687558, -0.135554671, 0.107365236, -0.0745012611, -0.121961415, 0.00332099153, 0.0623820536, -0.0855424553, -0.144670919, -0.00410610996, 0.018668985, -0.0468354598, 0.104753383, 0.116255291, -0.0909991711, 0.0423864201, -0.0167759657, 0.112893499, 0.0140526397, 0.0157002211, 0.025987532, -0.0515090972, 0.0492114387, 0.0286730602, -0.00728053227, 0.0730762854, -0.0576741025, 0.0987064838, -0.12626642, 0.0363303982, 0.00025613606, -0.0854930282, 0.0409880728, -0.0491628014, -0.0495841466, -0.0832021907, 0.109828413, -0.00949191209, 0.025237117, 0.122777909, 0.0256123319, 0.0638817549, 0.00852558389, 0.0977258906, 0.165678307, 0.0380590409, -0.040783532, -0.0961662456, 0.0668946505, -0.0157988425, -0.0765058249, -0.0761791319, 0.127417073, -0.00562030124, -0.0150924847, 0.0162233636, 0.0635270476, -0.121701874, -0.0227665529, -0.0745811015, 0.00387974456, 0.0041704569, -0.0789878815, -0.0486721024, -0.00843084604, 0.0702937096, 0.030550193, -0.0509378761, -0.0183612444, -0.141379282, 0.118152753, -0.0668954402, -0.0372721925, -0.0300644953, 0.0570926517, -0.0313790515, 0.0383626595, 0.12200132, 0.069827117, 0.0511526726, 0.105546087, 0.111735642, 0.0725364089, -0.0557615533, 0.060444653, -0.0400662571, -0.0745078549, -0.0652316064, -0.0708966032, -0.0220151078, 0.0539559312, 0.0375150554, 0.0141001325, 0.0504179634, -0.0686047524, -0.0137163773, -0.0515023954, 0.0290786456, 0.0783781409, -0.0577777997, 0.013601426, -0.037097238, -0.0802973881, -0.0311410725, 0.000239511253, 0.0391602069, -0.102556601, 0.0228124075, 0.0532910526, 0.00637396704, 0.211682871, -0.0590877682, -0.0185743347, -0.116268821, 0.123046994, 0.0638253465, 0.103012592, -0.0295602046, -0.0184217803, -0.126529723, -0.021587871, 0.0466953442, -0.0207868125, -0.0102520138, 0.0223338567, -0.0615631379, -0.0313155428, 0.0144809857, 0.0701513886, -0.0250683762, 0.0702576339, -0.104813933, 0.0414853878, 0.0486246869, -0.0420227423, 0.0235443022, 0.0312029328, -0.0468768179, -0.0021700263, 0.122100636, 0.0458291471, -0.0841060728, 0.0307521727, 0.120696224, 0.0763218403, 0.124105752, -0.0635750741, 0.0466547534, 0.0204870068, 0.0262179971, 0.00880821981, -0.134466439, 0.0516617745, 0.0791150853, 0.158821866, -0.0417293124, -0.0195431169, -0.0592326075, 0.0584496781, 0.0470124222, -0.0392942876, 0.0094333142, 0.0206860416, 0.160820901, -0.00310400408, 0.0299142431, 0.00139450654, 0.062466152, 0.05967924, -0.0433351211, 0.0331435986, 0.0972179025, 0.105120547, -0.0478204675, 0.0743556842, -0.0672744066, -0.046730414, -0.246408552, -0.0541513227, 0.00750867184, -0.0652973503, 0.0212405361, -0.02554431, 0.00203400478, 0.0351974927, 0.0219492614, -0.0213655662, 0.120339364, 0.0119028874, -0.034202572, -0.00784637406, -0.0541388094, -0.0597577617, 0.0158543289, 0.091164723, -7.52375927e-05, 0.0459715798, 0.0581619553, 0.0518091209, 0.00359082595, -0.0237384886, -0.147958845, 0.0622775517, 0.00865327567, -0.0153832324, -0.00439291075, -0.0402460471, 0.0388767943, 0.0856813192, -0.0089630885, 0.0840314776, 0.0315066054, -0.0487823747, 0.0760353208, -0.0752325878, 0.0017796047, -0.0281302053, 0.0624732561, 0.0957097262, 0.0376511998, -0.0715606511, -0.0852134004, 0.037225768, 0.0122167673, 0.0466136895, 0.038283091, 0.0952630118, 0.0974789783, -0.12276344, 0.00118430168, 0.0302159172, 0.00623338297, 0.018055059, 0.0586414635, 0.0171477292, -0.0526880771, -0.118420757, -0.124844752, 0.0284788664, -0.114810653, 0.0275984257, -0.0696739107, 0.0751996264, 0.095859915, 0.0687997341, -0.0259143673, 0.0121420603, -0.0324660055, 0.0405802354, -0.085328877, 0.119429722, -0.100314185, 0.102070868, -0.0252911821, 0.038893953, 0.0412346721, -0.0210889746, 0.129765391, 0.0169580691, 0.0226371624, -0.00887788087, -0.0572359003, 0.0157009233, 0.0193942357, -0.0108801918, -0.0912810713, -0.0476359725, -0.134074837, 0.0126453936, -0.0825806633, 0.0523258373, -0.0237158537, -0.0808548555, -0.091645591, 0.0902565494, 0.0146779232, 0.0990815386, -0.0994295329, -0.0455697812, 0.0555170365, -0.0137906522, 0.0581970885, -0.0395062715, -0.0858608931, -0.0830656365, 0.154364914, 0.14480707, 0.0541687235, -0.0914984494, 0.0245234314, -0.0803825408, 0.0533412918, 0.0108824316, 0.00130331982, -0.0745498165, 0.0868173093, -0.0637374967, 0.135478705, -0.0230534226, 0.0158655085, 0.0483710021, 0.0841864422, 0.135531038, 0.037712846, -0.0691346228, 0.0643537939, -0.00478052162, 0.111542173, -0.0323873013, -0.0721196979, 0.0629153326, -0.03225936, -0.0202114917, -0.0586395785, 0.0703757331, 0.105001338, -0.0352300443, -0.0207109638, -0.00277804397, -0.088710092, -0.00636978261, 0.0597423539, 0.1233472, -0.0532054417, -0.0184984189, -0.0356769115, -0.106631212, -0.078933306, -0.029100934, -0.0164433196, -0.100324057, 0.00681179203, 0.0538881905, 0.0577190667, 0.0235630125, -0.0408950746, -0.0765696466, 0.0572620928, 0.0715509504, -0.0141098583, -0.14256452, 0.0620078668, 0.0513346642, -0.014593279, -0.000190385617, 0.115069576, -0.00733298063, -0.0381898433, 0.0965593979, -0.082215935, 0.037181966, 0.057968311, -0.0169563778, -0.0351036116, 0.104300693, 0.131403923, -0.0407392234, 0.00248470437, -0.0625106692, 0.0529611409, 0.100966096, 0.0189072099, -0.0458419807, -0.0284237247, 0.0446987785, 0.0183654595, 0.0586776659, -0.0624799319, 0.116953477, 0.090016, 0.0165911783, -0.0229423959, -0.0926959291, 0.0235078447, -0.143053502, 0.0780783594, -0.0424500518, -0.0258744825, -0.13351348, -0.0939254463, -0.0294577107, 0.0331923179, -0.0493002273, 0.0673060417, -0.075317204, 0.0199663527, 0.0166395791, -0.0253233835, 0.0714993253, -0.0840470567, 0.116615638, -0.0817578733, 0.0800578892, 0.0296422839, 0.170557499, -0.1654616, -0.0277361833, -0.0246826354, 0.0284979492, -0.0261004046, -0.0193990432, -0.153675005, -0.000156990252, 0.0446386524, 0.00112404674, 0.00340267271, 0.110186473, -0.129498541, -0.0645064041, 0.0497275293, -0.01430069, -0.0417016521, 0.0662118047, 0.0380283259, 0.088968575, 0.0519468486, 0.0699722841, 0.0985773206, 0.01397039, -0.123004794, 0.050001882, 0.0688602924, 0.0884637237, -0.024484409, 0.0231193155, 0.0867063031, -0.117401488, 0.146742731, -0.0245518778, -0.00049746735, 0.107563034, 0.0153732263, -0.00138764642, 0.00719641149, -0.118613921, -0.0699281916, -0.0448083505, 0.0568592809, -0.03438925, -0.0568434261, 0.128248841, -0.0970832705, -0.131126106, -0.0322123691, 0.0494427308, 0.0349712223, -0.0516956002, -0.0108481338, -0.0205307081, -0.0627812296, -0.094834514, 0.0353070721, -0.0258042347, 0.139962509, 0.171861947, 0.00694552436, 0.0189717431, 0.0562504679, 0.0536639579, -0.012175221, 0.0922481269, -0.00224624015, -0.0172267184, -0.00408977456, -0.0315037183, -0.155455768, -0.0409466997, 0.13185519, 0.0294154324, -0.0134966858, -0.0774052441, -0.0542730987, -0.0419860855, -0.012225043, 0.081311509, 0.158177853, -0.0468696058, -0.0932726637, -0.0693122372, -0.00300208479, 0.0683663636, 0.0593294948, -0.0115551008, 0.179554924, 0.0512919687, -0.00133599411, 0.110675007, -0.0401133969, -0.000876663718, 0.151455745, -0.00121552218, 0.0146848718, -0.00242423825, -0.0363500565, -0.116146825, 0.079527013, 0.0865260661, 0.0545096248, -0.12196292, 0.0208703764, 0.0821463987, -0.0134822782, -0.027833946, 0.010675285, -0.0534569211, -0.15372014, 0.0209434144, 0.00385515532, -0.03036635, 0.0187385231, -0.0500814356, 0.00731410086, -0.0450109951, 0.0475450531, -0.0660711229, -0.0576170869, 0.0392976701, 0.0141733531, 0.105263107, 0.105541557, -0.0835994035, -0.0604783595, 0.0700645596, 0.00952682085, -0.060204614, 0.0383245014, -0.0303084739, 0.0449032895, -0.0314889662, -0.0117235109, -0.0435175374, -0.0120741315, -0.0456162468, -0.0304395314, 0.0392664373, 0.0543761477, -0.0223365463, 0.0479622632, -0.0356663093, -0.0946084857, -0.0987185538, -0.00450733677, -0.0622910261, -0.0854664817, -0.11624071, 0.0300633647, -0.0188361872, -0.196206644, -0.0151952319, 0.0356712975, 0.00420160685, 0.00529858842, -0.0407636985, -0.134199858, 0.0454469286, -0.0514911935, -0.0955984145, 0.0996576995, -0.0216490272, 0.0796884149, -0.0338479728, -0.0541275144, 0.114153914, -0.0927425176, 0.0597409792, 0.0275961626, -0.0266114324, -0.00144245848, -0.0843057185, -0.03371007, -0.000822213478, 0.137287915, 0.00845224597, 0.0294579789, -0.0588286072, -0.00748171657, 0.0366862677, -0.0881185085, -0.181755364, -0.0932161659, -0.0302605592, -0.004988058, -0.0171914734, 0.114152938, -0.0937477127, -0.107621804, 0.0418742374, 0.140122101, -0.109398291, -0.060850732, 0.0686470121, -0.000218321104, -0.0639985651, -0.0357726179, 0.110667303, 0.017532561, 0.0799096227, 0.0709084868, 0.0575583391, -0.0957374871, 0.0288257729, -0.0392640568, -0.124348633, 0.0544305295, 0.0763412863, -0.0880652219, 0.097671628, 0.047271423, -0.053128466, -0.0847817063, 0.0605234578, -0.0322612561, -0.0957455635, 0.163376689, -0.113794908, 0.0213765427, -0.0908470526, -0.0491742082, 0.0226370767, 0.0737887472, -0.0319020078, 0.0486837551, -0.0219347104, 0.0116338525, -0.0391337238, -0.0229025614, -0.055400338, 0.0399981774, -0.161445707, 0.0143578146, 0.108743295, -0.0870562717, -0.0278399661, -0.0423922464, -0.0586773343, -0.0430437848, -0.0837854445, -0.00241982192, 0.0739955232, -0.00983252376, 0.0226107929, -0.0281373821, -0.0663822368, -0.10870792, -0.0264889598, -0.0318740979, 0.0360140987, -0.0275817625, -0.0117399385, -0.0622121133, 0.0386478081, -0.138306975, 0.0722252876, 0.0681583658, 0.0357433297, -0.0503761508, -0.0888322741, 0.00609578472, -0.0550457835, -0.00491966493, 0.0018206574, -0.0777870715, 0.147252217, -0.0580721535, 0.00839607045, -0.0367960967, 0.0526871458, 0.112481609, -0.0370250121, 0.100097127, 0.0684277043, -0.0590134449, -0.000272998586, 0.0157443862, 0.0360369533, -0.00823564827, -0.11443729, -0.0748900771, 0.0570345223, 0.136014342, -0.00862678513, 0.0702614263, 0.0514154285, -0.0681594908, 0.0298552141, 0.00540684536, -0.0526974462, 0.0862854049, 0.0461132079, 0.10347601, 0.0749654993, -0.0231539886, -0.112434372, -0.0588796437, 0.0134588666, -0.131307006, -0.0329538956, 0.0385348871, 0.156908885, -0.0546470098, 0.00706227124, -0.00997575559, 0.0139146633, 0.0237259697, -0.00629263464, -0.0165242497, 0.090869844, 0.0364026949, -0.0375510603, -0.143859923, 0.0524707101, -0.0971896201, 0.00969352759, -0.0669112504, 0.100931376, -0.0398303121, -0.0936012641, -0.056639906, -0.0213063024, 0.175421089, -0.0735043213, -0.0395346321, -0.0607963353, -0.029217504, -0.0229287352, 0.042531345, -0.0905115232, -0.00708591565, -0.137183487, -0.0699275136, 0.107452646, -0.0319059044, -0.00441396236, -0.0106489789, 0.00246873125, 0.0293903332, -0.0112364143, 0.0890116245, -0.0172665641, -0.00711072702, 0.0278019793, 0.051202938, 0.054612495, -0.0475451201, -0.144114584, -0.0397719592, -0.113360614, 0.0785803273, 0.248093903, 0.0131256646, -0.0935446024, -0.0747676492, -0.00567668118, 0.00239985064, 0.0283464417, 0.111431696, -0.0532648116, -0.0453556739, -0.0236246549, -0.0972554907, -0.0118487664, 0.0293593854, -0.0276271068, 0.00488677248, 0.0133009003, 0.041428037, 0.0813874677, -0.00393976644, 0.0840215832, -0.0254320111, -0.0392817594, 0.00961663947, -0.085313648, -0.0234975703, -0.0803359449, 0.103493989, -0.0231693909, -0.0406989381, -0.057833001, -0.0455716588, 0.00552285463, -0.00918115489, -0.0363552719, -0.0460190773, -0.0786511749, -0.111753605, 0.0318435878, -0.0275966488, -0.146628007, -0.0202041827, 0.0246242601, 0.018335212, 0.0525075756, 0.0480933674, 0.015275049, 0.0815747604, 0.0505161509, -0.0541922376, -0.0505428798, 0.111340925, 0.0775246918, -0.0652684048, 0.0497954078, -0.202423543, -0.0580477528, 0.020171009, -0.00113054644, -0.0192843638, 0.0420398563, -0.0225126874, -0.00377615076, -0.0362481251, -0.0177948177, 0.0269957781, -0.00571646122, 0.0753164589, 0.0851424038, 0.0344276242, -0.0110771693, -0.0674054474, 0.0238144211, 0.0722684339, 0.127525941, 0.0353774205, 0.0332326517, 0.0574975386, 0.132011339, -0.021666646, 0.0812211335, -0.0385468937, -0.0912349299, -0.0816484094, 0.0864037871, 0.169749379, 0.0938792005, -0.0426299907, 0.0495092198, 0.044266887, 0.0522757173, 0.0168170929, -0.0512816086, 0.0146380551, 0.0567030497, 0.0319734029, 0.0424369946, 0.0125781037, -0.0639688969, -0.0218270272, -0.00753120333, -0.094087109, 0.0415724069, -0.0458106026, -0.191868842, -0.0353733376, -0.0827914998, 0.0222649202, -0.0110880127, 0.0588395298, -0.00075106509, 0.00630116276, 0.0508419052, -0.0973529369, 0.00889941677, 0.0150931329, -0.0762014017, -0.00210261345, 0.0544563234, -0.0157391671, 0.0114466082, -0.0318201222, -0.00051691226, -0.0407840647, -0.00694661075, 0.137765795, 0.0271868668, 0.0586328693, -0.0419846252, 0.0305384435, 0.0598569289, -0.0171761531, 0.0587193891, 0.0230484381, 0.12882179, 0.0120551828, -0.168238074, 0.0669286475, 0.0403562225, 0.0549735874, 0.066484943, -0.0145690329, 0.0632467121, -0.0359894931, 0.0815353915, -0.0462696441, -0.0617114268, 0.0324998535, 0.104943894, 0.0243134871, 0.0348146185, 0.111343443, 0.0185335688, -0.126225591, 0.0969006494, 0.0387630202, -0.197859943, -0.00749284029, -0.102993302, 0.093429096, -0.130881503, -0.0969738141, 0.159489989, -0.0507350154, -0.0478643775, 0.0019461792, -0.0112797022, -0.112410203, -0.00914694369, -0.0477013178, -0.0175735839, -0.0404180251, -0.0811169967, -0.0171765462, 0.0963852555, 0.114861697, -0.0139015261, -0.100321144, -0.0470585749, -0.0460179895, -0.162901118, -0.0248801392, -0.0205437746, -0.0337562151, 0.0522041097, -0.0410371646, -0.0846687555, -0.0636999235, 0.200840011, 0.0945674181, 0.0910367817, 0.0748383999, -0.140553772, -0.0284785368, -0.0362542495, 0.107232265, -0.0338969082, -0.0610294044, 0.0289454386, 0.0942899287, 0.0331130847, -0.0296364836, -0.0157973766, -0.110053211, -0.0952294171, -0.0308468044, -0.0917455107, -0.012321448, -0.026099572, -0.0903289616, 0.149475008, -0.0356912613, -0.0336054303, -0.0462723821, 0.0410968587, 0.0664142892, -0.0442651771, 0.0419820622, -0.00955121219, -0.0328969583, -0.0133415833, 0.0805753767, -0.0440384522, -0.0572364479, -0.0806434304, -0.199577808, 0.230586052, -0.0350115635, -0.0919062197, -0.142132744, 0.168537289, -0.00562704355, -0.0955159962, 0.0648066252, -0.0613829941, -0.0894394368, -0.0347663015, -0.028064115, 0.0362613648, 0.0463579334, -0.0798790306, -0.0732574761, -0.0253687128, -0.0559770465, 0.0480587594, -0.0656372085, 0.0877685621, -0.0300214272, 0.0177654028, -0.0479325876, -0.04533384, 0.00566974469, -0.160316736, 0.0640275702, 0.0861340314, -0.0507358126, -0.0361745469, 0.0520602651, -0.0654230267, 0.05035422, 0.0391078517, -0.0605994686, -0.0294262469, -0.00314886123, 0.0941899493, -0.0902123451, -0.0473316908, 0.03309476, -0.00887358468, 0.0519970991, -0.0706470236, -0.0585814975, 0.0448119715, 0.0293908119, -0.0922531039, 0.0633407086, -0.164037898, -0.0344860554, 0.0450999252, -0.00827317126, 0.0797850564, 0.0878356174, -0.168259695, -0.111685902, 0.0194611624, -0.0502003171, 0.0400763042, -0.000246921554, 0.0347175598, -0.0578241013, 0.0705874041, -0.0547405779, 0.0456695706, -0.0114778504, 0.00666502118, -0.158520162, 0.0391363762, -0.103737898, -0.0202049147, -0.088732928, -0.0948789492, 0.0870066583, -0.0883992463, 0.0831747726, 0.0661358535, -0.00944175199, -0.194340572, 0.00321928412, 0.0783763677, 0.00112029398, 0.0339062437, -0.0166905355, -0.057094533, -0.0835953802, -0.0406135097, 0.0742160231, -0.044803407, -0.174876824, 0.112007923, 0.147358492, -0.0847913846, 0.0327977575, 0.0154416123, 0.0593767762, -0.00806243159, 0.0516847745, -0.0334345698, -0.00635620393, -0.0670741349, 0.139667913, 0.0469381735, -0.0539213493, -0.0244122203, -0.0659745857, 0.0283477679, -0.0295619257, 0.0378655344, 0.0485721529, -0.0206418131, -0.111100182, -0.0611830056, -0.0195047855, -0.000287644565, 0.0513734743, -0.0807389319, 0.0663611367, 0.0745266005, 0.0250715297, -0.074418515, -0.0920155793, 0.0298504829, -0.0113703683, 0.00965473056, 0.00187846646, -0.138389483, 0.083949022, 0.0813331231, 0.0412819758, -0.0259420518, -0.0780557394, 0.0112823695, 0.0292894877, -0.121571183, -0.171000004, -0.082161963, -0.0934179276, 0.032158263, -0.0429277867, 0.0859632492, 0.143906415, 0.0723193884, 0.1921767, 0.0211715698, -0.119239479, 0.00303502637, 0.0327959321, -0.0355542824, -0.0364986621, 0.014449208, 0.0821491703, -0.0108046737, -0.09774068, -0.0262510162, -0.0463821851, -0.025814116, -0.113182858, -0.0296528637, 0.141963795, 0.069177866, 0.011556413, 0.00709964149, 0.0644153059, -0.0336896852, 0.0873855054, -0.0798419714, -0.0273210257, -0.117931627, -0.0242039915, -0.0473055542, -0.049700819, 0.0279959533, 0.120111533, -0.0517931357, -0.0758071691, 0.0162475444, 0.0594417267, -0.165750802, -0.0595090389, 0.024117101, -0.00721539045, 0.02062824, -0.0610174797, -0.047291778, 0.0229518041, -0.0178083591, 0.0143660717, 0.107656598, 0.0646652132, 0.0129710324, -0.0765416026, -0.0067758821, 0.071242258, -0.0673705488, -0.196762294, -0.0317336246, 0.0874641016, -0.0363835618, -0.0167499296, 0.0126019027, 0.0590260327, -0.0619911924, 0.125976726, 0.0454879105, -0.0814923048, -0.160627574, 0.0401536077, 0.11946094, -0.00205735117, 0.0649667308, 0.119357049, -0.0163080599, -0.0327946432, -0.0541737825, 0.103204623, -0.0368971452, -0.00818765908, -0.0605907142, 0.0254717674, -0.0940710902, -0.190521747, -0.102423266, -0.0435902327, -0.0440872647, 0.0942212269, -0.00657942891, 0.00986169092, 0.0419842377, -0.0898573399, -0.13850674, 0.0310922042, 0.110772438, 0.128877789, -0.0391735509, -0.0354640856, -0.0221875757, -0.109102696, -0.131654769, -0.00299015827, -0.0143673187, -0.0724790767, -0.0387414917, -0.0553217307, -0.0794467032, 0.0357225388, -0.0577824861, 0.127521515, 0.030323673, -0.0575866997, 0.0470415689, -0.02680251, -0.13124375, 0.14153403, 0.0602536276, -0.0151671181, -0.0162680708, 0.0525177345, 0.0274184011, 0.0358750187, -0.119836435, 0.0613141358, 0.0407154448, -0.0118777975, -0.0230017081, -0.00926114991, -0.0414987132, -0.0842045993, -0.00167208165, -0.0925509632, 0.0421595834, 0.0608234778, -0.130276754, 0.0267832708, 0.100988097, 0.0781755894, -0.0390111469, 0.0901702121, -0.057276465, 0.0248767994, 0.172336698, -0.020048501, 0.0744086504, -0.0542870872, 0.0197537728, 0.0848038197, -0.0120387282, -0.0234180801, -0.0143575976, -0.0196826849, -0.0373380929, 0.0507742353, 0.0573016703, -0.105674788, -0.0482716076, 0.0154178804, 0.0567820966, 0.0546647832, -0.077160351, -0.0974433571, 0.0261986218, 0.0682947934, 0.142600715, -0.0821557045, -0.0264292788, 0.0293401107, -0.141429424, 0.0557237118, 0.00814896636, -0.0856773034, -0.0153672369, -0.0419892743, -0.0394244827, 0.0818297863, -0.0586152971, -0.0249222666, 0.0107620507, 0.0225159116, 0.0488754958, 0.0784658343, 0.158379465, -0.00325796939, 0.0975780785, -0.0909784883, -0.00240113959, 0.028311016, -0.0576878339, -0.107952863, 0.0455746762, 0.0782887936, -0.0428143069, -0.0966097116, 0.0105752349, 0.147920817, 0.0276091732, 0.0509470589, 0.0948298052, -0.115800686, -0.0791827589, -0.0415750258, -0.0642590597, 0.051787965, -0.0664690211, 0.135570541, 6.43308667e-05, -0.0391023755, -0.0508662984, 0.0224460736, 0.0564484969, 0.053764686, -0.107197657, -0.00115409866, 0.0311301108, 0.0211292151, -0.0459631011, 0.0348635539, -0.0117480159, -0.0270452388, -0.00449803099, 0.109037757, 0.155846879, -0.0825168863, 0.122937411, 0.0165575948, 0.0443798937, 0.0524557307, 0.0123378197, 0.230386585, 0.00925843418, -0.147435188, 0.0187123716, 0.0921274424, 0.0463036858, 0.0319886357, 0.00493047945, -0.0185778253, 0.0484505594, 0.134464771, -0.0519553833, -0.0243367665, 0.106514797, 0.0361147523, 0.0137277758, 0.00527644157, 0.0497434065, -0.00503639504, -0.0432905667, 0.0993102491, 0.136526898, -0.0145881996, 0.130319893, -0.132631332, -0.066883117, 0.0614537522, -0.146018207, -0.0854729265, -0.0106974319, -0.0684075132, 0.000379471108, -0.0152550749, 0.0307253655, -0.0415801778, 0.0565482304, 0.0613053888, 0.0351135246, -0.00204717368, -0.0194362011, 0.119199343, -0.10788542, -0.121140428, -0.0756799057, 0.0656082779, 0.0473917872, 0.110425636, -0.10782776, 0.0833447948, 0.0206291992, -0.0329098925, 0.105064832, -0.027444927, 0.00177714229, 0.0579485819, 0.0476972051, 0.0915832892, -0.0460004956, -0.0286061596, -0.0868751183, -0.00388204306, -0.122030437, 0.0168477185, 0.0854151845, 0.0344677158, -0.109319732, -0.0454696715, -0.0337420478, 0.0016348036, 0.116318591, 0.091471374, -0.0618529841, 0.00717924815, 0.0219491664, 0.027185725, -0.0214611832, 0.00936102122, -0.0100392811, -0.122589931, 0.0584963523, -0.0140657034, -0.0762873739, 0.0760588795, 0.0238103811, -0.0771279335, -0.0201385953, 0.0819055736, 0.0235249512, -0.0114337914, 0.0701106191, 0.0395762213, 0.0140983667, 0.0242828913, 0.0286869016, 0.0211825147, -0.0424613357, 0.0431166589, -0.097460188, -0.00259585679, 0.0190237854, 0.0898538753, -0.0310720168, 0.0507076494, -0.0149203688, -0.0873094648, 0.0690678656, -0.0789354071, -0.0375652462, 0.013849549, 0.0499016792, 0.0156347491, 0.0342558399, 0.0526852161, 0.115731694, 0.113165185, -0.0557963699, 0.0368037485, 0.0216162018, 0.214696974, 0.000794485211, -0.0406426713, -0.0198553521, 0.0373584591, -0.0704259425, 0.029388763, 0.082738027, -0.0326178819, 0.09166722, -0.0369430296, 0.00916040316, -0.0170614962, 0.0870813802, -0.0095146168, -0.065076001, -0.102999263, -0.045840688, 0.0162314083, -0.0649379268, 0.0297924839, -0.0204978622, -0.0241616368, 0.0600432009, 0.159195215, 0.143640861, 0.0745456144, 0.0539212152, 0.00271478156, -0.0936590433, 0.0323141217, 0.0196025074, -0.000803589821, 0.0519903377, -0.120891005, 0.0062912032, 0.0357041061, 0.0307115577, 0.0233878214, 0.0397786349, -0.0911078379, 0.00382280257, 0.0125010032, -0.0251113549, 0.0125831477, 0.0556067452, 0.0666292682, 0.0994372368, 0.0410823897, 0.0671635717, -0.0785583779, 0.0100541897, -0.0105275586, 0.100008905, 0.00607637689, 0.119727626, 0.06037727, -0.0570261627, -0.0179527644, 0.0237348266, 0.0198590662, 0.097318396, -0.0709325224, -0.150020763, -0.0541847646, -0.00585578289, 0.00333797373, -0.028236445, -0.00830273796, 0.0893258899, 0.136049345, 0.0833097324, 0.00150818564, 0.0841375962, 0.044127617, 0.0420588702, 0.0320436023, 0.0824125558, -0.0333235189, -0.0897977799, 0.0601325929, -0.0908033848, -0.0204037391, -0.103487767, 0.084499523, 0.0478009656, -0.0516456328, 0.0319618322, -0.0162731893, -0.0307973847, -0.0242388286, -0.0598752722, 0.0676786974, -0.0532381423, 0.0455306582, -0.0513714179, -0.0223139729, -0.0721026957, -0.0332549997, 0.0154482415, 0.00276384782, -0.00769143552, -0.135057539, 0.0194987282, -0.0791820884, 0.027593242, 0.0468132161, 0.0648820028, 0.141864702, 0.0540276431, -0.0930785388, -0.0342094153, -0.0712071806, 0.0516552515, -0.0519339666, 0.141384766, -0.115820587, -0.0578783303, 0.0993592069, -0.0826922432, -0.0402599946, 0.0600859299, 0.052808255, 0.062896654, -0.0991227105, -0.0308523662, 0.0058810655, 0.0195116568, -0.176231444, -0.0120743476, 0.0466277748, -0.00479177758, 0.132687926, 0.0372997411, -0.0698493868, -0.114647776, 0.0988531783, -0.00462367944, 0.0126146749, 0.0215533301, -0.0302089714, 0.111634687, 0.0171016511, 0.0716648474, 0.0292715598, -0.0343657285, 0.0722840428, 0.00431878865, 0.169528246, -0.0553757697, 0.0625901446, 0.129925251, 0.0075961519, 0.0814568102, -0.000654119998, -0.0866291448, 0.122778445, 0.0197446793, -0.0894370601, -0.0221604332, -0.0719681457, -0.000667473301, 0.0250691995, 0.0285977963, -0.0907365084, 0.07515008, -0.165994599, 0.168218225, -0.137749895, 0.106884032, -0.129251719, 0.0266259871, 0.0769484565, -0.0372937955, 0.0479861833, -0.0484450944, 0.0363472104, -0.0782243684, -0.0511998497, -0.013238335, -0.0329197496, 0.0104758553, -0.0709497258, 0.0391665697, -0.127216831, -0.0404612347, -0.0867774114, -0.046600692, 0.00418355316, -0.0633166507, -0.0414735936, 0.0236057006, -0.0258368962, 0.0678422004, 0.112647943, -0.0324306339, -0.00988782942, 0.0839368254, 0.0120457122, -0.0703958571, -0.0518545657, -0.0366280451, -0.0344718434, -0.0195410885, 0.140279353, 0.0287122019, 0.034899421, -0.0190885291, -0.0903406516, 0.0937678069, 0.0595882423, 0.0444250442, 0.02489971, -0.0289831776, 0.0477713309, 0.160236746, -0.0507163815, -0.02798298, 0.0835297853, -0.145065278, 0.110856101, -0.0219675228, -0.09635894, 0.139262006, -0.0428989083, 0.006609309, -0.0212683361, -0.0233980827, 0.00470141508, 0.0974960998, 0.104721539, 0.0269472525, 0.0124460198, -0.0666405708, 0.00455601886, 0.0233568326, -0.140762657, 0.0594203956, 0.00405210583, -0.180983603, 0.0104133934, 0.00331818778, -0.0334692076, 0.0713636801, 0.0462374873, 0.0826871693, 0.0863402188, 0.134145707, -0.0676784068, 0.0348382145, -0.0834512562, 0.0684894025, 0.0506787188, -0.0485029928, 0.0136228791, 0.164052099, 0.0657436177, -0.000161466189, 0.00585474214, -0.00230954075, -0.0957160294, 0.0718223453, 0.0585715473, -0.0631539151, 0.0948207974, -0.0422124118, -0.0262737256, -0.0412255339, 0.0186428111, -0.13579911, -0.183053255, 0.00305974856, -0.024856139, -0.0873593986, 0.100135244, -0.0249364562, -0.0182432774, -0.0374694169, 0.112602696, 0.0115270391, 0.00774586573, 0.00832534954, -0.0187189281, -0.0247038193, -0.072468698, -0.0127941612, 0.0929326862, 0.0153889861, 0.0401442125, -0.105329812, -0.041904889, 0.0746989921, -0.0426267236, 0.096574001, 0.0588563308, -0.0723425001, 0.0519671626, -0.110282645, 0.023782514, -0.0220482349, 0.0455567315, 0.00126918801, 0.0148957735, -0.0828897879, 0.0330617018, -0.0603466406, -0.0312512703, 0.158161759, -0.064591296, -0.0302896984, -0.0546595864, 0.041126214, -0.0834092349, -0.0379186906, 0.159711421, -0.080117397, -0.0189905092, -0.0189962052, 0.0377800204, 0.0824783742, 0.0999648273, -0.030885186, 0.0940911844, -0.0122155016, -0.0698266551, -0.0508394614, 0.0794238448, 0.0523062013, -0.0470671318, 0.0817164108, 0.0626662672, 0.0733318478, 0.104500718, 0.0606436543, -0.0396260135, 0.0492423661, 0.0252361633, -0.053880997, -0.0710671544, -0.034930598, 0.0249724053, 0.039634496, 0.00128793344, -0.0316855088, -0.0832425132, 0.128735602, -0.107892126, 0.189235479, 0.114530109, -0.0733102486, 0.0611379035, -0.0727086216, -0.00784323364, 0.0649280772, 0.078512989, -0.0140992254, 0.0500521399, 0.0546547771, 0.032995224, -0.0924386531, 0.0342714824, -0.0288704298, -0.0537729412, 0.0160043482, -0.0571973547, -0.0930881575, -0.0060783294, 0.00658744713, -0.00991571881, 0.0334253199, -0.0391148813, -0.0716266036, 0.0784005821, 0.100003406, -0.049674537, -0.136607498, 0.0599353202, 0.00876861438, 0.123580955, 0.11543794, 0.027512813, 0.0601726808, 0.0825635195, 0.0102091115, -0.0660458058, 0.0296149608, 0.00901784003, 0.140400052, -0.140364692, -0.0125178769, 0.0600770488, 0.0589169003, 0.0683401376, 0.0202003792, -0.0620686933, -0.112169608, 0.0258502401, 0.112197705, 0.0135365054, 0.0189605858, -0.086132735, -0.169402003, 0.0953313708, 0.00955498405, -0.0141711263, 0.0974058509, -0.0825876519, 0.0700342059, 0.0554787591, 0.0475979745, 0.113273486, 0.0469833612, -0.095944792, -0.00116587523, 0.107693441, -0.0434525535, 0.0535380021, 0.00395460706, -0.0444919243, 0.109183334, 0.147456348, 0.0826073885, 0.134649783, -0.0860900283, -0.0745515525, 0.0465153717, -0.122678399, 0.0569026023, -0.0684145316, -0.0305911433, -0.0619250238, -0.0482132137, -0.0189730283, -0.0551335625, -0.116009459, 0.02166228, -0.0904422402, -0.0962748304, 0.0397973061, 0.0565618835, -0.0541109219, 0.00912805088, 0.00842884742, -0.00535425078, -0.0266479701, -0.0859368294, 0.0233013704, 0.042687472, -0.018398555, -0.0481752902, 0.0822771192, -0.022317227, -0.118334077, 0.095822528, 0.139224648, 0.0195650458, 0.0683586597, 0.0631345958, -0.0373875722, 0.00341564603, 0.107133001, -0.0751987696, 0.00454649981, -0.0362539589, 0.026337428, -0.0179972276, 6.35553151e-05, -0.0705527738, 0.0230018832, 0.0606943443, -0.038967438, -0.0266847778, 0.0172603615, 0.0308038648, 0.022909835, -0.0310519468, 0.0154562201, 0.0787664652, -0.121662647, -0.0801561549, -0.00359021639, -0.0524999462, -0.00503655523, -0.0436337888, -0.0619397163, 0.0351424366, 0.0792855993, -0.0914481431, 0.054709658, 0.0170378536, 0.0350544453, -0.0636989996, 0.0668064356, 0.0525544137, 0.0519481078, 0.0748329982, -0.0683197007, -0.110261567, -0.0808580518, 0.0433228835, 0.0686655864, 0.0811156705, 0.156877279, 0.0324891731, 0.025431687, 0.102199338, 0.0574450791, 0.141714647, 0.111159399, 0.0125291236, -0.0447607189, 0.130543992, -0.0637754649, -0.0112033971, 0.0106440624, -0.0678310171, 0.0161886699, 0.033586964, -0.0785687715, -0.000732215121, -0.100033045, -0.00619979948, 0.0352816507, 0.00844343752, -0.0454045013, -0.101458229, -0.119886011, -0.0570310503, 0.00495114177, 0.0789650828, -0.0153123513, 0.07088162, 0.00860105455, -0.0862798318, -0.0800941512, 0.0199356303, 0.0428098105, 0.0869083628, 0.0312335305, -0.0582196042, 0.110067889, 0.0443210714, 0.0505822003, -0.0973165855, -0.0469971225, -0.0390720591, 0.151471704, 0.127615348, -0.105041966, -0.164652064, 0.0131918658, 0.029172156, 0.00465614349, -0.0354489461, 0.0173196532, 0.0124960765, -0.200602576, 0.00305063999, -0.011325432, -0.0427099168, -0.0469666794, -0.0288568828, -0.0726884678, -0.00320445118, -0.020172514, 0.0339836776, -0.0170585364, -0.0856021419, 0.000350127928, -0.00189465168, 0.0373253897, -0.0414954796, 0.073211439, -0.0566916279, -0.012231566, 0.0222783666, 0.0329278037, -0.115158595, -0.138853624, -0.0693328455, -0.0101504438, 0.0382712074, -0.00926143676, 0.0709851384, 0.0712291747, 0.0422781147, 0.053045772, 0.054939948, 0.0537798926, 0.0823203847, -0.0454094484, 0.124955572, 0.0222275015, -0.0329840928, -0.097050406, -0.0406842232, -0.0315937251, -0.0451682471, 0.0331139192, -0.111749321, 0.0606486052, -0.076717943, 0.0591437481, 0.0165941566, -0.158840597, -0.00306601822, 0.0333832949, -0.0355267599, 0.111018218, -0.0104070455, 0.0489391163, -0.00862740353, -0.0600290075, -0.0773975477, -0.0431323797, 0.0192667395, 0.105983481, 0.0561273359, -0.091204077, -0.114225745, 0.103793919, 0.012235254, -0.115128316, -0.0581305996, 0.0234019887, 0.0715955943, -0.0840854943, -0.102567874, -0.0818333924, 0.0280918758, -0.0301763713, 0.0228692051, -0.0594820604, 0.0897795111, 0.106658682, 0.0206690338, 0.0726500899, -0.000891397242, 0.0139189754, -0.054154858, -0.0630462244, -0.108763322, 0.126787513, 0.00294042518, 0.0292959437, -0.0553980321, 0.0807077736, -0.0965617076, -0.0890631229, 0.0466582552, -0.00911538024, 0.156839207, -0.0626729354, -0.0245680921, -0.00179294869, -0.056965515, -0.0199423786, -0.115498662, 0.0221503396, 0.0872155279, 0.119776607, 0.0166656077, -0.0399951339, -0.0429340228, -0.0653482974, -0.033989653, -0.0458589531, -0.0407891795, -0.0253337026, -0.0725796819, -0.0302919783, 0.00206887163, -0.100360379, -0.071315363, -0.017575983, 0.0177510977, 0.0351644121, 0.0383973196, -0.0745397806, -0.0709501654, 0.195765108, -0.0271085314, 0.0249852221, -0.0700546056, 0.184820786, 0.158069536, -0.0409562513, -0.0287105516, -0.0858581439, 0.0129066352, -0.030616425, -0.0372961275, 0.0750120357, -0.00228865957, 0.000365508662, -0.0622223467, 0.102390289, 0.0501865447, -0.0586910993, -0.0958363265, 0.0167813376, -0.0460788198, 0.0475374013, 0.073757261, 0.0686880201, -0.016310079, -0.0307487864, 0.012816906, -0.0567861497, 0.117383681, 0.0600756668, -0.0127716083, -0.0240453258, -0.0374855399, -0.032605987, 0.0901284069, -0.133627295, 0.0372318402, 0.180233389, -0.042641554, -0.0745786205, 0.102745302, 0.0446086749, 0.141644612, 0.0281131864, -0.0547536165, -0.0813148469, -0.0966759175, 0.0440410338, 0.0347155966, -0.0452661924, 0.00467441976, 0.143894181, 0.0984901041, 0.000415101647, -0.0614643805, 0.00953144394, 0.0880256295, 0.0648551509, 0.0617447086, 0.152493358, -0.0478570797, 0.104216434, 0.0910557956, -0.065354012, 0.0716719031, 0.0858117864, -0.0790668055, 0.100356698, 0.125176936, 0.00570722762, 0.0199908521, -0.0199188571, 0.0151966773, -0.0859806389, 0.0459887758, 0.229563281, -0.055340413, 0.0785515308, -0.0705481991, -0.0218721218, -0.0860364884, 0.0521545634, -0.0791168362, 0.092071332, 0.0687095225, -0.0352584347, 0.0084028868, -0.0515908487, 0.067410484, -0.0238079429, 0.0491214432, 0.0763769448, 0.0616733208, -0.10592977, 0.0577273741, 0.0236162581, 0.0179329254, -0.0668587163, -0.000917315483, 0.100958973, -0.136879578, 0.0519942529, 0.0552516207, -0.117933288, -0.0284534171, 0.0147698354, 0.0290891677, -0.0483859926, -0.00171393529, 0.0671777129, 0.0262195617, 0.0175510049, 0.0993073359, 0.00920790061, 0.0365526564, 0.118519023, -0.0862539858, 0.0720768198, 0.141677991, -0.018712623, -0.0670909733, 0.0032716766, 0.033690609, -0.000137303025, -0.0312980786, 0.0564908609, 0.115278304, 0.0838204175, -0.106906064, -0.105256386, 0.0039839847, 0.143497258, -0.0308761299, 0.061087437, -0.0215484872, 0.213556752, -0.0191945173, 0.0867439806, 0.0362426117, 0.0124808261, -0.02415636, 0.161512941, 0.071432732, 0.0367532372, 0.0120303296, 0.0474461541, 0.0920784175, 0.0683402717, 0.0278418101, 0.0420726165, -0.051485911, -0.00894092023, 0.0546397753, 0.00826329738, 0.0242030192, 0.0114576034, 0.0699174181, 0.0751249939, -0.0101688132, -0.0607835576, -0.104924619, 0.00508963317, -0.110204637, -0.0232813805, 0.142941684, -0.0581625439, 0.0117709413, 0.019689925, 0.0111599695, -0.0325533599, -0.142398402, 0.0469465777, -0.0962782055, -0.0296663232, -0.0991843939, -0.0907072723, -0.018030135, -0.136653036, -0.00641700998, 0.0690531433, 0.0612690002, -0.127184689, 0.0164758004, -0.0353412777, 0.126112342, 0.0430115089, -0.0611712597, 0.0732707083, -0.0329353586, 0.0160628408, 0.0106481165, 0.0799932927, -0.029079929, -0.111094221, 0.138537467, 0.0436870679, 0.0114703607, -0.111047409, -0.0588934831, -0.143290088, 0.00713616796, 0.00893756747, -0.0305529404, 0.00438396959, -0.00538037438, -0.0742936879, -0.0868203044, 0.0736782998, -0.00870422367, -0.0734259933, 0.0238608457, 0.0103617096, -0.0459689163, 0.0194341168, 0.0505106598, 0.038368959, 0.048780188, -0.0726687014, -0.110066131, -0.067750439, -0.157951459, -0.0285825022, 0.0622866154, -0.031255234, 0.0788101628, -0.00532437488, -0.0541705601, 0.181852654, 0.0464031994, 0.0114014857, -0.115355566, 0.0505047888, 0.0553555712, 0.011652261, -0.0318466201, -0.0325593352, -0.107562304, 0.0409038886, -0.0569218919, 0.037518084, -0.0663177744, -0.010987144, 0.0359393656, 0.0968064517, 0.0664260089, -0.0963557586, -0.0316545814, -0.00830668956, -0.016299244, 0.131724447, -0.0682323277, -0.100451991, 0.0899666324, 0.0605907626, -0.0334617831, 0.00608175248, -0.00132036954, 0.144946083, -0.015863914, 0.130428657, 0.0414888225, 0.03145032, -0.012145143, 0.105927542, 0.0972640514, -0.0331205763, -0.048977606, -0.0166362859, 0.0798452944, -0.0234581437, 0.161201462, -0.0630989969, 0.0775372311, -0.0355709456, 0.104933083, -0.0266663842, 0.0230915528, 0.107127644, -0.124312878, -0.0319105722, 0.0134256873, -0.152985573, -0.116613597, 0.0173692219, -0.0704726353, 0.0289779007, 0.0375288725, 0.0732763112, -0.0757907927, -0.195766464, -0.0980283767, -0.00513102859, 0.0143520981, 0.113044247, -0.0562009402, -0.123434529, 0.0368995182, 0.0028431192, 0.136627197, -0.0138487108, -0.069396466, 0.0879209787, 0.113950782, 0.0165350158, -0.0697787404, 0.0165037923, 0.0319612734, 0.00848966371, -0.0742693692, 0.0245090649, -0.0677825734, 0.02509683, -0.0597349927, 0.131780028, 0.0651398599, 0.0184568018, 0.0326681882, 0.0139567442, -0.00476132333, 0.0173050445, -0.0241064765, -0.0518168993, -0.0752798617, 0.0386652574, 0.0384047478, -0.018362388, -0.101061665, -0.0666311234, 0.101437956, -0.0874377638, -0.0317256749, 0.0850132555, -0.0111166034, -0.0420253798, -0.0590298176, 0.00268510729, 0.104384378, -0.033026509, -0.0944487453, 0.0328986719, -0.0315738469, -0.127896726, 0.0722550005, 0.0570910573, 0.0532291643, 0.00170435198, -0.0596524999, 0.00574701605, -0.0424169526, 0.126607269, 0.0750704706, -0.125349313, 0.0210697092, -0.136739492, -0.0569494255, -0.0609738082, -0.0403983779, -0.0410580374, 0.13844195, 0.0848094821, -0.125428453, -0.112865232, 0.0516311377, -0.0986351818, -0.0494424626, -0.0234178081, 0.044481352, 0.107108541, -0.0497174039, -0.106645383, -0.0507276244, 0.0824460238, -0.151569441, 0.114093393, -0.0665538311, 0.068059355, 0.0118242092, -0.0422057286, -0.173799008, -0.00440534949, -0.0892028213, 0.00304216705, -0.0684691593, 0.0433448181, 0.0295414627, 0.00422838889, 0.13651593, -0.0920076668, 0.0499312393, -0.0532680899, 0.0698095188, -0.0335529149, -0.0184200816, 0.00152085349, -0.0769852102, -0.0194537211, 0.0329587795, 0.084027186, 0.0138547821, 0.078202188, -0.113860883, 0.081746459, 0.1273821, 0.0576579385, 0.0589885786, 0.137488559, -0.0280587077, -0.147009701, 0.0482914932, -0.0349069014, -0.0415082574, -0.0786461309, -0.0904545635, -0.0178104006, 0.0326328538, -0.0779492632, 0.0391764306, -0.00248269504, 0.041821897, -0.00617768522, 0.0309736803, 0.0183068309, -0.0023522526, 0.131349832, 0.0794798583, 0.0397143438, 0.0478656515, 0.0136936139, 0.0489361435, 0.0558214411, -0.00169046316, 0.0115834484, -0.00844283216, 0.0599297397, -0.0403334275, -0.0405900553, -0.0121230781, 0.106669635, 0.110829912, -0.0452369377, 0.0713214055, 0.0187946334, -0.0228895321, 0.0249673799, 0.0452177264, -0.101951599, -0.0477757826, 0.104328498, -0.10797099, -0.0486136638, -0.0292987712, 0.0669425651, -0.0583777986, 0.0370908305, 0.028847212, -0.0660194457, 0.0539241061, 0.0207896139, 0.0580766648, 0.0728344545, -0.0960628167, 0.0166663975, -0.0675754026, 0.0527179092, 0.0253911428, -0.0322320201, 0.000191444531, -0.0626192391, -0.0938816443, 0.0427594446, 0.0444745012, 0.0671123564, 0.116402999, -0.00334139913, 0.0760671645, 0.0691754073, -0.110883355, -0.018052483, -0.0751862302, -0.0639079809, 0.0157645084, -0.149932712, 0.0299264304, -0.17823188, 0.0385304317, -0.132355168, 0.0266840048, 0.0542500056, 0.0666455328, -0.092522651, -0.0835058093, 0.0800313652, -0.0826294273, -0.0597820953, -0.103087187, -0.0524287559, -0.117469326, 0.0530021451, 0.0314180478, 0.0173868798, -0.0561694875, -0.0524752513, 0.107553661, -0.0895222872, 0.035363283, -0.00804894418, 0.0827626139, -0.023751054, 0.0319075957, -0.0241621211, 0.108154953, 0.0550332405, 0.0688145459, 0.0629935786, -0.0339644738, 0.0941599458, -0.0688125864, -0.0261289347, -0.0469831042, -0.0747010112, -0.1975936, 0.10091415, -0.0841339156, -0.0335424654, 0.0286981687, 0.0692808703, -0.0667530447, 0.0430541411, 0.0215135142, -0.0122609325, -0.0251649506, 0.0593507327, 0.176167563, -0.0734691918, -0.0467854515, 0.000647263776, 0.038958177, -0.0285261609, 0.0124273915, -0.0466737039, 0.0187623464, 0.124909841, -0.166239634, 0.0446738228, 0.0110851061, 0.0547700152, 0.0490482748, 0.134703919, 0.0421581641, -0.0794193894, -0.0543411858, 0.0453204773, -0.0109050162, 0.0158124641, 0.0817929879, 0.0832850188, 0.0549521595, -0.00940894336, -0.0147470459, 0.0424956232, -0.0880125538, 0.177774161, 0.127763346, 0.124928072, 0.0601709485, 0.0640123338, 0.0203758813, -0.051416859, 0.057953991, -0.0709685087, -0.00976901688, -0.0335928351, 0.00619953498, 0.0378086716, 0.0417027101, -0.00208918098, 0.00262965634, -0.0185245723, 0.0205108598, 0.042619355, 0.146731392, 0.0441337712, -0.0846837461, -0.00324742123, 0.236852542, 0.0898044258, 0.020407008, -0.15276964, -0.0101641072, 0.0237147808, 0.0172680281, -0.00233229995, 0.131191328, 0.0216754414, -0.0336728096, 0.107479818, -0.0277084317, -0.1844064, 0.00492768548, 0.0109517844, -0.0393908992, -0.00126481801, 0.104402393, -0.0805563256, 0.0671683326, -0.028834559, 0.00854677334, -0.0218764003, -0.0414474383, -0.0489949323, -0.000848490745, -0.113781974, 0.0259864926, 0.00311553292, 0.0160832442, -0.0782885551, 0.0363949053, 0.00709262863, -0.0311835818, 0.056816116, 0.0280716978, -0.110789046, -0.107226349, -0.114018351, -0.112105981, -0.051748991, -0.0294137653, 0.0470993072, -0.0109183677, 0.0952649862, 0.0169891641, -0.029055912, 0.0548034087, -0.0231187064, -0.0509331226, -0.0425397605, -0.0886350796, 0.0664251149, 0.000766177662, 0.0235708579, 0.0986191481, 0.0169718452, 0.0350453779, -0.0181663595, -0.0581547208, -0.0111971665, -0.0658968091, -0.043942187, 0.0744755417, 0.0649959669, -0.00646108575, 0.0577539243, -0.035588719, 0.0617120005, 0.0129959956, -0.00798365474, -0.0934553295, -0.00565501768, -0.0376720279, 0.134627596, -0.0593289584, -0.022235956, 0.0201732926, -0.110076368, 0.0505789034, -0.0523465984, 0.0842581093, 0.0155403186, 0.0820551142, -0.0493090674, 0.225808814, 0.0257120468, 0.00689401105, -0.0957904756, 0.130746499, -0.0968430638, 0.0995664597, -0.054121986, 0.0299899653, 0.0616851412, -0.0309149232, -0.0588663667, 0.00374672562, 0.0229911096, 0.00757680833, 0.0249638297, -0.00211454183, -0.0953999609, 0.0296648555, 0.0276420079, -0.0173467435, 0.0349950381, -0.0239780173, -0.0750618353, 0.0558826625, -0.135295808, -0.0406377763, -0.0228079446, -0.0255099293, -0.0144131482, 0.105348289, 0.0330178663, -0.0323044285, -0.0620107092, 0.131417841, -0.0253877491, 0.0873237997, -0.0394588523, 0.130003497, 0.0544283539, -0.0228096507, 0.0344365835, 0.0589501187, -0.0384093933, -0.0729825944, -0.0472028404, 0.00675820373, 0.0377000533, 0.025417015, -0.150040045, -0.115042344, -0.0164607763, 0.10575477, 0.0255208723, -0.0214468297, -0.00740232365, -0.0733775645, -0.085227862, 0.0887256637, -0.0821226463, -0.0732457265, -0.0800393075, -0.157817408, 0.0516942963, -0.0149588697, -0.0229824521, 0.0223708227, 0.108997419, 0.0898767784, 0.0144321844, 0.000437498093, 0.0885114521, 0.0405967273, 0.0147995763, 0.134369314, -0.0147804739, 0.0423911065, 0.121686779, -0.0199723002, 0.0324794352, -0.0344413184, 0.0108162761, 0.0200632159, -0.0909346044, 0.0907277092, 0.078306593, 0.0123565141, 0.0495449752, -0.0268470664, -0.19156903, -0.0474564806, -0.0203771871, 0.0257022083, -0.0370838679, -0.104858413, -0.0181517266, -0.004468292, 0.00745896623, -0.0022775121, -0.0293494053, -0.0270710811, -0.107970081, -0.0305090789, -0.100271553, -0.10888052, 0.0533380061, 0.10615176, -0.0254803989, 0.0142585365, 0.0874576494, 0.0021774061, -0.0550973043, -0.0375173315, -0.0712005347, -0.0556420982, -0.0178135373, 0.0202902313, 0.116308086, 0.0801922977, 0.0404350646, -0.094611831, -0.0405631363, -0.0629749671, -0.0304389298, -0.0778223425, 0.0274351016, 0.0912509486, -0.101376347, -0.109884903, 0.118219361, -0.117630638, 0.033197917, 0.00980661903, -0.0233400688, 0.0876687616, -0.0866567641, -0.0495598651, 0.154081911, 0.066799514, 0.0663663745, 0.138981178, -0.104617655, -0.134632289, 0.0132512227, -0.0307451282, -0.0717537105, -0.0447786599, -0.0203792769, -0.00305938348, 0.128751531, 0.168384135, 0.134389818, -0.0488407984, -0.000193296, -0.0230348315, -0.0891407803, 0.0645165443, -0.0150886513, 0.0311952345, 0.0172327608, -0.0182059966, 0.0205209963, -0.023462031, -0.0115296096, 0.0937949345, -0.062077418, -0.044753857, -0.00663919561, -0.0111889178, -0.106608666, 0.115085535, 0.00561359525, 0.0392463915, 0.139113545, 0.142638013, 0.0229292717, 0.125224665, 0.0784767196, -0.134339631, 0.00184373744, -0.0163332913, -0.037552651, -0.0847556069, -0.102111034, 0.0670402348, -0.0362388343, -0.143356144, 0.00816862285, 0.171866357, 0.063321799, 0.0515059792, 0.0642708689, 0.0454857424, 0.0236697234, 0.105821952, 0.0092480965, -0.00954593718, -0.0710259974, -0.0341528915, -0.0791757852, 0.0946761966, -0.0109210648, 0.114886783, 0.177807823, 0.119987622, 0.0022838451, 0.00656085368, 0.0229036044, 0.0576986969, -0.0194735266, -0.0557837673, -0.00587408245, 0.00565860048, 0.0221642759, 0.0461966321, 0.00775645301, 0.0414951742, -0.0115494877, -0.0968217701, 0.046022784, -0.0580905527, -0.0181989633, 0.022852499, -0.0723620951, 0.142874643, -0.0302886758, -0.0984666646, 0.0232525952, -0.0980240777, -0.0456527174, -0.00293019903, -0.097713165, 0.113620192, -0.018971812, -0.0219054222, -0.116879433, 0.0463627949, -0.130884036, -0.0317850523, -0.0150047466, 0.040894188, 0.102204598, 0.150269806, 0.0201216973, 0.0339559913, -0.0181002952, -0.104960471, -0.0267044716, 0.0290627331, -0.0245765261, -0.071058929, -0.13309963, -0.00754409656, 0.032728754, 0.120368265, 0.0840021297, 0.121953458, 0.0370791778, -0.016948875, 0.123968489, -0.0218659379, 0.0870331824, 0.011598371, 0.0358568542, -0.0549993739, 0.0354933813, 0.107385799, 0.0247484297, 0.0363589413, -0.0932978243, 0.00257878006, -0.129064277, 0.0111397859, -0.0785455704, -0.0435388722, -0.0460782498, 0.0266925059, -0.0495381057, -0.102360234, -0.0679884255, -0.0235304758, -0.0381551832, -0.0561104901, 0.141988829, -0.078078486, 0.0651649013, 0.0301409364, -0.0386709869, -0.0861276835, -0.06776914, -0.0386363938, -0.0569600686, -0.0936848819, -0.186116084, 0.0288296659, 0.010812805, 0.00793905184, -0.0462868586, -0.0906251371, 0.150258929, 0.0796489045, 0.0377195105, 0.0914610624, 0.00676715001, -0.0510880947, -0.0859677643, -0.0254568122, 0.0497521162, -0.0127981463, 0.0270112157, -0.0329849198, 0.0815009847, -0.0126657169, 0.0565544777, -0.14730446, 0.0399446636, 0.0802432224, 0.0333384946, 0.0544420928, 0.085682556, -0.1993016, 0.0529618785, 0.0273188688, -0.111082606, -0.046358332, 0.0874589086, -0.0264321417, 0.0715716183, -0.0346798263, 0.0223852396, 0.0577339418, -0.0958287045, -0.120151833, 0.00864275172, -0.0160820521, 0.00365970843, 0.0863499194, 0.0390572399, 0.0824703574, -0.00912335794, -0.00690958649, -0.0363679193, -0.0325383544, -0.0292693563, 0.0690342039, -0.0164378732, 0.00357266515, -0.0945315361, 0.00905000698, -0.0426640883, 0.084148258, 0.0307582188, 0.0673260018, 0.0324155875, 0.0248095021, 0.0546956547, -0.169563293, 0.0235199165, 0.208287105, -0.068595916, -0.0589914434, 0.0206119567, -0.00962059386, 0.0512155183, 0.0895944834, 0.0827069134, 0.0629096627, -0.0445563346, -0.0354665592, -0.0346590281, -0.0655499771, -0.0373479873, 0.0698575899, -0.0468572788, 0.00708710589, -0.00173727423, -0.0926145092, 0.104473613, 0.0377659239, -0.0705457777, 0.023749087, -0.0678561479, 0.125114292, 0.055179134, -0.0156256072, -0.00088315492, 0.0195074286, -0.0321733728, -0.136137784, -0.0892990008, 0.074931927, -0.139921665, 0.149736241, -0.00113547593, -0.119224325, -0.138149425, 0.163096026, 0.111989059, 0.0714135095, 0.110901728, 0.0429112762, 0.11657019, -0.160976976, -0.074212864, 0.0048305355, -0.105347976, 0.0909552872, 0.0236025043, -0.0941404924, -0.0795364976, 0.0665476769, 0.0217442717, 0.0755219609, -0.0634106547, 0.0359948166, 0.0906661898, 0.0534381792, 0.0274045356, -0.0940109044, 0.00214707386, -0.0603406392, -0.0384378657, 0.0393172428, -0.0180536099, 0.0640648231, -0.160350576, -0.0605928935, -0.108627155, -0.0328229517, -0.0526959151, 0.0211077407, 0.133559987, 0.0900996923, 0.0283339117, -0.0361762606, 0.0774903893, 0.0309651326, -0.077206187, -0.142700225, 0.0507220514, -0.175183147, 0.0608116277, 0.016379755, 0.144942716, 0.0481477119, -0.117837735, 0.018508248, -0.0424480923, 0.0253082402, -0.0704792961, -0.052820012, 0.0263381302, 0.00419567712, -0.0866010785, -0.0889194682, 0.0321662389, -0.118707448, -0.0977562219, 0.000621002167, -0.118462905, 0.0978502259, -0.0253498629, -0.0458875671, -0.051405862, 0.0701094493, -0.0925895125, 0.0269318074, -0.0387994498, -0.0177200045, 0.0361462906, 0.032940004, 0.0911707282, -0.0253412202, 0.131375626, -0.076097846, 0.0516649634, 0.0129128927, 0.044285655, 0.0269309897, 0.0223179683, -0.0487635061, -0.0733353645, 0.0146101527, -0.00891945511, 0.100568205, 0.0520949662, -0.0144930556, 0.0657366961, -0.0298533905, -0.183018446, -0.0344359316, -0.0526576638, 0.204600394, -0.0510475226, -0.0618838072, -0.0188805908, 0.0744666457, 0.106323443, 0.0069219768, -0.0662630573, 0.123655081, 0.079134956, -0.0166491717, -0.025728751, 0.0176477507, -0.120832592, 0.0348780043, 0.132895634, -0.152824923, 0.0176192392, 0.0983903855, 0.000804595649, 0.0392432623, -0.0858294889, -0.00694064423, 0.0766717196, -0.0207373202, -0.143785551, -0.0299797244, 0.00368108228, -0.02576527, -0.0918034166, -0.0245569218, -0.0020073913, -0.134635925, -0.0244379062, -0.00205026567, 0.0436320864, -0.0382906646, 0.124861129, -0.0658158511, -0.0838000253, 0.0625896007, -0.187241822, 0.0442486778, -0.0854963809, 0.0744676366, 0.015948303, -0.0422934443, -0.0632212684, 0.0303207487, -0.0105451606, 0.0159170292, 0.0608507097, -0.0636942834, 0.0493633822, -0.156775504, 0.00367055833, -0.0044856444, -0.118679613, -0.0614755079, -0.109478787, -0.113873944, 0.0541704595, -0.0759271681, 0.0513200127, 0.0227294788, -0.00442646584, 0.0624753572, -0.0299119651, 0.0340797305, 0.0449048541, 0.065268077, 0.0243841615, -0.0443482772, -0.0178897921, -0.017998118, 0.117099263, -0.0903324708, -0.0930202976, 0.0174601749, -0.0082530342, 0.0238389187, -0.0269895345, 0.00585436868, 0.0552141257, 0.0576381721, -0.155392274, 0.0323198363, 0.124261506, 0.0385111682, 0.0172231607, -0.0813641548, -0.0470695235, 0.0632121563, -0.0595323779, 0.018977534, 0.0495419018, 0.114390008, -0.0611852705, 0.0584638566, -0.05169563, -0.0447621755, 0.0405260995, -0.0654804185, -0.0223629847, 0.0111893751, -0.0597181506, 0.0481003746, -0.0876153484, 0.0571012944, 0.0373661555, 0.00842267741, 0.0424995199, -0.0365535617, -0.103940263, 0.164833188, 0.081475459, -0.0621950999, -0.0220634304, 0.00333214551, -0.103024431, 0.059290383, -0.00829190947, -0.00786833931, 0.0418062247, -0.00335859787, 0.118728697, -0.0206394717, 0.0441573337, -0.0821953714, -0.112937331, -0.0872935355, 0.00823296793, 0.0686616898, -0.00996761862, 0.0819208771, 0.103608765, -0.133317322, -0.143641129, 0.0187726133, 0.0164246075, 0.0107233748, 0.0463518016, 0.119414046, 0.00115352124, 0.106320053, -0.0232305583, 0.145007864, 0.0707367361, 0.0352928489, -0.102848031, -0.0608059093, -0.0658036917, 0.0598252937, -0.0420819595, 0.0859991163, 0.0343810208, -0.0238903575, -0.0279339999, -0.00486056507, -0.0449833646, -0.028704524, -0.0549230054, -0.125461668, -0.0846189857, -0.00544487685, 0.138138548, 0.18346715, -0.10757079, 0.00334860012, -0.0436559319, 0.0171282887, 0.0511732697, 0.0205869693, -0.158152893, -0.0237202868, 0.0500039905, 0.00804132037, -0.178919747, 0.049530372, 0.0231576655, 0.016319206, 0.0968668461, -0.209181368, 0.0242683813, -0.0633693859, 0.143747747, 0.0669897944, -0.0720201135, 0.0511079021, 0.00224748626, -0.0249123648, -0.0882710144, -0.026280582, -0.0307737496, -0.107300185, -0.105721176, -0.11115665, -0.209473535, -0.0533579774, 0.0403167084, -0.137139887, 0.0712546259, -0.0053200461, -0.00831546076, -0.0903995559, 0.0744837746, 0.132631153, -0.0206565894, 0.133443296, -0.123549096, 0.00900856964, -0.0347793065, -0.0173467137, 0.0470211133, -0.0636748075, 0.0644437224, 0.0110963862, 0.010691151, 0.0257252157, -0.121936694, 0.0435509644, -0.00285037979, 0.0418016613, 0.0332998931, 0.0127451979, -0.080453068, -0.00660414994, -0.0891625136, 0.00468665361, -0.0160302259, 0.0267248079, 0.0152133033, 0.108307645, -0.0517366603, 0.0560837314, 0.0401830934, -0.00482201949, 0.0350291207, 0.0949657708, -0.027060559, 0.0701910704, -0.0418955274, 0.0724823996, 0.0422584601, 0.00114974752, 0.0695210099, -0.0699081048, 0.0320460238, -0.079946436, -0.098674804, 0.106608361, -0.0207979083, 0.0518062264, 0.128592819, 0.0216310043, -0.158794522, 0.0481886566, 0.0344376825, -0.103498466, -0.0388584435, -0.00339685567, 0.119976752, -0.121837057, -0.0361002609, -0.0467634946, 0.0227424484, 0.0812298506, 0.0057318625, -0.0632766932, 0.0133693535, -0.115805924, 0.0372774228, -0.128631905, 0.052809976, -0.0637927055, -0.0514348708, -0.0125545496, -0.0759181529, 0.0670369864, -0.129334778, 0.0128213912, 0.154368311, 0.0482923649, -0.105797492, 0.0687054098, -0.0472880341, 0.0421877354, 0.106991515, -0.00419089198, 0.0296891294, -0.0278291311, 0.119926207, -0.0632965714, 0.0724663958, 0.034995757, 0.0958595276, 0.00775001571, -0.0390481502, -0.0269152913, -0.0981106907, 0.0792592466, -0.0565083064, 0.0675349608, 0.0583877675, -0.0413221344, 0.0838775635, -0.0292064138, 0.0683145002, 0.0489856079, -0.00130998157, 0.0536718294, 0.0666105598, 0.031892512, -0.0458434671, 0.0538467243, 0.109850742, -0.00417516986, -0.0509028248, -0.142170504, -0.0366610698, 0.0718423426, -0.0225093924, 0.0383118689, -0.0554144755, 0.122152165, -0.0448820665, 0.116410255, 0.120842285, -0.140279487, 0.0613858178, 0.0650201887, -0.037952818, -0.0877776146, 0.0418614224, -0.187158108, 0.0190712661, 0.0696339682, -0.121901698, -0.104807861, 0.00705167651, 0.0914953873, -0.0124439057, 0.0169791616, -0.0378904678, -0.0500747412, 0.0369469672, 0.0846178979, 0.147575781, 0.0938130915, 0.0561358258, 0.0405266471, 0.00478235073, 0.0182364658, -0.0715994984, -0.0431600213, 0.172556713, 0.0006400235, 0.0317676365, -0.0478407927, 0.0609547161, -0.137460351, 0.0181176532, 0.00583034381, -0.0277956836, 0.0598901697, -0.0803982466, 0.0962693095, 0.0339596942, 0.152170867, -0.0431792364, 0.0741693377, -0.0776144266, -0.101780161, -0.0274014324, -0.0231655389, -0.072895214, -0.000511298655, -0.0507130511];
    bias_3_r : ARRAY[0..63] OF REAL := [0.211404547, 0.289471477, 0.350232184, -0.0113848262, 0.255106032, -0.0505001619, 0.393956006, 0.30565241, 0.215408534, -0.321017623, 0.146971986, 0.0140901972, 0.352487236, 0.073317118, 0.295657784, 0.195680931, 0.273608774, 0.247949466, -0.11806614, 0.244580895, -0.263936877, 0.299780279, 0.184798613, -0.0554735512, 0.345186561, 0.0326451622, 0.373724312, -0.0231367871, 0.362007052, 0.263970047, -0.101536416, 0.10940177, 0.303294301, 0.309194207, 0.367130488, 0.0412951261, 0.368920535, -0.00199001329, -0.0144892968, 0.218033642, 0.367789537, 0.388805985, 0.313740879, 0.32673353, 0.427658528, 0.0293739345, 0.169871822, -0.0308606736, 0.0321528874, 0.117100634, 0.105766714, 0.333601326, 0.314314336, -0.68898499, 0.30870831, -0.0834920183, -0.11542882, 0.321295649, 0.104272589, 0.312997669, 0.332255304, 0.352245361, 0.0179513358, 0.283515096];
    weights_3_h : ARRAY[0..4095] OF REAL := [-0.477327704, -0.223028138, 0.477383763, 0.272099614, -0.331715822, 0.392723799, -0.293869436, 0.293111712, 0.455964506, -0.370485485, -0.169337988, 0.358209044, -0.154706374, 0.319936365, 0.341514915, -0.402719289, 0.434456199, -0.47526449, -0.489136487, 0.58730334, -0.355098248, -0.302809507, 0.400321782, -0.371956021, 0.267092794, -0.463135689, 0.245020077, -0.399190784, -0.3084068, -0.313749343, 0.342046201, 0.564289451, 0.565605402, 0.579033673, 0.30539766, 0.45197311, -0.31735304, -0.48857221, 0.383875638, 0.302260935, 0.181652904, 0.315515608, -0.304400623, 0.285881907, 0.342444241, -0.290956706, -0.347757041, -0.304790974, 0.329997271, 0.307092458, 0.212757081, -0.246385187, -0.675582767, 0.27869159, -0.218399927, 0.649934232, 0.295164227, -0.504191816, 0.348629862, -0.788004518, -0.560513616, -0.37868908, 0.269324958, -0.386194885, 0.193138495, 0.0936199203, -0.371325284, -0.268244445, 0.284468323, -0.12238384, 0.208948225, -0.432277054, -0.20721513, 0.604005039, 0.275245756, 0.13828665, -0.0714443922, -0.0516165309, -0.545582175, 0.20568718, -0.181170657, 0.353475958, 0.459297806, -1.02305448, 0.308819354, 0.284700543, 0.00352787809, -0.0693232417, -0.21972768, 0.467387348, 0.0895780027, 0.0536244921, -0.0766994208, 0.446248025, 0.014726595, -0.51319015, -0.829305232, -0.732334197, -0.230438501, -0.527176559, 0.21426262, 0.720788836, -0.743974924, -0.29229632, -0.188690841, -0.0433681533, 0.0430677794, -0.570068121, -0.18835257, 0.152503192, 0.934911609, 0.225885972, -0.379429728, -0.208068192, -0.13282527, 0.118086673, 0.250476748, 0.0636733547, 0.155737996, -0.326886982, -0.424665511, 0.0709498152, -0.661783159, 0.405686229, 0.873163402, -0.0793672577, -0.4177818, 0.245727047, -0.175405353, -0.182268158, 0.395008862, 0.458469391, -0.411543816, 0.286715537, -0.214017823, 0.484770089, 0.241020083, -0.677324235, -0.476985693, 0.205288187, -0.320069313, 0.388286561, 0.530830264, -0.3388322, 0.462102681, -0.45303601, -0.569363117, 1.00542247, -0.387329727, -0.447940975, 0.195828974, -0.134499982, 0.127954915, -0.40173763, 0.196886495, -0.115446515, -0.0797588825, -0.58165437, 0.143406764, 0.49846068, 0.774460018, 0.545146048, 0.520931423, 0.562419355, -0.409500718, -0.861158252, 0.760374963, 0.581687093, 0.14180471, 0.300121695, -0.163008973, 0.539554894, 0.453706324, -0.350945413, -0.799297988, -0.450918794, 0.507954419, 0.0722613037, 0.14165011, 0.0171291456, -0.451630801, 0.339028627, -0.192155585, 0.502704501, 0.45119524, -0.238778964, 0.932323456, -0.594341278, -0.898570716, -0.0490389168, 0.511603117, -0.467601538, -0.405882061, -0.283297598, 0.739298701, 0.722658992, -0.26715821, 0.479726195, -0.532120645, -0.0237284917, 0.48330611, -0.323726654, -0.208368391, 0.232581526, -0.188637063, 0.318077564, 0.298525453, -0.850645363, 0.539557278, -0.377814859, -1.40523076, 0.465162724, -0.679179311, -0.241804957, 0.490303159, -0.195624158, 0.163719326, -0.237672776, 0.340154707, -0.157789201, -0.323773414, -0.332811028, 0.347858131, 0.352136403, 0.536489844, 0.31132561, 0.12756747, 0.476868987, -0.565818965, -0.488098741, 0.712121427, 0.354632258, 0.260619611, 0.48601073, -0.170348659, 0.188437447, 0.444436491, -0.191516027, -0.509016156, -0.303999394, 0.3035326, 0.426323533, 0.232193306, -0.302694231, -0.538741648, 0.337178558, -0.329310685, 1.2656703, 0.26894775, -0.53832674, 0.606308877, -1.39138579, -0.4849841, -0.118635602, 0.206906736, -0.590465903, -0.199698865, 0.0271727275, 0.279044747, 0.306948125, -0.0775341243, 0.0305152144, -0.290344119, 0.271196783, 0.355138123, -0.756615937, -0.33631447, 0.0121018663, 0.0225032959, 0.218690887, 0.450739831, -0.340195209, 0.321393847, -0.453326762, -0.424223185, 1.29127443, -0.450598478, -0.536069751, 0.133924276, -0.0862702057, 0.0843360797, -0.291461736, 0.162584856, 0.073226057, -0.0175837167, -0.559712708, -0.00935774576, 0.652041018, 1.12887228, 0.769396007, 0.220070481, 0.686632812, -0.390937507, -1.07226002, 1.04997945, 0.410393894, 0.276414692, 0.285110533, 0.187463403, 0.331211299, 0.240157336, -0.359538853, -1.06251729, -0.326777726, 0.335062295, 0.0289323889, 0.247402132, 0.152282834, -0.354610175, 0.138785884, -0.209046245, 0.367701799, 0.449430674, -0.39971137, 1.0538317, -0.411711067, -1.054932, -0.0593135431, 0.621842921, -0.248209327, 0.477279454, 0.215619951, -0.58452481, -0.387168229, 0.317550212, -0.459208816, 0.301971972, -0.190631434, -0.403445691, 0.433657497, 0.27659744, -0.268536121, 0.424349725, -0.477041692, -0.504639149, 0.611898065, -0.271073163, 0.398134053, 0.86002779, -0.541121185, 0.661311209, 0.171835855, -0.268515766, 0.370931357, -0.183438286, 0.413021863, -0.433557153, 0.295048714, 0.286439538, 0.461956412, -0.164179012, -0.331664711, -0.379812568, -0.527498066, -0.22169888, -0.193573356, 0.420137376, 0.509923577, -0.565212548, -0.406003714, -0.435218006, -0.211141258, 0.183033764, -0.326328188, -0.358321816, 0.263253033, 0.572903156, 0.108593255, -0.218963191, -0.393386781, -0.451561987, 0.272487462, 0.42083475, -0.320441037, 0.378210187, -0.800743878, -0.206348464, 0.493317813, -0.446035206, 0.908499122, 0.386151254, 0.357700586, -0.402182609, 0.459070325, 0.140864849, 0.288575321, -0.348540753, -0.425076783, 0.118181348, -0.243356273, 0.150108084, -0.444325507, -0.123226129, 0.473306119, 0.364770591, 0.00148743833, 0.0944404677, -0.306541115, -0.522351444, 0.498851001, -0.291609466, 0.26778546, 0.56175822, -0.910838962, 0.220005333, 0.245392412, -0.0919606686, 0.12009117, -0.270596415, 0.422408104, -0.247022122, 0.254039794, 0.247460261, 0.418485373, -0.0811505467, -0.418760002, -0.589756489, -0.569615185, -0.405208886, -0.295897305, 0.412519485, 0.577107072, -0.615277588, -0.450129092, -0.182284147, -0.281509578, 0.164060608, -0.51912117, -0.171782985, 0.26589784, 0.778394759, 0.445781618, -0.545298815, -0.346169353, -0.38436529, 0.154302657, 0.517731547, -0.123004794, 0.294294149, -0.45413813, -0.482562453, 0.281019598, -0.610744178, 0.363704741, 0.753128231, 0.086575456, -0.298806816, 0.24589105, 0.0509542264, -0.0878675953, -0.361967802, -0.14129588, 0.291017771, -0.0843326002, 0.128758132, -0.258407384, -0.0918218046, 0.707275033, 0.435013413, 0.0250871573, -0.025642937, -0.158087835, -0.674037695, 0.402723223, -0.0601783954, 0.288742483, 0.243659988, -0.825990617, 0.233642012, 0.269061714, -0.00234434125, -0.0981221199, -0.295686483, 0.219935164, -0.079252176, -0.0368116088, 0.0231886599, 0.375911981, 0.0211249851, -0.502770126, -0.684528112, -0.633163512, -0.299694657, -0.558346987, 0.0696757883, 0.671057284, -0.563194811, -0.547928572, 0.0158232022, -0.124067858, 0.0469608977, -0.375115931, -0.0409443192, 0.144540578, 0.627113402, 0.248610184, -0.504922211, 0.0778462961, 0.0162984747, 0.0167965312, 0.235533431, -0.208053276, 0.211524189, -0.272877842, -0.34588179, 0.178460166, -0.770073295, 0.325554669, 0.703614473, -0.0297916122, -0.327837318, 0.14476645, -0.44144997, -0.234786794, 0.529188812, 0.523501515, -0.357796252, 0.424868345, -0.517006397, 0.141995251, 0.379098713, -0.633924782, -0.251206756, 0.303300261, -0.401111096, 0.313024074, 0.616434216, -0.750947535, 0.386095852, -0.386080652, -0.715659797, 0.555656493, -0.676157176, -0.307923377, 0.264926344, -0.165334404, 0.311968446, -0.291944951, 0.305121362, -0.301692277, -0.412759036, -0.418982774, 0.274645507, 0.610886574, 0.565908909, 0.414676845, 0.207962871, 0.588509679, -0.404941797, -0.6643821, 0.66783911, 0.424814522, 0.481505871, 0.24890855, -0.242444739, 0.265006423, 0.439041078, -0.175621569, -0.500849247, -0.224863112, 0.277053595, 0.169953287, 0.346366912, -0.169367328, -0.483527571, 0.376635015, -0.450908452, 0.827903807, 0.32844761, -0.474182993, 0.488985538, -0.84350425, -0.501130641, -0.379122108, 0.504692018, -0.348160535, -0.394577801, -0.332454652, 0.620442033, 0.347108215, -0.362344354, 0.395488024, -0.402053118, 0.130479932, 0.457383066, -0.326182216, -0.125654116, 0.310799748, -0.326834619, 0.404181093, 0.532541454, -0.514216602, 0.280710787, -0.485759854, -1.04839063, 0.472379476, -0.611308753, -0.399096906, 0.353094399, -0.18524754, 0.0919896066, -0.21615237, 0.203743756, -0.380719543, -0.396900326, -0.270631969, 0.27788192, 0.400153369, 0.527069449, 0.39818123, 0.136097476, 0.476852208, -0.516976237, -0.425197482, 0.37682882, 0.359076917, 0.305471927, 0.3976219, -0.29075712, 0.280495822, 0.306257486, -0.0916249231, -0.550377309, -0.182597741, 0.316895187, 0.282076895, 0.494167656, -0.359965324, -0.625084102, 0.323182106, -0.241392806, 0.875507474, 0.19925873, -0.296331018, 0.463919044, -1.01431572, -0.572522163, -0.375802457, 0.474129498, -0.484108001, 0.288413167, 0.274932802, -0.710556924, -0.475689083, 0.546976268, -0.510572076, 0.488235116, -0.145688176, -0.398286849, 0.582664728, 0.363170892, -0.255636573, 0.209787473, -0.474498898, -0.612328053, 0.685234785, -0.581897259, 0.260182798, 0.670555294, -0.621553898, 0.635084927, 0.255827755, -0.425478548, 0.17255944, -0.266601831, 0.342834711, -0.223253682, 0.379250973, 0.261061937, 0.300956577, -0.462680608, -0.60275054, -0.428009123, -0.413296402, -0.417993307, -0.380859584, 0.484225571, 0.475330383, -0.430124938, -0.514763474, -0.297663152, -0.259608954, 0.3845824, -0.471717864, -0.46136874, 0.301499248, 0.500539005, 0.398300767, -0.402377456, -0.304875851, -0.270902991, 0.139693648, 0.46329838, -0.202600747, 0.52929157, -0.914714396, -0.263905555, 0.51817435, -0.66469872, 0.65652138, 0.703120649, 0.334961891, -0.464073271, 0.482738733, -0.402032852, -0.256628215, 0.60325563, 0.464955986, -0.488754064, 0.44054684, -0.351931095, 0.335125148, 0.383993655, -0.453640074, -0.357266277, 0.264695346, -0.423238248, 0.323907405, 0.363439411, -0.529959738, 0.442113191, -0.233310133, -0.54887563, 0.534587204, -0.416193873, -0.249545828, 0.218593985, -0.167820081, -0.0409015939, -0.30801788, 0.278022349, -0.213988036, -0.185186997, -0.215305299, 0.197828189, 0.241533354, 0.457693577, 0.322801739, 0.195181891, 0.416285813, -0.474574894, -0.573814929, 0.551088929, 0.432626188, 0.186370268, 0.417005748, -0.178998664, 0.369209796, 0.364946485, -0.255508095, -0.286388338, -0.304020703, 0.39779672, 0.201815382, 0.432966501, -0.0968573317, -0.54456532, 0.459975719, -0.403664708, 0.968537927, 0.221455663, -0.494535148, 0.299640477, -0.644444764, -0.410453022, -0.386866421, 0.267461985, -0.356428832, -0.328805238, -0.0637454614, 0.393411905, 0.468803138, -0.357432812, 0.378821403, -0.325893372, 0.350011259, 0.417902291, -0.618172526, -0.285892338, 0.0627596155, -0.391099364, 0.342592061, 0.523384273, -0.566791475, 0.385336578, -0.543573558, -0.475294858, 0.979063153, -0.267701507, -0.554845214, 0.276173621, -0.0819283798, 0.314517885, -0.230857477, 0.0595642999, -0.120733447, -0.276159704, -0.519333899, 0.207524702, 0.676103473, 0.855233908, 0.499728501, 0.328417093, 0.440930963, -0.268772095, -0.739480734, 0.7635445, 0.525407851, 0.154224113, 0.256070346, -0.0851509646, 0.390352964, 0.22515586, -0.271448046, -0.903774858, -0.486533314, 0.536528051, 0.175873756, 0.415732712, -0.0821277201, -0.344281822, 0.160368368, -0.330616474, 0.616188943, 0.417988837, -0.286683828, 0.702758849, -0.648998976, -0.853715777, -0.0481607579, 0.500560045, -0.462513, -0.552843332, -0.34522602, 0.706017435, 0.421820223, -0.36116761, 0.255278349, -0.421875745, 0.306022316, 0.586157978, -0.576375782, -0.374811351, 0.253098905, -0.238848642, 0.260446787, 0.519964099, -0.747914732, 0.380197048, -0.519582868, -0.866442919, 0.661144316, -0.496748656, -0.428809196, 0.522595227, -0.387359023, 0.242774397, -0.349623442, 0.180318043, -0.493550926, -0.224050626, -0.481433094, 0.229462758, 0.457891613, 0.391782224, 0.629506469, 0.194474161, 0.388027042, -0.407218933, -0.461699724, 0.504316986, 0.447760761, 0.455234855, 0.502935708, -0.297365248, 0.423520356, 0.430027187, -0.328196764, -0.539643645, -0.143298954, 0.291758806, 0.3875072, 0.36834985, -0.412410349, -0.748720109, 0.408659816, -0.520982742, 0.956483185, 0.219293684, -0.341582566, 0.395721704, -1.01725376, -0.595943451, -0.337810069, 0.295607686, -0.488323599, -0.349636436, -0.308000356, 0.490402669, 0.638465285, -0.486218452, 0.430971801, -0.352230936, 0.202724606, 0.32218647, -0.674066067, -0.439740092, 0.177810341, -0.311327368, 0.238911331, 0.568857551, -0.466204226, 0.309048265, -0.48708418, -0.624827981, 0.607511163, -0.47014752, -0.32180655, 0.231024921, -0.155010208, 0.0975646004, -0.353846371, 0.312885731, -0.177006781, -0.292344511, -0.628311932, 0.366413593, 0.578064263, 0.763272107, 0.473832756, 0.259060949, 0.629206419, -0.407530755, -0.828761935, 0.591798067, 0.584671795, 0.494536638, 0.220479235, -0.144863576, 0.566604674, 0.438300043, -0.360856116, -0.619844854, -0.392967105, 0.412362367, 0.352951437, 0.213788524, -0.193909869, -0.506160259, 0.221962705, -0.461049676, 0.636038899, 0.4712286, -0.372897178, 0.570715547, -0.735938251, -0.706887722, -0.32411629, 0.367031485, -0.453473657, 0.329574943, 0.113858491, -0.433573961, -0.597322106, 0.376203626, -0.308104128, 0.333011091, -0.308438241, -0.35983184, 0.433434129, 0.302102745, -0.279549867, 0.22821936, -0.439804673, -0.620297611, 0.670302868, -0.47142598, 0.484421641, 0.716174126, -0.639104605, 0.551014662, 0.40932253, -0.492379755, 0.189157993, -0.316898793, 0.253892779, -0.381210774, 0.252850324, 0.340161383, 0.555473149, -0.355789244, -0.498992503, -0.452613264, -0.398562074, -0.316708058, -0.313004225, 0.362591386, 0.449660271, -0.443094134, -0.485129714, -0.306576848, -0.421018839, 0.148315728, -0.235493913, -0.300601751, 0.155712843, 0.441041619, 0.160536632, -0.445706367, -0.244331717, -0.28677398, 0.328690678, 0.541368484, -0.240227968, 0.321249127, -0.718577266, -0.392744094, 0.272827089, -0.587734699, 0.649854302, 0.610579669, 0.318078816, -0.271371663, 0.379635185, -0.0426894836, 0.0169328637, 0.404992431, 0.357325703, -0.28137812, 0.100860856, -0.109935589, 0.310672909, 0.288043588, -0.741093874, -0.299798697, 0.13814421, 0.0261280425, 0.0171266366, 0.425724715, -0.442861974, 0.0923770443, -0.401256651, -0.474165499, 1.03819466, -0.386220872, -0.378698617, 0.057664983, -0.0632421151, 0.179827541, -0.40752545, 0.042543333, 0.025185233, 0.0572029725, -0.543838143, -0.0303743128, 0.4416278, 0.846494555, 0.552702963, 0.363539606, 0.561988175, -0.395481825, -0.757195771, 0.834630728, 0.296801209, 0.135583386, 0.242461458, 0.00149853434, 0.522064805, 0.121808387, -0.382256597, -0.944355726, -0.238420978, 0.349322855, 0.0415029116, 0.195602342, 0.0975472555, -0.451244146, 0.123684511, -0.0612902269, 0.54722321, 0.465005547, -0.32563898, 0.92168051, -0.422961742, -0.902706802, -0.0454702005, 0.475701034, -0.269188583, 0.431137741, 0.302249223, -0.365169317, -0.424596906, 0.409171462, -0.394324839, 0.455797195, -0.351036966, -0.339656293, 0.505931258, 0.316299289, -0.211256802, 0.225225851, -0.250558972, -0.390492499, 0.250553638, -0.300851762, 0.408233941, 0.419053882, -0.449558645, 0.2857427, 0.287398577, -0.175023362, 0.306584656, -0.200416088, 0.43390587, -0.139036909, 0.129665568, 0.126845345, 0.519663393, -0.327636778, -0.320798934, -0.543910921, -0.368158132, -0.395504296, -0.438559741, 0.41207847, 0.58443594, -0.585414469, -0.386796921, -0.195108861, -0.254426181, 0.371502966, -0.367399126, -0.421506017, 0.349295169, 0.570209265, 0.170539469, -0.401865393, -0.129753679, -0.146981284, 0.272144884, 0.411458701, -0.364425331, 0.214164123, -0.626362205, -0.327580601, 0.461556613, -0.465595633, 0.625617087, 0.539699614, 0.0691942871, -0.450905859, 0.369083643, 0.488014132, 0.308510482, -0.985760093, -0.656855106, 0.460517436, -0.374313235, 0.452514172, -0.243043512, -0.568539202, 0.400988013, 0.326916158, -0.137534708, 0.253734499, -0.31904614, -0.404188812, 0.772877038, -0.442900211, 0.326931804, 1.42899549, -0.716805339, 0.714970112, 0.220500067, -0.302772075, 0.337722123, 0.107022166, 0.263308704, -0.395402163, 0.190843195, 0.292111814, 0.302254111, -0.264495552, -0.320229203, -0.468786806, -0.398733824, -0.34744975, -0.560575843, 0.573619306, 0.717945099, -0.610519886, -0.272593498, -0.415558428, -0.278039813, 0.223500475, -0.333608121, -0.613316178, 0.0363137797, 0.530672193, 0.162215203, -0.175550312, -0.190970629, -0.542968452, 0.123111486, 0.764055014, -0.224358305, 0.401514381, -1.14394391, -0.358151048, 0.398012012, -0.429840177, 1.23222005, 0.550289273, 0.419542074, -0.246719256, 0.366144329, -0.226493016, -0.0867672637, 0.494269937, 0.345735371, -0.401583374, 0.313434929, -0.462404966, 0.364968777, 0.269517332, -0.529125035, -0.209614113, 0.262683421, -0.162425041, 0.422719598, 0.639131129, -0.326728851, 0.29691115, -0.270547688, -0.430654705, 0.425371289, -0.274355829, -0.408329993, 0.3738873, -0.271478355, 0.117712818, -0.31778717, 0.194500893, -0.35478574, -0.319126397, -0.41315937, 0.225813165, 0.456299156, 0.477703869, 0.570867181, 0.240507439, 0.523794234, -0.546395957, -0.482751936, 0.607023597, 0.244518608, 0.337806463, 0.210750669, -0.368023336, 0.424761921, 0.225456685, -0.314680427, -0.622482777, -0.443952829, 0.303335637, 0.173702255, 0.25203687, -0.125377074, -0.495982766, 0.125651434, -0.325726569, 0.678031385, 0.22161974, -0.337750196, 0.410270035, -0.607445538, -0.593451202, -0.101136215, 0.442320049, -0.446277022, 0.288560629, 0.150555223, -0.779746771, -0.559381187, 0.398118377, -0.333069712, 0.512455344, -0.232755899, -0.412902117, 0.438120782, 0.210418478, -0.178836808, 0.406812817, -0.264023304, -0.581604242, 0.858014107, -0.559283972, 0.289856821, 1.30308509, -0.600879848, 0.745255113, 0.319138259, -0.530548751, 0.265625685, -0.105322875, 0.403484702, -0.175625131, 0.449767977, 0.312865049, 0.267236799, -0.468998283, -0.539295316, -0.578932226, -0.418343246, -0.338175923, -0.327055544, 0.600691676, 0.69551158, -0.440372705, -0.475253642, -0.525151074, -0.440498412, 0.411674201, -0.322002083, -0.555084109, -0.026644798, 0.413151562, 0.335182786, -0.458753407, -0.322538793, -0.517705083, 0.360494882, 0.790223479, -0.318971336, 0.309954107, -1.18444574, -0.332045048, 0.528458416, -0.438204348, 1.2769779, 0.463581741, 0.346188903, -0.541043937, 0.472952843, -0.151076883, -0.0391670316, 0.484165132, 0.163757727, -0.155744925, 0.237383991, -0.098856166, 0.458446026, 0.26004383, -0.658104837, -0.488162577, 0.149263903, -0.251275361, 0.00616846327, 0.71037817, -0.320424646, 0.100915834, -0.569660246, -0.428083092, 1.01265335, -0.258638352, -0.331758499, 0.240801767, -0.211912602, 0.217610046, -0.300908387, 0.172748744, -0.0578850731, -0.089725554, -0.631647527, 0.0396588184, 0.48446086, 0.931545079, 0.477644712, 0.467726141, 0.360678792, -0.337131947, -0.714310169, 0.703947663, 0.48688671, 0.00236883806, 0.269856632, 0.000911458512, 0.396760881, 0.173451453, -0.223313868, -0.782667279, -0.446920216, 0.504058659, 0.226436675, 0.135301575, 0.0137502644, -0.295697212, 0.07708776, -0.296536386, 0.410770506, 0.25934276, -0.371930927, 0.880129695, -0.329439849, -0.953839064, -0.00357799907, 0.320931822, -0.294914871, 0.316993922, 0.386491984, -0.595305383, -0.621000111, 0.37464565, -0.438520551, 0.588068843, -0.179137543, -0.426252246, 0.422629029, 0.299157232, -0.163523972, 0.281377017, -0.450707316, -0.605161548, 0.558930933, -0.416764915, 0.420474023, 0.77181983, -0.512496769, 0.456202865, 0.28713274, -0.347833633, 0.155532271, -0.256846756, 0.305453092, -0.34788537, 0.306106925, 0.302135617, 0.519958258, -0.328972161, -0.437687069, -0.364500254, -0.602900267, -0.301467001, -0.345538378, 0.40527764, 0.668859303, -0.446932107, -0.321572036, -0.447129726, -0.431977034, 0.132199794, -0.410320789, -0.284836024, 0.280218333, 0.624450326, 0.241631314, -0.270135522, -0.231136993, -0.206530064, 0.164369702, 0.658122003, -0.235409796, 0.319439828, -0.844047725, -0.172972515, 0.42934078, -0.624288917, 0.651216745, 0.62214458, 0.28920868, -0.306190461, 0.508596659, 0.465467989, 0.356304526, -0.890000701, -0.493024111, 0.513009727, -0.512668431, 0.569935322, -0.20882903, -0.406313419, 0.425057709, 0.0926937088, -0.225285247, 0.374424994, -0.45082283, -0.375959128, 0.647611201, -0.422669321, 0.377288282, 0.988787174, -0.628787696, 0.72126776, 0.186070025, -0.370825142, 0.341421396, 0.112420022, 0.297329009, -0.215211868, 0.157667965, 0.324930221, 0.264982998, -0.225670323, -0.305468589, -0.442242056, -0.530349433, -0.274917603, -0.444238096, 0.541301429, 0.705904007, -0.544211388, -0.228262156, -0.223299339, -0.317610562, 0.236425012, -0.187866107, -0.446753472, 0.0985204503, 0.536803126, 0.0847401693, -0.34847939, -0.28480795, -0.439357877, 0.0954972357, 0.631364465, -0.178758129, 0.329071105, -0.956256747, -0.164466277, 0.35494101, -0.566812098, 1.06217372, 0.461021632, 0.336623818, -0.276855886, 0.427599818, -0.431912601, -0.217444614, 0.640483379, 0.324302703, -0.283906847, 0.271796942, -0.289066911, 0.470481485, 0.276978433, -0.54233408, -0.274462193, 0.297958046, -0.378045768, 0.253829062, 0.563533485, -0.421176434, 0.359822452, -0.48794505, -0.509410381, 0.625544548, -0.352221876, -0.403380096, 0.415013462, -0.286652893, 0.297795743, -0.451389909, 0.313659728, -0.291744769, -0.314239085, -0.379596859, 0.249631584, 0.403039992, 0.564996243, 0.510495424, 0.35699755, 0.619771063, -0.606117427, -0.67794311, 0.51534009, 0.333167613, 0.395176947, 0.415323824, -0.0689083189, 0.421069771, 0.469743133, -0.124462351, -0.567709386, -0.256274223, 0.264171898, 0.374026358, 0.207392007, -0.138830185, -0.572796941, 0.26487577, -0.482657969, 0.708209276, 0.296646059, -0.292218029, 0.748012424, -0.486979634, -0.697995782, -0.176561177, 0.611691058, -0.379391581, -0.39062345, -0.411017567, 0.866223156, 0.706337273, -0.402111232, 0.56058228, -0.544899106, 0.375838667, 0.475690663, -0.548797905, -0.269659221, 0.366319329, -0.434439659, 0.240379333, 0.307958692, -0.739541531, 0.652657211, -0.286324143, -1.53226817, 0.542305052, -0.793576777, -0.465901852, 0.417034954, -0.216747954, 0.0475536212, -0.233952254, 0.24702768, -0.338931412, -0.460048586, -0.495621622, 0.402857006, 0.428530186, 0.418013602, 0.414458543, 0.204654932, 0.3397277, -0.632151961, -0.759893477, 0.565124869, 0.35447821, 0.534128904, 0.289917767, -0.38015452, 0.496138215, 0.447544396, -0.277757704, -0.57324636, -0.339929491, 0.286599487, 0.424487829, 0.321267098, -0.401668042, -0.640672326, 0.38852036, -0.312558293, 1.13503742, 0.312915683, -0.451842874, 0.392264873, -1.27436757, -0.725945234, -0.454566032, 0.391351521, -0.514046371, 0.16079925, 0.210725769, -0.405412287, -0.316861272, 0.149214953, -0.35323894, 0.411222249, -0.327723145, -0.445907444, 0.69757092, 0.4237369, -0.188625678, 0.0774613917, -0.149058148, -0.471323401, 0.358809143, -0.351791233, 0.549129903, 0.588863492, -0.887951314, 0.471756995, 0.492872179, -0.382756084, 0.0816366002, -0.135769561, 0.463379323, -0.261050701, 0.292719781, 0.156909585, 0.455610722, -0.210006192, -0.568528354, -0.871279955, -0.544241428, -0.249187201, -0.580679417, 0.270824641, 0.800079048, -0.756231189, -0.550939262, -0.328521103, -0.119561553, 0.0194189325, -0.549140692, -0.204249993, 0.434082389, 0.660503983, 0.338215262, -0.5055058, -0.318888515, -0.30896017, -0.00862062443, 0.450840265, -0.0802882537, 0.21830225, -0.66549778, -0.317940623, 0.233479813, -0.621768594, 0.386966825, 0.789339066, 0.291289717, -0.396497995, 0.174070537, -0.388177931, -0.332033396, 0.943733513, 0.428894907, -0.421334684, 0.508803189, -0.345837325, 0.0400707796, 0.438002676, -0.569301665, -0.279780656, 0.223079726, -0.374037147, 0.346421629, 0.522622645, -0.566868246, 0.344092637, -0.423395425, -0.903560698, 0.657193184, -0.473076731, -0.318999141, 0.467569053, -0.333939135, 0.155065089, -0.139922574, 0.231326848, -0.422497123, -0.36896354, -0.499037743, 0.235308364, 0.566282034, 0.359879166, 0.435069978, 0.153725326, 0.474499553, -0.427220821, -0.678500175, 0.545710087, 0.404682159, 0.306849003, 0.376173109, -0.20642516, 0.351348698, 0.37668404, 0.0678337812, -0.420030922, -0.162219271, 0.185821801, 0.41966033, 0.363682985, -0.244284928, -0.618130982, 0.478689373, -0.270262152, 0.942919612, 0.225905895, -0.371593744, 0.378418505, -1.24545348, -0.572436631, -0.25611183, 0.281736225, -0.337322891, 0.120095894, 0.0458138362, -0.590941548, -0.362830758, 0.143806055, -0.36226353, 0.397725195, -0.467312008, -0.406470567, 0.658315778, 0.365121275, -0.195868224, 0.126190424, -0.331685543, -0.540272951, 0.518366635, -0.17168048, 0.459273279, 0.370512098, -1.00907397, 0.423638344, 0.324679941, -0.222556978, 0.0882237032, -0.227587491, 0.482755631, -0.108196519, 0.16863367, 0.054100126, 0.639589489, -0.11028415, -0.614035308, -1.01526451, -0.776605904, -0.447236985, -0.477974087, 0.231578916, 0.810127079, -0.956994772, -0.33736375, -0.361851811, -0.210540742, 0.0497537255, -0.314863205, -0.222965494, 0.297769547, 0.829195917, 0.420577615, -0.479922831, -0.1932109, -0.177411839, 0.142029166, 0.388717592, -0.258186758, 0.267783225, -0.645706236, -0.335402578, 0.183609232, -0.78569591, 0.650520921, 0.868913889, 0.0981106982, -0.4116413, 0.221889883, 0.31409514, -0.0168841016, -0.548824787, -0.45937115, 0.351160645, -0.0818493739, 0.373066097, -0.344443113, -0.381085783, 1.02282059, 0.321285933, -0.101764858, 0.192896143, -0.155903578, -0.684190929, 0.522310734, -0.393799186, 0.439627588, 0.748493135, -1.6595422, 0.449019045, 0.486280322, -0.28461802, 0.115419254, -0.302514464, 0.513807952, -0.186363235, 0.0939508677, 0.130765125, 0.679721415, -0.022032721, -0.743874371, -1.82264137, -0.860185266, -0.472115159, -0.727490306, 0.372781038, 1.38417804, -1.29241812, -0.535942554, -0.0400269739, -0.103019238, 0.111453742, -0.376251012, -0.36089462, 0.104617834, 1.92165339, 0.317137599, -0.531428576, -0.193516761, -0.137402773, 0.063355118, 0.349306852, -0.0617837831, 0.306067228, -0.640568137, -0.171641544, 0.409577489, -1.16000879, 0.679099798, 1.55457997, -0.0590775721, -0.581195414, 0.359650403, 0.475384116, 0.215332747, -0.911786973, -0.535001516, 0.423538387, -0.375832736, 0.380926251, -0.213422522, -0.441743195, 0.520301878, 0.0738486797, -0.203792587, 0.225653142, -0.500900984, -0.352563471, 0.642879963, -0.462786645, 0.216654375, 1.06189287, -0.544227242, 0.611953497, 0.260258466, -0.287598997, 0.442782819, -0.10331279, 0.321091861, -0.195554465, 0.256332159, 0.375735879, 0.439173549, -0.442848146, -0.297518045, -0.459702373, -0.540614903, -0.30653888, -0.287601888, 0.665254235, 0.412513703, -0.550573587, -0.451120049, -0.416260868, -0.331913412, 0.198240608, -0.20242241, -0.449633181, -0.0276320577, 0.446590245, 0.3299959, -0.366585106, -0.262439489, -0.325694323, 0.182583779, 0.46954295, -0.418800116, 0.477131039, -0.964160502, -0.319363981, 0.573387384, -0.56479162, 1.14394426, 0.565735996, 0.424945265, -0.226481229, 0.493830502, -0.412981153, -0.375823587, 0.737215638, 0.570785224, -0.323629379, 0.489963114, -0.574758351, 0.376042485, 0.52354306, -0.366570979, -0.318353593, 0.30906114, -0.365421176, 0.349539757, 0.299283206, -0.696141303, 0.347116262, -0.235132277, -0.916872561, 0.624709487, -0.47033748, -0.187180743, 0.386573792, -0.422119677, 0.0305087045, -0.281929165, 0.169989243, -0.453104675, -0.284178585, -0.30486244, 0.397361368, 0.525049567, 0.597838163, 0.491240352, 0.235518813, 0.225881934, -0.482109487, -0.486117691, 0.46542114, 0.253047436, 0.207687333, 0.237948924, -0.199165568, 0.44691816, 0.54960084, -0.212439716, -0.503438771, -0.233035192, 0.392413527, 0.438332915, 0.416876972, -0.155959249, -0.732186079, 0.320732772, -0.469835073, 0.827637196, 0.353363186, -0.324991733, 0.404210299, -0.864878178, -0.615257084, -0.202500567, 0.291328877, -0.566053033, 0.0874508694, -0.0195382517, -0.26613149, -0.406176984, 0.278051227, -0.213906258, 0.268738121, -0.198853984, -0.245324314, 0.665124059, 0.350464612, -0.00426692376, 0.0108659388, -0.201048553, -0.575250149, 0.292187661, -0.346289426, 0.533586383, 0.502590358, -0.66506511, 0.292921185, 0.30451104, -0.284007937, 0.147210762, -0.291302562, 0.426081091, -0.177212387, 0.0219840333, 0.113528401, 0.599709928, -0.0496736094, -0.440843016, -0.720499814, -0.715811372, -0.516294301, -0.460766047, 0.192094356, 0.694373429, -0.527056575, -0.300620675, -0.313924015, -0.129618391, -0.0570446029, -0.270844102, -0.336233318, 0.351289213, 0.777409077, 0.314562112, -0.463543475, -0.256572634, -0.100103155, -0.0737717301, 0.223827228, -0.206478432, 0.205807179, -0.391174227, -0.238219768, 0.132798344, -0.676143289, 0.542043924, 0.517598927, -0.0544856228, -0.481620997, 0.21524398, -0.243028104, -0.163744271, 0.576677859, 0.439167857, -0.184076488, 0.168333605, -0.330766976, 0.420736045, 0.274111062, -0.641604543, -0.296700835, 0.0656826124, -0.119610876, 0.0926019698, 0.550128818, -0.321108013, 0.146554098, -0.59891665, -0.359992892, 1.34891152, -0.332585424, -0.411800206, 0.208950475, -0.186248854, 0.185747251, -0.413295031, 0.124468625, -0.128618792, -0.274564058, -0.506177127, 0.216666251, 0.581105828, 1.06260896, 0.650262356, 0.441327751, 0.544335544, -0.398775637, -0.728176594, 0.990727246, 0.604771376, 0.242025897, 0.246481806, 0.0635329187, 0.349909067, 0.292281032, -0.26457721, -1.05096507, -0.399784714, 0.349184483, 0.127662018, 0.0902292132, 0.0907274708, -0.276808441, 0.0953731462, -0.337031752, 0.437619835, 0.347538531, -0.415724725, 0.947669744, -0.381604582, -1.13966286, -0.18662113, 0.525672495, -0.222771138, 0.409885228, 0.181371853, -0.46162796, -0.424802214, 0.326711148, -0.203998908, 0.408123285, -0.420484006, -0.272217184, 0.76048547, 0.515119731, -0.0933296978, 0.409145027, -0.321470916, -0.72881335, 0.488860458, -0.288540423, 0.613845468, 0.678315043, -0.898112297, 0.389775783, 0.524731636, -0.297094494, 0.161863849, -0.247477472, 0.45917359, -0.115731731, 0.155483097, 0.231482834, 0.418769807, -0.176665559, -0.585157752, -0.886291504, -0.705376208, -0.515281737, -0.396261424, 0.523047507, 0.835329235, -0.973869681, -0.497394949, -0.375061154, -0.440276712, 0.129687801, -0.444781601, -0.254213691, 0.179852232, 0.764155626, 0.394868851, -0.29218936, -0.180049241, -0.284795284, 0.149435118, 0.398981392, -0.29641214, 0.445781738, -0.746270061, -0.372758031, 0.376994699, -0.835753441, 0.478801936, 0.932245374, 0.170552269, -0.58489275, 0.381816447, 0.48789376, 0.400772721, -0.752847552, -0.499535441, 0.446504593, -0.33699733, 0.517591, -0.113535076, -0.409256637, 0.449244082, 0.192122892, -0.126278639, 0.420830876, -0.405703992, -0.464650601, 0.731547058, -0.445717573, 0.361120403, 0.960501015, -0.610710859, 0.535881579, 0.24686271, -0.367468953, 0.280776471, -0.247674271, 0.383428425, -0.294800282, 0.283032984, 0.309191495, 0.375214219, -0.426270634, -0.378553718, -0.530820072, -0.549305677, -0.28056702, -0.352196664, 0.431088388, 0.370129853, -0.555204034, -0.421654552, -0.491750449, -0.340274781, 0.397931695, -0.18644014, -0.342986912, 0.228953987, 0.534403563, 0.308754742, -0.362085879, -0.158810034, -0.374743491, 0.155526653, 0.650469542, -0.371493012, 0.368921071, -0.857041895, -0.249441326, 0.524518967, -0.42098698, 0.737317026, 0.421600848, 0.319834441, -0.218405604, 0.499209315, 0.369475812, 0.247101828, -0.409187824, -0.285732925, 0.290641516, -0.299312472, 0.332067758, -0.376642853, -0.271390468, 0.725094557, 0.292342991, -0.214276835, 0.251660913, -0.284254372, -0.736112356, 0.491976917, -0.204357207, 0.554132521, 0.409758359, -0.886488199, 0.252144128, 0.313474178, -0.168149337, 0.165345505, -0.348877728, 0.391794682, -0.312098622, 0.244126007, 0.165552765, 0.609793305, -0.187694117, -0.4168064, -0.538281262, -0.527159393, -0.413596004, -0.493292034, 0.304236323, 0.819169164, -0.865241706, -0.462231547, -0.196676031, -0.191255212, 0.261624455, -0.33057946, -0.18604283, 0.424600273, 0.785979986, 0.416870803, -0.309830725, -0.330239534, -0.17728816, 0.108429, 0.605147719, -0.252122492, 0.251037598, -0.50129813, -0.418912619, 0.411148965, -0.551536262, 0.495993406, 0.84234041, 0.188048735, -0.50608623, 0.364637583, -0.384309918, -0.391212225, 0.841116607, 0.537914276, -0.270776391, 0.230533093, -0.546946108, 0.244140178, 0.345368385, -0.603093922, -0.142137319, 0.0884019211, -0.24174346, 0.219795629, 0.273634315, -0.664947867, 0.540084302, -0.274016023, -1.12177527, 0.627060354, -0.59678781, -0.156358242, 0.262689561, -0.325996757, -0.0372905135, -0.264883995, 0.379849762, -0.391517431, -0.232241035, -0.286120713, 0.22352384, 0.449820071, 0.481535673, 0.570147336, 0.0741384476, 0.361522198, -0.40510112, -0.605552971, 0.632405043, 0.289219856, 0.363000095, 0.411892653, -0.146651626, 0.364796788, 0.438328624, -0.136313125, -0.413992584, -0.0620639771, 0.392394841, 0.258055389, 0.463164598, -0.19629328, -0.732971132, 0.414148003, -0.355665833, 1.04848206, 0.275394887, -0.614567935, 0.602525294, -1.39067745, -0.576803386, -0.385085493, 0.422306299, -0.40450123, 0.269389689, 0.316030174, -0.552360415, -0.438024879, 0.289036006, -0.392597258, 0.338405281, -0.13281852, -0.384657353, 0.554327309, 0.169573352, -0.131987825, 0.31911388, -0.341362178, -0.291610777, 0.733600318, -0.368896484, 0.292443722, 0.777043223, -0.45216462, 0.504087627, 0.197740391, -0.463237554, 0.373238415, -0.203284413, 0.230572298, -0.242228985, 0.319728345, 0.242422327, 0.220397592, -0.445341974, -0.374401301, -0.555892706, -0.490904301, -0.258437186, -0.444234222, 0.39764908, 0.488627434, -0.556188285, -0.398761451, -0.493797839, -0.489582747, 0.268681318, -0.427104145, -0.510954678, 0.105838746, 0.347195417, 0.183347389, -0.373264492, -0.346296936, -0.298220932, 0.275936007, 0.629091144, -0.368624121, 0.374072254, -0.86580801, -0.328984052, 0.577003062, -0.475551099, 1.0227052, 0.590043962, 0.383470744, -0.368406206, 0.553536415, 0.393583238, 0.309779227, -0.554365396, -0.38535139, 0.428513646, -0.195629299, 0.41048032, -0.252766937, -0.274031401, 0.45824936, 0.28105101, -0.160015211, 0.38542375, -0.382457107, -0.433201551, 0.399579316, -0.216419056, 0.345784843, 0.462602407, -0.660349786, 0.413877994, 0.302809894, -0.230250865, 0.253587872, -0.113286465, 0.300712019, -0.156404674, 0.288530618, 0.348006606, 0.461906075, -0.122462071, -0.536860168, -0.507788301, -0.580444396, -0.419831276, -0.243066341, 0.53788799, 0.537369907, -0.600037277, -0.466053933, -0.245911658, -0.329682887, 0.165540665, -0.288319468, -0.432209313, 0.28477782, 0.338071287, 0.25602442, -0.310828, -0.417393237, -0.446124554, 0.0644551143, 0.500903487, -0.236426741, 0.443310887, -0.700926185, -0.296836257, 0.477122337, -0.597384393, 0.69430697, 0.562427342, 0.298457295, -0.353467017, 0.383789986, -0.247371465, -0.203480422, 0.583611608, 0.268139154, -0.43694517, 0.363372177, -0.369097143, 0.259204566, 0.361795068, -0.586825669, -0.33919996, 0.114610553, -0.29522875, 0.13504006, 0.665973842, -0.363396794, 0.329544693, -0.399422258, -0.695483923, 0.768218815, -0.535257876, -0.468420833, 0.3680574, -0.179449856, 0.193810478, -0.462563217, 0.178024516, -0.0898036659, -0.267449468, -0.453599662, 0.157640412, 0.655802011, 0.66850996, 0.706598103, 0.284123182, 0.434089571, -0.292810559, -0.887778342, 0.695580781, 0.387305737, 0.222245499, 0.425396055, -0.103639573, 0.543849289, 0.268413097, -0.138714075, -0.766526341, -0.490518153, 0.404170156, 0.246892452, 0.366620004, -0.192014739, -0.629168987, 0.227558315, -0.405429155, 0.772421479, 0.502423882, -0.312957108, 0.763817549, -0.472828001, -0.925790489, -0.0528889261, 0.658507884, -0.283840716, -0.325200498, -0.139414474, 0.401559412, 0.228570744, -0.307639718, 0.278669387, -0.431588918, 0.460738182, 0.334268004, -0.757360518, -0.420996368, 0.049914252, -0.154565185, 0.144961759, 0.52449441, -0.359486669, 0.222480401, -0.436636657, -0.496427655, 0.945137143, -0.488757819, -0.444308817, 0.335362673, -0.271578759, 0.163565576, -0.451666355, 0.123458102, -0.240851939, -0.383218318, -0.445940673, 0.128106713, 0.610327899, 0.803149581, 0.669171751, 0.447072834, 0.497676134, -0.362726867, -0.730415165, 0.825091898, 0.351437598, 0.217528388, 0.360408157, -0.281360835, 0.603214562, 0.246845424, -0.306878477, -0.74486053, -0.379564077, 0.346566468, 0.168518886, 0.403990984, -0.127717942, -0.360213995, 0.350952804, -0.261595696, 0.554044366, 0.335477173, -0.419198751, 0.851325989, -0.683273196, -0.956246316, -0.181803375, 0.458820194, -0.297948629, 0.238015428, 0.0793840662, -0.496541321, -0.267986447, 0.240847871, -0.111892313, 0.283916324, -0.223188505, -0.113293678, 0.735074401, 0.289534718, 0.0644976869, 0.226398841, -0.00430864841, -0.450169176, 0.389421165, -0.0806062669, 0.442707628, 0.35259974, -0.8274858, 0.403373003, 0.346282929, -0.0932031572, 0.209753737, -0.37730664, 0.436992466, -0.0396686606, 0.169427603, 0.235724255, 0.575926065, 0.0262585115, -0.672419369, -0.765878379, -0.724586248, -0.250511557, -0.531025946, 0.200946376, 0.473256648, -0.631293476, -0.423229694, -0.245246649, -0.0285535324, -0.144437358, -0.549280822, -0.315312207, 0.230095178, 0.692253649, 0.359022915, -0.282209247, -0.0860122368, -0.0103105437, -0.0100394515, 0.24300167, -0.142850086, 0.278308928, -0.563721478, -0.501542866, 0.290684551, -0.600704074, 0.37248975, 0.537297487, 0.041685503, -0.538487375, 0.347824425, -0.313666195, -0.107675068, 0.410542667, 0.417645127, -0.155165136, 0.289373368, -0.185421929, 0.449024647, 0.317274034, -0.581352949, -0.41031608, 0.0431830361, -0.357916981, 0.189041391, 0.52964437, -0.338763297, 0.341493279, -0.257057071, -0.472512752, 0.883521914, -0.291867793, -0.392305583, 0.146180823, -0.100352801, 0.253875643, -0.498479694, 0.0707702637, -0.156596795, -0.254705995, -0.567901671, 0.376346976, 0.609128177, 0.635208845, 0.593142211, 0.362132549, 0.536599755, -0.328703612, -0.753822148, 0.560802877, 0.495339155, 0.138926998, 0.299738497, -0.270461142, 0.346564144, 0.307598233, -0.315763563, -0.578102589, -0.272445083, 0.422766209, 0.233591363, 0.303619862, -0.134720758, -0.448584944, 0.340417892, -0.227202311, 0.453481644, 0.47312063, -0.301582664, 0.564079463, -0.493751705, -0.686337292, -0.205262735, 0.54197365, -0.247620851, 0.0344309248, 0.189946458, -0.065027833, 0.000345474662, 0.205416724, -0.0480070785, 0.0912764668, 0.305920243, -0.1800019, -0.250887185, -0.221894979, -0.0942936316, 0.0655761287, -0.167775407, 0.318279624, 0.0301062688, -0.159910113, -0.299182057, -0.188728139, 0.214943707, -0.122218661, -0.225967675, -0.0444394425, 0.157053635, 0.287626475, -0.344853312, -0.259528875, 0.210367605, 0.0949606299, -0.319590539, -0.211907566, 0.305998772, 0.16340746, 0.285573572, 0.20619911, 0.212913722, 0.177616835, -0.306215405, 0.0922551677, 0.193863496, -0.0658633709, -0.132224262, 0.281344682, 0.299214423, -0.110345505, -0.231438458, -0.327115476, -0.28194657, 0.207359001, -0.202775285, -0.029759245, 0.303117305, -0.123671353, -0.044417344, 0.040638309, 0.0157539304, 0.394457281, -0.0379356518, 0.296513975, -0.169488579, -0.157276317, 0.0232879072, 0.304177105, 0.0541127808, -0.485945642, -0.36135, 0.660479724, 0.423538625, -0.337050855, 0.437062204, -0.543585837, 0.302641004, 0.558344603, -0.444594681, -0.383990467, 0.169267401, -0.207057133, 0.461357355, 0.513237119, -0.651970863, 0.383026451, -0.326919407, -0.960975647, 0.502709627, -0.60973686, -0.356365979, 0.452839136, -0.308545589, 0.106135018, -0.19845061, 0.246994868, -0.22833015, -0.280296147, -0.308169544, 0.200807467, 0.511359632, 0.538776994, 0.394334167, 0.344325304, 0.299391031, -0.601296484, -0.496858746, 0.587508976, 0.436448216, 0.385756701, 0.490168691, -0.3315458, 0.441373169, 0.476151615, -0.0619453527, -0.613934696, -0.407150745, 0.197971746, 0.309795618, 0.523114979, -0.132036999, -0.577990294, 0.470109522, -0.399931937, 1.03896189, 0.174513295, -0.359523207, 0.494046867, -0.862068057, -0.533078074, -0.192217931, 0.505256951, -0.388492256, 0.174100712, 0.195429489, -0.457197607, -0.502798319, 0.327439338, -0.392311245, 0.356427222, -0.270699501, -0.458460271, 0.380312681, 0.150350809, -0.176070854, 0.300542861, -0.360865742, -0.583856046, 0.515576422, -0.204642117, 0.45302555, 0.546301126, -0.498377115, 0.516420305, 0.462806493, -0.439206362, 0.106205963, -0.166298181, 0.339345574, -0.178185701, 0.297387213, 0.165833071, 0.501806438, -0.399785012, -0.499625087, -0.458599657, -0.34114632, -0.420146734, -0.242492482, 0.579106808, 0.352222472, -0.539884686, -0.235781401, -0.342602134, -0.2941145, 0.182296664, -0.229395986, -0.410523713, 0.250215411, 0.328568608, 0.171302572, -0.347481668, -0.15096432, -0.153256461, 0.0678987131, 0.560030401, -0.367725492, 0.373485118, -0.491174996, -0.276183546, 0.469605237, -0.451243699, 0.682902277, 0.449186891, 0.191687599, -0.447495073, 0.44682917, -0.354495764, -0.214953139, 0.570384383, 0.607290506, -0.309912205, 0.337733865, -0.572646797, 0.139874786, 0.39843756, -0.362487942, -0.388099432, 0.223540202, -0.424609244, 0.244639635, 0.29228881, -0.470054775, 0.567544639, -0.489977181, -0.852808058, 0.474919975, -0.647274852, -0.401068866, 0.248522773, -0.359556973, 0.149185821, -0.141178489, 0.192091435, -0.442445427, -0.349083036, -0.247978672, 0.416842848, 0.554330111, 0.359283447, 0.557251096, 0.189750567, 0.430174857, -0.515189767, -0.356198311, 0.489667922, 0.40158233, 0.480388343, 0.384018809, -0.228381172, 0.242658481, 0.539808214, -0.0599517152, -0.378246009, -0.223405883, 0.400687873, 0.300552547, 0.387052834, -0.340570301, -0.72891593, 0.238152713, -0.315393418, 0.909782052, 0.216166273, -0.423081666, 0.497089088, -0.979305148, -0.500800371, -0.341082841, 0.225481167, -0.490528077, -0.294875085, -0.176773831, 0.600279629, 0.441150874, -0.279734313, 0.32600674, -0.579203248, 0.155524611, 0.296192765, -0.558640122, -0.292823642, 0.359090835, -0.213707194, 0.463615358, 0.461322188, -0.528903782, 0.469456732, -0.23033765, -1.02339959, 0.628488541, -0.445650339, -0.367278874, 0.494078457, -0.353665709, 0.223716751, -0.312855095, 0.429643124, -0.438727379, -0.445991009, -0.269420981, 0.295045227, 0.442136496, 0.457582921, 0.333032966, 0.241505355, 0.431781411, -0.521913409, -0.452420682, 0.567804277, 0.428872555, 0.489490598, 0.461818755, -0.20265983, 0.396334797, 0.440459281, -0.237307161, -0.506970286, -0.274060309, 0.320778579, 0.432875425, 0.359549552, -0.381314784, -0.720901489, 0.296606034, -0.443178505, 1.15022051, 0.309405237, -0.350920677, 0.36626491, -0.937035382, -0.606027007, -0.309186429, 0.329207569, -0.517853975, -0.341044158, -0.154508501, 0.362724125, 0.332138211, -0.422617197, 0.324678153, -0.358543009, 0.27711913, 0.451690167, -0.497769266, -0.225744188, 0.274952829, -0.180933237, 0.142199531, 0.546207607, -0.35248965, 0.484285206, -0.409175098, -0.561070561, 0.446835548, -0.437814593, -0.419162661, 0.369103163, -0.33444792, 0.153142139, -0.270516485, 0.132258683, -0.420984417, -0.175909087, -0.475659609, 0.342963785, 0.426259041, 0.482439488, 0.40265584, 0.209301397, 0.482845098, -0.437490046, -0.515892982, 0.309698492, 0.198395401, 0.236715555, 0.313970566, -0.216576919, 0.291193485, 0.269574285, -0.276378274, -0.495629311, -0.368442267, 0.356579006, 0.366631597, 0.389299512, -0.113688044, -0.410548627, 0.188285008, -0.290006369, 0.767413974, 0.418548703, -0.420696855, 0.332758814, -0.527156353, -0.568532407, -0.365988404, 0.384107172, -0.429724753, -0.515623629, -0.31600827, 0.54113394, 0.62728399, -0.44118169, 0.48461917, -0.304099888, 0.244923845, 0.47913456, -0.511463344, -0.134884834, 0.178478643, -0.456481576, 0.464062244, 0.403155178, -0.516802311, 0.469760209, -0.274131417, -0.925406039, 0.683194399, -0.556314051, -0.262676477, 0.319428831, -0.337340951, 0.278574347, -0.369379222, 0.39447543, -0.424378663, -0.237108171, -0.363948077, 0.442252487, 0.446504354, 0.568018198, 0.405155897, 0.320903778, 0.470858127, -0.376504332, -0.40928328, 0.620316505, 0.461309552, 0.430827945, 0.365870148, -0.173717096, 0.238033175, 0.527404487, -0.141910002, -0.607519925, -0.433626264, 0.195883676, 0.27829209, 0.331122726, -0.242994428, -0.730860829, 0.306823045, -0.420194536, 0.879377782, 0.206099123, -0.504070103, 0.563019335, -0.874740064, -0.431201428, -0.162987113, 0.224800333, -0.392811447, 0.23666431, 0.124174878, -0.520936489, -0.260279119, 0.174009442, -0.315971017, 0.363126069, -0.423611611, -0.175672486, 0.54098326, 0.445020884, -0.0544905327, 0.154026121, -0.328295887, -0.456431121, 0.437881619, -0.438316405, 0.368522793, 0.355840951, -0.738659263, 0.419419199, 0.360655338, -0.374599993, 0.0870940313, -0.116249382, 0.405575573, -0.269013554, 0.101407722, 0.29289028, 0.527786374, -0.239587769, -0.453272611, -0.529340446, -0.449688733, -0.377864838, -0.531362355, 0.459060848, 0.676799119, -0.546671093, -0.550465941, -0.190264255, -0.371789336, 0.215232447, -0.321701318, -0.35528031, 0.358131886, 0.642617941, 0.458341151, -0.367478192, -0.172872797, -0.18079184, 0.119857892, 0.573992789, -0.25790152, 0.171199247, -0.448096454, -0.293333143, 0.41708523, -0.689325333, 0.531466544, 0.6960302, 0.105832472, -0.520439506, 0.18298763, 0.295250028, 0.0648750141, -0.547792971, -0.378030092, 0.218078449, -0.184435859, 0.23133783, -0.189135805, -0.389943302, 0.3212578, 0.330396056, -0.0594353154, 0.34091115, -0.229732171, -0.590282142, 0.338573754, -0.410895944, 0.420846045, 0.291860342, -0.659962118, 0.31692028, 0.453753024, -0.396362484, 0.168379754, -0.358299762, 0.347434103, -0.28468737, 0.357430845, 0.239723593, 0.432629526, -0.332877636, -0.45397532, -0.591729641, -0.454708219, -0.260705769, -0.296020895, 0.402255744, 0.534129441, -0.590010166, -0.513942361, -0.38513574, -0.177274898, 0.222672492, -0.437557369, -0.385776103, 0.376362562, 0.497511536, 0.261428744, -0.476261407, -0.180336773, -0.387253284, 0.138238996, 0.420188159, -0.293191105, 0.269250393, -0.383231163, -0.474132389, 0.193375021, -0.630862057, 0.396174699, 0.500936985, 0.182403222, -0.493527174, 0.192530602, 0.340060234, 0.383142263, -0.693232238, -0.380380481, 0.470381945, -0.258658886, 0.477341324, -0.245087311, -0.347030282, 0.371673018, 0.341406554, -0.302758545, 0.394184679, -0.237691626, -0.467933893, 0.744960487, -0.383957714, 0.236303031, 1.13399792, -0.597474992, 0.469922811, 0.231444806, -0.516190231, 0.304020286, -0.0542364232, 0.27130577, -0.317319512, 0.487157762, 0.477000058, 0.263333738, -0.348938048, -0.469136715, -0.613555372, -0.353967875, -0.163899779, -0.518040717, 0.483592957, 0.577883959, -0.616701543, -0.442135602, -0.491686165, -0.3167153, 0.215433553, -0.439656824, -0.523868144, 0.261042148, 0.364420444, 0.136963025, -0.461002827, -0.291728735, -0.258468658, 0.400962889, 0.481333166, -0.487069339, 0.311288059, -1.21948445, -0.330258608, 0.562764049, -0.519666493, 0.973513365, 0.36883828, 0.252141148, -0.277709395, 0.435908616, -0.294502944, -0.120495439, 0.618012846, 0.327623993, -0.393051773, 0.29589951, -0.31433475, 0.437040329, 0.416946799, -0.847911358, -0.495486438, -0.0218487848, -0.0938458666, 0.222067982, 0.793957949, -0.529143751, 0.477886498, -0.396578074, -0.701355875, 1.20411623, -0.524900913, -0.392517328, 0.24428764, -0.296788275, 0.321686357, -0.559090734, 0.00724298786, -0.171065554, -0.301436782, -0.580912232, 0.239976898, 0.563864052, 1.26303685, 0.668325007, 0.331461996, 0.546038687, -0.435142785, -1.11664522, 1.09541214, 0.448191643, 0.384961128, 0.375258654, 0.0559365153, 0.628695786, 0.305876464, -0.395852715, -1.28390658, -0.400222331, 0.300594538, 0.0435942449, 0.347624421, -0.0639878809, -0.527391016, 0.158750147, -0.373085976, 0.534933031, 0.381938428, -0.331843764, 0.950296462, -0.614255011, -1.3458612, -0.149373531, 0.543211162, -0.377014011, -0.336651742, -0.233295664, 0.797309339, 0.513071656, -0.458659798, 0.416595906, -0.479039162, 0.208397508, 0.369094044, -0.33914873, -0.123948902, 0.217620924, -0.443428725, 0.24789615, 0.270756036, -0.520253003, 0.439437777, -0.222539097, -0.93068707, 0.513027012, -0.627254486, -0.335910678, 0.297745198, -0.350271404, 0.0980542749, -0.397601038, 0.252478153, -0.361494482, -0.415535629, -0.328489363, 0.244084656, 0.325490683, 0.442657948, 0.509493828, 0.206637979, 0.250472814, -0.50072211, -0.490644038, 0.33298552, 0.196949959, 0.360783905, 0.265887409, -0.14296639, 0.211292595, 0.282961637, -0.214764073, -0.457740545, -0.377057016, 0.268329382, 0.443995386, 0.339058578, -0.166722327, -0.659231424, 0.259215534, -0.247541651, 0.951440156, 0.119866438, -0.331495941, 0.533548594, -1.04290521, -0.380973041, -0.38026461, 0.463556647, -0.553450346, 0.388274312, 0.314227313, -0.734515786, -0.415312618, 0.396463811, -0.465032965, 0.330259204, -0.136353105, -0.37911287, 0.456752777, 0.196156338, -0.226915464, 0.357480735, -0.301920533, -0.351103336, 0.490534633, -0.403399229, 0.374568343, 0.958853066, -0.411008984, 0.655613661, 0.408200473, -0.358712107, 0.41698119, -0.057735417, 0.362245679, -0.1919346, 0.459483832, 0.405272096, 0.312939048, -0.369709015, -0.284686863, -0.544496477, -0.448450774, -0.396722466, -0.351513207, 0.434725523, 0.566712618, -0.441553086, -0.422852814, -0.372797966, -0.262772977, 0.340972573, -0.375152946, -0.450661808, 0.133837804, 0.482885182, 0.109179661, -0.25703603, -0.175039023, -0.447719246, 0.122612499, 0.576418221, -0.245472148, 0.483302653, -0.937460661, -0.149299964, 0.530605853, -0.534834623, 0.859908164, 0.612307727, 0.33648929, -0.195717588, 0.37226367, 0.234359756, 0.0573784001, -0.480780452, -0.391622543, 0.208798051, -0.154145807, 0.189161777, -0.36538434, -0.253668606, 0.700959444, 0.286422849, -0.107619941, 0.173320502, -0.026170671, -0.641995609, 0.360915393, -0.287052065, 0.300064951, 0.417631716, -0.754731238, 0.223420814, 0.531779349, -0.285447836, 0.112132393, -0.320081294, 0.223516479, 0.0796050057, -0.0436959937, 0.0979389697, 0.522259831, 0.0310857296, -0.524198771, -0.530711055, -0.738940418, -0.345038652, -0.589956284, 0.25094974, 0.622439146, -0.727363586, -0.398103148, -0.0818379223, -0.0879493505, -0.00633695442, -0.450119436, -0.148047879, 0.352553815, 0.727132618, 0.340105951, -0.280110508, -0.0363540351, -0.201560363, 0.0324376076, 0.259978384, -0.0896535963, 0.0723608956, -0.396571308, -0.472210407, 0.201583266, -0.623772919, 0.373256624, 0.596561968, 0.170372009, -0.311935186, 0.22581917, -0.262734056, -0.205734208, 0.669653833, 0.548884273, -0.263559908, 0.382155478, -0.315499514, 0.106453419, 0.399859577, -0.253977865, -0.270770609, 0.192438766, -0.358980745, 0.452050358, 0.337466389, -0.601803601, 0.514998257, -0.248154074, -0.494003296, 0.527333379, -0.522102296, -0.296073616, 0.352668911, -0.273080915, 0.271502942, -0.314497381, 0.225861281, -0.193776995, -0.174735174, -0.500692964, 0.347684175, 0.526929259, 0.292768598, 0.298531443, 0.341743916, 0.442465752, -0.545993268, -0.43339932, 0.499211878, 0.393886477, 0.297906786, 0.392510653, -0.15197444, 0.467066497, 0.424802363, -0.119417347, -0.354376733, -0.396603137, 0.405060381, 0.290945709, 0.267006844, -0.308875382, -0.580213249, 0.448446721, -0.45384112, 0.637113988, 0.22468847, -0.44499284, 0.448179454, -0.695528984, -0.523058057, -0.20205234, 0.401423126, -0.299692124, -0.285832226, 0.00851056166, 0.446261317, 0.449846536, -0.147104949, 0.186150268, -0.341991156, 0.483379424, 0.409596086, -0.819293022, -0.427935719, -0.0609564856, -0.186954215, 0.22231397, 0.677733302, -0.430307955, 0.41937992, -0.53020221, -0.709738255, 1.39581501, -0.465620965, -0.406482309, 0.230612159, -0.127730966, 0.252974093, -0.327023417, 0.172929749, -0.179164842, -0.181214273, -0.630494654, 0.130540758, 0.800786495, 1.31670678, 0.651693225, 0.26879409, 0.717613041, -0.332398593, -1.13882279, 1.10321188, 0.628750741, 0.120193116, 0.169278011, 0.0102077844, 0.412785739, 0.243498132, -0.107576504, -1.41570306, -0.378706455, 0.558926582, 0.0833759829, 0.31381613, -0.0644204244, -0.374783784, 0.143002838, -0.351724088, 0.682405293, 0.445532829, -0.229264662, 1.07147574, -0.49398458, -1.41003466, -0.281465918, 0.399474233, -0.190109655, -0.300240487, -0.190270245, 0.290429056, 0.389570504, -0.41685605, 0.313826352, -0.353538096, 0.193838418, 0.17874822, -0.661477685, -0.218386546, 0.181119785, -0.27007553, 0.37187016, 0.545805931, -0.409519613, 0.313312501, -0.486589909, -0.514013529, 0.53758657, -0.388148338, -0.386788845, 0.236975595, -0.249515042, 0.352596641, -0.452643454, 0.0751595125, -0.199768692, -0.368431866, -0.564446449, 0.124738604, 0.551067472, 0.477803558, 0.645738363, 0.451337278, 0.36455822, -0.547371447, -0.558630824, 0.683180392, 0.508676529, 0.150767982, 0.334811896, -0.127142951, 0.520551682, 0.421019465, -0.380728275, -0.666364133, -0.208092257, 0.419620007, 0.251989931, 0.349487305, -0.100969084, -0.490674853, 0.104314096, -0.445262551, 0.700497091, 0.306501925, -0.290917009, 0.638085663, -0.611868978, -0.704333663, -0.236393571, 0.278745502, -0.160794124, 0.187537983, 0.193862125, -0.545814693, -0.429071397, 0.322655946, -0.339522034, 0.288719624, -0.320478141, -0.422625303, 0.679973006, 0.43120417, -0.175866529, 0.287333757, -0.24651818, -0.552334011, 0.582789361, -0.350291014, 0.340433657, 0.612520516, -0.698364496, 0.410984069, 0.496014744, -0.2112865, 0.172307029, -0.220764354, 0.23293744, -0.113850325, 0.151842833, 0.204290181, 0.624974251, -0.3173002, -0.616165519, -0.762767673, -0.581521392, -0.38164562, -0.364023566, 0.293084621, 0.684331954, -0.669203341, -0.578521132, -0.215825975, -0.309929729, 0.161461651, -0.481502086, -0.33366996, 0.407046795, 0.687428117, 0.432012111, -0.426859856, -0.190915257, -0.28371498, 0.112135045, 0.32552439, -0.376189739, 0.255220383, -0.659893572, -0.281848013, 0.271159649, -0.753100038, 0.696901441, 0.774981558, 0.263962597, -0.580399573, 0.207476303, -0.489746898, -0.318865716, 0.694255233, 0.589036345, -0.415274382, 0.450182855, -0.52728194, 0.16396296, 0.37136966, -0.397399455, -0.168249264, 0.171118036, -0.329902977, 0.449208915, 0.395524055, -0.750423372, 0.489338368, -0.368194759, -1.15998709, 0.620019853, -0.7576828, -0.205018669, 0.393452287, -0.447394371, 0.234547332, -0.427081048, 0.301175028, -0.476558894, -0.345771939, -0.409495801, 0.467222869, 0.548399627, 0.500039697, 0.378137559, 0.440289289, 0.491164953, -0.67148912, -0.57847774, 0.419943243, 0.335299194, 0.323250413, 0.377524287, -0.405551583, 0.467709899, 0.453525454, -0.108336598, -0.49214527, -0.241720945, 0.24566637, 0.437246531, 0.281952918, -0.337768018, -0.655142426, 0.224741742, -0.466080964, 1.07907832, 0.309440762, -0.374534786, 0.407602996, -1.12126684, -0.510153413, -0.174589857, 0.509226441, -0.596024573, 0.197434649, 0.104001492, -0.3198165, -0.32519263, 0.339605331, -0.314416826, 0.325983107, -0.343047291, -0.132974431, 0.81815207, 0.201130912, -0.0243123733, 0.0527296364, -0.0181351546, -0.478730559, 0.512533426, -0.200201452, 0.454898775, 0.605251253, -0.959287584, 0.476582855, 0.46511519, -0.073389031, 0.0493558347, -0.234351858, 0.489906907, -0.0115846926, 0.0954758003, 0.0923486948, 0.37821573, -0.0817371607, -0.744875193, -0.937383056, -0.51701045, -0.363589615, -0.375586689, 0.230454534, 0.888920665, -0.905913532, -0.344734728, -0.119335964, -0.100582771, -0.0639484748, -0.557996392, -0.198687643, 0.193681926, 1.00480378, 0.23948893, -0.548692167, -0.237381801, -0.222519547, -0.102165021, 0.280562282, -0.153881714, 0.144722894, -0.618686378, -0.229635522, 0.244115129, -0.770794094, 0.578632236, 1.04854047, 0.0756938905, -0.616603136, 0.10861589];
    recurrent_3_h : ARRAY[0..4095] OF REAL := [-0.0814854726, -0.0192965753, 0.0789262801, 0.0411406085, 0.0133345416, 0.0320188627, 0.0268287342, 0.098575674, 0.0197239444, 0.0170570016, 0.0375691243, 0.00974027067, -0.0348538384, 0.127068236, 0.0174264405, 0.113225967, 0.0694785044, -0.0788176358, 0.0529993363, 0.0676577315, -0.00359288044, -0.0408049487, 0.0645037144, -0.000435883179, -0.185998872, -0.0484710485, -0.0816430449, -0.0837951526, 0.0798519105, 0.0405569635, 0.0890566185, 0.0360047966, 0.0997576416, 0.0608237684, 0.0964706093, -0.00868162513, -0.108718976, 0.0455377959, -0.127817109, 0.034598954, 0.0658386946, 0.0902062431, 0.0447102711, 0.110850818, -0.10822577, -0.00176366791, -0.1578134, -0.0031897286, 0.0873728096, 0.0192435347, 0.000598257408, -0.00534118526, -0.06289424, 0.0543237627, 0.0102685485, -0.0766392127, 0.0172083843, -0.0324428305, -0.0644046962, 0.0433603153, 0.0116282376, 0.0277246814, -0.028188983, -0.092127122, 0.0713761374, 0.0740641654, 0.0193934143, 0.0861851647, -0.135807559, 0.0406226926, -0.0614926405, 0.0625797212, 0.0398422368, -0.0669911578, 0.105368845, 0.0588050187, -0.0192349926, -0.00367016345, 0.0765316337, -0.0240941439, 0.124655016, -0.0685237944, -0.0298877526, -0.107453629, -0.114462942, 0.0298811644, -0.0412020497, -0.0680356622, 0.08198829, 0.0671266764, 0.141011715, -0.108955503, 0.00767487474, -0.0263134968, -0.0382245034, -0.00829227827, -0.0490662754, -0.00504888594, -0.0578778498, -0.00452999398, -0.0257887766, -0.024094943, 0.0427409112, 0.182257861, 0.0536978841, 0.0288107246, -0.124135427, -0.0162076652, -0.0830906034, 0.0993471742, -0.00205180608, -0.0192750916, 0.0335743427, -0.010746954, 0.0416064188, 0.0425092839, 0.0763217732, -0.0269507729, -0.0376095176, -0.0840850174, 0.103590034, 0.0634661987, -0.0485707894, -0.135362148, -0.07549797, 0.117634244, -0.000415748334, 0.0653510541, 0.0405582041, -0.0844664723, -0.0534745008, -0.104245521, -0.040891327, -0.0525825433, 0.0440185517, 0.0694993064, 0.116974413, -0.00926593691, -0.0535617396, 0.00366610382, 0.050855957, 0.0667424276, 0.076435186, -0.125347257, 0.0312693715, -0.218390763, -0.0340445787, -0.00350955967, -0.0763550401, 0.0529564992, -0.0314787775, 0.029810477, -0.0718894303, -0.00991622731, 0.0670813322, 0.0509934798, -0.111424267, 0.148194313, 0.101489179, 0.0255741142, -0.110127077, 0.142647222, -0.0658696219, -0.0443728864, -0.0185198858, -0.108988307, 0.0414187089, -0.0581751317, -0.106079616, 0.0516243093, 0.0277372226, 0.0143314376, -0.104727075, -0.00395930745, 0.0917050466, 0.036209777, -0.0639554411, 0.0190380942, -0.082036227, -0.0430522598, 0.120325893, 0.044341255, -0.0262874365, 0.122560076, 0.0722675174, 0.0112938397, 0.0826819241, 0.140801668, -0.00693470985, -0.143158227, -0.0667897463, 0.0551305562, -0.0660582855, -0.0840694159, -0.201774463, -0.0808143318, 0.0204459652, -0.0805091262, -0.0514314324, 0.086621508, -0.019972384, 0.0697269142, 0.0801439807, -0.107793219, -0.0182074588, -0.037682306, 0.130044892, -0.0955766067, -0.0831588879, 0.014559716, -0.131067291, 0.0490752161, 0.11203061, 0.056660179, -0.0332784355, 0.0368628316, -0.0577385686, 0.101687275, -0.0243908167, 0.0317545906, -0.0498156808, 0.103358865, -0.0139978454, 0.0358166881, 0.118501097, -0.00132077187, -0.076020427, 0.0606940724, -0.00561159523, -0.0126780868, -0.15248692, 0.0325385891, 0.103686489, 0.0777438134, 0.111734673, -0.0146942325, 0.0624658316, -0.0260592327, 0.0342593491, 0.0526987091, 0.153397962, 0.012578873, 0.0223368406, 0.022732662, 0.0323334932, 0.00192690501, 0.155853719, -0.0188841671, -0.034229625, -0.116638057, -0.0345492139, 0.0173566677, 0.0428409353, 0.0695734099, -0.0880442858, 0.0729065686, 0.120992012, -0.0802285299, 0.170097202, -0.0124929547, 0.00698815892, 0.0169789419, -0.0330532752, -0.0208955593, -0.0945662484, 0.0137330554, -0.019574903, -0.0235930793, -0.0777337328, 0.111762121, 0.0232670885, -0.0713128671, -0.0559905767, 0.0478160717, 0.0293007158, 0.0418722071, 0.0608519875, 0.034675017, 0.0534267798, -0.0730765313, 0.0355616361, -0.012282202, 0.0249277949, -0.102093399, -0.0967272818, -0.0963730142, 0.0816735998, 0.125792161, -0.0747596696, -0.0144781265, -0.104787081, 0.0764187574, 0.121330157, -0.106906578, 0.058575578, -0.0980070978, -0.00227518752, 0.0111543592, 0.14027299, 0.00853795931, -0.00508823246, 0.13767986, -0.0324843042, -0.0966325998, 0.127950266, -0.0261407811, -0.0354549773, -0.0301502217, 0.0941592827, 0.0264327861, -0.0714561418, 0.0140698608, -0.0789159387, 0.00831018016, 0.0257221051, 0.126190424, -0.0692755729, -0.0622021519, -0.0098341275, 0.00592781231, 0.0521613136, -0.0226634201, 0.108450375, -0.0644210428, -0.0427489094, -0.012539804, 0.034737885, -0.04454289, 0.094007358, -0.213121518, 0.00931252353, 0.00689808279, -0.0219363961, 0.0552700087, -0.0720815957, 0.107797891, 0.0289382283, -0.0122516416, -0.027756881, -0.14954558, 0.133981004, 0.0155080631, 0.0937383473, -0.0370610394, -0.036308527, -0.10757535, -0.0292736068, 0.0913158357, -0.0255951732, -0.071827814, 0.0506477505, -0.0646002144, -0.091782026, -0.103335038, 0.147168487, -0.0559476502, 0.0518603101, 0.0846874267, 0.0487901233, 0.108146086, -0.087490581, 0.028688848, 0.0727105364, 0.079600811, -0.0486454591, 0.0721243843, 0.0166750103, 0.0583023727, -0.0257067531, -0.000845391303, -0.0355865359, -0.0593533888, -0.125758901, -0.0254528858, -0.157639965, 0.122022294, 0.0821343958, 0.0121467439, -0.0600851811, -0.00524813496, -0.00107267871, 0.0798011124, -0.0603280775, 0.0127256103, -0.0961495265, 0.0819807127, -0.089014031, -0.0675459057, 0.0232538357, 0.0451772958, 0.0720037073, -0.00161110307, 0.0975338221, -0.00135360286, -0.101388894, -0.00706165098, -0.0727991909, 0.0255892128, 0.0538133532, 0.071327284, -0.0615934543, -0.0809898525, -0.0331617296, -0.136261612, 0.0588698685, -0.0770790428, -0.102680333, 0.0188243501, 0.0302853081, 0.0163531806, 0.141216546, 0.0050297603, -0.019597711, -0.124074377, 0.115986295, 0.0230492167, 0.092672199, 0.0650038272, -0.0551722981, -0.0598487593, 0.0118252039, -0.0312254131, 0.0135671515, -0.046299994, -0.0392930359, 0.0330872759, -0.00160764158, -0.0612518042, -0.0837748498, -0.0547977313, -0.0544400886, 0.0210792422, 0.0538680404, 0.00474515557, -0.0188872237, -0.018180009, 0.0164556876, -0.0475738496, 0.12157543, -0.0967819691, -0.0598815978, 0.0273639522, -0.0985397696, -0.0664836168, -0.0643208325, 0.157129899, 0.0656617433, -0.0398358069, 0.0614418015, 0.216747984, -0.0336473361, 0.0630160719, -0.041756127, -0.090438962, -0.10895925, -0.0151612433, -0.0388511345, -0.0265313573, 0.0675288662, -0.0712825656, 0.00559772179, 0.148817271, 0.0186223574, 0.0694734305, -0.0698306561, 0.0821632147, 0.023453474, -0.0177625604, 0.0547127798, 0.049756173, 0.133104116, 0.0534175672, 0.0399441943, -0.0768370032, 0.0188250877, 0.0338728204, -0.16938214, 0.0136184543, -0.0372059941, 0.0454952382, 0.0554398, 0.0665775687, -0.00576402619, 0.114006989, 0.0220732726, 0.0500874817, -0.0487473235, 0.0962967649, -0.0625525713, -0.00653420389, -0.041575443, 0.0311930105, -0.029791832, 0.0689999983, 0.00458959769, -0.064472422, 0.00381559879, -0.110996231, 0.107624851, 0.0776014328, -0.0165557265, 0.0545652434, -0.02398834, 0.0211636443, -0.090277791, 0.123671643, 0.0038228156, -0.0428426638, 0.057123173, -0.0103270039, -0.0460167006, -0.0424827114, -0.0602993518, 0.0353726037, 0.0285762176, 0.00311186863, 0.00623007771, -0.0185233969, -0.0611157753, 0.0891965032, -0.0300280824, -0.0311615188, -0.0441223457, 0.0917677954, -0.0566205941, -0.0356463008, 0.0649248734, -0.12526457, -0.0269312095, 0.0369988903, -0.0115831438, -0.0411470011, -0.129782021, -0.0259651951, 0.0443037301, 0.0642121732, 0.0902121961, 0.137408137, -0.0848503858, 0.0204836316, 0.00812876038, 0.0144137349, 0.0262199081, -0.000904881861, -0.000609018258, 0.0209549796, 0.055321712, 0.0222451538, -0.121768117, -0.0235857777, 0.0472685657, -0.0451143906, -0.0986179784, -0.0401195846, -0.0330208838, 0.0867114365, 0.00304402597, 0.00186095014, 0.0426921509, 0.00287284143, -0.06281057, -0.0218146741, -0.0519862324, 0.0519039966, 0.130057991, 0.0735057816, -0.119574539, 0.0656085387, 0.0192519315, 0.0535424873, 0.0318356007, 0.0667994693, -0.154886812, 0.113748945, -0.0458672605, -0.0245250165, -0.0369493067, 0.0141960606, -0.0307653323, 0.0935062468, 0.065485619, -0.100963473, 0.191053107, -0.0558037199, -0.00151302665, -0.0613323674, 0.00489765219, 0.017088823, 0.00816752668, -0.0763265565, -0.0171313062, 0.0396030061, 0.0182253681, -0.0789322853, -0.0904842243, -0.017320957, 0.12033923, 0.0479416698, -0.0579523221, -0.0349941999, -0.0737884939, 0.0893755853, -0.0492203236, 0.0345975086, 0.0748756155, 0.031574931, -0.0574996993, -0.0414605848, -0.00592986867, -0.211724117, -0.152851686, 0.103620194, -0.0192455165, -0.0913382024, 0.0540000461, 0.0202528294, -0.0447318926, -0.0182958581, -0.0809874833, 0.00605034456, 0.014784079, 0.0598445684, 0.0352179557, -0.0735865161, 0.0985039175, 0.0263431855, 0.0266565308, 0.0760347694, 0.13909331, 0.0396100096, -0.235010266, 0.0348193459, 0.0385177955, -0.0210304111, 0.192817584, -0.0985148251, -0.0132797509, -0.0684133619, -0.0487778261, 0.0508381501, -0.0468438305, 0.0750653371, -0.0584874786, -0.0166681632, -0.105090663, 0.109042183, -0.100686267, 0.0926523507, 0.106955722, -0.0169380605, -0.0730493814, 0.149691254, 0.0468780324, 0.0161016695, -0.0533247441, 0.00323989149, -0.053974051, 0.0347923785, 0.108852185, 0.128028229, -0.0624134243, 0.0662307814, 0.0491992719, -0.00422449782, -0.0187873673, -0.0779604167, -0.0660356805, 0.0104759261, -0.122655123, -0.0868720487, 0.0616197884, 0.049584318, 0.014691012, -0.0485520102, -0.0751743391, 0.0209864173, -0.112359822, 0.126514718, -0.0403945595, -0.025346037, -0.0315166265, 0.0145783126, -0.0354765579, -0.0316554755, -0.0238025971, -0.0183946248, 0.0575497672, 0.049439773, 0.0156415105, -0.0338407457, -0.0162942, -0.0936263204, -0.0364862569, 0.0244779438, -0.0722951815, -0.117110163, 0.02470842, -0.0229848921, 0.106150478, -0.0234055258, 0.0364057608, -0.135178566, 0.105516925, -0.0627449304, 0.025232913, 0.0947535262, -0.0443718806, -0.0724740326, -0.0293204188, -0.00357807381, 0.0102455318, -0.0159719735, -0.0591221191, 0.0806587934, -0.0425145365, 0.047045663, -0.0435880646, -0.078207761, -0.0414206423, 0.00447744131, -0.0354393907, -0.0408014655, 0.0602022409, -0.0678982958, 0.0703518167, 0.108378991, -0.0511661023, -0.0182328783, -0.0605737269, -0.0301890429, -0.0551630966, 0.00768520124, -0.110727012, 0.00739408005, -0.186828896, -0.141738012, 0.152821541, -0.0067199124, 0.0317742191, 0.0481149554, 0.107150555, -0.0046456866, -0.0121925715, -0.108526014, 0.0991511941, 0.0589258522, 0.0793202296, -0.0861595273, 0.0195609853, 0.0406994224, -0.0150603354, 0.0482544713, -0.0906827897, 0.026193399, -0.115839884, -0.111916341, 0.00176167861, 0.0541164763, 0.0906799138, 0.0439846814, 0.00267879106, 0.0442864709, -0.0638696253, 0.000865995884, -0.0544654764, 0.0218691304, -0.024334576, 0.00822855532, 0.0591265038, 0.000598696992, -0.173971847, 0.187341824, 0.0311711002, -0.115362734, -0.14091152, 0.00509036705, 0.0740948766, -0.0132719018, -0.1538634, 0.0519612432, 0.100895002, -0.0455305725, 0.0349408239, -0.0396569818, 0.0162646547, -0.0628253222, 0.0149623957, -0.0761591569, -0.067038022, 0.0567291491, -0.0115640033, -0.12310382, 0.0153456051, 0.0261365995, -0.00158301182, 0.0688955933, -0.0150526986, -0.0419144668, -0.0858189166, -0.0221549645, -0.0814090595, 0.00748031028, -0.0477067642, 0.0846377611, 0.0814989284, 0.0424698517, -0.0446051806, 0.119475752, -0.0474177487, 0.0232976191, 2.86288559e-05, 0.0882164389, 0.117915064, -0.122286193, -0.082594052, -0.00397979468, -0.120276324, 0.0684959143, -0.0094874315, -0.0263404958, 0.0264270157, -0.0425064936, 0.030408198, 0.0444010012, 0.0288432315, -0.116888009, 0.0348403156, -0.127345368, -0.00221462548, 0.0839427561, -0.0583360605, 0.00646906486, -0.126093701, 0.0901082009, -0.11345911, 0.0232501011, -0.0398917533, -0.075740546, -0.0777630582, -0.0215390399, 0.0573985577, -0.0664281696, 0.0139244255, 0.0822378695, -0.0868723541, -0.0644526407, -0.0413177721, -0.0373630337, 0.074725315, 0.0198760182, 0.238774791, 0.000480882823, 0.146973342, -0.0438087285, 0.0210053455, -0.0476518944, 0.0700921118, -0.046215523, -0.00491245091, 0.116612412, -0.0539766103, -0.0231392421, -0.111935452, -0.0398099422, -0.0990347266, 0.0325184092, 0.0512922481, 0.0344113111, 0.04099489, -0.00529667363, 0.098762922, 0.0683466122, 0.0348195694, 0.0176171139, -0.0109903542, 0.0790873691, 0.00966604333, -0.0129369348, 0.00683330419, -0.1477516, 0.0131506315, -0.0942147598, -0.0606220663, -0.0697087795, 0.12897639, 0.125819787, 0.127462566, -0.130796269, -0.0318847187, -0.0541017577, -0.0710220337, 0.0319548063, 0.0484784655, -0.0833456367, 0.104416221, 0.0884514824, -0.0298784561, 0.00545195304, 0.00393914385, 0.180217415, -0.0419916697, -0.0388295129, -0.0210801885, -0.0985303819, 0.0308424477, -0.0293995664, -0.136730999, -0.0781954452, -0.0751239806, -0.127824411, 0.02346812, 0.0199848078, -0.0564694107, -0.105549797, -0.0490997583, -0.0215537027, -0.125966251, -0.00793886278, 0.112402536, 0.0460357703, -0.0970197842, 0.0360428169, 0.0909704044, -0.00488845445, 0.0602041259, -0.148838788, 0.0307073835, -0.119664438, 0.0977907553, -0.0584818907, -0.127177939, 0.101691186, -0.0500702485, -0.071391359, -0.0067316629, -0.0806362778, -0.0122225359, 0.0211955644, -0.027770441, 0.00372764096, 0.014971735, 0.010094665, 0.0299131721, 0.0425138883, -0.0504307114, -0.0968710408, 0.022818774, -0.018594075, -0.0278927796, 0.0345954448, 0.0309654102, 0.139828771, -0.0821411833, 0.0577695519, 0.014581183, 0.0716957003, -0.0795750916, -0.0606432706, 0.0648429319, 0.0562322102, 0.0133413039, -0.0868299752, 0.0934337527, 0.0354992002, -0.0141148129, -0.109865315, -0.0334577635, -0.096242331, 0.0114050489, 0.0945957601, -0.0225579925, 0.0670915917, 0.062363185, 0.0217214208, -0.135514319, 0.0564552322, -0.0463878363, 0.0140669513, -0.0390195698, -0.0332866646, -0.0231394097, 0.00866015442, 0.110395685, 0.139712736, -0.00856509246, -0.0202140808, -0.0637191013, -0.0218470022, 0.0505792089, 0.0140721239, -0.163294703, -0.0295530967, -0.035891261, 0.0550732948, -0.0232377499, -0.0182076506, 0.020572219, -0.00922282226, -0.042679809, 0.0690913424, 0.103285804, 0.0187672172, -0.084432207, -0.018480327, -0.0320419036, -0.0645342618, -0.0203374773, -0.0748507529, 0.18064329, 0.107685819, -0.00787636265, -0.0740540177, -0.0423652008, -0.0679801181, 0.0609641522, -0.0320399031, 0.130488232, -0.139181733, 0.027738709, -0.0237837918, -0.0416492298, 0.0861929581, 0.0453447551, -0.0122638159, -0.00358418492, 0.0130312154, 0.142131567, -0.0525563434, 0.0374514721, -0.278361261, -0.103083089, 0.0572038554, -0.0925511718, -0.0423664935, -0.0406515747, 0.0328615345, 0.00788263977, 0.0255986787, 0.0489936285, 0.0157014001, 0.0969976336, 0.0673143342, 0.0384454019, -0.0820726976, -0.119464785, 0.0662378669, 0.0176079124, -0.0653717965, 0.0807158649, -0.0395191312, -0.0441734344, 0.035682179, -0.0216369517, -0.0547301285, 0.0385114327, -0.0675674528, 0.064386636, -0.00892916601, -0.0853860378, -0.0403388627, -0.0137955323, -0.0079660397, -0.0607065223, -0.0771734193, -0.0302698184, -0.0709434301, -0.126736358, 0.0527005568, -0.0769583508, 0.0938322246, 0.0699062794, -0.0553395897, -0.078124173, 0.0375381298, -0.0296272896, 0.0516815223, -0.00348858535, -0.174458086, 0.120906889, -0.0485840626, -0.058952868, 0.0763350055, 0.124017775, 0.049220778, 0.027029492, 0.0800717175, -0.0427948348, -0.0720757321, 0.0563872904, 0.0478098877, -0.0327438712, 0.124894299, -0.0361689627, 0.00881732069, 0.0148479519, -0.0597984418, -0.104160495, 0.0817637891, -0.102677345, 0.014353578, -0.0131146312, -0.0629141182, 0.0233532414, -0.0576458424, -0.0407313854, 0.0819140375, 0.0799592435, 0.0245517902, -0.00226673298, -0.117883302, -0.00874280836, 0.0630186498, 0.0180511568, -0.0864587724, 0.0198795795, -0.045463793, 0.00537871383, 0.00525548402, 0.0297887903, 0.0285999216, -0.00921368226, 0.0653725788, -0.0809201747, 0.0645085126, -0.0491232648, 0.0156253614, 0.0181711018, -0.0428764597, -0.0789432675, -0.081858471, -0.0160164461, -0.0770956501, -0.0647167414, 0.0257139672, -0.0298938919, 0.08180172, 0.00204348378, -0.00999781303, 0.0234333351, 0.133766204, -0.0154174995, -0.00820135884, -0.0762263983, -0.0836507976, 0.0803018287, -0.00640827511, -0.0417413749, 0.0869801641, -0.00429981668, -0.0497169569, 0.0295637846, -0.0974320844, 0.0801439956, 0.00922070071, 0.00579300895, -0.0104648257, 0.0583571717, 0.0593466386, -0.0778260529, 0.0317886397, 0.119893447, -0.0661615953, 0.062702328, -0.0620942786, 0.0378547683, -0.000269612297, -0.0222870484, -0.102530479, -0.029686084, -0.0886763409, 0.0523997173, 0.0408445969, -0.0572608858, 0.0401265435, 0.0485404059, -0.119643465, 0.0316348076, -0.124418564, -0.00581553951, -0.0651025027, 0.231553227, 0.0868467391, -0.0643303916, -0.0186187401, 0.107610479, 0.0670118928, 0.003345415, 0.0190979186, 0.0473675244, 0.0245451815, 0.0763186291, 0.0333949029, -0.0293634944, 0.0173659772, -0.120647959, 0.115150526, 0.037421573, 0.0698179826, -0.108961686, 0.0455931984, 0.000210376456, -0.046899274, -0.115995303, -0.00141779333, 0.0489153825, -0.0698401108, -0.161397383, -0.00141991489, -0.0465725251, 0.0845248327, -0.0422395505, -0.0302315578, -0.0700481683, -0.0792448819, 0.00840363652, -0.0429288521, 0.0333831385, 0.0143478224, 0.0680661947, -0.00983876549, 0.00276218518, -0.138327628, -0.158029065, -0.061606165, 0.0796257779, -0.0719533488, 0.0366943665, -0.073024869, -0.0133639649, 0.0728572831, 0.0780148283, 0.000802894589, -0.00786045194, -0.0866034552, -0.0233533569, -0.00846383721, 0.00107602775, 0.0679003745, 0.14589192, 0.0838717669, 0.0657557547, -0.0575768799, 0.0471429303, -0.0183246173, 0.0733493492, -0.106923282, 0.036673069, 0.0290950835, -0.0066739507, -0.176835716, 0.0455783866, -0.0830275416, -0.0166184921, -0.0717226192, -0.16906327, 0.0413567014, 0.0666721538, 0.121657446, -0.0168469362, -0.071589604, 0.0492151454, 0.150245517, -0.00744849443, 0.036688786, 0.0148853846, 0.143496513, -0.106677443, -0.00377738103, 0.130240157, 0.0961677358, -0.0483830944, -0.0533252396, -0.0558958575, -0.0587435551, -0.0471863747, 0.0274546295, -0.00455031358, 0.152671129, -0.00452759489, 0.0198450424, 0.0892882496, 0.047615625, 0.0368035734, 0.117391482, 0.069509156, 0.0422603823, 0.00581758469, 0.054865323, 0.0964347795, -0.0813242495, 0.0565662682, -0.0331555605, 0.00256007444, 0.0171385929, -0.141754836, 0.0536107235, -0.00652080774, 0.0206656493, 0.0199916307, 0.0257186592, 0.0493282601, 0.0364555493, 0.00225205347, -0.0609959662, 0.0983685255, -0.170430332, 0.13926971, 0.126211256, -0.0434726365, -0.0863412768, 0.0850047767, -0.129416153, -0.01676948, -0.0442021042, -0.157091528, -0.0225310344, -0.126880839, 0.114073932, 0.0681565329, -0.0110374093, 0.103243686, 0.0314437076, 0.0178046897, -0.0883147791, 0.0996307209, -0.0759864748, 0.106075488, -0.0479057096, 0.048020076, -0.0221770257, 0.0870950297, 0.0886747539, -0.0086180903, 0.100509644, 0.102688968, -0.0428900011, 0.0470696762, 0.00363672804, -0.0063303262, 0.0105653387, -0.0434411094, 0.0254247542, -0.054897517, 0.0131881703, -0.0144290887, 0.0560137555, 0.0917306766, -0.0966982096, -0.0634434298, 0.0281065293, 0.0497760028, 0.077282235, -0.00285350066, -0.10189905, 0.102921128, -0.123005442, 0.0306916479, 0.0135944318, -0.0479210615, 0.0562534183, -0.19185783, -0.0953860581, 0.0645157844, -0.000782571733, 0.013786776, -0.0470033363, 0.0292213932, 0.0477219671, -0.101445727, 0.0189936887, -0.0241080429, -0.0662670806, -0.0212797467, 0.104987308, -0.112548925, 0.0970475078, -0.0197823402, 0.00148634985, -0.161885068, 0.1411549, 0.0358134024, 0.115680665, -0.0206926819, 0.015348413, -0.157771558, -0.083538644, -0.0901385322, 0.0155987553, -0.0408718027, -0.00824440178, -0.0196364, 0.00215512514, -0.0527868569, 0.120022118, 0.00736992061, -0.0261461362, 0.0481230207, -0.0812953711, 0.114198528, -0.0560671054, 0.0119590433, 0.139143959, 0.0231116526, -0.104707398, -0.0871268809, -0.0620228797, 0.0446613394, 0.0852409676, 0.0232791621, -0.0493073203, -0.122175001, -0.0743146241, -0.0970351323, -0.0322813652, -0.0230376031, -0.0747933164, 0.121797323, -0.0840328187, 0.182821229, 0.00267254747, 0.0346976668, 0.0289725326, -0.0111252572, -0.0236078594, -0.1362755, -0.0393440723, -0.039869599, -0.072801128, 0.00474104192, 0.0401104353, 0.031128373, -0.0375661589, 0.0981234908, -0.108892135, 0.0854332522, -0.100614265, 0.0620648228, -0.0946724862, 0.0276948623, 0.0799888819, -0.0238845237, -0.0382171869, -0.00498760119, 0.169999808, -0.0707746819, 0.0141820814, -0.0102484552, 0.0631627664, -0.004883321, -0.00955140963, 0.0335532203, -0.0903009176, 0.113554172, -0.0566767901, -0.0451321118, -0.0993601233, -0.0760187209, 0.0163101889, -0.0490140207, -0.0764138401, 0.0725791007, -0.032778874, 0.0713169724, 0.0636530221, -0.152569786, 0.0243993923, 0.0723212212, 0.0103602335, 0.0263289306, 0.112154886, 0.0905341506, 0.0342193283, 0.0545448586, 0.0113084335, -0.0643381625, 0.0082473997, -0.0725228712, -0.072711423, 0.0143926702, -0.0482516997, 0.0312177166, 0.0688024089, -0.0308066048, -0.00662764721, -0.0112344995, -0.0207642205, -0.0389785916, 0.0443165861, 0.00633093482, -0.0465511903, 0.0544905774, 0.0553966798, 0.000962100923, 0.0266012531, -0.0843920037, -0.167079523, 0.00344678294, -0.0810573623, 0.15070875, -0.0331101194, 0.114123136, -0.0225568712, -0.0176230837, 0.00988603011, 0.116972901, 0.0696514249, -0.0186434761, -0.0478475653, -0.0933808908, 0.159889385, -0.0408868194, -0.0198710598, -0.0154632078, 0.0247305688, -0.0267912764, -0.027883606, 0.0158543214, -0.00319262221, -0.011261275, 0.0731381178, 0.0616139174, 0.0586696975, -0.0678472072, -0.0454129875, 0.0754584596, -0.119438857, -0.0265938528, -0.10789749, 0.02866574, 0.14865832, 0.0880545527, 0.0348470993, -0.00962357968, -0.0345035829, -0.104515843, -0.0261899754, 0.037708655, -0.0984590501, -0.0180872008, -0.0691327602, -0.0333068855, 0.0305836722, 0.175035447, -0.12944904, -0.108516775, 0.0860668942, -0.053936474, -0.0133826192, -0.0959395021, 0.197356835, 0.0745769367, 0.00389399752, -0.032868892, -0.0853783563, 0.107811116, 0.111107975, 0.0311097205, -0.0910380483, 0.0032276623, -0.0549909212, 0.0134176295, 0.0511631444, 0.0414193794, 0.00317235477, 0.0898500681, -0.135848314, -0.0522413366, -0.159420639, -0.00305157714, 0.0386255533, 0.0291372277, -0.0885984898, -0.107466757, -0.0169878881, 0.00981041975, -0.0710143819, -0.122051045, -0.0637671649, 0.0386342034, 0.0928902775, 0.0227206014, 0.0287559219, -0.0440340862, -0.0868715644, 0.0140771419, 0.0950409174, 0.0169625469, -0.0600583479, -0.0682354867, 0.0235817283, -0.0693513602, 0.0654219612, -0.0319071636, -0.0191534534, 0.00270009041, -0.0966809914, 0.0543267839, -0.0966179818, 0.0533478707, 0.0473777466, 0.130858183, 0.0296896696, 0.110831179, -0.0794160515, 0.0891058296, -0.0746674836, -0.047442399, -0.00548080867, -0.0112081207, 0.0652866885, 0.018655736, -0.0504849851, 0.0934263095, -0.0137429051, 0.0306825303, -0.0171481334, 0.113898054, -0.0197691862, 0.01716391, -0.13725464, 0.160080954, -0.056644503, 0.0701243207, -0.0709521919, -0.00980228558, 0.0643183887, 0.0371039212, 0.172112271, 0.0266852025, -0.000314045697, 0.0352090076, 0.0782720819, -0.0268915538, -0.065240711, -0.0363622345, 0.00678189844, 0.0515537411, 0.0302088186, -0.0516999401, -0.0417689644, 0.0265829656, 0.0431901999, -0.047669176, -0.00715433434, -0.0398947671, -0.119628437, -0.0241764635, 0.0624189228, -0.0201673992, -0.109756812, -0.0724374354, 0.134150118, -0.0151170734, -0.10790728, 0.0218152143, 0.0434726067, -0.0754626244, -0.0895682871, -0.0746940523, 0.0798545033, 0.0490447059, -0.079427205, 0.0768660083, 0.134363741, -0.0893851966, -0.00989978015, 0.0592893064, 0.00601488166, 0.129167721, 0.0741336122, -0.0239292569, 0.0150100868, 0.0171410665, 0.0837964714, 0.0107440967, -0.0899902806, -0.0421808437, 0.14333652, 0.000882504741, -0.0283789635, -0.113518372, -0.119485527, 0.0271064285, -0.0126037691, -0.0302240029, -0.0556081943, -0.0852503479, -0.0272557475, -0.0232609026, -0.0675073713, 0.0605746955, 0.0169038232, -0.067426458, 0.0409276634, 0.0290825088, 0.0431087837, 0.0932073072, 0.0435449593, -0.0194333252, 0.0584137142, 0.00362193398, 0.0163618065, -0.0906330794, -0.0452677831, -0.107395664, 0.139208734, -0.0962576419, 0.0774556249, 0.0129028559, 0.0498936251, 0.0548831001, -0.0805293545, 0.00154444017, -0.0371510424, 0.0101845376, -0.154818743, -0.0077851247, -0.00720209349, 0.00499167852, 0.0433876552, 0.0626057312, -0.0534386337, 0.0327771008, 0.0748492405, 0.167353302, -0.0582256466, 0.0656488985, 0.0877349377, 0.0911114439, -0.033684805, -0.089890264, 0.112802006, 0.0697733462, 0.0105233509, -0.079758063, -0.0880320519, 0.0502214171, -0.0649921, 0.058669664, 0.0488339849, 0.000166147947, -0.0313328281, -0.0141187552, -0.0262500662, 0.086430274, 0.0312220976, 0.098366946, 0.0500786267, 0.0601362437, 0.0364454091, -0.0727507547, -0.00961787812, -0.0410132483, -0.0145145506, 0.0390949287, -0.00951914955, -0.00783446804, 0.0400613658, 0.0257792193, 0.0831083283, 0.0828651488, -0.0774267316, -0.00697443262, 0.0935089514, 0.0111638233, 0.0509233773, 0.0326655954, 0.0730861723, -0.178317621, -0.0233378243, 0.0365107656, -0.0567861274, -0.100251123, -0.0589826964, 0.0563125908, -0.0665871203, -0.00284511782, -0.0217932947, 0.0254806615, 0.00918012951, -0.0562544465, -0.00146721164, -0.0459353998, -0.00483963266, 0.0151962433, -0.0172823723, -0.010939464, -0.0505235195, -0.0148119424, -0.0467831343, -0.0790587291, -0.0456247032, 0.0541887097, -0.183028042, -0.0628453046, 0.0562240407, 0.064596042, 0.0402977951, -0.0902705193, -0.0543275364, -0.0671445355, 0.012307778, 0.0705013797, -0.0067007076, 0.0450508818, -0.0113195973, 0.0403822064, 0.0722088516, -0.0586804673, 0.0835686326, 0.116629913, -0.0618053786, 0.00126296934, -0.0307694152, 0.0223710835, 0.0577196926, -0.0216362979, -0.0806979835, -0.0328041427, 0.0271796659, 0.00863744225, 0.0390554368, 0.0131937107, 0.0795406327, -0.029518947, -0.00576462597, 0.0116117969, -0.0329764411, -0.0771837085, -0.102287009, -0.089663215, -0.218371257, 0.119085178, 0.0298947114, -0.038534712, -0.0590554103, -0.0107500628, -0.141160667, -0.0759352595, 0.117601112, -0.156553119, -0.011999514, -0.0650619566, -0.0730574876, -0.0246322155, -0.0698964298, -0.0485559702, -0.12944755, 0.00521457102, -0.0349291824, 0.0372204967, -0.132831231, 0.0268853568, -0.0678164959, 0.01158306, -0.0490771718, -0.129842356, -0.0273017623, 0.118581757, 0.0142164435, 0.0357958823, -0.135266781, 0.00959044602, -0.0602796748, 0.0601100251, 0.0731770322, 0.0262881704, -0.00786898099, -0.0921179354, -0.0371981561, 0.0295741931, 0.0243342854, 0.0789208785, -0.0568020456, -0.0867627934, -0.0332449675, -0.0421850346, -0.00150420517, 0.0511220172, -0.0336033963, 0.0623615161, -0.213038877, -0.0612739064, -0.026886005, -0.0112190992, -0.107592568, -0.158404768, 0.0247511286, -0.00325187342, 0.00806915201, -0.073451817, -0.0270244088, -0.186892807, -0.1511482, 0.07675457, 0.0333262496, 0.102376215, 0.0832969844, -0.0971427113, -0.0364518724, -0.0152430497, -0.127840132, 0.0834143609, 0.137075514, -0.00257097557, -0.00159274414, 0.0324123576, -0.0244972743, 0.0763535723, 0.0907546282, -0.00180239975, -0.00376731716, 0.13331072, 0.0758424923, -0.093535997, 0.0204091761, -0.0125161782, -0.134521812, -0.0275657028, -0.0810245574, 0.108791851, 0.000172570348, -0.100918159, -0.0968274102, -0.0810940862, -0.130157441, -0.0035761646, 0.0949944258, 0.0357959419, 0.102677576, -0.00810417254, -0.13290973, -0.090419367, -0.00868987292, -0.0630492195, -0.160759941, 0.0364927351, -0.0737517029, -0.0362737402, 0.038083896, 0.0794581026, -0.0493803881, 0.0407200716, -0.0497881584, -0.079237029, -0.0309528019, -0.0944269449, -0.0438238569, -0.041726768, 0.109497458, 0.0587373711, -0.135748714, 0.0756957531, -0.0297249965, -0.00938969664, 0.043221958, -0.0276608858, 0.0400940478, -0.00191638619, -0.0203203, -0.0793449506, 0.097187005, -0.0592457987, -0.0643090531, 0.0202469118, 0.0332247838, 0.0953644514, -0.0516278669, -0.131146327, -0.0792671144, -0.0597487278, -0.00294635445, 0.0967484415, -0.0312794521, 0.0133592859, 0.0706839263, -0.0293515176, -0.0438500978, -0.0517069995, 0.0330949873, -0.0315301344, 0.0448584333, -0.0420629829, -0.109620765, -0.164130181, -0.0980404168, 0.0248836204, 0.088697359, -0.113220185, -0.0422279499, -0.0472923331, -0.0464670584, 0.0527957492, 0.0145713305, -0.0128777456, -0.0992725566, -0.012445217, -0.155769691, -0.00321352668, -0.11781925, -0.0399204567, 0.0336041264, 0.109422341, 0.0170269795, -0.0438633002, -0.00304519292, -0.0239655524, 0.0205536298, 0.0797134042, -0.104388937, 0.0915353373, -0.0857452005, 0.0964980051, 0.0717691928, -0.12192674, -0.108307183, -0.0151441842, -0.0852235258, -0.0419365279, -0.0573839545, -0.000294502825, -0.091228053, 0.00850595906, -0.0173993055, -0.0732488334, 0.0468809865, -0.0340284184, 0.115676716, -0.0953338221, -0.0668268353, 0.0125814136, 0.0232165456, 0.0631158501, -0.0407331362, 0.0649367422, -0.150274932, -0.114792272, -0.0579118319, 0.0358544402, 0.0527209453, -0.0834443718, 0.0162117369, 0.0181254223, -0.0459999517, -0.00924878567, -0.0188188236, -0.200699046, 0.083431758, -0.0289405305, 0.100843623, -0.0543844067, -0.0213228483, -0.0823439136, 0.0506796241, -0.0783771649, 0.0163449757, 0.0561247207, 0.0255824793, -0.172806025, 0.0777617097, 0.116295606, -0.00262019318, -0.00658164173, 0.0238472763, -0.0476909094, 0.0135098621, -0.0669371486, 0.0111171473, -0.122062571, -0.0498253517, -0.0291282907, -0.173015878, 0.0420567915, -0.0911201611, 0.0584354028, 0.0305121839, 0.0397132039, 0.0658528209, 0.0387951732, -0.0431737304, 0.0818746313, -0.0564706326, -0.00999486633, -0.0379805788, -0.033199545, -0.0882304683, 0.00287892204, -0.0516074784, 0.0412358604, 0.131566599, 0.13412337, -0.0392659828, 0.0535762496, 0.0298382323, -0.0283444673, -0.0482411012, -0.0284610875, -0.0378182605, 0.0112354867, -0.0239805318, -0.00592691358, 0.154480234, 0.00800296944, -0.00739680696, 0.01570802, -0.128608316, 0.0373883285, 0.00223804824, 0.0431241132, -0.0234975219, -0.029798191, 0.0793395415, 0.0848310217, -0.0693508834, 0.00324432366, -0.144000366, -0.0398912765, -0.0685711354, -0.0200362187, -0.0482817702, 0.184426293, 0.0353978872, 0.135385722, -0.117208324, -0.0527831949, -0.0388038941, 0.104544699, -0.0188610889, -0.0286026523, 0.0971001685, -0.000703426078, 0.0268727504, -0.0154859498, -0.10792511, 0.157170147, -0.0427278765, -0.0264662243, 0.0401411764, -0.0388453826, 0.193847746, -0.0613880344, -0.00908031315, 0.111938514, 0.0168461613, 0.0317508988, 0.00498962402, -0.0748822838, -0.0916190371, -0.0108612515, -0.112528324, -0.0299282819, 0.038274128, -0.011974901, -0.0565649495, -0.0328519717, -0.0213433541, 0.129897207, -0.0328935012, -0.110759616, 0.0502097867, -0.0140230171, 0.0427038521, 0.0934353024, 0.0498347953, 0.0241618343, -0.0134589653, -0.0790630355, 0.0695633367, -0.0736205205, 0.0164346881, 0.0540283769, -0.123314232, -0.0443916172, -0.014228005, -0.0443573184, -0.0505989082, -0.0671131015, -0.0207865406, 0.0867469385, -0.143935561, 0.0978135914, 0.0641981065, -0.0140827606, -0.0885984749, 0.00961510837, -0.00615100656, -0.0863730758, 0.0572274551, 0.118623555, -0.00411961228, -0.0183738191, -0.00163236633, -0.0150230266, 0.0550976656, 0.0348100998, -0.00899617001, 0.0721205324, -0.0451185778, 0.0519079119, -0.0436058789, 0.0636622757, -0.0137794502, 0.00370390061, -0.0829177052, 0.00095188804, -0.0210709125, -0.0366235599, -0.0252530314, 0.0113218538, 0.0346394219, 0.0598685108, 0.0204074755, 0.0285690669, 0.133948505, -0.00939935073, 0.0975652859, 0.0343537554, 0.0170677174, -0.016463533, 0.0143543892, 0.0227485672, 0.0527459383, -0.145403877, 0.0538256764, -0.113765627, 0.0250843316, -0.031842351, 0.130124092, 0.132894307, 0.0850479752, 0.0246920604, -0.0833828896, 0.119493447, 0.117562339, 0.0258794446, 0.00648026913, -0.159253091, 0.0186034944, -0.0576140918, 0.0698988587, 0.00684992317, 0.0629072562, -0.16676414, -0.106456123, 0.132934898, 0.102742344, -0.0148053309, 0.0249220151, 0.0560664721, -0.136113957, 0.0519405454, 0.0143429618, -0.0377547815, 0.0269494578, -0.0424542576, -0.0378604382, -0.130487964, -0.00247203745, -0.126098335, -0.033814311, 0.0826421306, -0.122226387, 0.0033654999, 0.0505205169, -0.0212788582, -0.00628613494, 0.0552953109, -0.0479597673, -0.00329525396, 0.0209926255, -0.0205684248, 0.0478610024, 0.0806275979, -0.0743420571, -0.0931046903, 0.0527450331, -0.00999636948, 0.116710916, 0.0795818269, -0.042247206, 0.00203297473, 0.0550016873, -0.114586599, 0.126905248, 0.118282221, 0.0137572065, 0.0230594128, -0.0301910006, -0.0830214471, 0.00634433702, -0.0385019854, 0.045974113, 0.0223330148, -0.0154264048, -0.0188241377, 0.126796842, 0.0640706718, -0.0480389744, 0.0710388497, 7.29076564e-05, -0.0148876328, 0.0211679824, -0.013507612, -0.0415202789, -0.0301044956, -0.0432036407, -0.0804740116, -0.0297432039, -0.0194068104, -0.0929949358, 0.00407454977, 0.153331608, -0.0294467174, -0.0516009331, 0.011737382, -0.0235770624, 0.0614383221, -0.0587256067, -0.181149006, 0.0379187614, 0.0139180515, 0.126733571, -0.0525923893, -0.0963102728, 0.0340560302, 0.010048761, 0.0537804291, 0.00721588731, -0.0115360133, 0.0094257826, 0.141251072, -0.101650581, -0.0885887593, 0.0021282956, -0.0657165349, 0.0114656575, -0.0879223049, 0.0472398326, -0.0253054239, -0.0949798971, -0.0532924011, -0.110345133, -0.12598604, -0.0324145071, -0.117882788, -0.0235238336, 0.144998997, 0.0784391761, -0.0579266362, -0.037623588, 0.0221065655, 0.10861934, 0.0199468452, -0.0090676304, -0.0338938311, -0.0436233766, 0.0650386512, -0.0787329078, -0.0181119759, 0.102961294, -0.0252211094, -0.141934544, -0.0211859122, -0.0214212239, 0.0750921071, 0.0982615948, -0.0225319024, -0.0775617957, 0.0340965502, 0.107802778, -0.0417751148, -0.0193603709, 0.0165249649, -0.0958091095, -0.0096657183, 0.0185735859, -0.060692884, -0.0741733685, 0.0478498675, 0.140758082, 0.0878093168, 0.124422796, 0.0315869115, -0.0765189976, -0.158293381, -0.0663742274, -0.161471233, -0.00101692602, 0.0242872071, -0.018827172, -0.00992732495, 0.0574326739, -0.0708991811, 0.0418169796, 0.0214103982, 0.0277493, 0.0836243778, -0.114706472, -0.110778809, -0.00549926795, -0.0547126345, -0.0340471826, -0.0263265911, 0.0121591762, 0.0904770494, -0.0491277203, 0.055547826, 0.0116426498, 0.00450218469, 0.0239987187, -0.105099499, -0.0454495102, 0.181741923, 0.0572534874, -0.0400019772, 0.133353099, 0.020812327, 0.00370626338, 0.0576054901, -0.0590315312, -0.0551964603, 0.0629728138, 0.0279572792, -0.0744772702, 0.00956684351, -0.0706064776, 0.0634177253, 0.131110832, -0.0383560918, 0.0275039617, -0.00775681622, -0.0485731848, 0.0826426819, 0.0914519876, 0.0673530847, 0.11230211, -0.0202659685, -0.0253299512, 0.145047918, -0.0104174726, 0.12206649, 0.00895817019, 0.0214635525, -0.0384950005, 0.0974250734, 0.0578387864, -0.0336539596, 0.0341395587, 0.0233154371, 0.0867071003, 0.0834672004, -0.0215894487, 0.0957072973, -0.101723067, 0.0511676073, 0.0313554816, -0.0860508233, -0.0147732571, 0.00499431789, -0.0514711477, -0.00683964137, 0.02644879, -0.0171801373, -0.10945788, 0.121007361, 0.221389726, -0.0124760075, -0.0674972087, -0.149561465, 0.026429411, 0.0638324469, 0.0117955673, 0.0279138833, -0.020272702, 0.0516363829, 0.0422598794, -0.114757769, 0.00266931951, 0.0386949852, 0.0381801687, -0.00551658496, -0.0496969037, 0.0212384872, 0.00767339021, 0.0233013686, -0.0131994803, -0.0950405449, -0.115363941, -0.100356773, -0.041871652, 0.0446711816, -0.0411373973, 0.00625232514, 0.0883152261, 0.00292699318, 0.0855041817, 0.183508277, 0.0525820218, -0.0131733213, 0.0197753981, -0.0630000681, -0.0122047439, 0.0420472212, -0.00139854476, 0.0688946396, 0.105930798, -0.0156559572, 0.0936368257, 0.00706671504, -0.056444589, -0.108396575, 0.0138884149, -0.0538526848, -0.128820136, 0.0302302614, -0.111674353, 0.121688239, 0.0176053345, -0.10430266, 0.131543815, -0.0368286893, -0.103113487, -0.0715081543, -0.153515577, -0.104622796, 0.00369652454, 0.0772574842, 0.00716855377, 0.0859163627, -0.0379379131, 0.0117043816, 0.00218433887, -0.0561341755, -0.0711707398, -0.0604123734, 0.00601920066, 0.00673713721, 0.0530272275, -0.087426506, 0.0119247064, 0.0216195658, 0.0711690187, -0.0460512154, -0.0697385743, 0.0119794961, 0.0283777304, -0.084892951, 0.047121726, -0.0334042907, 0.028567221, -0.0157220569, 0.036880292, 0.0404169858, 0.0937352329, 0.0302604306, -0.0369935334, 0.00511695445, 0.00988284126, -0.0110902032, 0.103052162, 0.0853995383, 0.00195272965, -0.0113939494, -0.041175995, -0.0654686466, -0.0427516997, -0.145465791, 0.00170960696, 0.057869669, -0.0286980402, -0.00456581637, -0.085768804, -0.0539919809, 0.0158043746, 0.165604845, -0.027340278, -0.190521687, 0.075797081, 0.0119776074, 0.0335224271, 0.00701582991, 0.0292586386, -0.0574985072, 0.00961377472, -0.0490148328, -0.00297709648, 0.00284333713, -0.000433928333, 0.145019993, 0.0384721719, 0.0357460789, 0.126232311, -0.040336296, -0.0102300942, 0.119501092, -0.0390173979, -0.0487000942, -0.049991414, 0.0441951714, -0.0656402856, -0.00859091803, -0.0110485274, -0.0972131491, 0.0576536804, -0.173949748, -0.0703914985, 0.0491493195, 0.0730941743, 0.0783300772, 0.0708089247, 0.0507010035, 0.011911111, 0.0551151037, -0.0721687004, -0.0162433423, 0.020192109, 0.0923747048, 0.0203865096, 0.0873873755, -0.140714914, 0.0327500775, 0.014140388, -0.0651469007, 0.0345980227, 0.011195885, 0.0874392018, 0.0658201054, -0.0455558971, 0.0463316888, 0.0044172341, 0.0349625684, 0.0705547631, 0.0579739884, 0.0394821391, 0.125749066, 0.0352044329, 0.0180898402, 0.0983930379, 0.0521039143, 0.00767131895, -0.0869135037, -0.0102869906, -0.0738259256, -0.107947849, -0.034839794, -0.0593574271, -0.13112238, -0.11901968, 0.119414158, 0.0498590693, -0.105217464, -0.0373657681, -0.031966608, 0.0279503297, -0.0290230047, -0.0853976756, 0.0192912035, 0.0113811484, 0.142793164, 0.0543404594, -0.00275331782, -0.0411211476, -0.0437537879, -0.175868899, 0.0339396447, 0.0359358937, -0.00966062769, 0.0758331269, 0.0519977175, -0.116831876, 0.122007556, 0.0277519338, 0.138974085, -0.0515451841, 0.013362377, -0.00194710889, -0.024108164, -0.0320435092, 0.0878870934, -0.0230963212, -0.042228099, -0.0418023951, 0.155867562, 0.0163917653, 0.0963448435, -0.0340325385, -0.0556667112, -0.142566487, -0.0099136075, 0.209352762, -0.0376806483, -0.0146721434, 0.00145089068, -0.00487274118, -0.0763048232, -0.0218742155, 0.103745073, 0.0367730483, 0.0581323914, 0.0475413166, -0.153616562, -0.0449088328, -0.112986043, -0.02845864, -0.0427805707, -0.0357970595, -0.0357543342, 0.116666973, -0.045204781, -0.172904223, -0.0625614598, 0.0878430903, -0.0336587429, -0.0510490127, -0.00328099728, 0.0481171645, -0.0361189358, -0.00395132229, 0.048532743, 0.0747343302, -0.150656834, -0.0267654695, 0.065988034, 0.000906120986, 0.0526575483, -0.0886258855, -0.0326578878, -0.0392294563, -0.114601858, -0.0436432883, -0.0233603958, -0.0366286114, 0.0242132805, 0.046646174, -0.00596841611, 0.107337743, 0.100711152, 0.0962712914, -0.0196551755, -0.0379424095, -0.0149137788, -0.00352167524, 0.00364584103, -0.0446948335, -0.0481903926, -0.0171441138, -0.0307623744, -0.0520249456, -0.0215769466, -0.0831398889, 0.102580726, 0.0553011298, 0.0597906336, -0.0660742596, 0.0327185541, -0.0501872599, -0.0174297784, 0.0845402032, -0.0439116322, 0.00334379589, -0.0667040423, -0.00720180944, 0.0398931578, 0.0985840261, 0.0395776331, -0.0174181163, 0.0681332946, 0.0306725055, 0.0796344131, -0.0542774051, -0.00695079146, 0.00331622828, -0.0354855023, -0.024734579, -0.104051322, 0.0979310572, 0.111053832, -0.0395862758, 0.0508234426, 0.0743522495, 0.112601981, -0.0108194482, 0.0281996876, 0.0765923113, -0.0717236102, 0.159004852, 0.0928426981, 0.170626536, 0.0166542754, -0.0144605357, -0.0233754274, -0.126926482, 0.00886013359, -0.0221404657, 0.0173175037, -0.0316050202, 0.126515985, -0.0868917778, 0.171482056, 0.000556701794, 0.0924508423, 0.139084101, 0.109917842, -0.134655744, 0.101962559, 0.013568854, 0.0637116358, 0.106478803, 0.0461113527, 0.169571549, -0.0845821202, -0.0924094096, 0.0302632377, 0.0683329329, 0.00514531881, 0.164434299, 0.0242732447, 0.0178257711, 0.168122873, -0.0748524293, 0.0768326595, 0.125718981, 0.0113984775, 0.0914176553, -0.00384905934, 0.0749454051, -0.106595621, -0.004456806, 0.0573939309, -0.0508570671, -0.0259132627, -0.0837707222, -0.0911950693, 0.062700808, -0.0178347547, 0.0896601379, -0.0371693149, 0.0397659428, -0.0586689822, -0.0487654656, 0.00985174812, -0.0431361422, -0.0103281885, -0.0436234362, -0.00453014765, -0.0160913728, 0.00195264816, 0.0702505484, 0.0770360604, -0.0666011348, -0.128395498, -0.104411148, -0.117587678, 0.000573134981, 0.0101250224, -0.0282442681, 0.0171822198, 0.0782697201, 0.00239574723, -0.0798596889, -0.0255712122, -0.0991983712, -0.0479424968, -0.0651287064, 0.00909695122, 0.0286999997, 0.107792236, 0.0201869458, 0.129761383, 0.0120681971, 0.129636198, 0.030876562, -0.0569740236, 0.0125696817, 0.00621464849, 0.017092824, 0.00570657849, -0.00598617084, -0.041225329, 0.0295243431, -0.0221839678, -0.0352542624, 0.00819571223, 0.113492012, 0.0407709107, -0.0561432913, -0.0223866664, 0.0815185383, -0.0581509247, -0.0125219971, -0.0523082167, -0.0633664876, -0.0935018361, -0.0119582247, 0.121525399, -0.0465201139, -0.116775118, -0.0365208909, -0.0371810421, -0.112663895, 0.00683574378, -0.0989704579, 0.00214093737, -0.0367812067, 0.0180868953, -0.0585453287, -0.0212486722, -0.158388585, 0.0844327733, 0.0906519815, 0.0489695147, 0.0414573848, 0.0692197829, 0.0418851823, 0.0244824868, -0.0816810951, 0.0888817757, -0.0508183949, -0.088789925, 0.0785966963, -0.103541039, -0.0438995808, 0.0549837388, 0.0631930828, -0.0311866403, -0.0528068952, -0.000458076596, -0.0921617672, 0.0281930007, 0.0854556859, 0.1542577, 0.0876967907, 0.0826123059, 0.232156977, 0.0229519103, -0.030814413, 0.0359654352, 0.0792249665, 0.0734914243, 0.0297194421, 0.12659736, 0.105616376, 0.130550563, 0.0201957077, -0.158744067, 0.0149462121, -0.0611429513, -0.0496162809, -0.0840074569, -0.0463297591, -0.0214238595, 0.140511125, -0.0970251337, 0.0862722546, 0.0148826325, -0.0661468953, 0.0448164865, -0.00943928119, 0.170197755, 0.0304960068, 0.0266494136, -0.0164098088, 0.0421887636, 0.0587810464, -0.0198171325, -0.0166118629, -0.0128516201, 0.0712332726, -0.0262440406, -0.0257695001, 0.144736886, -0.0454605967, 0.0827688724, -0.105175555, 0.0854492635, 0.0372763723, -0.0393086672, -0.0433932096, -0.00199082866, -0.00664438307, -0.0665106848, 0.102266923, 0.200106829, 0.0514936373, 0.062575236, -0.12222188, -0.00965614989, -0.10842903, -0.0519748107, 0.0540346615, -0.0423696414, 0.0241926759, -0.00697272271, -0.0571990833, 0.0542127304, -0.00683669187, -0.0358720608, -0.0523957089, -0.00335288886, 0.0791841969, -0.0631926656, -0.000886259368, 0.160912022, 0.113086849, -0.0230797902, -0.115601629, -0.00374781527, -0.0388966948, -0.139379799, 0.112785511, -0.142339468, -0.125529379, -0.0601072349, -0.110232972, -0.0605999157, -0.0103344237, -0.00830904581, 0.0831668377, 0.017292574, 0.0398771241, 0.0214732271, 0.0823135525, 0.0139693758, 0.00157841854, 0.11886555, 0.0256661214, 0.133169919, -0.0465491563, 0.0687712431, -0.175382465, 0.0867511481, 0.0866570845, 0.0748714656, 0.045688156, -0.0761289895, 0.0661332235, 0.0861954689, 0.0729580745, 0.0148899965, -0.0253776368, -0.0456276014, -0.0161083508, 0.0115437303, -0.0153818261, 0.0868741348, -0.0882275328, 0.0707228035, 0.0998456255, 0.011327602, 0.0904787928, 0.0399920717, -0.0749375075, 0.00247166306, -0.0361021757, -0.126668707, -0.0503375903, 0.0633101314, -0.0163081326, -0.0129666403, 0.00958995894, 0.111958131, 0.0579606257, -0.0194422659, 0.0867757797, 0.0886274278, 0.11379382, -0.0136893839, 0.0386091657, 0.140771434, -0.0114353709, -0.0759116113, -0.00567827467, 0.0763429329, 0.0647702888, 0.0904307589, 0.0219500922, -0.0276538134, -0.0205843598, -0.0522674993, -0.00134441117, 0.129205391, 0.0696320534, 0.0557793975, 0.126799747, 0.107252121, 0.061958082, 0.0235393457, 0.051930923, -0.00306171365, -0.0450648591, -0.0375821628, 0.0596879274, -0.061171338, 0.0400689729, 0.0412523821, 0.0863733888, -0.0760089159, 0.0504633412, 0.0358135216, 0.0740757212, 0.0022061374, 0.0884475335, -0.000341153238, -0.0773504227, -0.0645802245, -0.0759093687, -0.0472579598, 0.0379689373, 0.0503579192, -0.0227510706, -0.0318921283, -0.0636509135, 0.0167824589, 0.0469228439, -0.0686417222, -0.0224289522, -0.116739154, -0.0366590023, -0.00713004917, 0.00225095917, 0.0232665855, -0.068639338, 0.0609753355, -0.116830498, -0.0711478218, 0.123511501, 0.0235070623, 0.0461065769, 0.0747356415, 0.0720939264, 0.00433993712, 0.0820146576, 0.069557704, 0.0107531231, -0.0327813998, 0.00303759053, 0.0307164751, 0.0211477932, -0.0687760338, -0.0758109912, 0.0396731943, -0.0592078567, 0.00160061009, 0.116870962, -0.127800584, 0.0479781218, 0.0467708185, 0.0786154717, -0.0823335052, 0.119760633, -0.11141441, 0.0265908577, -0.0524609499, 0.120253593, -0.00687352614, 0.0913991556, 0.0329756513, -0.0819903389, -0.0453966707, -0.00249208882, 0.0236762464, -0.0761071965, 0.0804237872, 0.106075808, 0.0286033526, 0.081977509, -0.0605856366, -0.0440501347, 0.0195822455, -0.0494956523, -0.0163362063, 0.0376294814, 0.0300236586, 0.00706194155, 0.0360870883, 0.10803137, 0.114604935, 0.106907368, 0.0261990167, 0.025890965, -0.0913227126, -0.0935981497, 0.185391679, 0.102065086, -0.0688922629, 0.0399040766, 0.0297738109, 0.000596365891, 0.0412646756, 0.0512274429, -0.124623746, -0.0459248126, -0.0313363522, 0.122049555, -0.000766901299, -0.0703695267, 0.0415504463, 0.139911398, 0.0679421127, 0.0302217659, -0.0152739808, 0.0120744314, 0.0357736871, 0.0544544384, -0.0690561086, 0.0109463455, 0.0249296762, 0.0186653174, -0.0291013829, -0.00324610109, 0.0695713609, -0.136896506, -0.0408418179, 0.0385437906, 0.031190034, -0.0783010945, 0.11616379, 0.00849272404, -0.0795347169, -0.0427973829, -0.0240525529, -0.0278865006, 0.0615595505, -0.0920619667, 0.0265126191, 0.124375701, -0.00754014961, 0.0605839938, -0.00936108828, -0.0976717398, -0.0971646011, 0.037894886, 0.0407787189, 0.0457353592, -0.0538839102, 0.0676756799, -0.0228612162, -0.0195428338, 0.0116100889, -0.0484733544, -0.0903081745, 0.0195736028, -0.177630827, -0.0424475297, -0.150964722, 0.0452550352, 0.0208111051, -0.00896799937, -0.0491741002, 0.070747979, -0.0901333243, -0.0358462296, -0.0416615084, 0.058083605, 0.0306156334, -0.0475451536, 0.0355117247, -0.0191579144, 0.127348647, 0.0233417489, -0.0105300415, -0.0514476039, 0.130523205, -0.0192206688, -0.00500579365, -0.02127425, 0.147623256, 0.0189047717, 0.0578304157, -0.0745900646, -0.116294131, -0.0905236304, 0.11783056, 0.0313080437, -0.117304355, 0.0563333407, -0.0425937027, -0.0149243101, -0.09566167, -0.118109919, -0.110766359, -0.0748157203, -0.00860852748, -0.0183044299, 0.0145282075, -0.0798267201, 0.0352287106, -0.153934568, 0.0180907808, 0.0400847048, -0.00181255862, 0.0976161212, -0.0077306591, -0.0462495685, -0.0855609477, 0.146166742, 0.119049467, -0.0308496356, 0.0242325962, -0.0348199941, -0.0325288065, -0.0175943989, -0.0934547186, 0.165575653, -0.00701182336, 0.0348708369, -0.0705262125, -0.0535933636, 0.0479519963, -0.106788114, 0.0836377293, -0.0230580494, -0.030803334, -0.0258164573, 0.0451489799, 0.0713042468, -0.0349851847, -0.103278354, -0.0427363738, -0.0513073057, 0.00717804022, -0.0678141862, -0.0282868147, 0.0327754542, 0.00344437035, -0.021794131, -0.0249118339, -0.132074341, -0.167451188, -0.0553339683, -0.0340443403, 0.0441243947, 0.0767783746, 0.0518309623, 0.053142339, -0.03464422, 0.0915156528, 0.0572075658, 0.0368602835, -0.122862265, 0.125554949, -0.0212506503, -0.028879609, 0.0728348345, 0.074088648, 0.0167630445, -0.0572193228, -0.0381724015, 0.12321689, 0.120577976, -0.00745597715, -0.00373940542, 0.0891999826, -0.100307591, -0.0272143763, -0.0464793816, 0.0808481872, -0.0214728303, -0.0114586502, 0.117915325, 0.0525748283, 0.0499168076, -0.0553271882, 0.0459340736, 0.0311813466, -0.0554301329, 0.119270027, -0.141592056, 0.0801190883, 0.0238559097, -0.0244946219, 0.0137403859, -0.0247483365, 0.0890131071, 0.0122417919, -0.0221369304, 0.134725109, 0.0171203725, -0.0616743043, -0.104806133, -0.043887794, 0.0243591964, -0.0707414448, 0.0545995533, -0.244177178, 0.00985076651, -0.00673175463, 0.00327755511, -0.0787141323, 0.0315161161, -0.054905612, -0.0245899297, 0.0200434048, -0.0167779438, -0.00633175578, -0.00168752554, 0.0146405138, 0.102586865, -0.141001478, 0.0254550986, 0.0282731801, 0.0347467586, 0.0325434059, -0.050280951, 0.18338868, 0.0346820056, -0.0438000076, -0.0990172401, -0.039733801, -0.028076401, 0.0997701958, -0.0247635506, -0.0885608494, 0.0252160151, 0.0274931937, 0.0407864675, -0.00188285112, 0.020264674, -0.0637085289, -0.0331827141, -0.0375841819, 0.0395974182, -0.0142489355, 0.00901054405, 0.0661969706, -0.0141161121, -0.133677304, -0.0379943736, 0.104471594, 0.00207850896, 0.0502881594, -0.0103730969, 0.0161753967, 0.102761641, 0.0681505501, -0.0854083449, -0.0660482645, 0.10789603, 0.121360719, -0.249932483, 0.043577794, -0.019488927, -0.0333441533, 0.0699044764, -0.0417760946, -0.0830878019, 0.0335712731, 0.0915890262, -0.0181932189, -1.87662663e-05, -0.0177107975, 0.0466791168, -0.0754079893, 0.0253002997, 0.198537499, -0.0213280898, -0.025934197, 0.0887482762, -0.00143241324, -0.0775671974, 0.0361523703, 0.0349732526, -0.100858748, -0.00825742539, -0.0823086947, -0.0676879585, -0.111404717, -0.00717196055, 0.156943232, 0.0420605578, 0.133920968, 0.0445161164, 0.0383869596, 0.127522886, 0.0221633837, -0.018852653, 0.148891225, 0.125538707, 0.0585277081, 0.007541053, -0.00326655805, 0.0190913379, -0.0821087062, 0.0579386801, 0.118444584, -0.0510979965, 0.0783319324, 0.0698043033, 0.00990374014, 0.0493937135, 0.0577939376, -0.0367200673, -0.054412514, -0.109961107, 0.0457087681, -0.0674096867, -0.104861669, -0.0329911038, -0.107919648, 0.0506276563, -0.0262097511, -0.0370987169, 0.115089066, -0.0547752641, -0.0348114185, 0.139484152, 0.0119006224, -0.0441697314, -0.108552918, 0.106704302, -0.0203959923, -0.0326148309, 0.00614642445, 0.0449354462, 0.0489949211, 0.0114523806, 0.0450277254, 0.121315338, 0.102272771, -0.0944834501, 0.092575267, -0.0403284207, 0.0216861926, 0.00450862665, -0.0592273101, 0.00570360571, -0.0967926979, -0.0910627022, -0.00712880678, -0.0250440538, 0.136949509, 0.0154127292, -0.0850391686, 0.0234602913, 0.00543305464, 0.0879383385, 0.0208250824, 0.0559528843, -0.0110894479, 0.0145522431, 0.135471657, 0.0212556887, 0.0144467633, 0.203706801, -0.0035531295, 0.0548708662, 0.140472278, -0.0227280222, 0.0714532286, 0.0695853531, -0.102898076, -0.0454968996, 0.0986656249, 0.110469475, 0.0370585546, -0.00549947098, -0.105551526, 0.089052707, -0.0938652977, -0.0917528048, -0.0288683102, -0.00569865108, 0.0564894304, -0.0824488103, 0.00415596366, 0.0122276712, 0.0612397604, 0.00702984305, 0.045586437, 0.0224325489, 0.0116679557, 0.104367994, 0.00187444873, -0.0533959605, -0.0969143659, 0.0603949167, 0.0610991865, -0.0280593596, 0.118755028, 0.163122639, -0.138794631, -0.0982856303, -0.0437370613, -0.0400318317, 0.0307425465, 0.00351504236, -0.0370394252, 0.0179562531, -0.0826809853, 0.0623588376, 0.0165627245, -0.00318234041, -0.221593887, 0.109638736, 0.0367929861, -0.00492305635, 0.0764009804, -0.0543240719, 0.00832460541, 0.0246482976, -0.0788863152, -0.0332067758, 0.0616043061, -0.21109958, -0.0462315455, -0.0243709795, 0.12805903, -0.12404044, 0.030349832, -0.0422639549, -0.0548278876, 0.115669861, 0.0864745677, -0.0318449363, 0.00868205354, 0.0428102463, 0.0293472409, 0.0725860298, -0.00305261649, -0.0225684382, 0.0127110137, -0.0456389897, -0.0668282583, -0.0378625616, 0.0442645028, 0.173314661, -0.052643083, 0.0150079504, 0.0173244383, 0.00870173331, 0.0481358767, -0.0213168375, 0.0177885741, 0.0484836027, -0.0253024288, 0.0580496639, -0.0112942867, 0.0664902106, -0.127707645, 0.155566022, -0.0657561421, 0.0964245349, 0.00386818405, 0.00187859917, -0.02726865, 0.034068726, 0.0160691291, -0.0390943512, -0.0815259814, -0.0481792055, 0.0673541129, 0.0301477201, -0.0904736668, 0.0712888315, 0.0729079992, -0.059337128, 0.0573410057, -0.073555395, -0.0689984858, -0.0625811219, 0.0529500842, -0.0561883114, 0.0769964159, 0.0505550019, 0.000728402287, -0.070477441, 0.0579672381, 0.101890601, -0.0232261382, 0.0331965685, -0.13476932, 0.0779082999, -0.0188822336, 0.0747630894, -0.0301496182, -0.00284632482, -0.0692487508, -0.0216729604, 0.160968274, -0.0487398952, -0.0273404717, 0.050436575, -0.0679521263, -0.218488425, 0.0673827305, -0.0169843659, -0.003985174, 0.128913343, -0.00705931336, 0.0715985522, -0.0235490371, -0.0697448403, 0.049252674, 0.00652051531, 0.0601320639, 0.0213046558, 0.0109692924, 0.0429657996, -0.174835622, -0.130821571, 0.102699831, 0.0806046799, 0.0338189378, 0.122710109, 0.019222524, -0.096650511, -0.0175743625, -0.0367461853, -0.124857023, 0.0774191171, 0.080327183, -0.0344017185, -0.114270456, -0.0034753317, 0.0288006812, 0.0443388335, 0.014642843, -0.1024535, 0.0593441091, 0.0772532597, -0.00851446763, 0.0876583084, 0.124778286, -0.0536802486, -0.0409024581, -0.0989011303, -0.0572285131, 0.0117281517, 0.021247806, 0.0173328109, -0.0679287314, 0.0592512637, 0.0371976048, -0.0846372098, 0.0498691611, 0.0432467423, 0.0368210562, 0.0556512997, -0.0579462983, -0.00415133499, 0.059488792, -0.0446038172, 0.097750172, -0.016106993, 0.0228777528, -0.0185083281, -0.0073051299, -0.0180141293, -0.00993139949, -0.0436107181, 0.035581328, -0.105229981, 0.0257416777, 0.092828095, -0.0869532079, 0.0912591293, 0.0479641408, 0.0192065462, -0.0746231526, -0.00535912719, -0.00916508213, -0.0579479821, 0.125106856, -0.029226372, -0.0246271715, -0.116364449, -0.00552114286, -0.023564972, 0.0158106312, -0.00883663632, 0.086115554, -0.0623098575, 0.0139099192, 0.0638796389, 0.08404769, -0.0410103686, 0.173401594, -0.103401519, -0.0626127943, -0.0580803752, 0.0124420989, 0.0831609741, -0.00756312162, 0.0207710881, 0.0159177668, 0.144318879, 0.074575834, -0.0103816949, -0.0032339131, -0.029581476, -0.104740039, 0.189521343, 0.0631510541, -0.0114794131, 0.0336302407, 0.0695150122, -0.0663278848, -0.00947028026, 0.0796912834, 0.117743649, -0.0355180204, -0.0403854102, -0.0393885002, 0.114623398, 0.122436151, 0.12554881, -0.076746434, 0.0528300032, 0.084031716, -0.103645802, -0.146345764, -0.0427184589, -0.0977167636, -0.141606271, 0.0692159384, -0.0181116704, -0.120115615, -0.0101953847, 0.0760765225, 0.0554642305, 0.000105306506, -0.0047814101, -0.0269510858, -0.125877321, -0.141362876, -0.121428445, 0.100611567, -0.0299713388, 0.0269113686, 0.0415728725, 0.165701568, 0.0359493531, 0.0818786994, 0.0318259075, -0.0558618456, 0.0194035377, 0.056799829, 0.0331340544, -0.0671101585, -0.0700573176, 0.0376645476, -0.0909235179, 0.0566633083, -0.0423257649, -0.123594165, 0.026218446, -0.12405815, -0.0305393357, -0.0208273903, 0.0113523966, 0.0103740282, -0.0453835651, -0.0157404374, -0.0896555334, -0.143528402, 0.128691524, -0.0391090289, -0.0135176145, 0.0219401699, -0.109882608, 0.0331697166, -0.112585135, -0.182065874, 0.077039957, -0.00479537249, 0.0636857823, -0.0363294184, 0.0772058442, -0.0258613601, -0.160521716, -0.117557757, -0.0483435877, 0.0140365288, 0.0360953435, -0.0815866441, -0.0412564129, 0.00797186326, -0.0999645889, 0.00220270455, 0.0667368174, 0.0200745277, -0.0253414474, 0.0040999949, 0.143322214, 0.0579100028, 0.0961008891, 0.00519804657, -0.0552583858, 0.104603909, 0.0475944132, -0.0181248486, 0.0693280995, -0.0443166457, 0.0621352941, 0.0530473851, 0.0355710611, -0.0889870003, 0.0598861016, -0.0278735906, 0.0632814839, -0.0215976648, -0.11186105, -0.099360846, 0.0478967354, 0.129642054, -0.0641585365, 0.0809434652, 0.12299259, 0.0165501498, 0.044932235, -0.0917557701, 0.11085023, 0.00117426179, -0.0625073239, -0.0624597371, -0.161765128, -0.0117147248, -0.131242961, -0.0102577172, 0.0281911381, -0.0956992656, 0.120214455, 0.0611006394, 0.0452139191, 0.00106171332, -0.0305562951, -0.0058944067, -0.0535558127, -0.0557085425, 0.0984686315, -0.0755340382, -0.0857185647, 0.029177431, -0.0294365548, 0.0448531359, -0.0881679505, -0.0566896051, 0.0818277374, 0.171184421, 0.0391540192, 0.0264476165, -0.0424234644, 0.00381949544, 0.0557178929, -0.00430215895, 0.0519038811, -0.0217410438, -0.0639868975, 0.0107317418, -0.0457099602, -0.0515033007, -0.00533560105, 0.101076961, -0.0996893495, 0.110352285, 0.0275920294, -0.126547217, 0.0580787845, -0.0648229197, 0.0641894937, 0.0190863106, -0.0730425566, -0.0441494212, -0.0377254561, -0.00119296182, 0.0298135336, -0.055152528, -0.0692317933, -0.133605316, 0.102659523, 0.00388940051, 0.110093594, -0.0825676173, -0.153323025, -0.0475650169, 0.0295819063, 0.0981707796, 0.0889128968, -0.0153834652, 0.0210752022, -0.0495757982, 0.0258275159, -0.0230260268, 0.0365365446, -0.0103806965, 0.0280630793, 0.0804096013, -0.0812752768, 0.0715501979, 0.0769598112, -0.0793469474, -0.0544905476, -0.120476916, 0.0758223608, -0.0434372351, -0.0345638357, -0.116654873, -0.00733613782, 0.0018581152, -0.0251683071, 0.0275420249, -0.0133311432, 0.02410152, -0.0494358316, 0.0597402379, 0.0644570887, 0.0644316301, -0.10921298, 0.0997109562, 0.000376366079, 0.119578719, -0.0456936583, 0.110384509, -0.0454241335, 0.115739658, -0.0350133367, 0.0300470926, 0.0534853637, 0.000776473433, 0.0301366635, -0.098016873, 0.0700167418, -0.233400077, 0.0236323681, 0.161524281, 0.010498126, 0.0271028839, -0.0192050189, 0.0778874606, 0.120771617, -0.0141737051, 0.0373958796, -0.0652192086, 0.113831788, -0.0542669669, 0.0246119127, -0.0946244225, -0.0857878923, -0.0324967988, 0.0309826005, 0.061101079, 0.0833132565, -0.0271196496, 0.035355188, -0.134274811, -0.0367200524, 0.039295841, -0.0480492152, 0.0820622668, -0.0221788306, -0.00728615187, 0.211294726, -0.0996121317, -0.0951313376, 0.0882309228, 0.0507182628, 0.0955223814, -0.0135086589, -0.0100876577, -0.104710273, -0.0837924182, -0.00485351775, 0.140761971, 0.0304966271, -0.00328581966, 0.0630469769, -0.0528654195, 0.00146873784, 0.070460178, -0.00982738007, -0.0246508308, 0.0094127208, 0.0792464614, 0.0270396024, -0.0288467649, 0.0683740824, 0.0343907848, -0.0171846393, 0.101047479, -0.0562119856, -0.104776561, 0.0199727528, -0.105037361, 0.0388257988, -0.0307911783, -0.0515712202, -0.00239409413, 0.0136426426, -0.00552344508, 0.0488392264, 0.0432750806, -0.0318257213, 0.0592304394, -0.0536281317, 0.0502378196, -0.0556555688];
    bias_w_3_h : ARRAY[0..63] OF REAL := [0.0991463065, -0.116468273, 0.138851866, -0.0278104451, 0.109091796, 0.00748556852, -0.14681308, -0.125416145, 0.0911259875, -0.007215071, -0.0655900463, 0.0117500499, 0.138449639, 0.0438438281, 0.131512955, -0.0941261575, 0.114508875, -0.106850296, 0.0109656742, 0.100971431, 0.00989976991, 0.122776113, -0.0815143511, 0.0247511063, 0.151071012, 0.0270412229, -0.144494727, -0.0250454061, -0.138304651, -0.113388814, 0.0156560782, 0.0580180995, -0.130460665, 0.130777717, -0.147577867, -0.0267437994, -0.144388303, -0.0317561962, -0.0075275274, -0.0961027741, 0.143372744, 0.156992108, -0.123628758, 0.128169924, 0.143014401, 0.01310274, -0.0771420449, 0.00980290584, 0.0187610406, 0.0503772497, 0.0593717098, -0.129526407, -0.125063941, 0.00348926126, 0.131469816, -0.0135045191, 0.0106752291, -0.124533199, 0.0468791761, 0.122625463, 0.13421531, -0.145920694, 0.0187235065, -0.121972054];
    bias_r_3_h : ARRAY[0..63] OF REAL := [0.213432834, -0.161678195, 0.256692797, -0.0889138281, 0.165887326, -0.0884462819, -0.27341947, -0.168622971, 0.192972749, 0.016962342, -0.191151828, 0.130318716, 0.270743728, 0.142349645, 0.253203601, -0.221500397, 0.170809239, -0.19833906, 0.0530763082, 0.221980438, -0.0285716169, 0.184993401, -0.214608163, 0.0641558841, 0.288412601, 0.160010368, -0.266304582, -0.0861380771, -0.252676189, -0.209977716, 0.0482637659, 0.184551656, -0.19582215, 0.224073783, -0.276625097, -0.156061158, -0.293882459, -0.105265953, -0.0959337279, -0.204042628, 0.264214009, 0.313724399, -0.184004784, 0.25386411, 0.154165655, 0.137930378, -0.192821845, 0.0848548487, 0.141432852, 0.171690077, 0.166555926, -0.253184497, -0.235516116, 0.00120966323, 0.229147851, 0.0655627847, -0.0512111448, -0.184087113, 0.153496757, 0.241964057, 0.270176709, -0.28698346, 0.118432842, -0.196983278];
